# B&R Automation Studio project Panasonic_LinkaPowerCP2_A2021055 (part 2)

### IoMap.iom - 5PC900_TS17_00/IoMap.iom
```iecst
VAR_CONFIG
	Cyclic#1.P1_Pracovisko.IN.ModulWeidmuller_IO_KomOK AT %IX."P1_IOmodul_PowerlinkMaster".ModuleOk;
	Cyclic#1.P1_Pracovisko.IN.Robot_KomOK AT %IX."P1_Robot_IRB120_R1".ModuleOk;
	Cyclic#1.P1_Pracovisko.IN.Skrutkovacka_K30_KomOK AT %IX."P1_SkrutkovackaK30".ModuleOk;
	Cyclic#1.P1_Pracovisko.IN.Skrutkovacka_M5_KomOK AT %IX."P1_SkrutkovackaM5".ModuleOk;
	Cyclic#1.P1_Pracovisko.IN.Skrutkovacka_M4_KomOK AT %IX."P1_SkrutkovackaM4".ModuleOk;
	Cyclic#1.P1_Pracovisko.IN.ModulFesto_IO_KomOK AT %IX."P1_IOmaster".ModuleOk;
	Cyclic#1.::P1_Pracovisko.IN.SmartKamera3_KomOK AT %IX."P1_CAM_3".ModuleOk;
	Cyclic#1.P1_Pracovisko.IN.SmartKamera5_KomOK AT %IX."P1_CAM_5".ModuleOk;
	Cyclic#1.P1_Pracovisko.COM_Weidmuller.AB1_2_8DI AT %IB."P1_IOmodul_PowerlinkMaster".DigitalInput_I6000_S01;
	Cyclic#1.P1_Pracovisko.COM_Weidmuller.AB1_3_8DI AT %IB."P1_IOmodul_PowerlinkMaster".DigitalInput_I6000_S02;
	Cyclic#1.P1_Pracovisko.COM_Weidmuller.AB1_4_8DI AT %IB."P1_IOmodul_PowerlinkMaster".DigitalInput_I6000_S03;
	Cyclic#1.P1_Pracovisko.COM_Weidmuller.AB1_5_8DI AT %IB."P1_IOmodul_PowerlinkMaster".DigitalInput_I6000_S04;
	Cyclic#1.P1_Pracovisko.COM_Weidmuller.AB1_6_8DO AT %QB."P1_IOmodul_PowerlinkMaster".DigitalOutput_I6200_S01;
	Cyclic#1.P1_Pracovisko.COM_Weidmuller.AB1_7_8DO AT %QB."P1_IOmodul_PowerlinkMaster".DigitalOutput_I6200_S02;
	Cyclic#1.P1_Pracovisko.COM_Weidmuller.AB1_9_8DO AT %QB."P1_IOmodul_PowerlinkMaster".DigitalOutput_I6200_S03;
	Cyclic#1.P1_Pracovisko.COM_Weidmuller.AB1_10_8DO AT %QB."P1_IOmodul_PowerlinkMaster".DigitalOutput_I6200_S04;
	Cyclic#1.P1_Pracovisko.COM_Festo.DS1_1_Port0_IN[0] AT %IB."P1_IOmaster".Module007_Inputs001;
	Cyclic#1.P1_Pracovisko.COM_Festo.DS1_1_Port0_IN[1] AT %IB."P1_IOmaster".Module007_Inputs002;
	Cyclic#1.P1_Pracovisko.COM_Festo.DM1_1_4DI[0] AT %IX."P1_IOmaster".Module001_Bit_0_Bit_0;
	Cyclic#1.P1_Pracovisko.COM_Festo.DM1_1_4DI[1] AT %IX."P1_IOmaster".Module001_Bit_1_Bit_1;
	Cyclic#1.P1_Pracovisko.COM_Festo.DM1_1_4DI[2] AT %IX."P1_IOmaster".Module001_Bit_2_Bit_2;
	Cyclic#1.P1_Pracovisko.COM_Festo.DM1_1_4DI[3] AT %IX."P1_IOmaster".Module001_Bit_3_Bit_3;
	Cyclic#1.P1_Pracovisko.COM_Festo.DM1_1_4DO[0] AT %QX."P1_IOmaster".Module001_Bit_0_Bit_1;
	Cyclic#1.P1_Pracovisko.COM_Festo.DM1_1_4DO[1] AT %QX."P1_IOmaster".Module001_Bit_1_Bit_2;
	Cyclic#1.P1_Pracovisko.COM_Festo.DM1_1_4DO[2] AT %QX."P1_IOmaster".Module001_Bit_2_Bit_3;
	Cyclic#1.P1_Pracovisko.COM_Festo.DM1_1_4DO[3] AT %QX."P1_IOmaster".Module001_Bit_3_Bit_4;
	Cyclic#1.P1_Pracovisko.COM_Festo.DI1_1_8DI[0] AT %IX."P1_IOmaster".Module002_Bit_0_Bit_0;
	Cyclic#1.P1_Pracovisko.COM_Festo.DI1_1_8DI[1] AT %IX."P1_IOmaster".Module002_Bit_1_Bit_1;
	Cyclic#1.P1_Pracovisko.COM_Festo.DI1_1_8DI[2] AT %IX."P1_IOmaster".Module002_Bit_2_Bit_2;
	Cyclic#1.P1_Pracovisko.COM_Festo.DI1_1_8DI[3] AT %IX."P1_IOmaster".Module002_Bit_3_Bit_3;
	Cyclic#1.P1_Pracovisko.COM_Festo.DI1_1_8DI[4] AT %IX."P1_IOmaster".Module002_Bit_4_Bit_4;
	Cyclic#1.P1_Pracovisko.COM_Festo.DI1_1_8DI[5] AT %IX."P1_IOmaster".Module002_Bit_5_Bit_5;
	Cyclic#1.P1_Pracovisko.COM_Festo.DI1_1_8DI[6] AT %IX."P1_IOmaster".Module002_Bit_6_Bit_6;
	Cyclic#1.P1_Pracovisko.COM_Festo.DI1_1_8DI[7] AT %IX."P1_IOmaster".Module002_Bit_7_Bit_7;
	Cyclic#1.P1_Pracovisko.COM_Festo.DI1_5_8DI[0] AT %IX."P1_IOmaster".Module003_Bit_0_Bit_0;
	Cyclic#1.P1_Pracovisko.COM_Festo.DI1_5_8DI[1] AT %IX."P1_IOmaster".Module003_Bit_1_Bit_1;
	Cyclic#1.P1_Pracovisko.COM_Festo.DI1_5_8DI[2] AT %IX."P1_IOmaster".Module003_Bit_2_Bit_2;
	Cyclic#1.P1_Pracovisko.COM_Festo.DI1_5_8DI[3] AT %IX."P1_IOmaster".Module003_Bit_3_Bit_3;
	Cyclic#1.P1_Pracovisko.COM_Festo.DI1_5_8DI[4] AT %IX."P1_IOmaster".Module003_Bit_4_Bit_4;
	Cyclic#1.P1_Pracovisko.COM_Festo.DI1_5_8DI[5] AT %IX."P1_IOmaster".Module003_Bit_5_Bit_5;
	Cyclic#1.P1_Pracovisko.COM_Festo.DI1_5_8DI[6] AT %IX."P1_IOmaster".Module003_Bit_6_Bit_6;
	Cyclic#1.P1_Pracovisko.COM_Festo.DI1_5_8DI[7] AT %IX."P1_IOmaster".Module003_Bit_7_Bit_7;
	Cyclic#1.P1_Pracovisko.COM_Festo.DI1_3_8DI[0] AT %IX."P1_IOmaster".Module004_Bit_0_Bit_0;
	Cyclic#1.P1_Pracovisko.COM_Festo.DI1_3_8DI[1] AT %IX."P1_IOmaster".Module004_Bit_1_Bit_1;
	Cyclic#1.P1_Pracovisko.COM_Festo.DI1_3_8DI[2] AT %IX."P1_IOmaster".Module004_Bit_2_Bit_2;
	Cyclic#1.P1_Pracovisko.COM_Festo.DI1_3_8DI[3] AT %IX."P1_IOmaster".Module004_Bit_3_Bit_3;
	Cyclic#1.P1_Pracovisko.COM_Festo.DI1_3_8DI[4] AT %IX."P1_IOmaster".Module004_Bit_4_Bit_4;
	Cyclic#1.P1_Pracovisko.COM_Festo.DI1_3_8DI[5] AT %IX."P1_IOmaster".Module004_Bit_5_Bit_5;
	Cyclic#1.P1_Pracovisko.COM_Festo.DI1_3_8DI[6] AT %IX."P1_IOmaster".Module004_Bit_6_Bit_6;
	Cyclic#1.P1_Pracovisko.COM_Festo.DI1_3_8DI[7] AT %IX."P1_IOmaster".Module004_Bit_7_Bit_7;
	Cyclic#1.P1_Pracovisko.COM_Festo.DI1_4_8DI[0] AT %IX."P1_IOmaster".Module005_Bit_0_Bit_0;
	Cyclic#1.P1_Pracovisko.COM_Festo.DI1_4_8DI[1] AT %IX."P1_IOmaster".Module005_Bit_1_Bit_1;
	Cyclic#1.P1_Pracovisko.COM_Festo.DI1_4_8DI[2] AT %IX."P1_IOmaster".Module005_Bit_2_Bit_2;
	Cyclic#1.P1_Pracovisko.COM_Festo.DI1_4_8DI[3] AT %IX."P1_IOmaster".Module005_Bit_3_Bit_3;
	Cyclic#1.P1_Pracovisko.COM_Festo.DI1_4_8DI[4] AT %IX."P1_IOmaster".Module005_Bit_4_Bit_4;
	Cyclic#1.P1_Pracovisko.COM_Festo.DI1_4_8DI[5] AT %IX."P1_IOmaster".Module005_Bit_5_Bit_5;
	Cyclic#1.P1_Pracovisko.COM_Festo.DI1_4_8DI[6] AT %IX."P1_IOmaster".Module005_Bit_6_Bit_6;
	Cyclic#1.P1_Pracovisko.COM_Festo.DI1_4_8DI[7] AT %IX."P1_IOmaster".Module005_Bit_7_Bit_7;
	Cyclic#1.P1_Pracovisko.COM_Festo.DI1_2_8DI[0] AT %IX."P1_IOmaster".Module006_Bit_0_Bit_0;
	Cyclic#1.P1_Pracovisko.COM_Festo.DI1_2_8DI[1] AT %IX."P1_IOmaster".Module006_Bit_1_Bit_1;
	Cyclic#1.P1_Pracovisko.COM_Festo.DI1_2_8DI[2] AT %IX."P1_IOmaster".Module006_Bit_2_Bit_2;
	Cyclic#1.P1_Pracovisko.COM_Festo.DI1_2_8DI[3] AT %IX."P1_IOmaster".Module006_Bit_3_Bit_3;
	Cyclic#1.P1_Pracovisko.COM_Festo.DI1_2_8DI[4] AT %IX."P1_IOmaster".Module006_Bit_4_Bit_4;
	Cyclic#1.P1_Pracovisko.COM_Festo.DI1_2_8DI[5] AT %IX."P1_IOmaster".Module006_Bit_5_Bit_5;
	Cyclic#1.P1_Pracovisko.COM_Festo.DI1_2_8DI[6] AT %IX."P1_IOmaster".Module006_Bit_6_Bit_6;
	Cyclic#1.P1_Pracovisko.COM_Festo.DI1_2_8DI[7] AT %IX."P1_IOmaster".Module006_Bit_7_Bit_7;
	Cyclic#1.P1_Pracovisko.COM_Festo.DS1_1_Port0_OUT[0] AT %QB."P1_IOmaster".Module007_Outputs001;
	Cyclic#1.P1_Pracovisko.COM_Festo.DS1_1_Port0_OUT[1] AT %QB."P1_IOmaster".Module007_Outputs002;
	Cyclic#1.P1_Pracovisko.COM_Festo.DS1_1_Port1_IN[0] AT %IB."P1_IOmaster".Module007_Inputs003;
	Cyclic#1.P1_Pracovisko.COM_Festo.DS1_1_Port1_IN[1] AT %IB."P1_IOmaster".Module007_Inputs004;
	Cyclic#1.P1_Pracovisko.COM_Festo.DS1_1_Port1_IN[2] AT %IB."P1_IOmaster".Module007_Inputs005;
	Cyclic#1.P1_Pracovisko.COM_Festo.DS1_1_Port1_IN[3] AT %IB."P1_IOmaster".Module007_Inputs006;
	Cyclic#1.P1_Pracovisko.COM_Festo.DS1_1_Port1_IN[4] AT %IB."P1_IOmaster".Module007_Inputs007;
	Cyclic#1.P1_Pracovisko.COM_Festo.DS1_1_Port1_IN[5] AT %IB."P1_IOmaster".Module007_Inputs008;
	Cyclic#1.P1_Pracovisko.COM_Festo.DS1_1_Port1_IN[6] AT %IB."P1_IOmaster".Module007_Inputs009;
	Cyclic#1.P1_Pracovisko.COM_Festo.DS1_1_Port1_IN[7] AT %IB."P1_IOmaster".Module007_Inputs010;
	Cyclic#1.P1_Pracovisko.COM_Festo.DS1_1_Port1_IN[8] AT %IB."P1_IOmaster".Module007_Inputs011;
	Cyclic#1.P1_Pracovisko.COM_Festo.DS1_1_Port1_IN[9] AT %IB."P1_IOmaster".Module007_Inputs012;
	Cyclic#1.P1_Pracovisko.COM_Festo.DS1_1_Port1_IN[10] AT %IB."P1_IOmaster".Module007_Inputs013;
	Cyclic#1.P1_Pracovisko.COM_Festo.DS1_1_Port1_IN[11] AT %IB."P1_IOmaster".Module007_Inputs014;
	Cyclic#1.P1_Pracovisko.COM_Festo.DS1_1_Port1_IN[12] AT %IB."P1_IOmaster".Module007_Inputs015;
	Cyclic#1.P1_Pracovisko.COM_Festo.DS1_1_Port1_IN[13] AT %IB."P1_IOmaster".Module007_Inputs016;
	Cyclic#1.P1_Pracovisko.COM_Festo.DS1_1_Port1_IN[14] AT %IB."P1_IOmaster".Module007_Inputs017;
	Cyclic#1.P1_Pracovisko.COM_Festo.DS1_1_Port1_IN[15] AT %IB."P1_IOmaster".Module007_Inputs018;
	Cyclic#1.P1_Pracovisko.COM_Festo.DS1_1_Port1_OUT[0] AT %QB."P1_IOmaster".Module007_Outputs003;
	Cyclic#1.P1_Pracovisko.COM_Festo.DS1_1_Port1_OUT[1] AT %QB."P1_IOmaster".Module007_Outputs004;
	Cyclic#1.P1_Pracovisko.COM_Festo.DS1_1_Port1_OUT[2] AT %QB."P1_IOmaster".Module007_Outputs005;
	Cyclic#1.P1_Pracovisko.COM_Festo.DS1_1_Port1_OUT[3] AT %QB."P1_IOmaster".Module007_Outputs006;
	Cyclic#1.P1_Pracovisko.COM_Festo.DS1_1_Port1_OUT[4] AT %QB."P1_IOmaster".Module007_Outputs007;
	Cyclic#1.P1_Pracovisko.COM_Festo.DS1_1_Port1_OUT[5] AT %QB."P1_IOmaster".Module007_Outputs008;
	Cyclic#1.P1_Pracovisko.COM_Festo.DS1_1_Port1_OUT[6] AT %QB."P1_IOmaster".Module007_Outputs009;
	Cyclic#1.P1_Pracovisko.COM_Festo.DS1_1_Port1_OUT[7] AT %QB."P1_IOmaster".Module007_Outputs010;
	Cyclic#1.P1_Pracovisko.COM_Festo.DS1_1_Port1_OUT[8] AT %QB."P1_IOmaster".Module007_Outputs011;
	Cyclic#1.P1_Pracovisko.COM_Festo.DS1_1_Port1_OUT[9] AT %QB."P1_IOmaster".Module007_Outputs012;
	Cyclic#1.P1_Pracovisko.COM_Festo.DS1_1_Port1_OUT[10] AT %QB."P1_IOmaster".Module007_Outputs013;
	Cyclic#1.P1_Pracovisko.COM_Festo.DS1_1_Port1_OUT[11] AT %QB."P1_IOmaster".Module007_Outputs014;
	Cyclic#1.P1_Pracovisko.COM_Festo.DS1_1_Port1_OUT[12] AT %QB."P1_IOmaster".Module007_Outputs015;
	Cyclic#1.P1_Pracovisko.COM_Festo.DS1_1_Port1_OUT[13] AT %QB."P1_IOmaster".Module007_Outputs016;
	Cyclic#1.P1_Pracovisko.COM_Festo.DS1_1_Port1_OUT[14] AT %QB."P1_IOmaster".Module007_Outputs017;
	Cyclic#1.P1_Pracovisko.COM_Festo.DS1_1_Port1_OUT[15] AT %QB."P1_IOmaster".Module007_Outputs018;
	Cyclic#1.P1_Pracovisko.COM_Festo.DS1_1_Port2_IN[0] AT %IB."P1_IOmaster".Module007_Inputs019;
	Cyclic#1.P1_Pracovisko.COM_Festo.DS1_1_Port2_IN[1] AT %IB."P1_IOmaster".Module007_Inputs020;
	Cyclic#1.P1_Pracovisko.COM_Festo.DS1_1_Port2_IN[2] AT %IB."P1_IOmaster".Module007_Inputs021;
	Cyclic#1.P1_Pracovisko.COM_Festo.DS1_1_Port2_IN[3] AT %IB."P1_IOmaster".Module007_Inputs022;
	Cyclic#1.P1_Pracovisko.COM_Festo.DS1_1_Port2_IN[4] AT %IB."P1_IOmaster".Module007_Inputs023;
	Cyclic#1.P1_Pracovisko.COM_Festo.DS1_1_Port2_IN[5] AT %IB."P1_IOmaster".Module007_Inputs024;
	Cyclic#1.P1_Pracovisko.COM_Festo.DS1_1_Port2_IN[6] AT %IB."P1_IOmaster".Module007_Inputs025;
	Cyclic#1.P1_Pracovisko.COM_Festo.DS1_1_Port2_IN[7] AT %IB."P1_IOmaster".Module007_Inputs026;
	Cyclic#1.P1_Pracovisko.COM_Festo.DS1_1_Port2_IN[8] AT %IB."P1_IOmaster".Module007_Inputs027;
	Cyclic#1.P1_Pracovisko.COM_Festo.DS1_1_Port2_IN[9] AT %IB."P1_IOmaster".Module007_Inputs028;
	Cyclic#1.P1_Pracovisko.COM_Festo.DS1_1_Port2_IN[10] AT %IB."P1_IOmaster".Module007_Inputs029;
	Cyclic#1.P1_Pracovisko.COM_Festo.DS1_1_Port2_IN[11] AT %IB."P1_IOmaster".Module007_Inputs030;
	Cyclic#1.P1_Pracovisko.COM_Festo.DS1_1_Port2_IN[12] AT %IB."P1_IOmaster".Module007_Inputs031;
	Cyclic#1.P1_Pracovisko.COM_Festo.DS1_1_Port2_IN[13] AT %IB."P1_IOmaster".Module007_Inputs032;
	Cyclic#1.P1_Pracovisko.COM_Festo.DS1_1_Port2_IN[14] AT %IB."P1_IOmaster".Module007_Inputs033;
	Cyclic#1.P1_Pracovisko.COM_Festo.DS1_1_Port2_IN[15] AT %IB."P1_IOmaster".Module007_Inputs034;
	Cyclic#1.P1_Pracovisko.COM_Festo.DS1_1_Port2_IN[16] AT %IB."P1_IOmaster".Module007_Inputs035;
	Cyclic#1.P1_Pracovisko.COM_Festo.DS1_1_Port2_IN[17] AT %IB."P1_IOmaster".Module007_Inputs036;
	Cyclic#1.P1_Pracovisko.COM_Festo.DS1_1_Port2_IN[18] AT %IB."P1_IOmaster".Module007_Inputs037;
	Cyclic#1.P1_Pracovisko.COM_Festo.DS1_1_Port2_IN[19] AT %IB."P1_IOmaster".Module007_Inputs038;
	Cyclic#1.P1_Pracovisko.COM_Festo.DS1_1_Port2_IN[20] AT %IB."P1_IOmaster".Module007_Inputs039;
	Cyclic#1.P1_Pracovisko.COM_Festo.DS1_1_Port2_IN[21] AT %IB."P1_IOmaster".Module007_Inputs040;
	Cyclic#1.P1_Pracovisko.COM_Festo.DS1_1_Port2_IN[22] AT %IB."P1_IOmaster".Module007_Inputs041;
	Cyclic#1.P1_Pracovisko.COM_Festo.DS1_1_Port2_IN[23] AT %IB."P1_IOmaster".Module007_Inputs042;
	Cyclic#1.P1_Pracovisko.COM_Festo.DS1_1_Port2_IN[24] AT %IB."P1_IOmaster".Module007_Inputs043;
	Cyclic#1.P1_Pracovisko.COM_Festo.DS1_1_Port2_IN[25] AT %IB."P1_IOmaster".Module007_Inputs044;
	Cyclic#1.P1_Pracovisko.COM_Festo.DS1_1_Port2_IN[26] AT %IB."P1_IOmaster".Module007_Inputs045;
	Cyclic#1.P1_Pracovisko.COM_Festo.DS1_1_Port2_IN[27] AT %IB."P1_IOmaster".Module007_Inputs046;
	Cyclic#1.P1_Pracovisko.COM_Festo.DS1_1_Port2_IN[28] AT %IB."P1_IOmaster".Module007_Inputs047;
	Cyclic#1.P1_Pracovisko.COM_Festo.DS1_1_Port2_IN[29] AT %IB."P1_IOmaster".Module007_Inputs048;
	Cyclic#1.P1_Pracovisko.COM_Festo.DS1_1_Port2_IN[30] AT %IB."P1_IOmaster".Module007_Inputs049;
	Cyclic#1.P1_Pracovisko.COM_Festo.DS1_1_Port2_IN[31] AT %IB."P1_IOmaster".Module007_Inputs050;
	Cyclic#1.P1_Pracovisko.COM_Festo.DS1_1_Port2_OUT[0] AT %QB."P1_IOmaster".Module007_Outputs019;
	Cyclic#1.P1_Pracovisko.COM_Festo.DS1_1_Port2_OUT[1] AT %QB."P1_IOmaster".Module007_Outputs020;
	Cyclic#1.P1_Pracovisko.COM_Festo.DS1_1_Port2_OUT[2] AT %QB."P1_IOmaster".Module007_Outputs021;
	Cyclic#1.P1_Pracovisko.COM_Festo.DS1_1_Port2_OUT[3] AT %QB."P1_IOmaster".Module007_Outputs022;
	Cyclic#1.P1_Pracovisko.COM_Festo.DS1_1_Port2_OUT[4] AT %QB."P1_IOmaster".Module007_Outputs023;
	Cyclic#1.P1_Pracovisko.COM_Festo.DS1_1_Port2_OUT[5] AT %QB."P1_IOmaster".Module007_Outputs024;
	Cyclic#1.P1_Pracovisko.COM_Festo.DS1_1_Port2_OUT[6] AT %QB."P1_IOmaster".Module007_Outputs025;
	Cyclic#1.P1_Pracovisko.COM_Festo.DS1_1_Port2_OUT[7] AT %QB."P1_IOmaster".Module007_Outputs026;
	Cyclic#1.P1_Pracovisko.COM_Festo.DS1_1_Port2_OUT[8] AT %QB."P1_IOmaster".Module007_Outputs027;
	Cyclic#1.P1_Pracovisko.COM_Festo.DS1_1_Port2_OUT[9] AT %QB."P1_IOmaster".Module007_Outputs028;
	Cyclic#1.P1_Pracovisko.COM_Festo.DS1_1_Port2_OUT[10] AT %QB."P1_IOmaster".Module007_Outputs029;
	Cyclic#1.P1_Pracovisko.COM_Festo.DS1_1_Port2_OUT[11] AT %QB."P1_IOmaster".Module007_Outputs030;
	Cyclic#1.P1_Pracovisko.COM_Festo.DS1_1_Port2_OUT[12] AT %QB."P1_IOmaster".Module007_Outputs031;
	Cyclic#1.P1_Pracovisko.COM_Festo.DS1_1_Port2_OUT[13] AT %QB."P1_IOmaster".Module007_Outputs032;
	Cyclic#1.P1_Pracovisko.COM_Festo.DS1_1_Port2_OUT[14] AT %QB."P1_IOmaster".Module007_Outputs033;
	Cyclic#1.P1_Pracovisko.COM_Festo.DS1_1_Port2_OUT[15] AT %QB."P1_IOmaster".Module007_Outputs034;
	Cyclic#1.P1_Pracovisko.COM_Festo.DS1_1_Port2_OUT[16] AT %QB."P1_IOmaster".Module007_Outputs035;
	Cyclic#1.P1_Pracovisko.COM_Festo.DS1_1_Port2_OUT[17] AT %QB."P1_IOmaster".Module007_Outputs036;
	Cyclic#1.P1_Pracovisko.COM_Festo.DS1_1_Port2_OUT[18] AT %QB."P1_IOmaster".Module007_Outputs037;
	Cyclic#1.P1_Pracovisko.COM_Festo.DS1_1_Port2_OUT[19] AT %QB."P1_IOmaster".Module007_Outputs038;
	Cyclic#1.P1_Pracovisko.COM_Festo.DS1_1_Port2_OUT[20] AT %QB."P1_IOmaster".Module007_Outputs039;
	Cyclic#1.P1_Pracovisko.COM_Festo.DS1_1_Port2_OUT[21] AT %QB."P1_IOmaster".Module007_Outputs040;
	Cyclic#1.P1_Pracovisko.COM_Festo.DS1_1_Port2_OUT[22] AT %QB."P1_IOmaster".Module007_Outputs041;
	Cyclic#1.P1_Pracovisko.COM_Festo.DS1_1_Port2_OUT[23] AT %QB."P1_IOmaster".Module007_Outputs042;
	Cyclic#1.P1_Pracovisko.COM_Festo.DS1_1_Port2_OUT[24] AT %QB."P1_IOmaster".Module007_Outputs043;
	Cyclic#1.P1_Pracovisko.COM_Festo.DS1_1_Port2_OUT[25] AT %QB."P1_IOmaster".Module007_Outputs044;
	Cyclic#1.P1_Pracovisko.COM_Festo.DS1_1_Port2_OUT[26] AT %QB."P1_IOmaster".Module007_Outputs045;
	Cyclic#1.P1_Pracovisko.COM_Festo.DS1_1_Port2_OUT[27] AT %QB."P1_IOmaster".Module007_Outputs046;
	Cyclic#1.P1_Pracovisko.COM_Festo.DS1_1_Port2_OUT[28] AT %QB."P1_IOmaster".Module007_Outputs047;
	Cyclic#1.P1_Pracovisko.COM_Festo.DS1_1_Port2_OUT[29] AT %QB."P1_IOmaster".Module007_Outputs048;
	Cyclic#1.P1_Pracovisko.COM_Festo.DS1_1_Port2_OUT[30] AT %QB."P1_IOmaster".Module007_Outputs049;
	Cyclic#1.P1_Pracovisko.COM_Festo.DS1_1_Port2_OUT[31] AT %QB."P1_IOmaster".Module007_Outputs050;
	Cyclic#1.P1_Pracovisko.COM_Festo.DS1_1_Port3_IN[0] AT %IB."P1_IOmaster".Module007_Inputs051;
	Cyclic#1.P1_Pracovisko.COM_Festo.DS1_1_Port3_IN[1] AT %IB."P1_IOmaster".Module007_Inputs052;
	Cyclic#1.P1_Pracovisko.COM_Festo.DS1_1_Port3_IN[2] AT %IB."P1_IOmaster".Module007_Inputs053;
	Cyclic#1.P1_Pracovisko.COM_Festo.DS1_1_Port3_IN[3] AT %IB."P1_IOmaster".Module007_Inputs054;
	Cyclic#1.P1_Pracovisko.COM_Festo.DS1_1_Port3_IN[4] AT %IB."P1_IOmaster".Module007_Inputs055;
	Cyclic#1.P1_Pracovisko.COM_Festo.DS1_1_Port3_IN[5] AT %IB."P1_IOmaster".Module007_Inputs056;
	Cyclic#1.P1_Pracovisko.COM_Festo.DS1_1_Port3_IN[6] AT %IB."P1_IOmaster".Module007_Inputs057;
	Cyclic#1.P1_Pracovisko.COM_Festo.DS1_1_Port3_IN[7] AT %IB."P1_IOmaster".Module007_Inputs058;
	Cyclic#1.P1_Pracovisko.COM_Festo.DS1_1_Port3_IN[8] AT %IB."P1_IOmaster".Module007_Inputs059;
	Cyclic#1.P1_Pracovisko.COM_Festo.DS1_1_Port3_IN[9] AT %IB."P1_IOmaster".Module007_Inputs060;
	Cyclic#1.P1_Pracovisko.COM_Festo.DS1_1_Port3_IN[10] AT %IB."P1_IOmaster".Module007_Inputs061;
	Cyclic#1.P1_Pracovisko.COM_Festo.DS1_1_Port3_IN[11] AT %IB."P1_IOmaster".Module007_Inputs062;
	Cyclic#1.P1_Pracovisko.COM_Festo.DS1_1_Port3_IN[12] AT %IB."P1_IOmaster".Module007_Inputs063;
	Cyclic#1.P1_Pracovisko.COM_Festo.DS1_1_Port3_IN[13] AT %IB."P1_IOmaster".Module007_Inputs064;
	Cyclic#1.P1_Pracovisko.COM_Festo.DS1_1_Port3_IN[14] AT %IB."P1_IOmaster".Module007_Inputs065;
	Cyclic#1.P1_Pracovisko.COM_Festo.DS1_1_Port3_IN[15] AT %IB."P1_IOmaster".Module007_Inputs066;
	Cyclic#1.P1_Pracovisko.COM_Festo.DS1_1_Port3_IN[16] AT %IB."P1_IOmaster".Module007_Inputs067;
	Cyclic#1.P1_Pracovisko.COM_Festo.DS1_1_Port3_IN[17] AT %IB."P1_IOmaster".Module007_Inputs068;
	Cyclic#1.P1_Pracovisko.COM_Festo.DS1_1_Port3_IN[18] AT %IB."P1_IOmaster".Module007_Inputs069;
	Cyclic#1.P1_Pracovisko.COM_Festo.DS1_1_Port3_IN[19] AT %IB."P1_IOmaster".Module007_Inputs070;
	Cyclic#1.P1_Pracovisko.COM_Festo.DS1_1_Port3_IN[20] AT %IB."P1_IOmaster".Module007_Inputs071;
	Cyclic#1.P1_Pracovisko.COM_Festo.DS1_1_Port3_IN[21] AT %IB."P1_IOmaster".Module007_Inputs072;
	Cyclic#1.P1_Pracovisko.COM_Festo.DS1_1_Port3_IN[22] AT %IB."P1_IOmaster".Module007_Inputs073;
	Cyclic#1.P1_Pracovisko.COM_Festo.DS1_1_Port3_IN[23] AT %IB."P1_IOmaster".Module007_Inputs074;
	Cyclic#1.P1_Pracovisko.COM_Festo.DS1_1_Port3_IN[24] AT %IB."P1_IOmaster".Module007_Inputs075;
	Cyclic#1.P1_Pracovisko.COM_Festo.DS1_1_Port3_IN[25] AT %IB."P1_IOmaster".Module007_Inputs076;
	Cyclic#1.P1_Pracovisko.COM_Festo.DS1_1_Port3_IN[26] AT %IB."P1_IOmaster".Module007_Inputs077;
	Cyclic#1.P1_Pracovisko.COM_Festo.DS1_1_Port3_IN[27] AT %IB."P1_IOmaster".Module007_Inputs078;
	Cyclic#1.P1_Pracovisko.COM_Festo.DS1_1_Port3_IN[28] AT %IB."P1_IOmaster".Module007_Inputs079;
	Cyclic#1.P1_Pracovisko.COM_Festo.DS1_1_Port3_IN[29] AT %IB."P1_IOmaster".Module007_Inputs080;
	Cyclic#1.P1_Pracovisko.COM_Festo.DS1_1_Port3_IN[30] AT %IB."P1_IOmaster".Module007_Inputs081;
	Cyclic#1.P1_Pracovisko.COM_Festo.DS1_1_Port3_IN[31] AT %IB."P1_IOmaster".Module007_Inputs082;
	Cyclic#1.P1_Pracovisko.COM_Festo.DS1_1_Port3_OUT[0] AT %QB."P1_IOmaster".Module007_Outputs051;
	Cyclic#1.P1_Pracovisko.COM_Festo.DS1_1_Port3_OUT[1] AT %QB."P1_IOmaster".Module007_Outputs052;
	Cyclic#1.P1_Pracovisko.COM_Festo.DS1_1_Port3_OUT[2] AT %QB."P1_IOmaster".Module007_Outputs053;
	Cyclic#1.P1_Pracovisko.COM_Festo.DS1_1_Port3_OUT[3] AT %QB."P1_IOmaster".Module007_Outputs054;
	Cyclic#1.P1_Pracovisko.COM_Festo.DS1_1_Port3_OUT[4] AT %QB."P1_IOmaster".Module007_Outputs055;
	Cyclic#1.P1_Pracovisko.COM_Festo.DS1_1_Port3_OUT[5] AT %QB."P1_IOmaster".Module007_Outputs056;
	Cyclic#1.P1_Pracovisko.COM_Festo.DS1_1_Port3_OUT[6] AT %QB."P1_IOmaster".Module007_Outputs057;
	Cyclic#1.P1_Pracovisko.COM_Festo.DS1_1_Port3_OUT[7] AT %QB."P1_IOmaster".Module007_Outputs058;
	Cyclic#1.P1_Pracovisko.COM_Festo.DS1_1_Port3_OUT[8] AT %QB."P1_IOmaster".Module007_Outputs059;
	Cyclic#1.P1_Pracovisko.COM_Festo.DS1_1_Port3_OUT[9] AT %QB."P1_IOmaster".Module007_Outputs060;
	Cyclic#1.P1_Pracovisko.COM_Festo.DS1_1_Port3_OUT[10] AT %QB."P1_IOmaster".Module007_Outputs061;
	Cyclic#1.P1_Pracovisko.COM_Festo.DS1_1_Port3_OUT[11] AT %QB."P1_IOmaster".Module007_Outputs062;
	Cyclic#1.P1_Pracovisko.COM_Festo.DS1_1_Port3_OUT[12] AT %QB."P1_IOmaster".Module007_Outputs063;
	Cyclic#1.P1_Pracovisko.COM_Festo.DS1_1_Port3_OUT[13] AT %QB."P1_IOmaster".Module007_Outputs064;
	Cyclic#1.P1_Pracovisko.COM_Festo.DS1_1_Port3_OUT[14] AT %QB."P1_IOmaster".Module007_Outputs065;
	Cyclic#1.P1_Pracovisko.COM_Festo.DS1_1_Port3_OUT[15] AT %QB."P1_IOmaster".Module007_Outputs066;
	Cyclic#1.P1_Pracovisko.COM_Festo.DS1_1_Port3_OUT[16] AT %QB."P1_IOmaster".Module007_Outputs067;
	Cyclic#1.P1_Pracovisko.COM_Festo.DS1_1_Port3_OUT[17] AT %QB."P1_IOmaster".Module007_Outputs068;
	Cyclic#1.P1_Pracovisko.COM_Festo.DS1_1_Port3_OUT[18] AT %QB."P1_IOmaster".Module007_Outputs069;
	Cyclic#1.P1_Pracovisko.COM_Festo.DS1_1_Port3_OUT[19] AT %QB."P1_IOmaster".Module007_Outputs070;
	Cyclic#1.P1_Pracovisko.COM_Festo.DS1_1_Port3_OUT[20] AT %QB."P1_IOmaster".Module007_Outputs071;
	Cyclic#1.P1_Pracovisko.COM_Festo.DS1_1_Port3_OUT[21] AT %QB."P1_IOmaster".Module007_Outputs072;
	Cyclic#1.P1_Pracovisko.COM_Festo.DS1_1_Port3_OUT[22] AT %QB."P1_IOmaster".Module007_Outputs073;
	Cyclic#1.P1_Pracovisko.COM_Festo.DS1_1_Port3_OUT[23] AT %QB."P1_IOmaster".Module007_Outputs074;
	Cyclic#1.P1_Pracovisko.COM_Festo.DS1_1_Port3_OUT[24] AT %QB."P1_IOmaster".Module007_Outputs075;
	Cyclic#1.P1_Pracovisko.COM_Festo.DS1_1_Port3_OUT[25] AT %QB."P1_IOmaster".Module007_Outputs076;
	Cyclic#1.P1_Pracovisko.COM_Festo.DS1_1_Port3_OUT[26] AT %QB."P1_IOmaster".Module007_Outputs077;
	Cyclic#1.P1_Pracovisko.COM_Festo.DS1_1_Port3_OUT[27] AT %QB."P1_IOmaster".Module007_Outputs078;
	Cyclic#1.P1_Pracovisko.COM_Festo.DS1_1_Port3_OUT[28] AT %QB."P1_IOmaster".Module007_Outputs079;
	Cyclic#1.P1_Pracovisko.COM_Festo.DS1_1_Port3_OUT[29] AT %QB."P1_IOmaster".Module007_Outputs080;
	Cyclic#1.P1_Pracovisko.COM_Festo.DS1_1_Port3_OUT[30] AT %QB."P1_IOmaster".Module007_Outputs081;
	Cyclic#1.P1_Pracovisko.COM_Festo.DS1_1_Port3_OUT[31] AT %QB."P1_IOmaster".Module007_Outputs082;
	Cyclic#1.P1_Pracovisko.COM_Festo.DS1_2_Port0_IN[0] AT %IB."P1_IOmaster".Module008_Inputs001;
	Cyclic#1.P1_Pracovisko.COM_Festo.DS1_2_Port0_IN[1] AT %IB."P1_IOmaster".Module008_Inputs002;
	Cyclic#1.P1_Pracovisko.COM_Festo.DS1_2_Port0_OUT[0] AT %QB."P1_IOmaster".Module008_Outputs001;
	Cyclic#1.P1_Pracovisko.COM_Festo.DS1_2_Port0_OUT[1] AT %QB."P1_IOmaster".Module008_Outputs002;
	Cyclic#1.P3_Pracovisko.IN.ModulWeidmuller_IO_KomOK AT %IX."P3_IOmodul_PowerlinkMaster".ModuleOk;
	Cyclic#1.P3_Pracovisko.COM_Weidmuller.AB3_5_8DI AT %IB."P3_IOmodul_PowerlinkMaster".DigitalInput_I6000_S01;
	Cyclic#1.P3_Pracovisko.COM_Weidmuller.AB3_6_8DI AT %IB."P3_IOmodul_PowerlinkMaster".DigitalInput_I6000_S02;
	Cyclic#1.P3_Pracovisko.COM_Weidmuller.AB3_7_8DI AT %IB."P3_IOmodul_PowerlinkMaster".DigitalInput_I6000_S03;
	Cyclic#1.P3_Pracovisko.COM_Weidmuller.AB3_8_8DI AT %IB."P3_IOmodul_PowerlinkMaster".DigitalInput_I6000_S04;
	Cyclic#1.P3_Pracovisko.COM_Weidmuller.AB3_9_8DO AT %QB."P3_IOmodul_PowerlinkMaster".DigitalOutput_I6200_S01;
	Cyclic#1.P3_Pracovisko.COM_Weidmuller.AB3_10_8DO AT %QB."P3_IOmodul_PowerlinkMaster".DigitalOutput_I6200_S02;
	Cyclic#1.P3_Pracovisko.COM_Weidmuller.AB3_12_8DO AT %QB."P3_IOmodul_PowerlinkMaster".DigitalOutput_I6200_S03;
	Cyclic#1.P1_Robot.COM_IN.BYTE_IN[0] AT %IB."P1_Robot_IRB120_R1".Module001_Input_0;
	Cyclic#1.P1_Robot.COM_IN.BYTE_IN[1] AT %IB."P1_Robot_IRB120_R1".Module001_Input_1;
	Cyclic#1.P1_Robot.COM_IN.BYTE_IN[2] AT %IB."P1_Robot_IRB120_R1".Module001_Input_2;
	Cyclic#1.P1_Robot.COM_IN.BYTE_IN[3] AT %IB."P1_Robot_IRB120_R1".Module001_Input_3;
	Cyclic#1.P1_Robot.COM_IN.BYTE_IN[4] AT %IB."P1_Robot_IRB120_R1".Module001_Input_4;
	Cyclic#1.P1_Robot.COM_IN.BYTE_IN[5] AT %IB."P1_Robot_IRB120_R1".Module001_Input_5;
	Cyclic#1.P1_Robot.COM_IN.BYTE_IN[6] AT %IB."P1_Robot_IRB120_R1".Module001_Input_6;
	Cyclic#1.P1_Robot.COM_IN.BYTE_IN[7] AT %IB."P1_Robot_IRB120_R1".Module001_Input_7;
	Cyclic#1.P1_Robot.COM_IN.BYTE_IN[8] AT %IB."P1_Robot_IRB120_R1".Module001_Input_8;
	Cyclic#1.P1_Robot.COM_IN.BYTE_IN[9] AT %IB."P1_Robot_IRB120_R1".Module001_Input_9;
	Cyclic#1.P1_Robot.COM_IN.BYTE_IN[10] AT %IB."P1_Robot_IRB120_R1".Module001_Input_10;
	Cyclic#1.P1_Robot.COM_IN.BYTE_IN[11] AT %IB."P1_Robot_IRB120_R1".Module001_Input_11;
	Cyclic#1.P1_Robot.COM_IN.BYTE_IN[12] AT %IB."P1_Robot_IRB120_R1".Module001_Input_12;
	Cyclic#1.P1_Robot.COM_IN.BYTE_IN[13] AT %IB."P1_Robot_IRB120_R1".Module001_Input_13;
	Cyclic#1.P1_Robot.COM_IN.BYTE_IN[14] AT %IB."P1_Robot_IRB120_R1".Module001_Input_14;
	Cyclic#1.P1_Robot.COM_IN.BYTE_IN[15] AT %IB."P1_Robot_IRB120_R1".Module001_Input_15;
	Cyclic#1.P1_Robot.COM_IN.BYTE_IN[16] AT %IB."P1_Robot_IRB120_R1".Module001_Input_16;
	Cyclic#1.P1_Robot.COM_IN.BYTE_IN[17] AT %IB."P1_Robot_IRB120_R1".Module001_Input_17;
	Cyclic#1.P1_Robot.COM_IN.BYTE_IN[18] AT %IB."P1_Robot_IRB120_R1".Module001_Input_18;
	Cyclic#1.P1_Robot.COM_IN.BYTE_IN[19] AT %IB."P1_Robot_IRB120_R1".Module001_Input_19;
	Cyclic#1.P1_Robot.COM_IN.BYTE_IN[20] AT %IB."P1_Robot_IRB120_R1".Module001_Input_20;
	Cyclic#1.P1_Robot.COM_IN.BYTE_IN[21] AT %IB."P1_Robot_IRB120_R1".Module001_Input_21;
	Cyclic#1.P1_Robot.COM_IN.BYTE_IN[22] AT %IB."P1_Robot_IRB120_R1".Module001_Input_22;
	Cyclic#1.P1_Robot.COM_IN.BYTE_IN[23] AT %IB."P1_Robot_IRB120_R1".Module001_Input_23;
	Cyclic#1.P1_Robot.COM_IN.BYTE_IN[24] AT %IB."P1_Robot_IRB120_R1".Module001_Input_24;
	Cyclic#1.P1_Robot.COM_IN.BYTE_IN[25] AT %IB."P1_Robot_IRB120_R1".Module001_Input_25;
	Cyclic#1.P1_Robot.COM_IN.BYTE_IN[26] AT %IB."P1_Robot_IRB120_R1".Module001_Input_26;
	Cyclic#1.P1_Robot.COM_IN.BYTE_IN[27] AT %IB."P1_Robot_IRB120_R1".Module001_Input_27;
	Cyclic#1.P1_Robot.COM_IN.BYTE_IN[28] AT %IB."P1_Robot_IRB120_R1".Module001_Input_28;
	Cyclic#1.P1_Robot.COM_IN.BYTE_IN[29] AT %IB."P1_Robot_IRB120_R1".Module001_Input_29;
	Cyclic#1.P1_Robot.COM_IN.BYTE_IN[30] AT %IB."P1_Robot_IRB120_R1".Module001_Input_30;
	Cyclic#1.P1_Robot.COM_IN.BYTE_IN[31] AT %IB."P1_Robot_IRB120_R1".Module001_Input_31;
	Cyclic#1.P1_Robot.COM_IN.BYTE_IN[32] AT %IB."P1_Robot_IRB120_R1".Module001_Input_32;
	Cyclic#1.P1_Robot.COM_IN.BYTE_IN[33] AT %IB."P1_Robot_IRB120_R1".Module001_Input_33;
	Cyclic#1.P1_Robot.COM_IN.BYTE_IN[34] AT %IB."P1_Robot_IRB120_R1".Module001_Input_34;
	Cyclic#1.P1_Robot.COM_IN.BYTE_IN[35] AT %IB."P1_Robot_IRB120_R1".Module001_Input_35;
	Cyclic#1.P1_Robot.COM_IN.BYTE_IN[36] AT %IB."P1_Robot_IRB120_R1".Module001_Input_36;
	Cyclic#1.P1_Robot.COM_IN.BYTE_IN[37] AT %IB."P1_Robot_IRB120_R1".Module001_Input_37;
	Cyclic#1.P1_Robot.COM_IN.BYTE_IN[38] AT %IB."P1_Robot_IRB120_R1".Module001_Input_38;
	Cyclic#1.P1_Robot.COM_IN.BYTE_IN[39] AT %IB."P1_Robot_IRB120_R1".Module001_Input_39;
	Cyclic#1.P1_Robot.COM_IN.BYTE_IN[40] AT %IB."P1_Robot_IRB120_R1".Module001_Input_40;
	Cyclic#1.P1_Robot.COM_IN.BYTE_IN[41] AT %IB."P1_Robot_IRB120_R1".Module001_Input_41;
	Cyclic#1.P1_Robot.COM_IN.BYTE_IN[42] AT %IB."P1_Robot_IRB120_R1".Module001_Input_42;
	Cyclic#1.P1_Robot.COM_IN.BYTE_IN[43] AT %IB."P1_Robot_IRB120_R1".Module001_Input_43;
	Cyclic#1.P1_Robot.COM_IN.BYTE_IN[44] AT %IB."P1_Robot_IRB120_R1".Module001_Input_44;
	Cyclic#1.P1_Robot.COM_IN.BYTE_IN[45] AT %IB."P1_Robot_IRB120_R1".Module001_Input_45;
	Cyclic#1.P1_Robot.COM_IN.BYTE_IN[46] AT %IB."P1_Robot_IRB120_R1".Module001_Input_46;
	Cyclic#1.P1_Robot.COM_IN.BYTE_IN[47] AT %IB."P1_Robot_IRB120_R1".Module001_Input_47;
	Cyclic#1.P1_Robot.COM_IN.BYTE_IN[48] AT %IB."P1_Robot_IRB120_R1".Module001_Input_48;
	Cyclic#1.P1_Robot.COM_IN.BYTE_IN[49] AT %IB."P1_Robot_IRB120_R1".Module001_Input_49;
	Cyclic#1.P1_Robot.COM_IN.BYTE_IN[50] AT %IB."P1_Robot_IRB120_R1".Module001_Input_50;
	Cyclic#1.P1_Robot.COM_IN.BYTE_IN[51] AT %IB."P1_Robot_IRB120_R1".Module001_Input_51;
	Cyclic#1.P1_Robot.COM_IN.BYTE_IN[52] AT %IB."P1_Robot_IRB120_R1".Module001_Input_52;
	Cyclic#1.P1_Robot.COM_IN.BYTE_IN[53] AT %IB."P1_Robot_IRB120_R1".Module001_Input_53;
	Cyclic#1.P1_Robot.COM_IN.BYTE_IN[54] AT %IB."P1_Robot_IRB120_R1".Module001_Input_54;
	Cyclic#1.P1_Robot.COM_IN.BYTE_IN[55] AT %IB."P1_Robot_IRB120_R1".Module001_Input_55;
	Cyclic#1.P1_Robot.COM_IN.BYTE_IN[56] AT %IB."P1_Robot_IRB120_R1".Module001_Input_56;
	Cyclic#1.P1_Robot.COM_IN.BYTE_IN[57] AT %IB."P1_Robot_IRB120_R1".Module001_Input_57;
	Cyclic#1.P1_Robot.COM_IN.BYTE_IN[58] AT %IB."P1_Robot_IRB120_R1".Module001_Input_58;
	Cyclic#1.P1_Robot.COM_IN.BYTE_IN[59] AT %IB."P1_Robot_IRB120_R1".Module001_Input_59;
	Cyclic#1.P1_Robot.COM_IN.BYTE_IN[60] AT %IB."P1_Robot_IRB120_R1".Module001_Input_60;
	Cyclic#1.P1_Robot.COM_IN.BYTE_IN[61] AT %IB."P1_Robot_IRB120_R1".Module001_Input_61;
	Cyclic#1.P1_Robot.COM_IN.BYTE_IN[62] AT %IB."P1_Robot_IRB120_R1".Module001_Input_62;
	Cyclic#1.P1_Robot.COM_IN.BYTE_IN[63] AT %IB."P1_Robot_IRB120_R1".Module001_Input_63;
	Cyclic#1.P1_Robot.COM_OUT.BYTE_OUT[0] AT %QB."P1_Robot_IRB120_R1".Module002_Output_0;
	Cyclic#1.P1_Robot.COM_OUT.BYTE_OUT[1] AT %QB."P1_Robot_IRB120_R1".Module002_Output_1;
	Cyclic#1.P1_Robot.COM_OUT.BYTE_OUT[2] AT %QB."P1_Robot_IRB120_R1".Module002_Output_2;
	Cyclic#1.P1_Robot.COM_OUT.BYTE_OUT[3] AT %QB."P1_Robot_IRB120_R1".Module002_Output_3;
	Cyclic#1.P1_Robot.COM_OUT.BYTE_OUT[4] AT %QB."P1_Robot_IRB120_R1".Module002_Output_4;
	Cyclic#1.P1_Robot.COM_OUT.BYTE_OUT[5] AT %QB."P1_Robot_IRB120_R1".Module002_Output_5;
	Cyclic#1.P1_Robot.COM_OUT.BYTE_OUT[6] AT %QB."P1_Robot_IRB120_R1".Module002_Output_6;
	Cyclic#1.P1_Robot.COM_OUT.BYTE_OUT[7] AT %QB."P1_Robot_IRB120_R1".Module002_Output_7;
	Cyclic#1.P1_Robot.COM_OUT.BYTE_OUT[8] AT %QB."P1_Robot_IRB120_R1".Module002_Output_8;
	Cyclic#1.P1_Robot.COM_OUT.BYTE_OUT[9] AT %QB."P1_Robot_IRB120_R1".Module002_Output_9;
	Cyclic#1.P1_Robot.COM_OUT.BYTE_OUT[10] AT %QB."P1_Robot_IRB120_R1".Module002_Output_10;
	Cyclic#1.P1_Robot.COM_OUT.BYTE_OUT[11] AT %QB."P1_Robot_IRB120_R1".Module002_Output_11;
	Cyclic#1.P1_Robot.COM_OUT.BYTE_OUT[12] AT %QB."P1_Robot_IRB120_R1".Module002_Output_12;
	Cyclic#1.P1_Robot.COM_OUT.BYTE_OUT[13] AT %QB."P1_Robot_IRB120_R1".Module002_Output_13;
	Cyclic#1.P1_Robot.COM_OUT.BYTE_OUT[14] AT %QB."P1_Robot_IRB120_R1".Module002_Output_14;
	Cyclic#1.P1_Robot.COM_OUT.BYTE_OUT[15] AT %QB."P1_Robot_IRB120_R1".Module002_Output_15;
	Cyclic#1.P1_Robot.COM_OUT.BYTE_OUT[16] AT %QB."P1_Robot_IRB120_R1".Module002_Output_16;
	Cyclic#1.P1_Robot.COM_OUT.BYTE_OUT[17] AT %QB."P1_Robot_IRB120_R1".Module002_Output_17;
	Cyclic#1.P1_Robot.COM_OUT.BYTE_OUT[18] AT %QB."P1_Robot_IRB120_R1".Module002_Output_18;
	Cyclic#1.P1_Robot.COM_OUT.BYTE_OUT[19] AT %QB."P1_Robot_IRB120_R1".Module002_Output_19;
	Cyclic#1.P1_Robot.COM_OUT.BYTE_OUT[20] AT %QB."P1_Robot_IRB120_R1".Module002_Output_20;
	Cyclic#1.P1_Robot.COM_OUT.BYTE_OUT[21] AT %QB."P1_Robot_IRB120_R1".Module002_Output_21;
	Cyclic#1.P1_Robot.COM_OUT.BYTE_OUT[22] AT %QB."P1_Robot_IRB120_R1".Module002_Output_22;
	Cyclic#1.P1_Robot.COM_OUT.BYTE_OUT[23] AT %QB."P1_Robot_IRB120_R1".Module002_Output_23;
	Cyclic#1.P1_Robot.COM_OUT.BYTE_OUT[24] AT %QB."P1_Robot_IRB120_R1".Module002_Output_24;
	Cyclic#1.P1_Robot.COM_OUT.BYTE_OUT[25] AT %QB."P1_Robot_IRB120_R1".Module002_Output_25;
	Cyclic#1.P1_Robot.COM_OUT.BYTE_OUT[26] AT %QB."P1_Robot_IRB120_R1".Module002_Output_26;
	Cyclic#1.P1_Robot.COM_OUT.BYTE_OUT[27] AT %QB."P1_Robot_IRB120_R1".Module002_Output_27;
	Cyclic#1.P1_Robot.COM_OUT.BYTE_OUT[28] AT %QB."P1_Robot_IRB120_R1".Module002_Output_28;
	Cyclic#1.P1_Robot.COM_OUT.BYTE_OUT[29] AT %QB."P1_Robot_IRB120_R1".Module002_Output_29;
	Cyclic#1.P1_Robot.COM_OUT.BYTE_OUT[30] AT %QB."P1_Robot_IRB120_R1".Module002_Output_30;
	Cyclic#1.P1_Robot.COM_OUT.BYTE_OUT[31] AT %QB."P1_Robot_IRB120_R1".Module002_Output_31;
	Cyclic#1.P1_Robot.COM_OUT.BYTE_OUT[32] AT %QB."P1_Robot_IRB120_R1".Module002_Output_32;
	Cyclic#1.P1_Robot.COM_OUT.BYTE_OUT[33] AT %QB."P1_Robot_IRB120_R1".Module002_Output_33;
	Cyclic#1.P1_Robot.COM_OUT.BYTE_OUT[34] AT %QB."P1_Robot_IRB120_R1".Module002_Output_34;
	Cyclic#1.P1_Robot.COM_OUT.BYTE_OUT[35] AT %QB."P1_Robot_IRB120_R1".Module002_Output_35;
	Cyclic#1.P1_Robot.COM_OUT.BYTE_OUT[36] AT %QB."P1_Robot_IRB120_R1".Module002_Output_36;
	Cyclic#1.P1_Robot.COM_OUT.BYTE_OUT[37] AT %QB."P1_Robot_IRB120_R1".Module002_Output_37;
	Cyclic#1.P1_Robot.COM_OUT.BYTE_OUT[38] AT %QB."P1_Robot_IRB120_R1".Module002_Output_38;
	Cyclic#1.P1_Robot.COM_OUT.BYTE_OUT[39] AT %QB."P1_Robot_IRB120_R1".Module002_Output_39;
	Cyclic#1.P1_Robot.COM_OUT.BYTE_OUT[40] AT %QB."P1_Robot_IRB120_R1".Module002_Output_40;
	Cyclic#1.P1_Robot.COM_OUT.BYTE_OUT[41] AT %QB."P1_Robot_IRB120_R1".Module002_Output_41;
	Cyclic#1.P1_Robot.COM_OUT.BYTE_OUT[42] AT %QB."P1_Robot_IRB120_R1".Module002_Output_42;
	Cyclic#1.P1_Robot.COM_OUT.BYTE_OUT[43] AT %QB."P1_Robot_IRB120_R1".Module002_Output_43;
	Cyclic#1.P1_Robot.COM_OUT.BYTE_OUT[44] AT %QB."P1_Robot_IRB120_R1".Module002_Output_44;
	Cyclic#1.P1_Robot.COM_OUT.BYTE_OUT[45] AT %QB."P1_Robot_IRB120_R1".Module002_Output_45;
	Cyclic#1.P1_Robot.COM_OUT.BYTE_OUT[46] AT %QB."P1_Robot_IRB120_R1".Module002_Output_46;
	Cyclic#1.P1_Robot.COM_OUT.BYTE_OUT[47] AT %QB."P1_Robot_IRB120_R1".Module002_Output_47;
	Cyclic#1.P1_Robot.COM_OUT.BYTE_OUT[48] AT %QB."P1_Robot_IRB120_R1".Module002_Output_48;
	Cyclic#1.P1_Robot.COM_OUT.BYTE_OUT[49] AT %QB."P1_Robot_IRB120_R1".Module002_Output_49;
	Cyclic#1.P1_Robot.COM_OUT.BYTE_OUT[50] AT %QB."P1_Robot_IRB120_R1".Module002_Output_50;
	Cyclic#1.P1_Robot.COM_OUT.BYTE_OUT[51] AT %QB."P1_Robot_IRB120_R1".Module002_Output_51;
	Cyclic#1.P1_Robot.COM_OUT.BYTE_OUT[52] AT %QB."P1_Robot_IRB120_R1".Module002_Output_52;
	Cyclic#1.P1_Robot.COM_OUT.BYTE_OUT[53] AT %QB."P1_Robot_IRB120_R1".Module002_Output_53;
	Cyclic#1.P1_Robot.COM_OUT.BYTE_OUT[54] AT %QB."P1_Robot_IRB120_R1".Module002_Output_54;
	Cyclic#1.P1_Robot.COM_OUT.BYTE_OUT[55] AT %QB."P1_Robot_IRB120_R1".Module002_Output_55;
	Cyclic#1.P1_Robot.COM_OUT.BYTE_OUT[56] AT %QB."P1_Robot_IRB120_R1".Module002_Output_56;
	Cyclic#1.P1_Robot.COM_OUT.BYTE_OUT[57] AT %QB."P1_Robot_IRB120_R1".Module002_Output_57;
	Cyclic#1.P1_Robot.COM_OUT.BYTE_OUT[58] AT %QB."P1_Robot_IRB120_R1".Module002_Output_58;
	Cyclic#1.P1_Robot.COM_OUT.BYTE_OUT[59] AT %QB."P1_Robot_IRB120_R1".Module002_Output_59;
	Cyclic#1.P1_Robot.COM_OUT.BYTE_OUT[60] AT %QB."P1_Robot_IRB120_R1".Module002_Output_60;
	Cyclic#1.P1_Robot.COM_OUT.BYTE_OUT[61] AT %QB."P1_Robot_IRB120_R1".Module002_Output_61;
	Cyclic#1.P1_Robot.COM_OUT.BYTE_OUT[62] AT %QB."P1_Robot_IRB120_R1".Module002_Output_62;
	Cyclic#1.P1_Robot.COM_OUT.BYTE_OUT[63] AT %QB."P1_Robot_IRB120_R1".Module002_Output_63;
	Cyclic#1.P1_Srobovanie.PAR.K30_AtlasCopcoInputs[0] AT %ID."P1_SkrutkovackaK30".Module001_Input_I_00;
	Cyclic#1.P1_Srobovanie.PAR.K30_AtlasCopcoInputs[1] AT %ID."P1_SkrutkovackaK30".Module001_Input_I_01;
	Cyclic#1.P1_Srobovanie.PAR.K30_AtlasCopcoInputs[2] AT %ID."P1_SkrutkovackaK30".Module002_Input_I_00;
	Cyclic#1.P1_Srobovanie.PAR.K30_AtlasCopcoInputs[3] AT %ID."P1_SkrutkovackaK30".Module002_Input_I_01;
	Cyclic#1.P1_Srobovanie.PAR.K30_AtlasCopcoInputs[4] AT %ID."P1_SkrutkovackaK30".Module003_Input_I_00;
	Cyclic#1.P1_Srobovanie.PAR.K30_AtlasCopcoInputs[5] AT %ID."P1_SkrutkovackaK30".Module003_Input_I_01;
	Cyclic#1.P1_Srobovanie.PAR.K30_AtlasCopcoInputs[6] AT %ID."P1_SkrutkovackaK30".Module004_Input_I_00;
	Cyclic#1.P1_Srobovanie.PAR.K30_AtlasCopcoInputs[7] AT %ID."P1_SkrutkovackaK30".Module004_Input_I_01;
	Cyclic#1.P1_Srobovanie.PAR.K30_AtlasCopcoOutputs[0] AT %QD."P1_SkrutkovackaK30".Module005_Output_O_00;
	Cyclic#1.P1_Srobovanie.PAR.K30_AtlasCopcoOutputs[1] AT %QD."P1_SkrutkovackaK30".Module005_Output_O_01;
	Cyclic#1.P1_Srobovanie.PAR.K30_AtlasCopcoOutputs[2] AT %QD."P1_SkrutkovackaK30".Module006_Output_O_00;
	Cyclic#1.P1_Srobovanie.PAR.K30_AtlasCopcoOutputs[3] AT %QD."P1_SkrutkovackaK30".Module006_Output_O_01;
	Cyclic#1.P1_Srobovanie.PAR.K30_AtlasCopcoOutputs[4] AT %QD."P1_SkrutkovackaK30".Module007_Output_O_00;
	Cyclic#1.P1_Srobovanie.PAR.K30_AtlasCopcoOutputs[5] AT %QD."P1_SkrutkovackaK30".Module007_Output_O_01;
	Cyclic#1.P1_Srobovanie.PAR.K30_AtlasCopcoOutputs[6] AT %QD."P1_SkrutkovackaK30".Module008_Output_O_00;
	Cyclic#1.P1_Srobovanie.PAR.K30_AtlasCopcoOutputs[7] AT %QD."P1_SkrutkovackaK30".Module008_Output_O_01;
	Cyclic#1.P1_Srobovanie.PAR.M5_AtlasCopcoInputs[0] AT %ID."P1_SkrutkovackaM5".Module001_Input_I_00;
	Cyclic#1.P1_Srobovanie.PAR.M5_AtlasCopcoInputs[1] AT %ID."P1_SkrutkovackaM5".Module001_Input_I_01;
	Cyclic#1.P1_Srobovanie.PAR.M5_AtlasCopcoInputs[2] AT %ID."P1_SkrutkovackaM5".Module002_Input_I_00;
	Cyclic#1.P1_Srobovanie.PAR.M5_AtlasCopcoInputs[3] AT %ID."P1_SkrutkovackaM5".Module002_Input_I_01;
	Cyclic#1.P1_Srobovanie.PAR.M5_AtlasCopcoInputs[4] AT %ID."P1_SkrutkovackaM5".Module003_Input_I_00;
	Cyclic#1.P1_Srobovanie.PAR.M5_AtlasCopcoInputs[5] AT %ID."P1_SkrutkovackaM5".Module003_Input_I_01;
	Cyclic#1.P1_Srobovanie.PAR.M5_AtlasCopcoInputs[6] AT %ID."P1_SkrutkovackaM5".Module004_Input_I_00;
	Cyclic#1.P1_Srobovanie.PAR.M5_AtlasCopcoInputs[7] AT %ID."P1_SkrutkovackaM5".Module004_Input_I_01;
	Cyclic#1.P1_Srobovanie.PAR.M5_AtlasCopcoOutputs[0] AT %QD."P1_SkrutkovackaM5".Module005_Output_O_00;
	Cyclic#1.P1_Srobovanie.PAR.M5_AtlasCopcoOutputs[1] AT %QD."P1_SkrutkovackaM5".Module005_Output_O_01;
	Cyclic#1.P1_Srobovanie.PAR.M5_AtlasCopcoOutputs[2] AT %QD."P1_SkrutkovackaM5".Module006_Output_O_00;
	Cyclic#1.P1_Srobovanie.PAR.M5_AtlasCopcoOutputs[3] AT %QD."P1_SkrutkovackaM5".Module006_Output_O_01;
	Cyclic#1.P1_Srobovanie.PAR.M5_AtlasCopcoOutputs[4] AT %QD."P1_SkrutkovackaM5".Module007_Output_O_00;
	Cyclic#1.P1_Srobovanie.PAR.M5_AtlasCopcoOutputs[5] AT %QD."P1_SkrutkovackaM5".Module007_Output_O_01;
	Cyclic#1.P1_Srobovanie.PAR.M5_AtlasCopcoOutputs[6] AT %QD."P1_SkrutkovackaM5".Module008_Output_O_00;
	Cyclic#1.P1_Srobovanie.PAR.M5_AtlasCopcoOutputs[7] AT %QD."P1_SkrutkovackaM5".Module008_Output_O_01;
	Cyclic#1.P1_Srobovanie.PAR.M4_AtlasCopcoInputs[0] AT %ID."P1_SkrutkovackaM4".Module001_Input_I_00;
	Cyclic#1.P1_Srobovanie.PAR.M4_AtlasCopcoInputs[1] AT %ID."P1_SkrutkovackaM4".Module001_Input_I_01;
	Cyclic#1.P1_Srobovanie.PAR.M4_AtlasCopcoInputs[2] AT %ID."P1_SkrutkovackaM4".Module002_Input_I_00;
	Cyclic#1.P1_Srobovanie.PAR.M4_AtlasCopcoInputs[3] AT %ID."P1_SkrutkovackaM4".Module002_Input_I_01;
	Cyclic#1.P1_Srobovanie.PAR.M4_AtlasCopcoInputs[4] AT %ID."P1_SkrutkovackaM4".Module003_Input_I_00;
	Cyclic#1.P1_Srobovanie.PAR.M4_AtlasCopcoInputs[5] AT %ID."P1_SkrutkovackaM4".Module003_Input_I_01;
	Cyclic#1.P1_Srobovanie.PAR.M4_AtlasCopcoInputs[6] AT %ID."P1_SkrutkovackaM4".Module004_Input_I_00;
	Cyclic#1.P1_Srobovanie.PAR.M4_AtlasCopcoInputs[7] AT %ID."P1_SkrutkovackaM4".Module004_Input_I_01;
	Cyclic#1.P1_Srobovanie.PAR.M4_AtlasCopcoOutputs[0] AT %QD."P1_SkrutkovackaM4".Module005_Output_O_00;
	Cyclic#1.P1_Srobovanie.PAR.M4_AtlasCopcoOutputs[1] AT %QD."P1_SkrutkovackaM4".Module005_Output_O_01;
	Cyclic#1.P1_Srobovanie.PAR.M4_AtlasCopcoOutputs[2] AT %QD."P1_SkrutkovackaM4".Module006_Output_O_00;
	Cyclic#1.P1_Srobovanie.PAR.M4_AtlasCopcoOutputs[3] AT %QD."P1_SkrutkovackaM4".Module006_Output_O_01;
	Cyclic#1.P1_Srobovanie.PAR.M4_AtlasCopcoOutputs[4] AT %QD."P1_SkrutkovackaM4".Module007_Output_O_00;
	Cyclic#1.P1_Srobovanie.PAR.M4_AtlasCopcoOutputs[5] AT %QD."P1_SkrutkovackaM4".Module007_Output_O_01;
	Cyclic#1.P1_Srobovanie.PAR.M4_AtlasCopcoOutputs[6] AT %QD."P1_SkrutkovackaM4".Module008_Output_O_00;
	Cyclic#1.P1_Srobovanie.PAR.M4_AtlasCopcoOutputs[7] AT %QD."P1_SkrutkovackaM4".Module008_Output_O_01;
	Cyclic#1.P3_Pracovisko.IN.Skrutkovacka_K40_KomOK AT %IX."P3_SkrutkovackaK40".ModuleOk;
	Cyclic#1.P3_Pracovisko.IN.Skrutkovacka_M5_KomOK AT %IX."P3_SkrutkovackaM5".ModuleOk;
	Cyclic#1.P3_Srobovanie.PAR.K40_AtlasCopcoInputs[0] AT %ID."P3_SkrutkovackaK40".Module001_Input_I_00;
	Cyclic#1.P3_Srobovanie.PAR.K40_AtlasCopcoInputs[1] AT %ID."P3_SkrutkovackaK40".Module001_Input_I_01;
	Cyclic#1.P3_Srobovanie.PAR.K40_AtlasCopcoInputs[2] AT %ID."P3_SkrutkovackaK40".Module002_Input_I_00;
	Cyclic#1.P3_Srobovanie.PAR.K40_AtlasCopcoInputs[3] AT %ID."P3_SkrutkovackaK40".Module002_Input_I_01;
	Cyclic#1.P3_Srobovanie.PAR.K40_AtlasCopcoInputs[4] AT %ID."P3_SkrutkovackaK40".Module003_Input_I_00;
	Cyclic#1.P3_Srobovanie.PAR.K40_AtlasCopcoInputs[5] AT %ID."P3_SkrutkovackaK40".Module003_Input_I_01;
	Cyclic#1.P3_Srobovanie.PAR.K40_AtlasCopcoInputs[6] AT %ID."P3_SkrutkovackaK40".Module004_Input_I_00;
	Cyclic#1.P3_Srobovanie.PAR.K40_AtlasCopcoInputs[7] AT %ID."P3_SkrutkovackaK40".Module004_Input_I_01;
	Cyclic#1.P3_Srobovanie.PAR.K40_AtlasCopcoOutputs[0] AT %QD."P3_SkrutkovackaK40".Module005_Output_O_00;
	Cyclic#1.P3_Srobovanie.PAR.K40_AtlasCopcoOutputs[1] AT %QD."P3_SkrutkovackaK40".Module005_Output_O_01;
	Cyclic#1.P3_Srobovanie.PAR.K40_AtlasCopcoOutputs[2] AT %QD."P3_SkrutkovackaK40".Module006_Output_O_00;
	Cyclic#1.P3_Srobovanie.PAR.K40_AtlasCopcoOutputs[3] AT %QD."P3_SkrutkovackaK40".Module006_Output_O_01;
	Cyclic#1.P3_Srobovanie.PAR.K40_AtlasCopcoOutputs[4] AT %QD."P3_SkrutkovackaK40".Module007_Output_O_00;
	Cyclic#1.P3_Srobovanie.PAR.K40_AtlasCopcoOutputs[5] AT %QD."P3_SkrutkovackaK40".Module007_Output_O_01;
	Cyclic#1.P3_Srobovanie.PAR.K40_AtlasCopcoOutputs[6] AT %QD."P3_SkrutkovackaK40".Module008_Output_O_00;
	Cyclic#1.P3_Srobovanie.PAR.K40_AtlasCopcoOutputs[7] AT %QD."P3_SkrutkovackaK40".Module008_Output_O_01;
	Cyclic#1.P3_Srobovanie.PAR.M5_AtlasCopcoInputs[0] AT %ID."P3_SkrutkovackaM5".Module001_Input_I_00;
	Cyclic#1.P3_Srobovanie.PAR.M5_AtlasCopcoInputs[1] AT %ID."P3_SkrutkovackaM5".Module001_Input_I_01;
	Cyclic#1.P3_Srobovanie.PAR.M5_AtlasCopcoInputs[2] AT %ID."P3_SkrutkovackaM5".Module002_Input_I_00;
	Cyclic#1.P3_Srobovanie.PAR.M5_AtlasCopcoInputs[3] AT %ID."P3_SkrutkovackaM5".Module002_Input_I_01;
	Cyclic#1.P3_Srobovanie.PAR.M5_AtlasCopcoInputs[4] AT %ID."P3_SkrutkovackaM5".Module003_Input_I_00;
	Cyclic#1.P3_Srobovanie.PAR.M5_AtlasCopcoInputs[5] AT %ID."P3_SkrutkovackaM5".Module003_Input_I_01;
	Cyclic#1.P3_Srobovanie.PAR.M5_AtlasCopcoInputs[6] AT %ID."P3_SkrutkovackaM5".Module004_Input_I_00;
	Cyclic#1.P3_Srobovanie.PAR.M5_AtlasCopcoInputs[7] AT %ID."P3_SkrutkovackaM5".Module004_Input_I_01;
	Cyclic#1.P3_Srobovanie.PAR.M5_AtlasCopcoOutputs[0] AT %QD."P3_SkrutkovackaM5".Module005_Output_O_00;
	Cyclic#1.P3_Srobovanie.PAR.M5_AtlasCopcoOutputs[1] AT %QD."P3_SkrutkovackaM5".Module005_Output_O_01;
	Cyclic#1.P3_Srobovanie.PAR.M5_AtlasCopcoOutputs[2] AT %QD."P3_SkrutkovackaM5".Module006_Output_O_00;
	Cyclic#1.P3_Srobovanie.PAR.M5_AtlasCopcoOutputs[3] AT %QD."P3_SkrutkovackaM5".Module006_Output_O_01;
	Cyclic#1.P3_Srobovanie.PAR.M5_AtlasCopcoOutputs[4] AT %QD."P3_SkrutkovackaM5".Module007_Output_O_00;
	Cyclic#1.P3_Srobovanie.PAR.M5_AtlasCopcoOutputs[5] AT %QD."P3_SkrutkovackaM5".Module007_Output_O_01;
	Cyclic#1.P3_Srobovanie.PAR.M5_AtlasCopcoOutputs[6] AT %QD."P3_SkrutkovackaM5".Module008_Output_O_00;
	Cyclic#1.P3_Srobovanie.PAR.M5_AtlasCopcoOutputs[7] AT %QD."P3_SkrutkovackaM5".Module008_Output_O_01;
	Cyclic#1.P1_Pracovisko.IN.VentilovyTerminal_KomOK AT %IX."P1_VentilovyTerminal_VT1".ModuleOk;
	Cyclic#1.P1_Pracovisko.COM_VentilovyTerminal[0] AT %QB."P1_VentilovyTerminal_VT1".ValveCoils1_8_I2000_S01;
	Cyclic#1.P1_Pracovisko.COM_VentilovyTerminal[1] AT %QB."P1_VentilovyTerminal_VT1".ValveCoils9_16_I2000_S02;
	Cyclic#1.P1_Pracovisko.COM_VentilovyTerminal[2] AT %QB."P1_VentilovyTerminal_VT1".ValveCoils17_24_I2000_S03;
	Cyclic#1.P1_Pracovisko.COM_VentilovyTerminal[3] AT %QB."P1_VentilovyTerminal_VT1".ValveCoils25_32_I2000_S04;
	Cyclic#1.P1_Pracovisko.COM_VentilovyTerminal[4] AT %QB."P1_VentilovyTerminal_VT1".ValveCoils33_40_I2000_S05;
	Cyclic#1.P1_Pracovisko.COM_VentilovyTerminal[5] AT %QB."P1_VentilovyTerminal_VT1".ValveCoils41_48_I2000_S06;
	Cyclic#1.P3_Pracovisko.IN.VentilovyTerminal_KomOK AT %IX."P3_VentilovyTerminal_VT3".ModuleOk;
	Cyclic#1.P3_Pracovisko.COM_VentilovyTerminal[0] AT %QB."P3_VentilovyTerminal_VT3".ValveCoils1_8_I2000_S01;
	Cyclic#1.P3_Pracovisko.COM_VentilovyTerminal[1] AT %QB."P3_VentilovyTerminal_VT3".ValveCoils9_16_I2000_S02;
	Cyclic#1.P3_Pracovisko.COM_VentilovyTerminal[2] AT %QB."P3_VentilovyTerminal_VT3".ValveCoils17_24_I2000_S03;
	Cyclic#1.P3_Pracovisko.COM_VentilovyTerminal[3] AT %QB."P3_VentilovyTerminal_VT3".ValveCoils25_32_I2000_S04;
	Cyclic#1.P3_Pracovisko.COM_VentilovyTerminal[4] AT %QB."P3_VentilovyTerminal_VT3".ValveCoils33_40_I2000_S05;
	Cyclic#1.P3_Pracovisko.COM_VentilovyTerminal[5] AT %QB."P3_VentilovyTerminal_VT3".ValveCoils41_48_I2000_S06;
	Cyclic#1.P1_Pracovisko.IN.ServoZdvihuVytahu_KomOK AT %IX."P1_ServoZdvihuVstupVytahu".ModuleOk;
	Cyclic#1.P1_Vytah.ServoZdvihuVytahu.IN_forMapping.Status_word_1 AT %IW."P1_ServoZdvihuVstupVytahu".Module001_Status_word_1;
	Cyclic#1.P1_Vytah.ServoZdvihuVytahu.IN_forMapping.Position_Statusword_1 AT %IW."P1_ServoZdvihuVstupVytahu".Module001_Position_Statusword_1;
	Cyclic#1.P1_Vytah.ServoZdvihuVytahu.IN_forMapping.Position_Statusword_2 AT %IW."P1_ServoZdvihuVstupVytahu".Module001_Position_Statusword_2;
	Cyclic#1.P1_Vytah.ServoZdvihuVytahu.IN_forMapping.Status_word_2 AT %IW."P1_ServoZdvihuVstupVytahu".Module001_Status_word_2;
	Cyclic#1.P1_Vytah.ServoZdvihuVytahu.IN_forMapping.Report_word AT %IW."P1_ServoZdvihuVstupVytahu".Module001_Report_word;
	Cyclic#1.P1_Vytah.ServoZdvihuVytahu.IN_forMapping.Position_actual_value_A AT %ID."P1_ServoZdvihuVstupVytahu".Module001_Position_actual_value_A;
	Cyclic#1.P1_Vytah.ServoZdvihuVytahu.IN_forMapping.Speed_actual_value_B AT %ID."P1_ServoZdvihuVstupVytahu".Module001_Speed_actual_value_B;
	Cyclic#1.P1_Vytah.ServoZdvihuVytahu.IN_forMapping.Fault_Code AT %IW."P1_ServoZdvihuVstupVytahu".Module001_Fault_Code;
	Cyclic#1.P1_Vytah.ServoZdvihuVytahu.IN_forMapping.Warn_Code AT %IW."P1_ServoZdvihuVstupVytahu".Module001_Warn_Code;
	Cyclic#1.P1_Vytah.ServoZdvihuVytahu.IN_forMapping.User AT %IW."P1_ServoZdvihuVstupVytahu".Module001_User;
	Cyclic#1.P1_Vytah.ServoZdvihuVytahu.IN_forMapping.Status_word_or_actual_value_0 AT %IW."P1_ServoZdvihuVstupVytahu".Module001_Status_word_or_actual_value_I_00;
	Cyclic#1.P1_Vytah.ServoZdvihuVytahu.IN_forMapping.Status_word_or_actual_value_1 AT %IW."P1_ServoZdvihuVstupVytahu".Module001_Status_word_or_actual_value_I_01;
	Cyclic#1.P1_Vytah.ServoZdvihuVytahu.IN_forMapping.Status_word_or_actual_value_2 AT %IW."P1_ServoZdvihuVstupVytahu".Module001_Status_word_or_actual_value_I_02;
	Cyclic#1.P1_Vytah.ServoZdvihuVytahu.IN_forMapping.Status_word_or_actual_value_3 AT %IW."P1_ServoZdvihuVstupVytahu".Module001_Status_word_or_actual_value_I_03;
	Cyclic#1.P1_Vytah.ServoZdvihuVytahu.IN_forMapping.Status_word_or_actual_value_4 AT %IW."P1_ServoZdvihuVstupVytahu".Module001_Status_word_or_actual_value_I_04;
	Cyclic#1.P1_Vytah.ServoZdvihuVytahu.IN_forMapping.Status_word_or_actual_value_5 AT %IW."P1_ServoZdvihuVstupVytahu".Module001_Status_word_or_actual_value_I_05;
	Cyclic#1.P1_Vytah.ServoZdvihuVytahu.IN_forMapping.Status_word_or_actual_value_6 AT %IW."P1_ServoZdvihuVstupVytahu".Module001_Status_word_or_actual_value_I_06;
	Cyclic#1.P1_Vytah.ServoZdvihuVytahu.IN_forMapping.Status_word_or_actual_value_7 AT %IW."P1_ServoZdvihuVstupVytahu".Module001_Status_word_or_actual_value_I_07;
	Cyclic#1.P1_Vytah.ServoZdvihuVytahu.IN_forMapping.Status_word_or_actual_value_8 AT %IW."P1_ServoZdvihuVstupVytahu".Module001_Status_word_or_actual_value_I_08;
	Cyclic#1.P1_Vytah.ServoZdvihuVytahu.IN_forMapping.Status_word_or_actual_value_9 AT %IW."P1_ServoZdvihuVstupVytahu".Module001_Status_word_or_actual_value_I_09;
	Cyclic#1.P1_Vytah.ServoZdvihuVytahu.IN_forMapping.Status_word_or_actual_value_10 AT %IW."P1_ServoZdvihuVstupVytahu".Module001_Status_word_or_actual_value_I_10;
	Cyclic#1.P1_Vytah.ServoZdvihuVytahu.IN_forMapping.Status_word_or_actual_value_11 AT %IW."P1_ServoZdvihuVstupVytahu".Module001_Status_word_or_actual_value_I_11;
	Cyclic#1.P1_Vytah.ServoZdvihuVytahu.IN_forMapping.Status_word_or_actual_value_12 AT %IW."P1_ServoZdvihuVstupVytahu".Module001_Status_word_or_actual_value_I_12;
	Cyclic#1.P1_Vytah.ServoZdvihuVytahu.IN_forMapping.Status_word_or_actual_value_13 AT %IW."P1_ServoZdvihuVstupVytahu".Module001_Status_word_or_actual_value_I_13;
	Cyclic#1.P1_Vytah.ServoZdvihuVytahu.IN_forMapping.Status_word_or_actual_value_14 AT %IW."P1_ServoZdvihuVstupVytahu".Module001_Status_word_or_actual_value_I_14;
	Cyclic#1.P1_Vytah.ServoZdvihuVytahu.IN_forMapping.Status_word_or_actual_value_15 AT %IW."P1_ServoZdvihuVstupVytahu".Module001_Status_word_or_actual_value_I_15;
	Cyclic#1.P1_Vytah.ServoZdvihuVytahu.OUT_forMapping.Control_word_1 AT %QW."P1_ServoZdvihuVstupVytahu".Module001_Control_word_1;
	Cyclic#1.P1_Vytah.ServoZdvihuVytahu.OUT_forMapping.Position_Controlword_1 AT %QW."P1_ServoZdvihuVstupVytahu".Module001_Position_Controlword_1;
	Cyclic#1.P1_Vytah.ServoZdvihuVytahu.OUT_forMapping.Position_Controlword_2 AT %QW."P1_ServoZdvihuVstupVytahu".Module001_Position_Controlword_2;
	Cyclic#1.P1_Vytah.ServoZdvihuVytahu.OUT_forMapping.Control_word_2 AT %QW."P1_ServoZdvihuVstupVytahu".Module001_Control_word_2;
	Cyclic#1.P1_Vytah.ServoZdvihuVytahu.OUT_forMapping.Override AT %QW."P1_ServoZdvihuVstupVytahu".Module001_Override;
	Cyclic#1.P1_Vytah.ServoZdvihuVytahu.OUT_forMapping.MDI_target_position AT %QD."P1_ServoZdvihuVstupVytahu".Module001_MDI_target_position;
	Cyclic#1.P1_Vytah.ServoZdvihuVytahu.OUT_forMapping.MDI_velocity AT %QD."P1_ServoZdvihuVstupVytahu".Module001_MDI_velocity;
	Cyclic#1.P1_Vytah.ServoZdvihuVytahu.OUT_forMapping.MDI_acceleration AT %QW."P1_ServoZdvihuVstupVytahu".Module001_MDI_acceleartion;
	Cyclic#1.P1_Vytah.ServoZdvihuVytahu.OUT_forMapping.MDI_decceleration AT %QW."P1_ServoZdvihuVstupVytahu".Module001_MDI_deceleration;
	Cyclic#1.P1_Vytah.ServoZdvihuVytahu.OUT_forMapping.User1 AT %QW."P1_ServoZdvihuVstupVytahu".Module001_User1;
	Cyclic#1.P1_Vytah.ServoZdvihuVytahu.OUT_forMapping.Control_word_or_setpoint_0 AT %QW."P1_ServoZdvihuVstupVytahu".Module001_Control_word_or_setpoint_O_00;
	Cyclic#1.P1_Vytah.ServoZdvihuVytahu.OUT_forMapping.Control_word_or_setpoint_1 AT %QW."P1_ServoZdvihuVstupVytahu".Module001_Control_word_or_setpoint_O_01;
	Cyclic#1.P1_Vytah.ServoZdvihuVytahu.OUT_forMapping.Control_word_or_setpoint_2 AT %QW."P1_ServoZdvihuVstupVytahu".Module001_Control_word_or_setpoint_O_02;
	Cyclic#1.P1_Vytah.ServoZdvihuVytahu.OUT_forMapping.Control_word_or_setpoint_3 AT %QW."P1_ServoZdvihuVstupVytahu".Module001_Control_word_or_setpoint_O_03;
	Cyclic#1.P1_Vytah.ServoZdvihuVytahu.OUT_forMapping.Control_word_or_setpoint_4 AT %QW."P1_ServoZdvihuVstupVytahu".Module001_Control_word_or_setpoint_O_04;
	Cyclic#1.P1_Vytah.ServoZdvihuVytahu.OUT_forMapping.Control_word_or_setpoint_5 AT %QW."P1_ServoZdvihuVstupVytahu".Module001_Control_word_or_setpoint_O_05;
	Cyclic#1.P1_Vytah.ServoZdvihuVytahu.OUT_forMapping.Control_word_or_setpoint_6 AT %QW."P1_ServoZdvihuVstupVytahu".Module001_Control_word_or_setpoint_O_06;
	Cyclic#1.P1_Vytah.ServoZdvihuVytahu.OUT_forMapping.Control_word_or_setpoint_7 AT %QW."P1_ServoZdvihuVstupVytahu".Module001_Control_word_or_setpoint_O_07;
	Cyclic#1.P1_Vytah.ServoZdvihuVytahu.OUT_forMapping.Control_word_or_setpoint_8 AT %QW."P1_ServoZdvihuVstupVytahu".Module001_Control_word_or_setpoint_O_08;
	Cyclic#1.P1_Vytah.ServoZdvihuVytahu.OUT_forMapping.Control_word_or_setpoint_9 AT %QW."P1_ServoZdvihuVstupVytahu".Module001_Control_word_or_setpoint_O_09;
	Cyclic#1.P1_Vytah.ServoZdvihuVytahu.OUT_forMapping.Control_word_or_setpoint_10 AT %QW."P1_ServoZdvihuVstupVytahu".Module001_Control_word_or_setpoint_O_10;
	Cyclic#1.P1_Vytah.ServoZdvihuVytahu.OUT_forMapping.Control_word_or_setpoint_11 AT %QW."P1_ServoZdvihuVstupVytahu".Module001_Control_word_or_setpoint_O_11;
	Cyclic#1.P1_Vytah.ServoZdvihuVytahu.OUT_forMapping.Control_word_or_setpoint_12 AT %QW."P1_ServoZdvihuVstupVytahu".Module001_Control_word_or_setpoint_O_12;
	Cyclic#1.P1_Vytah.ServoZdvihuVytahu.OUT_forMapping.Control_word_or_setpoint_13 AT %QW."P1_ServoZdvihuVstupVytahu".Module001_Control_word_or_setpoint_O_13;
	Cyclic#1.P1_Vytah.ServoZdvihuVytahu.OUT_forMapping.Control_word_or_setpoint_14 AT %QW."P1_ServoZdvihuVstupVytahu".Module001_Control_word_or_setpoint_O_14;
	Cyclic#1.P1_Vytah.ServoZdvihuVytahu.OUT_forMapping.Control_word_or_setpoint_15 AT %QW."P1_ServoZdvihuVstupVytahu".Module001_Control_word_or_setpoint_O_15;
	Cyclic#1.P1_Pracovisko.IN.ServoManipulatorOsX_KomOK AT %IX."P1_ServoManipOsX".ModuleOk;
	Cyclic#1.P1_Srobovanie.ServoManipulOsX.IN_forMapping.Status_word_1 AT %IW."P1_ServoManipOsX".Module001_Status_word_1;
	Cyclic#1.P1_Srobovanie.ServoManipulOsX.IN_forMapping.Position_Statusword_1 AT %IW."P1_ServoManipOsX".Module001_Position_Statusword_1;
	Cyclic#1.P1_Srobovanie.ServoManipulOsX.IN_forMapping.Position_Statusword_2 AT %IW."P1_ServoManipOsX".Module001_Position_Statusword_2;
	Cyclic#1.P1_Srobovanie.ServoManipulOsX.IN_forMapping.Status_word_2 AT %IW."P1_ServoManipOsX".Module001_Status_word_2;
	Cyclic#1.P1_Srobovanie.ServoManipulOsX.IN_forMapping.Report_word AT %IW."P1_ServoManipOsX".Module001_Report_word;
	Cyclic#1.P1_Srobovanie.ServoManipulOsX.IN_forMapping.Position_actual_value_A AT %ID."P1_ServoManipOsX".Module001_Position_actual_value_A;
	Cyclic#1.P1_Srobovanie.ServoManipulOsX.IN_forMapping.Speed_actual_value_B AT %ID."P1_ServoManipOsX".Module001_Speed_actual_value_B;
	Cyclic#1.P1_Srobovanie.ServoManipulOsX.IN_forMapping.Fault_Code AT %IW."P1_ServoManipOsX".Module001_Fault_Code;
	Cyclic#1.P1_Srobovanie.ServoManipulOsX.IN_forMapping.Warn_Code AT %IW."P1_ServoManipOsX".Module001_Warn_Code;
	Cyclic#1.P1_Srobovanie.ServoManipulOsX.IN_forMapping.User AT %IW."P1_ServoManipOsX".Module001_User;
	Cyclic#1.P1_Srobovanie.ServoManipulOsX.IN_forMapping.Status_word_or_actual_value_0 AT %IW."P1_ServoManipOsX".Module001_Status_word_or_actual_value_I_00;
	Cyclic#1.P1_Srobovanie.ServoManipulOsX.IN_forMapping.Status_word_or_actual_value_1 AT %IW."P1_ServoManipOsX".Module001_Status_word_or_actual_value_I_01;
	Cyclic#1.P1_Srobovanie.ServoManipulOsX.IN_forMapping.Status_word_or_actual_value_2 AT %IW."P1_ServoManipOsX".Module001_Status_word_or_actual_value_I_02;
	Cyclic#1.P1_Srobovanie.ServoManipulOsX.IN_forMapping.Status_word_or_actual_value_3 AT %IW."P1_ServoManipOsX".Module001_Status_word_or_actual_value_I_03;
	Cyclic#1.P1_Srobovanie.ServoManipulOsX.IN_forMapping.Status_word_or_actual_value_4 AT %IW."P1_ServoManipOsX".Module001_Status_word_or_actual_value_I_04;
	Cyclic#1.P1_Srobovanie.ServoManipulOsX.IN_forMapping.Status_word_or_actual_value_5 AT %IW."P1_ServoManipOsX".Module001_Status_word_or_actual_value_I_05;
	Cyclic#1.P1_Srobovanie.ServoManipulOsX.IN_forMapping.Status_word_or_actual_value_6 AT %IW."P1_ServoManipOsX".Module001_Status_word_or_actual_value_I_06;
	Cyclic#1.P1_Srobovanie.ServoManipulOsX.IN_forMapping.Status_word_or_actual_value_7 AT %IW."P1_ServoManipOsX".Module001_Status_word_or_actual_value_I_07;
	Cyclic#1.P1_Srobovanie.ServoManipulOsX.IN_forMapping.Status_word_or_actual_value_8 AT %IW."P1_ServoManipOsX".Module001_Status_word_or_actual_value_I_08;
	Cyclic#1.P1_Srobovanie.ServoManipulOsX.IN_forMapping.Status_word_or_actual_value_9 AT %IW."P1_ServoManipOsX".Module001_Status_word_or_actual_value_I_09;
	Cyclic#1.P1_Srobovanie.ServoManipulOsX.IN_forMapping.Status_word_or_actual_value_10 AT %IW."P1_ServoManipOsX".Module001_Status_word_or_actual_value_I_10;
	Cyclic#1.P1_Srobovanie.ServoManipulOsX.IN_forMapping.Status_word_or_actual_value_11 AT %IW."P1_ServoManipOsX".Module001_Status_word_or_actual_value_I_11;
	Cyclic#1.P1_Srobovanie.ServoManipulOsX.IN_forMapping.Status_word_or_actual_value_12 AT %IW."P1_ServoManipOsX".Module001_Status_word_or_actual_value_I_12;
	Cyclic#1.P1_Srobovanie.ServoManipulOsX.IN_forMapping.Status_word_or_actual_value_13 AT %IW."P1_ServoManipOsX".Module001_Status_word_or_actual_value_I_13;
	Cyclic#1.P1_Srobovanie.ServoManipulOsX.IN_forMapping.Status_word_or_actual_value_14 AT %IW."P1_ServoManipOsX".Module001_Status_word_or_actual_value_I_14;
	Cyclic#1.P1_Srobovanie.ServoManipulOsX.IN_forMapping.Status_word_or_actual_value_15 AT %IW."P1_ServoManipOsX".Module001_Status_word_or_actual_value_I_15;
	Cyclic#1.P1_Srobovanie.ServoManipulOsX.OUT_forMapping.Control_word_1 AT %QW."P1_ServoManipOsX".Module001_Control_word_1;
	Cyclic#1.P1_Srobovanie.ServoManipulOsX.OUT_forMapping.Position_Controlword_1 AT %QW."P1_ServoManipOsX".Module001_Position_Controlword_1;
	Cyclic#1.P1_Srobovanie.ServoManipulOsX.OUT_forMapping.Position_Controlword_2 AT %QW."P1_ServoManipOsX".Module001_Position_Controlword_2;
	Cyclic#1.P1_Srobovanie.ServoManipulOsX.OUT_forMapping.Control_word_2 AT %QW."P1_ServoManipOsX".Module001_Control_word_2;
	Cyclic#1.P1_Srobovanie.ServoManipulOsX.OUT_forMapping.Override AT %QW."P1_ServoManipOsX".Module001_Override;
	Cyclic#1.P1_Srobovanie.ServoManipulOsX.OUT_forMapping.MDI_target_position AT %QD."P1_ServoManipOsX".Module001_MDI_target_position;
	Cyclic#1.P1_Srobovanie.ServoManipulOsX.OUT_forMapping.MDI_velocity AT %QD."P1_ServoManipOsX".Module001_MDI_velocity;
	Cyclic#1.P1_Srobovanie.ServoManipulOsX.OUT_forMapping.MDI_acceleration AT %QW."P1_ServoManipOsX".Module001_MDI_acceleartion;
	Cyclic#1.P1_Srobovanie.ServoManipulOsX.OUT_forMapping.MDI_decceleration AT %QW."P1_ServoManipOsX".Module001_MDI_deceleration;
	Cyclic#1.P1_Srobovanie.ServoManipulOsX.OUT_forMapping.User1 AT %QW."P1_ServoManipOsX".Module001_User1;
	Cyclic#1.P1_Srobovanie.ServoManipulOsX.OUT_forMapping.Control_word_or_setpoint_0 AT %QW."P1_ServoManipOsX".Module001_Control_word_or_setpoint_O_00;
	Cyclic#1.P1_Srobovanie.ServoManipulOsX.OUT_forMapping.Control_word_or_setpoint_1 AT %QW."P1_ServoManipOsX".Module001_Control_word_or_setpoint_O_01;
	Cyclic#1.P1_Srobovanie.ServoManipulOsX.OUT_forMapping.Control_word_or_setpoint_2 AT %QW."P1_ServoManipOsX".Module001_Control_word_or_setpoint_O_02;
	Cyclic#1.P1_Srobovanie.ServoManipulOsX.OUT_forMapping.Control_word_or_setpoint_3 AT %QW."P1_ServoManipOsX".Module001_Control_word_or_setpoint_O_03;
	Cyclic#1.P1_Srobovanie.ServoManipulOsX.OUT_forMapping.Control_word_or_setpoint_4 AT %QW."P1_ServoManipOsX".Module001_Control_word_or_setpoint_O_04;
	Cyclic#1.P1_Srobovanie.ServoManipulOsX.OUT_forMapping.Control_word_or_setpoint_5 AT %QW."P1_ServoManipOsX".Module001_Control_word_or_setpoint_O_05;
	Cyclic#1.P1_Srobovanie.ServoManipulOsX.OUT_forMapping.Control_word_or_setpoint_6 AT %QW."P1_ServoManipOsX".Module001_Control_word_or_setpoint_O_06;
	Cyclic#1.P1_Srobovanie.ServoManipulOsX.OUT_forMapping.Control_word_or_setpoint_7 AT %QW."P1_ServoManipOsX".Module001_Control_word_or_setpoint_O_07;
	Cyclic#1.P1_Srobovanie.ServoManipulOsX.OUT_forMapping.Control_word_or_setpoint_8 AT %QW."P1_ServoManipOsX".Module001_Control_word_or_setpoint_O_08;
	Cyclic#1.P1_Srobovanie.ServoManipulOsX.OUT_forMapping.Control_word_or_setpoint_9 AT %QW."P1_ServoManipOsX".Module001_Control_word_or_setpoint_O_09;
	Cyclic#1.P1_Srobovanie.ServoManipulOsX.OUT_forMapping.Control_word_or_setpoint_10 AT %QW."P1_ServoManipOsX".Module001_Control_word_or_setpoint_O_10;
	Cyclic#1.P1_Srobovanie.ServoManipulOsX.OUT_forMapping.Control_word_or_setpoint_11 AT %QW."P1_ServoManipOsX".Module001_Control_word_or_setpoint_O_11;
	Cyclic#1.P1_Srobovanie.ServoManipulOsX.OUT_forMapping.Control_word_or_setpoint_12 AT %QW."P1_ServoManipOsX".Module001_Control_word_or_setpoint_O_12;
	Cyclic#1.P1_Srobovanie.ServoManipulOsX.OUT_forMapping.Control_word_or_setpoint_13 AT %QW."P1_ServoManipOsX".Module001_Control_word_or_setpoint_O_13;
	Cyclic#1.P1_Srobovanie.ServoManipulOsX.OUT_forMapping.Control_word_or_setpoint_14 AT %QW."P1_ServoManipOsX".Module001_Control_word_or_setpoint_O_14;
	Cyclic#1.P1_Srobovanie.ServoManipulOsX.OUT_forMapping.Control_word_or_setpoint_15 AT %QW."P1_ServoManipOsX".Module001_Control_word_or_setpoint_O_15;
	Cyclic#1.P1_Pracovisko.IN.ServoManipulatorOsY_KomOK AT %IX."P1_ServoManipOsY".ModuleOk;
	Cyclic#1.P1_Srobovanie.ServoManipulOsY.IN_forMapping.Status_word_1 AT %IW."P1_ServoManipOsY".Module001_Status_word_1;
	Cyclic#1.P1_Srobovanie.ServoManipulOsY.IN_forMapping.Position_Statusword_1 AT %IW."P1_ServoManipOsY".Module001_Position_Statusword_1;
	Cyclic#1.P1_Srobovanie.ServoManipulOsY.IN_forMapping.Position_Statusword_2 AT %IW."P1_ServoManipOsY".Module001_Position_Statusword_2;
	Cyclic#1.P1_Srobovanie.ServoManipulOsY.IN_forMapping.Status_word_2 AT %IW."P1_ServoManipOsY".Module001_Status_word_2;
	Cyclic#1.P1_Srobovanie.ServoManipulOsY.IN_forMapping.Report_word AT %IW."P1_ServoManipOsY".Module001_Report_word;
	Cyclic#1.P1_Srobovanie.ServoManipulOsY.IN_forMapping.Position_actual_value_A AT %ID."P1_ServoManipOsY".Module001_Position_actual_value_A;
	Cyclic#1.P1_Srobovanie.ServoManipulOsY.IN_forMapping.Speed_actual_value_B AT %ID."P1_ServoManipOsY".Module001_Speed_actual_value_B;
	Cyclic#1.P1_Srobovanie.ServoManipulOsY.IN_forMapping.Fault_Code AT %IW."P1_ServoManipOsY".Module001_Fault_Code;
	Cyclic#1.P1_Srobovanie.ServoManipulOsY.IN_forMapping.Warn_Code AT %IW."P1_ServoManipOsY".Module001_Warn_Code;
	Cyclic#1.P1_Srobovanie.ServoManipulOsY.IN_forMapping.User AT %IW."P1_ServoManipOsY".Module001_User;
	Cyclic#1.P1_Srobovanie.ServoManipulOsY.IN_forMapping.Status_word_or_actual_value_0 AT %IW."P1_ServoManipOsY".Module001_Status_word_or_actual_value_I_00;
	Cyclic#1.P1_Srobovanie.ServoManipulOsY.IN_forMapping.Status_word_or_actual_value_1 AT %IW."P1_ServoManipOsY".Module001_Status_word_or_actual_value_I_01;
	Cyclic#1.P1_Srobovanie.ServoManipulOsY.IN_forMapping.Status_word_or_actual_value_2 AT %IW."P1_ServoManipOsY".Module001_Status_word_or_actual_value_I_02;
	Cyclic#1.P1_Srobovanie.ServoManipulOsY.IN_forMapping.Status_word_or_actual_value_3 AT %IW."P1_ServoManipOsY".Module001_Status_word_or_actual_value_I_03;
	Cyclic#1.P1_Srobovanie.ServoManipulOsY.IN_forMapping.Status_word_or_actual_value_4 AT %IW."P1_ServoManipOsY".Module001_Status_word_or_actual_value_I_04;
	Cyclic#1.P1_Srobovanie.ServoManipulOsY.IN_forMapping.Status_word_or_actual_value_5 AT %IW."P1_ServoManipOsY".Module001_Status_word_or_actual_value_I_05;
	Cyclic#1.P1_Srobovanie.ServoManipulOsY.IN_forMapping.Status_word_or_actual_value_6 AT %IW."P1_ServoManipOsY".Module001_Status_word_or_actual_value_I_06;
	Cyclic#1.P1_Srobovanie.ServoManipulOsY.IN_forMapping.Status_word_or_actual_value_7 AT %IW."P1_ServoManipOsY".Module001_Status_word_or_actual_value_I_07;
	Cyclic#1.P1_Srobovanie.ServoManipulOsY.IN_forMapping.Status_word_or_actual_value_8 AT %IW."P1_ServoManipOsY".Module001_Status_word_or_actual_value_I_08;
	Cyclic#1.P1_Srobovanie.ServoManipulOsY.IN_forMapping.Status_word_or_actual_value_9 AT %IW."P1_ServoManipOsY".Module001_Status_word_or_actual_value_I_09;
	Cyclic#1.P1_Srobovanie.ServoManipulOsY.IN_forMapping.Status_word_or_actual_value_10 AT %IW."P1_ServoManipOsY".Module001_Status_word_or_actual_value_I_10;
	Cyclic#1.P1_Srobovanie.ServoManipulOsY.IN_forMapping.Status_word_or_actual_value_11 AT %IW."P1_ServoManipOsY".Module001_Status_word_or_actual_value_I_11;
	Cyclic#1.P1_Srobovanie.ServoManipulOsY.IN_forMapping.Status_word_or_actual_value_12 AT %IW."P1_ServoManipOsY".Module001_Status_word_or_actual_value_I_12;
	Cyclic#1.P1_Srobovanie.ServoManipulOsY.IN_forMapping.Status_word_or_actual_value_13 AT %IW."P1_ServoManipOsY".Module001_Status_word_or_actual_value_I_13;
	Cyclic#1.P1_Srobovanie.ServoManipulOsY.IN_forMapping.Status_word_or_actual_value_14 AT %IW."P1_ServoManipOsY".Module001_Status_word_or_actual_value_I_14;
	Cyclic#1.P1_Srobovanie.ServoManipulOsY.IN_forMapping.Status_word_or_actual_value_15 AT %IW."P1_ServoManipOsY".Module001_Status_word_or_actual_value_I_15;
	Cyclic#1.P1_Srobovanie.ServoManipulOsY.OUT_forMapping.Control_word_1 AT %QW."P1_ServoManipOsY".Module001_Control_word_1;
	Cyclic#1.P1_Srobovanie.ServoManipulOsY.OUT_forMapping.Position_Controlword_1 AT %QW."P1_ServoManipOsY".Module001_Position_Controlword_1;
	Cyclic#1.P1_Srobovanie.ServoManipulOsY.OUT_forMapping.Position_Controlword_2 AT %QW."P1_ServoManipOsY".Module001_Position_Controlword_2;
	Cyclic#1.P1_Srobovanie.ServoManipulOsY.OUT_forMapping.Control_word_2 AT %QW."P1_ServoManipOsY".Module001_Control_word_2;
	Cyclic#1.P1_Srobovanie.ServoManipulOsY.OUT_forMapping.Override AT %QW."P1_ServoManipOsY".Module001_Override;
	Cyclic#1.P1_Srobovanie.ServoManipulOsY.OUT_forMapping.MDI_target_position AT %QD."P1_ServoManipOsY".Module001_MDI_target_position;
	Cyclic#1.P1_Srobovanie.ServoManipulOsY.OUT_forMapping.MDI_velocity AT %QD."P1_ServoManipOsY".Module001_MDI_velocity;
	Cyclic#1.P1_Srobovanie.ServoManipulOsY.OUT_forMapping.MDI_acceleration AT %QW."P1_ServoManipOsY".Module001_MDI_acceleartion;
	Cyclic#1.P1_Srobovanie.ServoManipulOsY.OUT_forMapping.MDI_decceleration AT %QW."P1_ServoManipOsY".Module001_MDI_deceleration;
	Cyclic#1.P1_Srobovanie.ServoManipulOsY.OUT_forMapping.User1 AT %QW."P1_ServoManipOsY".Module001_User1;
	Cyclic#1.P1_Srobovanie.ServoManipulOsY.OUT_forMapping.Control_word_or_setpoint_0 AT %QW."P1_ServoManipOsY".Module001_Control_word_or_setpoint_O_00;
	Cyclic#1.P1_Srobovanie.ServoManipulOsY.OUT_forMapping.Control_word_or_setpoint_1 AT %QW."P1_ServoManipOsY".Module001_Control_word_or_setpoint_O_01;
	Cyclic#1.P1_Srobovanie.ServoManipulOsY.OUT_forMapping.Control_word_or_setpoint_2 AT %QW."P1_ServoManipOsY".Module001_Control_word_or_setpoint_O_02;
	Cyclic#1.P1_Srobovanie.ServoManipulOsY.OUT_forMapping.Control_word_or_setpoint_3 AT %QW."P1_ServoManipOsY".Module001_Control_word_or_setpoint_O_03;
	Cyclic#1.P1_Srobovanie.ServoManipulOsY.OUT_forMapping.Control_word_or_setpoint_4 AT %QW."P1_ServoManipOsY".Module001_Control_word_or_setpoint_O_04;
	Cyclic#1.P1_Srobovanie.ServoManipulOsY.OUT_forMapping.Control_word_or_setpoint_5 AT %QW."P1_ServoManipOsY".Module001_Control_word_or_setpoint_O_05;
	Cyclic#1.P1_Srobovanie.ServoManipulOsY.OUT_forMapping.Control_word_or_setpoint_6 AT %QW."P1_ServoManipOsY".Module001_Control_word_or_setpoint_O_06;
	Cyclic#1.P1_Srobovanie.ServoManipulOsY.OUT_forMapping.Control_word_or_setpoint_7 AT %QW."P1_ServoManipOsY".Module001_Control_word_or_setpoint_O_07;
	Cyclic#1.P1_Srobovanie.ServoManipulOsY.OUT_forMapping.Control_word_or_setpoint_8 AT %QW."P1_ServoManipOsY".Module001_Control_word_or_setpoint_O_08;
	Cyclic#1.P1_Srobovanie.ServoManipulOsY.OUT_forMapping.Control_word_or_setpoint_9 AT %QW."P1_ServoManipOsY".Module001_Control_word_or_setpoint_O_09;
	Cyclic#1.P1_Srobovanie.ServoManipulOsY.OUT_forMapping.Control_word_or_setpoint_10 AT %QW."P1_ServoManipOsY".Module001_Control_word_or_setpoint_O_10;
	Cyclic#1.P1_Srobovanie.ServoManipulOsY.OUT_forMapping.Control_word_or_setpoint_11 AT %QW."P1_ServoManipOsY".Module001_Control_word_or_setpoint_O_11;
	Cyclic#1.P1_Srobovanie.ServoManipulOsY.OUT_forMapping.Control_word_or_setpoint_12 AT %QW."P1_ServoManipOsY".Module001_Control_word_or_setpoint_O_12;
	Cyclic#1.P1_Srobovanie.ServoManipulOsY.OUT_forMapping.Control_word_or_setpoint_13 AT %QW."P1_ServoManipOsY".Module001_Control_word_or_setpoint_O_13;
	Cyclic#1.P1_Srobovanie.ServoManipulOsY.OUT_forMapping.Control_word_or_setpoint_14 AT %QW."P1_ServoManipOsY".Module001_Control_word_or_setpoint_O_14;
	Cyclic#1.P1_Srobovanie.ServoManipulOsY.OUT_forMapping.Control_word_or_setpoint_15 AT %QW."P1_ServoManipOsY".Module001_Control_word_or_setpoint_O_15;
	Cyclic#1.P1_Pracovisko.IN.ServoManipulatorOsZ_M5_KomOK AT %IX."P1_ServoManipOsZ_M5".ModuleOk;
	Cyclic#1.P1_Srobovanie.ServoManipulOsZ_M5.IN_forMapping.Status_word_1 AT %IW."P1_ServoManipOsZ_M5".Module001_Status_word_1;
	Cyclic#1.P1_Srobovanie.ServoManipulOsZ_M5.IN_forMapping.Position_Statusword_1 AT %IW."P1_ServoManipOsZ_M5".Module001_Position_Statusword_1;
	Cyclic#1.P1_Srobovanie.ServoManipulOsZ_M5.IN_forMapping.Position_Statusword_2 AT %IW."P1_ServoManipOsZ_M5".Module001_Position_Statusword_2;
	Cyclic#1.P1_Srobovanie.ServoManipulOsZ_M5.IN_forMapping.Status_word_2 AT %IW."P1_ServoManipOsZ_M5".Module001_Status_word_2;
	Cyclic#1.P1_Srobovanie.ServoManipulOsZ_M5.IN_forMapping.Report_word AT %IW."P1_ServoManipOsZ_M5".Module001_Report_word;
	Cyclic#1.P1_Srobovanie.ServoManipulOsZ_M5.IN_forMapping.Position_actual_value_A AT %ID."P1_ServoManipOsZ_M5".Module001_Position_actual_value_A;
	Cyclic#1.P1_Srobovanie.ServoManipulOsZ_M5.IN_forMapping.Speed_actual_value_B AT %ID."P1_ServoManipOsZ_M5".Module001_Speed_actual_value_B;
	Cyclic#1.P1_Srobovanie.ServoManipulOsZ_M5.IN_forMapping.Fault_Code AT %IW."P1_ServoManipOsZ_M5".Module001_Fault_Code;
	Cyclic#1.P1_Srobovanie.ServoManipulOsZ_M5.IN_forMapping.Warn_Code AT %IW."P1_ServoManipOsZ_M5".Module001_Warn_Code;
	Cyclic#1.P1_Srobovanie.ServoManipulOsZ_M5.IN_forMapping.User AT %IW."P1_ServoManipOsZ_M5".Module001_User;
	Cyclic#1.P1_Srobovanie.ServoManipulOsZ_M5.IN_forMapping.Status_word_or_actual_value_0 AT %IW."P1_ServoManipOsZ_M5".Module001_Status_word_or_actual_value_I_00;
	Cyclic#1.P1_Srobovanie.ServoManipulOsZ_M5.IN_forMapping.Status_word_or_actual_value_1 AT %IW."P1_ServoManipOsZ_M5".Module001_Status_word_or_actual_value_I_01;
	Cyclic#1.P1_Srobovanie.ServoManipulOsZ_M5.IN_forMapping.Status_word_or_actual_value_2 AT %IW."P1_ServoManipOsZ_M5".Module001_Status_word_or_actual_value_I_02;
	Cyclic#1.P1_Srobovanie.ServoManipulOsZ_M5.IN_forMapping.Status_word_or_actual_value_3 AT %IW."P1_ServoManipOsZ_M5".Module001_Status_word_or_actual_value_I_03;
	Cyclic#1.P1_Srobovanie.ServoManipulOsZ_M5.IN_forMapping.Status_word_or_actual_value_4 AT %IW."P1_ServoManipOsZ_M5".Module001_Status_word_or_actual_value_I_04;
	Cyclic#1.P1_Srobovanie.ServoManipulOsZ_M5.IN_forMapping.Status_word_or_actual_value_5 AT %IW."P1_ServoManipOsZ_M5".Module001_Status_word_or_actual_value_I_05;
	Cyclic#1.P1_Srobovanie.ServoManipulOsZ_M5.IN_forMapping.Status_word_or_actual_value_6 AT %IW."P1_ServoManipOsZ_M5".Module001_Status_word_or_actual_value_I_06;
	Cyclic#1.P1_Srobovanie.ServoManipulOsZ_M5.IN_forMapping.Status_word_or_actual_value_7 AT %IW."P1_ServoManipOsZ_M5".Module001_Status_word_or_actual_value_I_07;
	Cyclic#1.P1_Srobovanie.ServoManipulOsZ_M5.IN_forMapping.Status_word_or_actual_value_8 AT %IW."P1_ServoManipOsZ_M5".Module001_Status_word_or_actual_value_I_08;
	Cyclic#1.P1_Srobovanie.ServoManipulOsZ_M5.IN_forMapping.Status_word_or_actual_value_9 AT %IW."P1_ServoManipOsZ_M5".Module001_Status_word_or_actual_value_I_09;
	Cyclic#1.P1_Srobovanie.ServoManipulOsZ_M5.IN_forMapping.Status_word_or_actual_value_10 AT %IW."P1_ServoManipOsZ_M5".Module001_Status_word_or_actual_value_I_10;
	Cyclic#1.P1_Srobovanie.ServoManipulOsZ_M5.IN_forMapping.Status_word_or_actual_value_11 AT %IW."P1_ServoManipOsZ_M5".Module001_Status_word_or_actual_value_I_11;
	Cyclic#1.P1_Srobovanie.ServoManipulOsZ_M5.IN_forMapping.Status_word_or_actual_value_12 AT %IW."P1_ServoManipOsZ_M5".Module001_Status_word_or_actual_value_I_12;
	Cyclic#1.P1_Srobovanie.ServoManipulOsZ_M5.IN_forMapping.Status_word_or_actual_value_13 AT %IW."P1_ServoManipOsZ_M5".Module001_Status_word_or_actual_value_I_13;
	Cyclic#1.P1_Srobovanie.ServoManipulOsZ_M5.IN_forMapping.Status_word_or_actual_value_14 AT %IW."P1_ServoManipOsZ_M5".Module001_Status_word_or_actual_value_I_14;
	Cyclic#1.P1_Srobovanie.ServoManipulOsZ_M5.IN_forMapping.Status_word_or_actual_value_15 AT %IW."P1_ServoManipOsZ_M5".Module001_Status_word_or_actual_value_I_15;
	Cyclic#1.P1_Srobovanie.ServoManipulOsZ_M5.OUT_forMapping.Control_word_1 AT %QW."P1_ServoManipOsZ_M5".Module001_Control_word_1;
	Cyclic#1.P1_Srobovanie.ServoManipulOsZ_M5.OUT_forMapping.Position_Controlword_1 AT %QW."P1_ServoManipOsZ_M5".Module001_Position_Controlword_1;
	Cyclic#1.P1_Srobovanie.ServoManipulOsZ_M5.OUT_forMapping.Position_Controlword_2 AT %QW."P1_ServoManipOsZ_M5".Module001_Position_Controlword_2;
	Cyclic#1.P1_Srobovanie.ServoManipulOsZ_M5.OUT_forMapping.Control_word_2 AT %QW."P1_ServoManipOsZ_M5".Module001_Control_word_2;
	Cyclic#1.P1_Srobovanie.ServoManipulOsZ_M5.OUT_forMapping.Override AT %QW."P1_ServoManipOsZ_M5".Module001_Override;
	Cyclic#1.P1_Srobovanie.ServoManipulOsZ_M5.OUT_forMapping.MDI_target_position AT %QD."P1_ServoManipOsZ_M5".Module001_MDI_target_position;
	Cyclic#1.P1_Srobovanie.ServoManipulOsZ_M5.OUT_forMapping.MDI_velocity AT %QD."P1_ServoManipOsZ_M5".Module001_MDI_velocity;
	Cyclic#1.P1_Srobovanie.ServoManipulOsZ_M5.OUT_forMapping.MDI_acceleration AT %QW."P1_ServoManipOsZ_M5".Module001_MDI_acceleartion;
	Cyclic#1.P1_Srobovanie.ServoManipulOsZ_M5.OUT_forMapping.MDI_decceleration AT %QW."P1_ServoManipOsZ_M5".Module001_MDI_deceleration;
	Cyclic#1.P1_Srobovanie.ServoManipulOsZ_M5.OUT_forMapping.User1 AT %QW."P1_ServoManipOsZ_M5".Module001_User1;
	Cyclic#1.P1_Srobovanie.ServoManipulOsZ_M5.OUT_forMapping.Control_word_or_setpoint_0 AT %QW."P1_ServoManipOsZ_M5".Module001_Control_word_or_setpoint_O_00;
	Cyclic#1.P1_Srobovanie.ServoManipulOsZ_M5.OUT_forMapping.Control_word_or_setpoint_1 AT %QW."P1_ServoManipOsZ_M5".Module001_Control_word_or_setpoint_O_01;
	Cyclic#1.P1_Srobovanie.ServoManipulOsZ_M5.OUT_forMapping.Control_word_or_setpoint_2 AT %QW."P1_ServoManipOsZ_M5".Module001_Control_word_or_setpoint_O_02;
	Cyclic#1.P1_Srobovanie.ServoManipulOsZ_M5.OUT_forMapping.Control_word_or_setpoint_3 AT %QW."P1_ServoManipOsZ_M5".Module001_Control_word_or_setpoint_O_03;
	Cyclic#1.P1_Srobovanie.ServoManipulOsZ_M5.OUT_forMapping.Control_word_or_setpoint_4 AT %QW."P1_ServoManipOsZ_M5".Module001_Control_word_or_setpoint_O_04;
	Cyclic#1.P1_Srobovanie.ServoManipulOsZ_M5.OUT_forMapping.Control_word_or_setpoint_5 AT %QW."P1_ServoManipOsZ_M5".Module001_Control_word_or_setpoint_O_05;
	Cyclic#1.P1_Srobovanie.ServoManipulOsZ_M5.OUT_forMapping.Control_word_or_setpoint_6 AT %QW."P1_ServoManipOsZ_M5".Module001_Control_word_or_setpoint_O_06;
	Cyclic#1.P1_Srobovanie.ServoManipulOsZ_M5.OUT_forMapping.Control_word_or_setpoint_7 AT %QW."P1_ServoManipOsZ_M5".Module001_Control_word_or_setpoint_O_07;
	Cyclic#1.P1_Srobovanie.ServoManipulOsZ_M5.OUT_forMapping.Control_word_or_setpoint_8 AT %QW."P1_ServoManipOsZ_M5".Module001_Control_word_or_setpoint_O_08;
	Cyclic#1.P1_Srobovanie.ServoManipulOsZ_M5.OUT_forMapping.Control_word_or_setpoint_9 AT %QW."P1_ServoManipOsZ_M5".Module001_Control_word_or_setpoint_O_09;
	Cyclic#1.P1_Srobovanie.ServoManipulOsZ_M5.OUT_forMapping.Control_word_or_setpoint_10 AT %QW."P1_ServoManipOsZ_M5".Module001_Control_word_or_setpoint_O_10;
	Cyclic#1.P1_Srobovanie.ServoManipulOsZ_M5.OUT_forMapping.Control_word_or_setpoint_11 AT %QW."P1_ServoManipOsZ_M5".Module001_Control_word_or_setpoint_O_11;
	Cyclic#1.P1_Srobovanie.ServoManipulOsZ_M5.OUT_forMapping.Control_word_or_setpoint_12 AT %QW."P1_ServoManipOsZ_M5".Module001_Control_word_or_setpoint_O_12;
	Cyclic#1.P1_Srobovanie.ServoManipulOsZ_M5.OUT_forMapping.Control_word_or_setpoint_13 AT %QW."P1_ServoManipOsZ_M5".Module001_Control_word_or_setpoint_O_13;
	Cyclic#1.P1_Srobovanie.ServoManipulOsZ_M5.OUT_forMapping.Control_word_or_setpoint_14 AT %QW."P1_ServoManipOsZ_M5".Module001_Control_word_or_setpoint_O_14;
	Cyclic#1.P1_Srobovanie.ServoManipulOsZ_M5.OUT_forMapping.Control_word_or_setpoint_15 AT %QW."P1_ServoManipOsZ_M5".Module001_Control_word_or_setpoint_O_15;
	Cyclic#1.P1_Pracovisko.IN.ServoManipulatorOsZ_M4_KomOK AT %IX."P1_ServoManipOsZ_M4".ModuleOk;
	Cyclic#1.P1_Srobovanie.ServoManipulOsZ_M4.IN_forMapping.Status_word_1 AT %IW."P1_ServoManipOsZ_M4".Module001_Status_word_1;
	Cyclic#1.P1_Srobovanie.ServoManipulOsZ_M4.IN_forMapping.Position_Statusword_1 AT %IW."P1_ServoManipOsZ_M4".Module001_Position_Statusword_1;
	Cyclic#1.P1_Srobovanie.ServoManipulOsZ_M4.IN_forMapping.Position_Statusword_2 AT %IW."P1_ServoManipOsZ_M4".Module001_Position_Statusword_2;
	Cyclic#1.P1_Srobovanie.ServoManipulOsZ_M4.IN_forMapping.Status_word_2 AT %IW."P1_ServoManipOsZ_M4".Module001_Status_word_2;
	Cyclic#1.P1_Srobovanie.ServoManipulOsZ_M4.IN_forMapping.Report_word AT %IW."P1_ServoManipOsZ_M4".Module001_Report_word;
	Cyclic#1.P1_Srobovanie.ServoManipulOsZ_M4.IN_forMapping.Position_actual_value_A AT %ID."P1_ServoManipOsZ_M4".Module001_Position_actual_value_A;
	Cyclic#1.P1_Srobovanie.ServoManipulOsZ_M4.IN_forMapping.Speed_actual_value_B AT %ID."P1_ServoManipOsZ_M4".Module001_Speed_actual_value_B;
	Cyclic#1.P1_Srobovanie.ServoManipulOsZ_M4.IN_forMapping.Fault_Code AT %IW."P1_ServoManipOsZ_M4".Module001_Fault_Code;
	Cyclic#1.P1_Srobovanie.ServoManipulOsZ_M4.IN_forMapping.Warn_Code AT %IW."P1_ServoManipOsZ_M4".Module001_Warn_Code;
	Cyclic#1.P1_Srobovanie.ServoManipulOsZ_M4.IN_forMapping.User AT %IW."P1_ServoManipOsZ_M4".Module001_User;
	Cyclic#1.P1_Srobovanie.ServoManipulOsZ_M4.IN_forMapping.Status_word_or_actual_value_0 AT %IW."P1_ServoManipOsZ_M4".Module001_Status_word_or_actual_value_I_00;
	Cyclic#1.P1_Srobovanie.ServoManipulOsZ_M4.IN_forMapping.Status_word_or_actual_value_1 AT %IW."P1_ServoManipOsZ_M4".Module001_Status_word_or_actual_value_I_01;
	Cyclic#1.P1_Srobovanie.ServoManipulOsZ_M4.IN_forMapping.Status_word_or_actual_value_2 AT %IW."P1_ServoManipOsZ_M4".Module001_Status_word_or_actual_value_I_02;
	Cyclic#1.P1_Srobovanie.ServoManipulOsZ_M4.IN_forMapping.Status_word_or_actual_value_3 AT %IW."P1_ServoManipOsZ_M4".Module001_Status_word_or_actual_value_I_03;
	Cyclic#1.P1_Srobovanie.ServoManipulOsZ_M4.IN_forMapping.Status_word_or_actual_value_4 AT %IW."P1_ServoManipOsZ_M4".Module001_Status_word_or_actual_value_I_04;
	Cyclic#1.P1_Srobovanie.ServoManipulOsZ_M4.IN_forMapping.Status_word_or_actual_value_5 AT %IW."P1_ServoManipOsZ_M4".Module001_Status_word_or_actual_value_I_05;
	Cyclic#1.P1_Srobovanie.ServoManipulOsZ_M4.IN_forMapping.Status_word_or_actual_value_6 AT %IW."P1_ServoManipOsZ_M4".Module001_Status_word_or_actual_value_I_06;
	Cyclic#1.P1_Srobovanie.ServoManipulOsZ_M4.IN_forMapping.Status_word_or_actual_value_7 AT %IW."P1_ServoManipOsZ_M4".Module001_Status_word_or_actual_value_I_07;
	Cyclic#1.P1_Srobovanie.ServoManipulOsZ_M4.IN_forMapping.Status_word_or_actual_value_8 AT %IW."P1_ServoManipOsZ_M4".Module001_Status_word_or_actual_value_I_08;
	Cyclic#1.P1_Srobovanie.ServoManipulOsZ_M4.IN_forMapping.Status_word_or_actual_value_9 AT %IW."P1_ServoManipOsZ_M4".Module001_Status_word_or_actual_value_I_09;
	Cyclic#1.P1_Srobovanie.ServoManipulOsZ_M4.IN_forMapping.Status_word_or_actual_value_10 AT %IW."P1_ServoManipOsZ_M4".Module001_Status_word_or_actual_value_I_10;
	Cyclic#1.P1_Srobovanie.ServoManipulOsZ_M4.IN_forMapping.Status_word_or_actual_value_11 AT %IW."P1_ServoManipOsZ_M4".Module001_Status_word_or_actual_value_I_11;
	Cyclic#1.P1_Srobovanie.ServoManipulOsZ_M4.IN_forMapping.Status_word_or_actual_value_12 AT %IW."P1_ServoManipOsZ_M4".Module001_Status_word_or_actual_value_I_12;
	Cyclic#1.P1_Srobovanie.ServoManipulOsZ_M4.IN_forMapping.Status_word_or_actual_value_13 AT %IW."P1_ServoManipOsZ_M4".Module001_Status_word_or_actual_value_I_13;
	Cyclic#1.P1_Srobovanie.ServoManipulOsZ_M4.IN_forMapping.Status_word_or_actual_value_14 AT %IW."P1_ServoManipOsZ_M4".Module001_Status_word_or_actual_value_I_14;
	Cyclic#1.P1_Srobovanie.ServoManipulOsZ_M4.IN_forMapping.Status_word_or_actual_value_15 AT %IW."P1_ServoManipOsZ_M4".Module001_Status_word_or_actual_value_I_15;
	Cyclic#1.P1_Srobovanie.ServoManipulOsZ_M4.OUT_forMapping.Control_word_1 AT %QW."P1_ServoManipOsZ_M4".Module001_Control_word_1;
	Cyclic#1.P1_Srobovanie.ServoManipulOsZ_M4.OUT_forMapping.Position_Controlword_1 AT %QW."P1_ServoManipOsZ_M4".Module001_Position_Controlword_1;
	Cyclic#1.P1_Srobovanie.ServoManipulOsZ_M4.OUT_forMapping.Position_Controlword_2 AT %QW."P1_ServoManipOsZ_M4".Module001_Position_Controlword_2;
	Cyclic#1.P1_Srobovanie.ServoManipulOsZ_M4.OUT_forMapping.Control_word_2 AT %QW."P1_ServoManipOsZ_M4".Module001_Control_word_2;
	Cyclic#1.P1_Srobovanie.ServoManipulOsZ_M4.OUT_forMapping.Override AT %QW."P1_ServoManipOsZ_M4".Module001_Override;
	Cyclic#1.P1_Srobovanie.ServoManipulOsZ_M4.OUT_forMapping.MDI_target_position AT %QD."P1_ServoManipOsZ_M4".Module001_MDI_target_position;
	Cyclic#1.P1_Srobovanie.ServoManipulOsZ_M4.OUT_forMapping.MDI_velocity AT %QD."P1_ServoManipOsZ_M4".Module001_MDI_velocity;
	Cyclic#1.P1_Srobovanie.ServoManipulOsZ_M4.OUT_forMapping.MDI_acceleration AT %QW."P1_ServoManipOsZ_M4".Module001_MDI_acceleartion;
	Cyclic#1.P1_Srobovanie.ServoManipulOsZ_M4.OUT_forMapping.MDI_decceleration AT %QW."P1_ServoManipOsZ_M4".Module001_MDI_deceleration;
	Cyclic#1.P1_Srobovanie.ServoManipulOsZ_M4.OUT_forMapping.User1 AT %QW."P1_ServoManipOsZ_M4".Module001_User1;
	Cyclic#1.P1_Srobovanie.ServoManipulOsZ_M4.OUT_forMapping.Control_word_or_setpoint_0 AT %QW."P1_ServoManipOsZ_M4".Module001_Control_word_or_setpoint_O_00;
	Cyclic#1.P1_Srobovanie.ServoManipulOsZ_M4.OUT_forMapping.Control_word_or_setpoint_1 AT %QW."P1_ServoManipOsZ_M4".Module001_Control_word_or_setpoint_O_01;
	Cyclic#1.P1_Srobovanie.ServoManipulOsZ_M4.OUT_forMapping.Control_word_or_setpoint_2 AT %QW."P1_ServoManipOsZ_M4".Module001_Control_word_or_setpoint_O_02;
	Cyclic#1.P1_Srobovanie.ServoManipulOsZ_M4.OUT_forMapping.Control_word_or_setpoint_3 AT %QW."P1_ServoManipOsZ_M4".Module001_Control_word_or_setpoint_O_03;
	Cyclic#1.P1_Srobovanie.ServoManipulOsZ_M4.OUT_forMapping.Control_word_or_setpoint_4 AT %QW."P1_ServoManipOsZ_M4".Module001_Control_word_or_setpoint_O_04;
	Cyclic#1.P1_Srobovanie.ServoManipulOsZ_M4.OUT_forMapping.Control_word_or_setpoint_5 AT %QW."P1_ServoManipOsZ_M4".Module001_Control_word_or_setpoint_O_05;
	Cyclic#1.P1_Srobovanie.ServoManipulOsZ_M4.OUT_forMapping.Control_word_or_setpoint_6 AT %QW."P1_ServoManipOsZ_M4".Module001_Control_word_or_setpoint_O_06;
	Cyclic#1.P1_Srobovanie.ServoManipulOsZ_M4.OUT_forMapping.Control_word_or_setpoint_7 AT %QW."P1_ServoManipOsZ_M4".Module001_Control_word_or_setpoint_O_07;
	Cyclic#1.P1_Srobovanie.ServoManipulOsZ_M4.OUT_forMapping.Control_word_or_setpoint_8 AT %QW."P1_ServoManipOsZ_M4".Module001_Control_word_or_setpoint_O_08;
	Cyclic#1.P1_Srobovanie.ServoManipulOsZ_M4.OUT_forMapping.Control_word_or_setpoint_9 AT %QW."P1_ServoManipOsZ_M4".Module001_Control_word_or_setpoint_O_09;
	Cyclic#1.P1_Srobovanie.ServoManipulOsZ_M4.OUT_forMapping.Control_word_or_setpoint_10 AT %QW."P1_ServoManipOsZ_M4".Module001_Control_word_or_setpoint_O_10;
	Cyclic#1.P1_Srobovanie.ServoManipulOsZ_M4.OUT_forMapping.Control_word_or_setpoint_11 AT %QW."P1_ServoManipOsZ_M4".Module001_Control_word_or_setpoint_O_11;
	Cyclic#1.P1_Srobovanie.ServoManipulOsZ_M4.OUT_forMapping.Control_word_or_setpoint_12 AT %QW."P1_ServoManipOsZ_M4".Module001_Control_word_or_setpoint_O_12;
	Cyclic#1.P1_Srobovanie.ServoManipulOsZ_M4.OUT_forMapping.Control_word_or_setpoint_13 AT %QW."P1_ServoManipOsZ_M4".Module001_Control_word_or_setpoint_O_13;
	Cyclic#1.P1_Srobovanie.ServoManipulOsZ_M4.OUT_forMapping.Control_word_or_setpoint_14 AT %QW."P1_ServoManipOsZ_M4".Module001_Control_word_or_setpoint_O_14;
	Cyclic#1.P1_Srobovanie.ServoManipulOsZ_M4.OUT_forMapping.Control_word_or_setpoint_15 AT %QW."P1_ServoManipOsZ_M4".Module001_Control_word_or_setpoint_O_15;
	Cyclic#1.P3_Pracovisko.IN.ServoManipulatorOsY_KomOK AT %IX."P3_ServoManipulatoraOsY".ModuleOk;
	Cyclic#1.P3_Srobovanie.ServoManipulOsY.IN_forMapping.Status_word_1 AT %IW."P3_ServoManipulatoraOsY".Module001_Status_word_1;
	Cyclic#1.P3_Srobovanie.ServoManipulOsY.IN_forMapping.Position_Statusword_1 AT %IW."P3_ServoManipulatoraOsY".Module001_Position_Statusword_1;
	Cyclic#1.P3_Srobovanie.ServoManipulOsY.IN_forMapping.Position_Statusword_2 AT %IW."P3_ServoManipulatoraOsY".Module001_Position_Statusword_2;
	Cyclic#1.P3_Srobovanie.ServoManipulOsY.IN_forMapping.Status_word_2 AT %IW."P3_ServoManipulatoraOsY".Module001_Status_word_2;
	Cyclic#1.P3_Srobovanie.ServoManipulOsY.IN_forMapping.Report_word AT %IW."P3_ServoManipulatoraOsY".Module001_Report_word;
	Cyclic#1.P3_Srobovanie.ServoManipulOsY.IN_forMapping.Position_actual_value_A AT %ID."P3_ServoManipulatoraOsY".Module001_Position_actual_value_A;
	Cyclic#1.P3_Srobovanie.ServoManipulOsY.IN_forMapping.Speed_actual_value_B AT %ID."P3_ServoManipulatoraOsY".Module001_Speed_actual_value_B;
	Cyclic#1.P3_Srobovanie.ServoManipulOsY.IN_forMapping.Fault_Code AT %IW."P3_ServoManipulatoraOsY".Module001_Fault_Code;
	Cyclic#1.P3_Srobovanie.ServoManipulOsY.IN_forMapping.Warn_Code AT %IW."P3_ServoManipulatoraOsY".Module001_Warn_Code;
	Cyclic#1.P3_Srobovanie.ServoManipulOsY.IN_forMapping.User AT %IW."P3_ServoManipulatoraOsY".Module001_User;
	Cyclic#1.P3_Srobovanie.ServoManipulOsY.IN_forMapping.Status_word_or_actual_value_0 AT %IW."P3_ServoManipulatoraOsY".Module001_Status_word_or_actual_value_I_00;
	Cyclic#1.P3_Srobovanie.ServoManipulOsY.IN_forMapping.Status_word_or_actual_value_1 AT %IW."P3_ServoManipulatoraOsY".Module001_Status_word_or_actual_value_I_01;
	Cyclic#1.P3_Srobovanie.ServoManipulOsY.IN_forMapping.Status_word_or_actual_value_2 AT %IW."P3_ServoManipulatoraOsY".Module001_Status_word_or_actual_value_I_02;
	Cyclic#1.P3_Srobovanie.ServoManipulOsY.IN_forMapping.Status_word_or_actual_value_3 AT %IW."P3_ServoManipulatoraOsY".Module001_Status_word_or_actual_value_I_03;
	Cyclic#1.P3_Srobovanie.ServoManipulOsY.IN_forMapping.Status_word_or_actual_value_4 AT %IW."P3_ServoManipulatoraOsY".Module001_Status_word_or_actual_value_I_04;
	Cyclic#1.P3_Srobovanie.ServoManipulOsY.IN_forMapping.Status_word_or_actual_value_5 AT %IW."P3_ServoManipulatoraOsY".Module001_Status_word_or_actual_value_I_05;
	Cyclic#1.P3_Srobovanie.ServoManipulOsY.IN_forMapping.Status_word_or_actual_value_6 AT %IW."P3_ServoManipulatoraOsY".Module001_Status_word_or_actual_value_I_06;
	Cyclic#1.P3_Srobovanie.ServoManipulOsY.IN_forMapping.Status_word_or_actual_value_7 AT %IW."P3_ServoManipulatoraOsY".Module001_Status_word_or_actual_value_I_07;
	Cyclic#1.P3_Srobovanie.ServoManipulOsY.IN_forMapping.Status_word_or_actual_value_8 AT %IW."P3_ServoManipulatoraOsY".Module001_Status_word_or_actual_value_I_08;
	Cyclic#1.P3_Srobovanie.ServoManipulOsY.IN_forMapping.Status_word_or_actual_value_9 AT %IW."P3_ServoManipulatoraOsY".Module001_Status_word_or_actual_value_I_09;
	Cyclic#1.P3_Srobovanie.ServoManipulOsY.IN_forMapping.Status_word_or_actual_value_10 AT %IW."P3_ServoManipulatoraOsY".Module001_Status_word_or_actual_value_I_10;
	Cyclic#1.P3_Srobovanie.ServoManipulOsY.IN_forMapping.Status_word_or_actual_value_11 AT %IW."P3_ServoManipulatoraOsY".Module001_Status_word_or_actual_value_I_11;
	Cyclic#1.P3_Srobovanie.ServoManipulOsY.IN_forMapping.Status_word_or_actual_value_12 AT %IW."P3_ServoManipulatoraOsY".Module001_Status_word_or_actual_value_I_12;
	Cyclic#1.P3_Srobovanie.ServoManipulOsY.IN_forMapping.Status_word_or_actual_value_13 AT %IW."P3_ServoManipulatoraOsY".Module001_Status_word_or_actual_value_I_13;
	Cyclic#1.P3_Srobovanie.ServoManipulOsY.IN_forMapping.Status_word_or_actual_value_14 AT %IW."P3_ServoManipulatoraOsY".Module001_Status_word_or_actual_value_I_14;
	Cyclic#1.P3_Srobovanie.ServoManipulOsY.IN_forMapping.Status_word_or_actual_value_15 AT %IW."P3_ServoManipulatoraOsY".Module001_Status_word_or_actual_value_I_15;
	Cyclic#1.P3_Srobovanie.ServoManipulOsY.OUT_forMapping.Control_word_1 AT %QW."P3_ServoManipulatoraOsY".Module001_Control_word_1;
	Cyclic#1.P3_Srobovanie.ServoManipulOsY.OUT_forMapping.Position_Controlword_1 AT %QW."P3_ServoManipulatoraOsY".Module001_Position_Controlword_1;
	Cyclic#1.P3_Srobovanie.ServoManipulOsY.OUT_forMapping.Position_Controlword_2 AT %QW."P3_ServoManipulatoraOsY".Module001_Position_Controlword_2;
	Cyclic#1.P3_Srobovanie.ServoManipulOsY.OUT_forMapping.Control_word_2 AT %QW."P3_ServoManipulatoraOsY".Module001_Control_word_2;
	Cyclic#1.P3_Srobovanie.ServoManipulOsY.OUT_forMapping.Override AT %QW."P3_ServoManipulatoraOsY".Module001_Override;
	Cyclic#1.P3_Srobovanie.ServoManipulOsY.OUT_forMapping.MDI_target_position AT %QD."P3_ServoManipulatoraOsY".Module001_MDI_target_position;
	Cyclic#1.P3_Srobovanie.ServoManipulOsY.OUT_forMapping.MDI_velocity AT %QD."P3_ServoManipulatoraOsY".Module001_MDI_velocity;
	Cyclic#1.P3_Srobovanie.ServoManipulOsY.OUT_forMapping.MDI_acceleration AT %QW."P3_ServoManipulatoraOsY".Module001_MDI_acceleartion;
	Cyclic#1.P3_Srobovanie.ServoManipulOsY.OUT_forMapping.MDI_decceleration AT %QW."P3_ServoManipulatoraOsY".Module001_MDI_deceleration;
	Cyclic#1.P3_Srobovanie.ServoManipulOsY.OUT_forMapping.User1 AT %QW."P3_ServoManipulatoraOsY".Module001_User1;
	Cyclic#1.P3_Srobovanie.ServoManipulOsY.OUT_forMapping.Control_word_or_setpoint_0 AT %QW."P3_ServoManipulatoraOsY".Module001_Control_word_or_setpoint_O_00;
	Cyclic#1.P3_Srobovanie.ServoManipulOsY.OUT_forMapping.Control_word_or_setpoint_1 AT %QW."P3_ServoManipulatoraOsY".Module001_Control_word_or_setpoint_O_01;
	Cyclic#1.P3_Srobovanie.ServoManipulOsY.OUT_forMapping.Control_word_or_setpoint_2 AT %QW."P3_ServoManipulatoraOsY".Module001_Control_word_or_setpoint_O_02;
	Cyclic#1.P3_Srobovanie.ServoManipulOsY.OUT_forMapping.Control_word_or_setpoint_3 AT %QW."P3_ServoManipulatoraOsY".Module001_Control_word_or_setpoint_O_03;
	Cyclic#1.P3_Srobovanie.ServoManipulOsY.OUT_forMapping.Control_word_or_setpoint_4 AT %QW."P3_ServoManipulatoraOsY".Module001_Control_word_or_setpoint_O_04;
	Cyclic#1.P3_Srobovanie.ServoManipulOsY.OUT_forMapping.Control_word_or_setpoint_5 AT %QW."P3_ServoManipulatoraOsY".Module001_Control_word_or_setpoint_O_05;
	Cyclic#1.P3_Srobovanie.ServoManipulOsY.OUT_forMapping.Control_word_or_setpoint_6 AT %QW."P3_ServoManipulatoraOsY".Module001_Control_word_or_setpoint_O_06;
	Cyclic#1.P3_Srobovanie.ServoManipulOsY.OUT_forMapping.Control_word_or_setpoint_7 AT %QW."P3_ServoManipulatoraOsY".Module001_Control_word_or_setpoint_O_07;
	Cyclic#1.P3_Srobovanie.ServoManipulOsY.OUT_forMapping.Control_word_or_setpoint_8 AT %QW."P3_ServoManipulatoraOsY".Module001_Control_word_or_setpoint_O_08;
	Cyclic#1.P3_Srobovanie.ServoManipulOsY.OUT_forMapping.Control_word_or_setpoint_9 AT %QW."P3_ServoManipulatoraOsY".Module001_Control_word_or_setpoint_O_09;
	Cyclic#1.P3_Srobovanie.ServoManipulOsY.OUT_forMapping.Control_word_or_setpoint_10 AT %QW."P3_ServoManipulatoraOsY".Module001_Control_word_or_setpoint_O_10;
	Cyclic#1.P3_Srobovanie.ServoManipulOsY.OUT_forMapping.Control_word_or_setpoint_11 AT %QW."P3_ServoManipulatoraOsY".Module001_Control_word_or_setpoint_O_11;
	Cyclic#1.P3_Srobovanie.ServoManipulOsY.OUT_forMapping.Control_word_or_setpoint_12 AT %QW."P3_ServoManipulatoraOsY".Module001_Control_word_or_setpoint_O_12;
	Cyclic#1.P3_Srobovanie.ServoManipulOsY.OUT_forMapping.Control_word_or_setpoint_13 AT %QW."P3_ServoManipulatoraOsY".Module001_Control_word_or_setpoint_O_13;
	Cyclic#1.P3_Srobovanie.ServoManipulOsY.OUT_forMapping.Control_word_or_setpoint_14 AT %QW."P3_ServoManipulatoraOsY".Module001_Control_word_or_setpoint_O_14;
	Cyclic#1.P3_Srobovanie.ServoManipulOsY.OUT_forMapping.Control_word_or_setpoint_15 AT %QW."P3_ServoManipulatoraOsY".Module001_Control_word_or_setpoint_O_15;
	Cyclic#1.P3_Pracovisko.IN.ServoManipulatorOsZ_M5_KomOK AT %IX."P3_ServoManipOsZ_M5".ModuleOk;
	Cyclic#1.P3_Srobovanie.ServoManipulOsZ_M5.IN_forMapping.Status_word_1 AT %IW."P3_ServoManipOsZ_M5".Module001_Status_word_1;
	Cyclic#1.P3_Srobovanie.ServoManipulOsZ_M5.IN_forMapping.Position_Statusword_1 AT %IW."P3_ServoManipOsZ_M5".Module001_Position_Statusword_1;
	Cyclic#1.P3_Srobovanie.ServoManipulOsZ_M5.IN_forMapping.Position_Statusword_2 AT %IW."P3_ServoManipOsZ_M5".Module001_Position_Statusword_2;
	Cyclic#1.P3_Srobovanie.ServoManipulOsZ_M5.IN_forMapping.Status_word_2 AT %IW."P3_ServoManipOsZ_M5".Module001_Status_word_2;
	Cyclic#1.P3_Srobovanie.ServoManipulOsZ_M5.IN_forMapping.Report_word AT %IW."P3_ServoManipOsZ_M5".Module001_Report_word;
	Cyclic#1.P3_Srobovanie.ServoManipulOsZ_M5.IN_forMapping.Position_actual_value_A AT %ID."P3_ServoManipOsZ_M5".Module001_Position_actual_value_A;
	Cyclic#1.P3_Srobovanie.ServoManipulOsZ_M5.IN_forMapping.Speed_actual_value_B AT %ID."P3_ServoManipOsZ_M5".Module001_Speed_actual_value_B;
	Cyclic#1.P3_Srobovanie.ServoManipulOsZ_M5.IN_forMapping.Fault_Code AT %IW."P3_ServoManipOsZ_M5".Module001_Fault_Code;
	Cyclic#1.P3_Srobovanie.ServoManipulOsZ_M5.IN_forMapping.Warn_Code AT %IW."P3_ServoManipOsZ_M5".Module001_Warn_Code;
	Cyclic#1.P3_Srobovanie.ServoManipulOsZ_M5.IN_forMapping.User AT %IW."P3_ServoManipOsZ_M5".Module001_User;
	Cyclic#1.P3_Srobovanie.ServoManipulOsZ_M5.IN_forMapping.Status_word_or_actual_value_0 AT %IW."P3_ServoManipOsZ_M5".Module001_Status_word_or_actual_value_I_00;
	Cyclic#1.P3_Srobovanie.ServoManipulOsZ_M5.IN_forMapping.Status_word_or_actual_value_1 AT %IW."P3_ServoManipOsZ_M5".Module001_Status_word_or_actual_value_I_01;
	Cyclic#1.P3_Srobovanie.ServoManipulOsZ_M5.IN_forMapping.Status_word_or_actual_value_2 AT %IW."P3_ServoManipOsZ_M5".Module001_Status_word_or_actual_value_I_02;
	Cyclic#1.P3_Srobovanie.ServoManipulOsZ_M5.IN_forMapping.Status_word_or_actual_value_3 AT %IW."P3_ServoManipOsZ_M5".Module001_Status_word_or_actual_value_I_03;
	Cyclic#1.P3_Srobovanie.ServoManipulOsZ_M5.IN_forMapping.Status_word_or_actual_value_4 AT %IW."P3_ServoManipOsZ_M5".Module001_Status_word_or_actual_value_I_04;
	Cyclic#1.P3_Srobovanie.ServoManipulOsZ_M5.IN_forMapping.Status_word_or_actual_value_5 AT %IW."P3_ServoManipOsZ_M5".Module001_Status_word_or_actual_value_I_05;
	Cyclic#1.P3_Srobovanie.ServoManipulOsZ_M5.IN_forMapping.Status_word_or_actual_value_6 AT %IW."P3_ServoManipOsZ_M5".Module001_Status_word_or_actual_value_I_06;
	Cyclic#1.P3_Srobovanie.ServoManipulOsZ_M5.IN_forMapping.Status_word_or_actual_value_7 AT %IW."P3_ServoManipOsZ_M5".Module001_Status_word_or_actual_value_I_07;
	Cyclic#1.P3_Srobovanie.ServoManipulOsZ_M5.IN_forMapping.Status_word_or_actual_value_8 AT %IW."P3_ServoManipOsZ_M5".Module001_Status_word_or_actual_value_I_08;
	Cyclic#1.P3_Srobovanie.ServoManipulOsZ_M5.IN_forMapping.Status_word_or_actual_value_9 AT %IW."P3_ServoManipOsZ_M5".Module001_Status_word_or_actual_value_I_09;
	Cyclic#1.P3_Srobovanie.ServoManipulOsZ_M5.IN_forMapping.Status_word_or_actual_value_10 AT %IW."P3_ServoManipOsZ_M5".Module001_Status_word_or_actual_value_I_10;
	Cyclic#1.P3_Srobovanie.ServoManipulOsZ_M5.IN_forMapping.Status_word_or_actual_value_11 AT %IW."P3_ServoManipOsZ_M5".Module001_Status_word_or_actual_value_I_11;
	Cyclic#1.P3_Srobovanie.ServoManipulOsZ_M5.IN_forMapping.Status_word_or_actual_value_12 AT %IW."P3_ServoManipOsZ_M5".Module001_Status_word_or_actual_value_I_12;
	Cyclic#1.P3_Srobovanie.ServoManipulOsZ_M5.IN_forMapping.Status_word_or_actual_value_13 AT %IW."P3_ServoManipOsZ_M5".Module001_Status_word_or_actual_value_I_13;
	Cyclic#1.P3_Srobovanie.ServoManipulOsZ_M5.IN_forMapping.Status_word_or_actual_value_14 AT %IW."P3_ServoManipOsZ_M5".Module001_Status_word_or_actual_value_I_14;
	Cyclic#1.P3_Srobovanie.ServoManipulOsZ_M5.IN_forMapping.Status_word_or_actual_value_15 AT %IW."P3_ServoManipOsZ_M5".Module001_Status_word_or_actual_value_I_15;
	Cyclic#1.P3_Srobovanie.ServoManipulOsZ_M5.OUT_forMapping.Control_word_1 AT %QW."P3_ServoManipOsZ_M5".Module001_Control_word_1;
	Cyclic#1.P3_Srobovanie.ServoManipulOsZ_M5.OUT_forMapping.Position_Controlword_1 AT %QW."P3_ServoManipOsZ_M5".Module001_Position_Controlword_1;
	Cyclic#1.P3_Srobovanie.ServoManipulOsZ_M5.OUT_forMapping.Position_Controlword_2 AT %QW."P3_ServoManipOsZ_M5".Module001_Position_Controlword_2;
	Cyclic#1.P3_Srobovanie.ServoManipulOsZ_M5.OUT_forMapping.Control_word_2 AT %QW."P3_ServoManipOsZ_M5".Module001_Control_word_2;
	Cyclic#1.P3_Srobovanie.ServoManipulOsZ_M5.OUT_forMapping.Override AT %QW."P3_ServoManipOsZ_M5".Module001_Override;
	Cyclic#1.P3_Srobovanie.ServoManipulOsZ_M5.OUT_forMapping.MDI_target_position AT %QD."P3_ServoManipOsZ_M5".Module001_MDI_target_position;
	Cyclic#1.P3_Srobovanie.ServoManipulOsZ_M5.OUT_forMapping.MDI_velocity AT %QD."P3_ServoManipOsZ_M5".Module001_MDI_velocity;
	Cyclic#1.P3_Srobovanie.ServoManipulOsZ_M5.OUT_forMapping.MDI_acceleration AT %QW."P3_ServoManipOsZ_M5".Module001_MDI_acceleartion;
	Cyclic#1.P3_Srobovanie.ServoManipulOsZ_M5.OUT_forMapping.MDI_decceleration AT %QW."P3_ServoManipOsZ_M5".Module001_MDI_deceleration;
	Cyclic#1.P3_Srobovanie.ServoManipulOsZ_M5.OUT_forMapping.User1 AT %QW."P3_ServoManipOsZ_M5".Module001_User1;
	Cyclic#1.P3_Srobovanie.ServoManipulOsZ_M5.OUT_forMapping.Control_word_or_setpoint_0 AT %QW."P3_ServoManipOsZ_M5".Module001_Control_word_or_setpoint_O_00;
	Cyclic#1.P3_Srobovanie.ServoManipulOsZ_M5.OUT_forMapping.Control_word_or_setpoint_1 AT %QW."P3_ServoManipOsZ_M5".Module001_Control_word_or_setpoint_O_01;
	Cyclic#1.P3_Srobovanie.ServoManipulOsZ_M5.OUT_forMapping.Control_word_or_setpoint_2 AT %QW."P3_ServoManipOsZ_M5".Module001_Control_word_or_setpoint_O_02;
	Cyclic#1.P3_Srobovanie.ServoManipulOsZ_M5.OUT_forMapping.Control_word_or_setpoint_3 AT %QW."P3_ServoManipOsZ_M5".Module001_Control_word_or_setpoint_O_03;
	Cyclic#1.P3_Srobovanie.ServoManipulOsZ_M5.OUT_forMapping.Control_word_or_setpoint_4 AT %QW."P3_ServoManipOsZ_M5".Module001_Control_word_or_setpoint_O_04;
	Cyclic#1.P3_Srobovanie.ServoManipulOsZ_M5.OUT_forMapping.Control_word_or_setpoint_5 AT %QW."P3_ServoManipOsZ_M5".Module001_Control_word_or_setpoint_O_05;
	Cyclic#1.P3_Srobovanie.ServoManipulOsZ_M5.OUT_forMapping.Control_word_or_setpoint_6 AT %QW."P3_ServoManipOsZ_M5".Module001_Control_word_or_setpoint_O_06;
	Cyclic#1.P3_Srobovanie.ServoManipulOsZ_M5.OUT_forMapping.Control_word_or_setpoint_7 AT %QW."P3_ServoManipOsZ_M5".Module001_Control_word_or_setpoint_O_07;
	Cyclic#1.P3_Srobovanie.ServoManipulOsZ_M5.OUT_forMapping.Control_word_or_setpoint_8 AT %QW."P3_ServoManipOsZ_M5".Module001_Control_word_or_setpoint_O_08;
	Cyclic#1.P3_Srobovanie.ServoManipulOsZ_M5.OUT_forMapping.Control_word_or_setpoint_9 AT %QW."P3_ServoManipOsZ_M5".Module001_Control_word_or_setpoint_O_09;
	Cyclic#1.P3_Srobovanie.ServoManipulOsZ_M5.OUT_forMapping.Control_word_or_setpoint_10 AT %QW."P3_ServoManipOsZ_M5".Module001_Control_word_or_setpoint_O_10;
	Cyclic#1.P3_Srobovanie.ServoManipulOsZ_M5.OUT_forMapping.Control_word_or_setpoint_11 AT %QW."P3_ServoManipOsZ_M5".Module001_Control_word_or_setpoint_O_11;
	Cyclic#1.P3_Srobovanie.ServoManipulOsZ_M5.OUT_forMapping.Control_word_or_setpoint_12 AT %QW."P3_ServoManipOsZ_M5".Module001_Control_word_or_setpoint_O_12;
	Cyclic#1.P3_Srobovanie.ServoManipulOsZ_M5.OUT_forMapping.Control_word_or_setpoint_13 AT %QW."P3_ServoManipOsZ_M5".Module001_Control_word_or_setpoint_O_13;
	Cyclic#1.P3_Srobovanie.ServoManipulOsZ_M5.OUT_forMapping.Control_word_or_setpoint_14 AT %QW."P3_ServoManipOsZ_M5".Module001_Control_word_or_setpoint_O_14;
	Cyclic#1.P3_Srobovanie.ServoManipulOsZ_M5.OUT_forMapping.Control_word_or_setpoint_15 AT %QW."P3_ServoManipOsZ_M5".Module001_Control_word_or_setpoint_O_15;
	Cyclic#1.P3_Pracovisko.IN.LeakageTesterA_KomOK AT %IX."P3_AteqLeakageTesterA".ModuleOk;
	Cyclic#1.AteqLeakageTester_A.Profinet_PLC_INPUTS[1] AT %IB."P3_AteqLeakageTesterA".Module001_Inputs001;
	Cyclic#1.AteqLeakageTester_A.Profinet_PLC_INPUTS[2] AT %IB."P3_AteqLeakageTesterA".Module001_Inputs002;
	Cyclic#1.AteqLeakageTester_A.Profinet_PLC_INPUTS[3] AT %IB."P3_AteqLeakageTesterA".Module001_Inputs003;
	Cyclic#1.AteqLeakageTester_A.Profinet_PLC_INPUTS[4] AT %IB."P3_AteqLeakageTesterA".Module001_Inputs004;
	Cyclic#1.AteqLeakageTester_A.Profinet_PLC_INPUTS[5] AT %IB."P3_AteqLeakageTesterA".Module001_Inputs005;
	Cyclic#1.AteqLeakageTester_A.Profinet_PLC_INPUTS[6] AT %IB."P3_AteqLeakageTesterA".Module001_Inputs006;
	Cyclic#1.AteqLeakageTester_A.Profinet_PLC_INPUTS[7] AT %IB."P3_AteqLeakageTesterA".Module001_Inputs007;
	Cyclic#1.AteqLeakageTester_A.Profinet_PLC_INPUTS[8] AT %IB."P3_AteqLeakageTesterA".Module001_Inputs008;
	Cyclic#1.AteqLeakageTester_A.Profinet_PLC_INPUTS[9] AT %IB."P3_AteqLeakageTesterA".Module001_Inputs009;
	Cyclic#1.AteqLeakageTester_A.Profinet_PLC_INPUTS[10] AT %IB."P3_AteqLeakageTesterA".Module001_Inputs010;
	Cyclic#1.AteqLeakageTester_A.Profinet_PLC_INPUTS[11] AT %IB."P3_AteqLeakageTesterA".Module001_Inputs011;
	Cyclic#1.AteqLeakageTester_A.Profinet_PLC_INPUTS[12] AT %IB."P3_AteqLeakageTesterA".Module001_Inputs012;
	Cyclic#1.AteqLeakageTester_A.Profinet_PLC_INPUTS[13] AT %IB."P3_AteqLeakageTesterA".Module001_Inputs013;
	Cyclic#1.AteqLeakageTester_A.Profinet_PLC_INPUTS[24] AT %IB."P3_AteqLeakageTesterA".Module001_Inputs024;
	Cyclic#1.AteqLeakageTester_A.Profinet_PLC_INPUTS[25] AT %IB."P3_AteqLeakageTesterA".Module001_Inputs025;
	Cyclic#1.AteqLeakageTester_A.Profinet_PLC_INPUTS[26] AT %IB."P3_AteqLeakageTesterA".Module001_Inputs026;
	Cyclic#1.AteqLeakageTester_A.Profinet_PLC_INPUTS[27] AT %IB."P3_AteqLeakageTesterA".Module001_Inputs027;
	Cyclic#1.AteqLeakageTester_A.Profinet_PLC_INPUTS[35] AT %IB."P3_AteqLeakageTesterA".Module001_Inputs035;
	Cyclic#1.AteqLeakageTester_A.Profinet_PLC_INPUTS[36] AT %IB."P3_AteqLeakageTesterA".Module001_Inputs036;
	Cyclic#1.AteqLeakageTester_A.Profinet_PLC_INPUTS[41] AT %IB."P3_AteqLeakageTesterA".Module001_Inputs041;
	Cyclic#1.AteqLeakageTester_A.Profinet_PLC_INPUTS[42] AT %IB."P3_AteqLeakageTesterA".Module001_Inputs042;
	Cyclic#1.AteqLeakageTester_A.Profinet_PLC_INPUTS[47] AT %IB."P3_AteqLeakageTesterA".Module001_Inputs047;
	Cyclic#1.AteqLeakageTester_A.Profinet_PLC_INPUTS[48] AT %IB."P3_AteqLeakageTesterA".Module001_Inputs048;
	Cyclic#1.AteqLeakageTester_A.Profinet_PLC_INPUTS[53] AT %IB."P3_AteqLeakageTesterA".Module001_Inputs053;
	Cyclic#1.AteqLeakageTester_A.Profinet_PLC_INPUTS[54] AT %IB."P3_AteqLeakageTesterA".Module001_Inputs054;
	Cyclic#1.AteqLeakageTester_A.Profinet_PLC_OUTPUTS[1] AT %QB."P3_AteqLeakageTesterA".Module005_Outputs001;
	Cyclic#1.AteqLeakageTester_A.Profinet_PLC_OUTPUTS[7] AT %QB."P3_AteqLeakageTesterA".Module005_Outputs007;
	Cyclic#1.AteqLeakageTester_A.Profinet_PLC_OUTPUTS[8] AT %QB."P3_AteqLeakageTesterA".Module005_Outputs008;
	Cyclic#1.AteqLeakageTester_A.PocetCitanychParametrov AT %QB."P3_AteqLeakageTesterA".Module005_Outputs033;
	Cyclic#1.AteqLeakageTester_A.IdentifikaciaParametra_1 AT %QB."P3_AteqLeakageTesterA".Module005_Outputs035;
	Cyclic#1.AteqLeakageTester_A.IdentifikaciaParametra_2 AT %QB."P3_AteqLeakageTesterA".Module005_Outputs037;
	Cyclic#1.AteqLeakageTester_A.IdentifikaciaParametra_3 AT %QB."P3_AteqLeakageTesterA".Module005_Outputs039;
	Cyclic#1.AteqLeakageTester_A.IdentifikaciaParametra_4 AT %QB."P3_AteqLeakageTesterA".Module005_Outputs041;
	Cyclic#1.P3_Pracovisko.IN.LeakageTesterB_KomOK AT %IX."P3_AteqLeakageTesterB".ModuleOk;
	Cyclic#1.AteqLeakageTester_B.Profinet_PLC_INPUTS[1] AT %IB."P3_AteqLeakageTesterB".Module001_Inputs001;
	Cyclic#1.AteqLeakageTester_B.Profinet_PLC_INPUTS[2] AT %IB."P3_AteqLeakageTesterB".Module001_Inputs002;
	Cyclic#1.AteqLeakageTester_B.Profinet_PLC_INPUTS[3] AT %IB."P3_AteqLeakageTesterB".Module001_Inputs003;
	Cyclic#1.AteqLeakageTester_B.Profinet_PLC_INPUTS[4] AT %IB."P3_AteqLeakageTesterB".Module001_Inputs004;
	Cyclic#1.AteqLeakageTester_B.Profinet_PLC_INPUTS[5] AT %IB."P3_AteqLeakageTesterB".Module001_Inputs005;
	Cyclic#1.AteqLeakageTester_B.Profinet_PLC_INPUTS[6] AT %IB."P3_AteqLeakageTesterB".Module001_Inputs006;
	Cyclic#1.AteqLeakageTester_B.Profinet_PLC_INPUTS[7] AT %IB."P3_AteqLeakageTesterB".Module001_Inputs007;
	Cyclic#1.AteqLeakageTester_B.Profinet_PLC_INPUTS[8] AT %IB."P3_AteqLeakageTesterB".Module001_Inputs008;
	Cyclic#1.AteqLeakageTester_B.Profinet_PLC_INPUTS[9] AT %IB."P3_AteqLeakageTesterB".Module001_Inputs009;
	Cyclic#1.AteqLeakageTester_B.Profinet_PLC_INPUTS[10] AT %IB."P3_AteqLeakageTesterB".Module001_Inputs010;
	Cyclic#1.AteqLeakageTester_B.Profinet_PLC_INPUTS[11] AT %IB."P3_AteqLeakageTesterB".Module001_Inputs011;
	Cyclic#1.AteqLeakageTester_B.Profinet_PLC_INPUTS[12] AT %IB."P3_AteqLeakageTesterB".Module001_Inputs012;
	Cyclic#1.AteqLeakageTester_B.Profinet_PLC_INPUTS[13] AT %IB."P3_AteqLeakageTesterB".Module001_Inputs013;
	Cyclic#1.AteqLeakageTester_B.Profinet_PLC_INPUTS[24] AT %IB."P3_AteqLeakageTesterB".Module001_Inputs024;
	Cyclic#1.AteqLeakageTester_B.Profinet_PLC_INPUTS[25] AT %IB."P3_AteqLeakageTesterB".Module001_Inputs025;
	Cyclic#1.AteqLeakageTester_B.Profinet_PLC_INPUTS[26] AT %IB."P3_AteqLeakageTesterB".Module001_Inputs026;
	Cyclic#1.AteqLeakageTester_B.Profinet_PLC_INPUTS[27] AT %IB."P3_AteqLeakageTesterB".Module001_Inputs027;
	Cyclic#1.AteqLeakageTester_B.Profinet_PLC_INPUTS[35] AT %IB."P3_AteqLeakageTesterB".Module001_Inputs035;
	Cyclic#1.AteqLeakageTester_B.Profinet_PLC_INPUTS[36] AT %IB."P3_AteqLeakageTesterB".Module001_Inputs036;
	Cyclic#1.AteqLeakageTester_B.Profinet_PLC_INPUTS[41] AT %IB."P3_AteqLeakageTesterB".Module001_Inputs041;
	Cyclic#1.AteqLeakageTester_B.Profinet_PLC_INPUTS[42] AT %IB."P3_AteqLeakageTesterB".Module001_Inputs042;
	Cyclic#1.AteqLeakageTester_B.Profinet_PLC_INPUTS[47] AT %IB."P3_AteqLeakageTesterB".Module001_Inputs047;
	Cyclic#1.AteqLeakageTester_B.Profinet_PLC_INPUTS[48] AT %IB."P3_AteqLeakageTesterB".Module001_Inputs048;
	Cyclic#1.AteqLeakageTester_B.Profinet_PLC_INPUTS[53] AT %IB."P3_AteqLeakageTesterB".Module001_Inputs053;
	Cyclic#1.AteqLeakageTester_B.Profinet_PLC_INPUTS[54] AT %IB."P3_AteqLeakageTesterB".Module001_Inputs054;
	Cyclic#1.AteqLeakageTester_B.Profinet_PLC_OUTPUTS[1] AT %QB."P3_AteqLeakageTesterB".Module005_Outputs001;
	Cyclic#1.AteqLeakageTester_B.Profinet_PLC_OUTPUTS[7] AT %QB."P3_AteqLeakageTesterB".Module005_Outputs007;
	Cyclic#1.AteqLeakageTester_B.Profinet_PLC_OUTPUTS[8] AT %QB."P3_AteqLeakageTesterB".Module005_Outputs008;
	Cyclic#1.AteqLeakageTester_B.PocetCitanychParametrov AT %QB."P3_AteqLeakageTesterB".Module005_Outputs033;
	Cyclic#1.AteqLeakageTester_B.IdentifikaciaParametra_1 AT %QB."P3_AteqLeakageTesterB".Module005_Outputs035;
	Cyclic#1.AteqLeakageTester_B.IdentifikaciaParametra_2 AT %QB."P3_AteqLeakageTesterB".Module005_Outputs037;
	Cyclic#1.AteqLeakageTester_B.IdentifikaciaParametra_3 AT %QB."P3_AteqLeakageTesterB".Module005_Outputs039;
	Cyclic#1.AteqLeakageTester_B.IdentifikaciaParametra_4 AT %QB."P3_AteqLeakageTesterB".Module005_Outputs041;
	Cyclic#1.P3_Pracovisko.COM_VentilovyTerminal[6] AT %QB."P3_VentilovyTerminal_VT3".ValveCoils49_56_I2000_S07;
	Cyclic#1.P3_Pracovisko.COM_VentilovyTerminal[7] AT %QB."P3_VentilovyTerminal_VT3".ValveCoils57_64_I2000_S08;
	Cyclic#1.P3_Pracovisko.COM_VentilovyTerminal[8] AT %QB."P3_VentilovyTerminal_VT3".ValveCoils65_72_I2000_S09;
	Cyclic#1.P2_Pracovisko.IN.ModulFesto_IO_KomOK AT %IX."P2_IOmaster".ModuleOk;
	Cyclic#1.P2_Pracovisko.COM_Festo.DI2_1_8DI[0] AT %IX."P2_IOmaster".Module001_Bit_0_Bit_0;
	Cyclic#1.P2_Pracovisko.COM_Festo.DI2_1_8DI[1] AT %IX."P2_IOmaster".Module001_Bit_1_Bit_1;
	Cyclic#1.P2_Pracovisko.COM_Festo.DI2_1_8DI[2] AT %IX."P2_IOmaster".Module001_Bit_2_Bit_2;
	Cyclic#1.P2_Pracovisko.COM_Festo.DI2_1_8DI[3] AT %IX."P2_IOmaster".Module001_Bit_3_Bit_3;
	Cyclic#1.P2_Pracovisko.COM_Festo.DI2_1_8DI[4] AT %IX."P2_IOmaster".Module001_Bit_4_Bit_4;
	Cyclic#1.P2_Pracovisko.COM_Festo.DI2_1_8DI[5] AT %IX."P2_IOmaster".Module001_Bit_5_Bit_5;
	Cyclic#1.P2_Pracovisko.COM_Festo.DI2_1_8DI[6] AT %IX."P2_IOmaster".Module001_Bit_6_Bit_6;
	Cyclic#1.P2_Pracovisko.COM_Festo.DI2_1_8DI[7] AT %IX."P2_IOmaster".Module001_Bit_7_Bit_7;
	Cyclic#1.P2_Pracovisko.COM_Festo.DI2_5_8DI[0] AT %IX."P2_IOmaster".Module002_Bit_0_Bit_0;
	Cyclic#1.P2_Pracovisko.COM_Festo.DI2_5_8DI[1] AT %IX."P2_IOmaster".Module002_Bit_1_Bit_1;
	Cyclic#1.P2_Pracovisko.COM_Festo.DI2_5_8DI[2] AT %IX."P2_IOmaster".Module002_Bit_2_Bit_2;
	Cyclic#1.P2_Pracovisko.COM_Festo.DI2_5_8DI[3] AT %IX."P2_IOmaster".Module002_Bit_3_Bit_3;
	Cyclic#1.P2_Pracovisko.COM_Festo.DI2_5_8DI[4] AT %IX."P2_IOmaster".Module002_Bit_4_Bit_4;
	Cyclic#1.P2_Pracovisko.COM_Festo.DI2_5_8DI[5] AT %IX."P2_IOmaster".Module002_Bit_5_Bit_5;
	Cyclic#1.P2_Pracovisko.COM_Festo.DI2_5_8DI[6] AT %IX."P2_IOmaster".Module002_Bit_6_Bit_6;
	Cyclic#1.P2_Pracovisko.COM_Festo.DI2_5_8DI[7] AT %IX."P2_IOmaster".Module002_Bit_7_Bit_7;
	Cyclic#1.P2_Pracovisko.COM_Festo.DI2_6_8DI[0] AT %IX."P2_IOmaster".Module003_Bit_0_Bit_0;
	Cyclic#1.P2_Pracovisko.COM_Festo.DI2_6_8DI[1] AT %IX."P2_IOmaster".Module003_Bit_1_Bit_1;
	Cyclic#1.P2_Pracovisko.COM_Festo.DI2_6_8DI[2] AT %IX."P2_IOmaster".Module003_Bit_2_Bit_2;
	Cyclic#1.P2_Pracovisko.COM_Festo.DI2_6_8DI[3] AT %IX."P2_IOmaster".Module003_Bit_3_Bit_3;
	Cyclic#1.P2_Pracovisko.COM_Festo.DI2_6_8DI[4] AT %IX."P2_IOmaster".Module003_Bit_4_Bit_4;
	Cyclic#1.P2_Pracovisko.COM_Festo.DI2_6_8DI[5] AT %IX."P2_IOmaster".Module003_Bit_5_Bit_5;
	Cyclic#1.P2_Pracovisko.COM_Festo.DI2_6_8DI[6] AT %IX."P2_IOmaster".Module003_Bit_6_Bit_6;
	Cyclic#1.P2_Pracovisko.COM_Festo.DI2_6_8DI[7] AT %IX."P2_IOmaster".Module003_Bit_7_Bit_7;
	Cyclic#1.P2_Pracovisko.COM_Festo.DI2_7_8DI[0] AT %IX."P2_IOmaster".Module004_Bit_0_Bit_0;
	Cyclic#1.P2_Pracovisko.COM_Festo.DI2_7_8DI[1] AT %IX."P2_IOmaster".Module004_Bit_1_Bit_1;
	Cyclic#1.P2_Pracovisko.COM_Festo.DI2_7_8DI[2] AT %IX."P2_IOmaster".Module004_Bit_2_Bit_2;
	Cyclic#1.P2_Pracovisko.COM_Festo.DI2_7_8DI[3] AT %IX."P2_IOmaster".Module004_Bit_3_Bit_3;
	Cyclic#1.P2_Pracovisko.COM_Festo.DI2_7_8DI[4] AT %IX."P2_IOmaster".Module004_Bit_4_Bit_4;
	Cyclic#1.P2_Pracovisko.COM_Festo.DI2_7_8DI[5] AT %IX."P2_IOmaster".Module004_Bit_5_Bit_5;
	Cyclic#1.P2_Pracovisko.COM_Festo.DI2_7_8DI[6] AT %IX."P2_IOmaster".Module004_Bit_6_Bit_6;
	Cyclic#1.P2_Pracovisko.COM_Festo.DI2_7_8DI[7] AT %IX."P2_IOmaster".Module004_Bit_7_Bit_7;
	Cyclic#1.P2_Pracovisko.COM_Festo.DI2_8_8DI[0] AT %IX."P2_IOmaster".Module005_Bit_0_Bit_0;
	Cyclic#1.P2_Pracovisko.COM_Festo.DI2_8_8DI[1] AT %IX."P2_IOmaster".Module005_Bit_1_Bit_1;
	Cyclic#1.P2_Pracovisko.COM_Festo.DI2_8_8DI[2] AT %IX."P2_IOmaster".Module005_Bit_2_Bit_2;
	Cyclic#1.P2_Pracovisko.COM_Festo.DI2_8_8DI[3] AT %IX."P2_IOmaster".Module005_Bit_3_Bit_3;
	Cyclic#1.P2_Pracovisko.COM_Festo.DI2_8_8DI[4] AT %IX."P2_IOmaster".Module005_Bit_4_Bit_4;
	Cyclic#1.P2_Pracovisko.COM_Festo.DI2_8_8DI[5] AT %IX."P2_IOmaster".Module005_Bit_5_Bit_5;
	Cyclic#1.P2_Pracovisko.COM_Festo.DI2_8_8DI[6] AT %IX."P2_IOmaster".Module005_Bit_6_Bit_6;
	Cyclic#1.P2_Pracovisko.COM_Festo.DI2_8_8DI[7] AT %IX."P2_IOmaster".Module005_Bit_7_Bit_7;
	Cyclic#1.P2_Pracovisko.COM_Festo.DM2_1_4DI[0] AT %IX."P2_IOmaster".Module006_Bit_0_Bit_0;
	Cyclic#1.P2_Pracovisko.COM_Festo.DM2_1_4DI[1] AT %IX."P2_IOmaster".Module006_Bit_1_Bit_1;
	Cyclic#1.P2_Pracovisko.COM_Festo.DM2_1_4DI[2] AT %IX."P2_IOmaster".Module006_Bit_2_Bit_2;
	Cyclic#1.P2_Pracovisko.COM_Festo.DM2_1_4DI[3] AT %IX."P2_IOmaster".Module006_Bit_3_Bit_3;
	Cyclic#1.P2_Pracovisko.COM_Festo.DM2_1_4DO[0] AT %QX."P2_IOmaster".Module006_Bit_0_Bit_1;
	Cyclic#1.P2_Pracovisko.COM_Festo.DM2_1_4DO[1] AT %QX."P2_IOmaster".Module006_Bit_1_Bit_2;
	Cyclic#1.P2_Pracovisko.COM_Festo.DM2_1_4DO[2] AT %QX."P2_IOmaster".Module006_Bit_2_Bit_3;
	Cyclic#1.P2_Pracovisko.COM_Festo.DM2_1_4DO[3] AT %QX."P2_IOmaster".Module006_Bit_3_Bit_4;
	Cyclic#1.P2_Pracovisko.COM_Festo.DI2_2_8DI[0] AT %IX."P2_IOmaster".Module007_Bit_0_Bit_0;
	Cyclic#1.P2_Pracovisko.COM_Festo.DI2_2_8DI[1] AT %IX."P2_IOmaster".Module007_Bit_1_Bit_1;
	Cyclic#1.P2_Pracovisko.COM_Festo.DI2_2_8DI[2] AT %IX."P2_IOmaster".Module007_Bit_2_Bit_2;
	Cyclic#1.P2_Pracovisko.COM_Festo.DI2_2_8DI[3] AT %IX."P2_IOmaster".Module007_Bit_3_Bit_3;
	Cyclic#1.P2_Pracovisko.COM_Festo.DI2_2_8DI[4] AT %IX."P2_IOmaster".Module007_Bit_4_Bit_4;
	Cyclic#1.P2_Pracovisko.COM_Festo.DI2_2_8DI[5] AT %IX."P2_IOmaster".Module007_Bit_5_Bit_5;
	Cyclic#1.P2_Pracovisko.COM_Festo.DI2_2_8DI[6] AT %IX."P2_IOmaster".Module007_Bit_6_Bit_6;
	Cyclic#1.P2_Pracovisko.COM_Festo.DI2_2_8DI[7] AT %IX."P2_IOmaster".Module007_Bit_7_Bit_7;
	Cyclic#1.P2_Pracovisko.COM_Festo.DI2_3_8DI[0] AT %IX."P2_IOmaster".Module008_Bit_0_Bit_0;
	Cyclic#1.P2_Pracovisko.COM_Festo.DI2_3_8DI[1] AT %IX."P2_IOmaster".Module008_Bit_1_Bit_1;
	Cyclic#1.P2_Pracovisko.COM_Festo.DI2_3_8DI[2] AT %IX."P2_IOmaster".Module008_Bit_2_Bit_2;
	Cyclic#1.P2_Pracovisko.COM_Festo.DI2_3_8DI[3] AT %IX."P2_IOmaster".Module008_Bit_3_Bit_3;
	Cyclic#1.P2_Pracovisko.COM_Festo.DI2_3_8DI[4] AT %IX."P2_IOmaster".Module008_Bit_4_Bit_4;
	Cyclic#1.P2_Pracovisko.COM_Festo.DI2_3_8DI[5] AT %IX."P2_IOmaster".Module008_Bit_5_Bit_5;
	Cyclic#1.P2_Pracovisko.COM_Festo.DI2_3_8DI[6] AT %IX."P2_IOmaster".Module008_Bit_6_Bit_6;
	Cyclic#1.P2_Pracovisko.COM_Festo.DI2_3_8DI[7] AT %IX."P2_IOmaster".Module008_Bit_7_Bit_7;
	Cyclic#1.P2_Pracovisko.COM_Festo.DI2_4_8DI[0] AT %IX."P2_IOmaster".Module009_Bit_0_Bit_0;
	Cyclic#1.P2_Pracovisko.COM_Festo.DI2_4_8DI[1] AT %IX."P2_IOmaster".Module009_Bit_1_Bit_1;
	Cyclic#1.P2_Pracovisko.COM_Festo.DI2_4_8DI[2] AT %IX."P2_IOmaster".Module009_Bit_2_Bit_2;
	Cyclic#1.P2_Pracovisko.COM_Festo.DI2_4_8DI[3] AT %IX."P2_IOmaster".Module009_Bit_3_Bit_3;
	Cyclic#1.P2_Pracovisko.COM_Festo.DI2_4_8DI[4] AT %IX."P2_IOmaster".Module009_Bit_4_Bit_4;
	Cyclic#1.P2_Pracovisko.COM_Festo.DI2_4_8DI[5] AT %IX."P2_IOmaster".Module009_Bit_5_Bit_5;
	Cyclic#1.P2_Pracovisko.COM_Festo.DI2_4_8DI[6] AT %IX."P2_IOmaster".Module009_Bit_6_Bit_6;
	Cyclic#1.P2_Pracovisko.COM_Festo.DI2_4_8DI[7] AT %IX."P2_IOmaster".Module009_Bit_7_Bit_7;
	Cyclic#1.P2_Pracovisko.COM_Festo.DS2_2_Port0_IN[0] AT %IB."P2_IOmaster".Module010_Inputs001;
	Cyclic#1.P2_Pracovisko.COM_Festo.DS2_2_Port0_IN[1] AT %IB."P2_IOmaster".Module010_Inputs002;
	Cyclic#1.P2_Pracovisko.COM_Festo.DS2_2_Port0_IN[2] AT %IB."P2_IOmaster".Module010_Inputs003;
	Cyclic#1.P2_Pracovisko.COM_Festo.DS2_2_Port0_IN[3] AT %IB."P2_IOmaster".Module010_Inputs004;
	Cyclic#1.P2_Pracovisko.COM_Festo.DS2_2_Port0_IN[4] AT %IB."P2_IOmaster".Module010_Inputs005;
	Cyclic#1.P2_Pracovisko.COM_Festo.DS2_2_Port0_IN[5] AT %IB."P2_IOmaster".Module010_Inputs006;
	Cyclic#1.P2_Pracovisko.COM_Festo.DS2_2_Port0_IN[6] AT %IB."P2_IOmaster".Module010_Inputs007;
	Cyclic#1.P2_Pracovisko.COM_Festo.DS2_2_Port0_IN[7] AT %IB."P2_IOmaster".Module010_Inputs008;
	Cyclic#1.P2_Pracovisko.COM_Festo.DS2_2_Port0_IN[8] AT %IB."P2_IOmaster".Module010_Inputs009;
	Cyclic#1.P2_Pracovisko.COM_Festo.DS2_2_Port0_IN[9] AT %IB."P2_IOmaster".Module010_Inputs010;
	Cyclic#1.P2_Pracovisko.COM_Festo.DS2_2_Port0_IN[10] AT %IB."P2_IOmaster".Module010_Inputs011;
	Cyclic#1.P2_Pracovisko.COM_Festo.DS2_2_Port0_IN[11] AT %IB."P2_IOmaster".Module010_Inputs012;
	Cyclic#1.P2_Pracovisko.COM_Festo.DS2_2_Port0_IN[12] AT %IB."P2_IOmaster".Module010_Inputs013;
	Cyclic#1.P2_Pracovisko.COM_Festo.DS2_2_Port0_IN[13] AT %IB."P2_IOmaster".Module010_Inputs014;
	Cyclic#1.P2_Pracovisko.COM_Festo.DS2_2_Port0_IN[14] AT %IB."P2_IOmaster".Module010_Inputs015;
	Cyclic#1.P2_Pracovisko.COM_Festo.DS2_2_Port0_IN[15] AT %IB."P2_IOmaster".Module010_Inputs016;
	Cyclic#1.P2_Pracovisko.COM_Festo.DS2_2_Port0_IN[16] AT %IB."P2_IOmaster".Module010_Inputs017;
	Cyclic#1.P2_Pracovisko.COM_Festo.DS2_2_Port0_IN[17] AT %IB."P2_IOmaster".Module010_Inputs018;
	Cyclic#1.P2_Pracovisko.COM_Festo.DS2_2_Port0_IN[18] AT %IB."P2_IOmaster".Module010_Inputs019;
	Cyclic#1.P2_Pracovisko.COM_Festo.DS2_2_Port0_IN[19] AT %IB."P2_IOmaster".Module010_Inputs020;
	Cyclic#1.P2_Pracovisko.COM_Festo.DS2_2_Port0_IN[20] AT %IB."P2_IOmaster".Module010_Inputs021;
	Cyclic#1.P2_Pracovisko.COM_Festo.DS2_2_Port0_IN[21] AT %IB."P2_IOmaster".Module010_Inputs022;
	Cyclic#1.P2_Pracovisko.COM_Festo.DS2_2_Port0_IN[22] AT %IB."P2_IOmaster".Module010_Inputs023;
	Cyclic#1.P2_Pracovisko.COM_Festo.DS2_2_Port0_IN[23] AT %IB."P2_IOmaster".Module010_Inputs024;
	Cyclic#1.P2_Pracovisko.COM_Festo.DS2_2_Port0_IN[24] AT %IB."P2_IOmaster".Module010_Inputs025;
	Cyclic#1.P2_Pracovisko.COM_Festo.DS2_2_Port0_IN[25] AT %IB."P2_IOmaster".Module010_Inputs026;
	Cyclic#1.P2_Pracovisko.COM_Festo.DS2_2_Port0_IN[26] AT %IB."P2_IOmaster".Module010_Inputs027;
	Cyclic#1.P2_Pracovisko.COM_Festo.DS2_2_Port0_IN[27] AT %IB."P2_IOmaster".Module010_Inputs028;
	Cyclic#1.P2_Pracovisko.COM_Festo.DS2_2_Port0_IN[28] AT %IB."P2_IOmaster".Module010_Inputs029;
	Cyclic#1.P2_Pracovisko.COM_Festo.DS2_2_Port0_IN[29] AT %IB."P2_IOmaster".Module010_Inputs030;
	Cyclic#1.P2_Pracovisko.COM_Festo.DS2_2_Port0_IN[30] AT %IB."P2_IOmaster".Module010_Inputs031;
	Cyclic#1.P2_Pracovisko.COM_Festo.DS2_2_Port0_IN[31] AT %IB."P2_IOmaster".Module010_Inputs032;
	Cyclic#1.P2_Pracovisko.COM_Festo.DS2_2_Port1_IN[0] AT %IB."P2_IOmaster".Module010_Inputs033;
	Cyclic#1.P2_Pracovisko.COM_Festo.DS2_2_Port1_IN[1] AT %IB."P2_IOmaster".Module010_Inputs034;
	Cyclic#1.P2_Pracovisko.COM_Festo.DS2_2_Port1_IN[2] AT %IB."P2_IOmaster".Module010_Inputs035;
	Cyclic#1.P2_Pracovisko.COM_Festo.DS2_2_Port1_IN[3] AT %IB."P2_IOmaster".Module010_Inputs036;
	Cyclic#1.P2_Pracovisko.COM_Festo.DS2_2_Port1_IN[4] AT %IB."P2_IOmaster".Module010_Inputs037;
	Cyclic#1.P2_Pracovisko.COM_Festo.DS2_2_Port1_IN[5] AT %IB."P2_IOmaster".Module010_Inputs038;
	Cyclic#1.P2_Pracovisko.COM_Festo.DS2_2_Port1_IN[6] AT %IB."P2_IOmaster".Module010_Inputs039;
	Cyclic#1.P2_Pracovisko.COM_Festo.DS2_2_Port1_IN[7] AT %IB."P2_IOmaster".Module010_Inputs040;
	Cyclic#1.P2_Pracovisko.COM_Festo.DS2_2_Port1_IN[8] AT %IB."P2_IOmaster".Module010_Inputs041;
	Cyclic#1.P2_Pracovisko.COM_Festo.DS2_2_Port1_IN[9] AT %IB."P2_IOmaster".Module010_Inputs042;
	Cyclic#1.P2_Pracovisko.COM_Festo.DS2_2_Port1_IN[10] AT %IB."P2_IOmaster".Module010_Inputs043;
	Cyclic#1.P2_Pracovisko.COM_Festo.DS2_2_Port1_IN[11] AT %IB."P2_IOmaster".Module010_Inputs044;
	Cyclic#1.P2_Pracovisko.COM_Festo.DS2_2_Port1_IN[12] AT %IB."P2_IOmaster".Module010_Inputs045;
	Cyclic#1.P2_Pracovisko.COM_Festo.DS2_2_Port1_IN[13] AT %IB."P2_IOmaster".Module010_Inputs046;
	Cyclic#1.P2_Pracovisko.COM_Festo.DS2_2_Port1_IN[14] AT %IB."P2_IOmaster".Module010_Inputs047;
	Cyclic#1.P2_Pracovisko.COM_Festo.DS2_2_Port1_IN[15] AT %IB."P2_IOmaster".Module010_Inputs048;
	Cyclic#1.P2_Pracovisko.COM_Festo.DS2_2_Port1_IN[16] AT %IB."P2_IOmaster".Module010_Inputs049;
	Cyclic#1.P2_Pracovisko.COM_Festo.DS2_2_Port1_IN[17] AT %IB."P2_IOmaster".Module010_Inputs050;
	Cyclic#1.P2_Pracovisko.COM_Festo.DS2_2_Port1_IN[18] AT %IB."P2_IOmaster".Module010_Inputs051;
	Cyclic#1.P2_Pracovisko.COM_Festo.DS2_2_Port1_IN[19] AT %IB."P2_IOmaster".Module010_Inputs052;
	Cyclic#1.P2_Pracovisko.COM_Festo.DS2_2_Port1_IN[20] AT %IB."P2_IOmaster".Module010_Inputs053;
	Cyclic#1.P2_Pracovisko.COM_Festo.DS2_2_Port1_IN[21] AT %IB."P2_IOmaster".Module010_Inputs054;
	Cyclic#1.P2_Pracovisko.COM_Festo.DS2_2_Port1_IN[22] AT %IB."P2_IOmaster".Module010_Inputs055;
	Cyclic#1.P2_Pracovisko.COM_Festo.DS2_2_Port1_IN[23] AT %IB."P2_IOmaster".Module010_Inputs056;
	Cyclic#1.P2_Pracovisko.COM_Festo.DS2_2_Port1_IN[24] AT %IB."P2_IOmaster".Module010_Inputs057;
	Cyclic#1.P2_Pracovisko.COM_Festo.DS2_2_Port1_IN[25] AT %IB."P2_IOmaster".Module010_Inputs058;
	Cyclic#1.P2_Pracovisko.COM_Festo.DS2_2_Port1_IN[26] AT %IB."P2_IOmaster".Module010_Inputs059;
	Cyclic#1.P2_Pracovisko.COM_Festo.DS2_2_Port1_IN[27] AT %IB."P2_IOmaster".Module010_Inputs060;
	Cyclic#1.P2_Pracovisko.COM_Festo.DS2_2_Port1_IN[28] AT %IB."P2_IOmaster".Module010_Inputs061;
	Cyclic#1.P2_Pracovisko.COM_Festo.DS2_2_Port1_IN[29] AT %IB."P2_IOmaster".Module010_Inputs062;
	Cyclic#1.P2_Pracovisko.COM_Festo.DS2_2_Port1_IN[30] AT %IB."P2_IOmaster".Module010_Inputs063;
	Cyclic#1.P2_Pracovisko.COM_Festo.DS2_2_Port1_IN[31] AT %IB."P2_IOmaster".Module010_Inputs064;
	Cyclic#1.P2_Pracovisko.COM_Festo.DS2_2_Port2_IN[0] AT %IB."P2_IOmaster".Module010_Inputs065;
	Cyclic#1.P2_Pracovisko.COM_Festo.DS2_2_Port2_IN[1] AT %IB."P2_IOmaster".Module010_Inputs066;
	Cyclic#1.P2_Pracovisko.COM_Festo.DS2_2_Port2_IN[2] AT %IB."P2_IOmaster".Module010_Inputs067;
	Cyclic#1.P2_Pracovisko.COM_Festo.DS2_2_Port2_IN[3] AT %IB."P2_IOmaster".Module010_Inputs068;
	Cyclic#1.P2_Pracovisko.COM_Festo.DS2_2_Port2_IN[4] AT %IB."P2_IOmaster".Module010_Inputs069;
	Cyclic#1.P2_Pracovisko.COM_Festo.DS2_2_Port2_IN[5] AT %IB."P2_IOmaster".Module010_Inputs070;
	Cyclic#1.P2_Pracovisko.COM_Festo.DS2_2_Port2_IN[6] AT %IB."P2_IOmaster".Module010_Inputs071;
	Cyclic#1.P2_Pracovisko.COM_Festo.DS2_2_Port2_IN[7] AT %IB."P2_IOmaster".Module010_Inputs072;
	Cyclic#1.P2_Pracovisko.COM_Festo.DS2_2_Port2_IN[8] AT %IB."P2_IOmaster".Module010_Inputs073;
	Cyclic#1.P2_Pracovisko.COM_Festo.DS2_2_Port2_IN[9] AT %IB."P2_IOmaster".Module010_Inputs074;
	Cyclic#1.P2_Pracovisko.COM_Festo.DS2_2_Port2_IN[10] AT %IB."P2_IOmaster".Module010_Inputs075;
	Cyclic#1.P2_Pracovisko.COM_Festo.DS2_2_Port2_IN[11] AT %IB."P2_IOmaster".Module010_Inputs076;
	Cyclic#1.P2_Pracovisko.COM_Festo.DS2_2_Port2_IN[12] AT %IB."P2_IOmaster".Module010_Inputs077;
	Cyclic#1.P2_Pracovisko.COM_Festo.DS2_2_Port2_IN[13] AT %IB."P2_IOmaster".Module010_Inputs078;
	Cyclic#1.P2_Pracovisko.COM_Festo.DS2_2_Port2_IN[14] AT %IB."P2_IOmaster".Module010_Inputs079;
	Cyclic#1.P2_Pracovisko.COM_Festo.DS2_2_Port2_IN[15] AT %IB."P2_IOmaster".Module010_Inputs080;
	Cyclic#1.P2_Pracovisko.COM_Festo.DS2_2_Port2_IN[16] AT %IB."P2_IOmaster".Module010_Inputs081;
	Cyclic#1.P2_Pracovisko.COM_Festo.DS2_2_Port2_IN[17] AT %IB."P2_IOmaster".Module010_Inputs082;
	Cyclic#1.P2_Pracovisko.COM_Festo.DS2_2_Port2_IN[18] AT %IB."P2_IOmaster".Module010_Inputs083;
	Cyclic#1.P2_Pracovisko.COM_Festo.DS2_2_Port2_IN[19] AT %IB."P2_IOmaster".Module010_Inputs084;
	Cyclic#1.P2_Pracovisko.COM_Festo.DS2_2_Port2_IN[20] AT %IB."P2_IOmaster".Module010_Inputs085;
	Cyclic#1.P2_Pracovisko.COM_Festo.DS2_2_Port2_IN[21] AT %IB."P2_IOmaster".Module010_Inputs086;
	Cyclic#1.P2_Pracovisko.COM_Festo.DS2_2_Port2_IN[22] AT %IB."P2_IOmaster".Module010_Inputs087;
	Cyclic#1.P2_Pracovisko.COM_Festo.DS2_2_Port2_IN[23] AT %IB."P2_IOmaster".Module010_Inputs088;
	Cyclic#1.P2_Pracovisko.COM_Festo.DS2_2_Port2_IN[24] AT %IB."P2_IOmaster".Module010_Inputs089;
	Cyclic#1.P2_Pracovisko.COM_Festo.DS2_2_Port2_IN[25] AT %IB."P2_IOmaster".Module010_Inputs090;
	Cyclic#1.P2_Pracovisko.COM_Festo.DS2_2_Port2_IN[26] AT %IB."P2_IOmaster".Module010_Inputs091;
	Cyclic#1.P2_Pracovisko.COM_Festo.DS2_2_Port2_IN[27] AT %IB."P2_IOmaster".Module010_Inputs092;
	Cyclic#1.P2_Pracovisko.COM_Festo.DS2_2_Port2_IN[28] AT %IB."P2_IOmaster".Module010_Inputs093;
	Cyclic#1.P2_Pracovisko.COM_Festo.DS2_2_Port2_IN[29] AT %IB."P2_IOmaster".Module010_Inputs094;
	Cyclic#1.P2_Pracovisko.COM_Festo.DS2_2_Port2_IN[30] AT %IB."P2_IOmaster".Module010_Inputs095;
	Cyclic#1.P2_Pracovisko.COM_Festo.DS2_2_Port2_IN[31] AT %IB."P2_IOmaster".Module010_Inputs096;
	Cyclic#1.P2_Pracovisko.COM_Festo.DS2_2_Port3_IN[0] AT %IB."P2_IOmaster".Module010_Inputs097;
	Cyclic#1.P2_Pracovisko.COM_Festo.DS2_2_Port3_IN[1] AT %IB."P2_IOmaster".Module010_Inputs098;
	Cyclic#1.P2_Pracovisko.COM_Festo.DS2_2_Port3_IN[2] AT %IB."P2_IOmaster".Module010_Inputs099;
	Cyclic#1.P2_Pracovisko.COM_Festo.DS2_2_Port3_IN[3] AT %IB."P2_IOmaster".Module010_Inputs100;
	Cyclic#1.P2_Pracovisko.COM_Festo.DS2_2_Port3_IN[4] AT %IB."P2_IOmaster".Module010_Inputs101;
	Cyclic#1.P2_Pracovisko.COM_Festo.DS2_2_Port3_IN[5] AT %IB."P2_IOmaster".Module010_Inputs102;
	Cyclic#1.P2_Pracovisko.COM_Festo.DS2_2_Port3_IN[6] AT %IB."P2_IOmaster".Module010_Inputs103;
	Cyclic#1.P2_Pracovisko.COM_Festo.DS2_2_Port3_IN[7] AT %IB."P2_IOmaster".Module010_Inputs104;
	Cyclic#1.P2_Pracovisko.COM_Festo.DS2_2_Port3_IN[8] AT %IB."P2_IOmaster".Module010_Inputs105;
	Cyclic#1.P2_Pracovisko.COM_Festo.DS2_2_Port3_IN[9] AT %IB."P2_IOmaster".Module010_Inputs106;
	Cyclic#1.P2_Pracovisko.COM_Festo.DS2_2_Port3_IN[10] AT %IB."P2_IOmaster".Module010_Inputs107;
	Cyclic#1.P2_Pracovisko.COM_Festo.DS2_2_Port3_IN[11] AT %IB."P2_IOmaster".Module010_Inputs108;
	Cyclic#1.P2_Pracovisko.COM_Festo.DS2_2_Port3_IN[12] AT %IB."P2_IOmaster".Module010_Inputs109;
	Cyclic#1.P2_Pracovisko.COM_Festo.DS2_2_Port3_IN[13] AT %IB."P2_IOmaster".Module010_Inputs110;
	Cyclic#1.P2_Pracovisko.COM_Festo.DS2_2_Port3_IN[14] AT %IB."P2_IOmaster".Module010_Inputs111;
	Cyclic#1.P2_Pracovisko.COM_Festo.DS2_2_Port3_IN[15] AT %IB."P2_IOmaster".Module010_Inputs112;
	Cyclic#1.P2_Pracovisko.COM_Festo.DS2_2_Port3_IN[16] AT %IB."P2_IOmaster".Module010_Inputs113;
	Cyclic#1.P2_Pracovisko.COM_Festo.DS2_2_Port3_IN[17] AT %IB."P2_IOmaster".Module010_Inputs114;
	Cyclic#1.P2_Pracovisko.COM_Festo.DS2_2_Port3_IN[18] AT %IB."P2_IOmaster".Module010_Inputs115;
	Cyclic#1.P2_Pracovisko.COM_Festo.DS2_2_Port3_IN[19] AT %IB."P2_IOmaster".Module010_Inputs116;
	Cyclic#1.P2_Pracovisko.COM_Festo.DS2_2_Port3_IN[20] AT %IB."P2_IOmaster".Module010_Inputs117;
	Cyclic#1.P2_Pracovisko.COM_Festo.DS2_2_Port3_IN[21] AT %IB."P2_IOmaster".Module010_Inputs118;
	Cyclic#1.P2_Pracovisko.COM_Festo.DS2_2_Port3_IN[22] AT %IB."P2_IOmaster".Module010_Inputs119;
	Cyclic#1.P2_Pracovisko.COM_Festo.DS2_2_Port3_IN[23] AT %IB."P2_IOmaster".Module010_Inputs120;
	Cyclic#1.P2_Pracovisko.COM_Festo.DS2_2_Port3_IN[24] AT %IB."P2_IOmaster".Module010_Inputs121;
	Cyclic#1.P2_Pracovisko.COM_Festo.DS2_2_Port3_IN[25] AT %IB."P2_IOmaster".Module010_Inputs122;
	Cyclic#1.P2_Pracovisko.COM_Festo.DS2_2_Port3_IN[26] AT %IB."P2_IOmaster".Module010_Inputs123;
	Cyclic#1.P2_Pracovisko.COM_Festo.DS2_2_Port3_IN[27] AT %IB."P2_IOmaster".Module010_Inputs124;
	Cyclic#1.P2_Pracovisko.COM_Festo.DS2_2_Port3_IN[28] AT %IB."P2_IOmaster".Module010_Inputs125;
	Cyclic#1.P2_Pracovisko.COM_Festo.DS2_2_Port3_IN[29] AT %IB."P2_IOmaster".Module010_Inputs126;
	Cyclic#1.P2_Pracovisko.COM_Festo.DS2_2_Port3_IN[30] AT %IB."P2_IOmaster".Module010_Inputs127;
	Cyclic#1.P2_Pracovisko.COM_Festo.DS2_2_Port3_IN[31] AT %IB."P2_IOmaster".Module010_Inputs128;
	Cyclic#1.P2_Pracovisko.COM_Festo.DS2_2_Port0_OUT[0] AT %QB."P2_IOmaster".Module010_Outputs001;
	Cyclic#1.P2_Pracovisko.COM_Festo.DS2_2_Port0_OUT[1] AT %QB."P2_IOmaster".Module010_Outputs002;
	Cyclic#1.P2_Pracovisko.COM_Festo.DS2_2_Port0_OUT[2] AT %QB."P2_IOmaster".Module010_Outputs003;
	Cyclic#1.P2_Pracovisko.COM_Festo.DS2_2_Port0_OUT[3] AT %QB."P2_IOmaster".Module010_Outputs004;
	Cyclic#1.P2_Pracovisko.COM_Festo.DS2_2_Port0_OUT[4] AT %QB."P2_IOmaster".Module010_Outputs005;
	Cyclic#1.P2_Pracovisko.COM_Festo.DS2_2_Port0_OUT[5] AT %QB."P2_IOmaster".Module010_Outputs006;
	Cyclic#1.P2_Pracovisko.COM_Festo.DS2_2_Port0_OUT[6] AT %QB."P2_IOmaster".Module010_Outputs007;
	Cyclic#1.P2_Pracovisko.COM_Festo.DS2_2_Port0_OUT[7] AT %QB."P2_IOmaster".Module010_Outputs008;
	Cyclic#1.P2_Pracovisko.COM_Festo.DS2_2_Port0_OUT[8] AT %QB."P2_IOmaster".Module010_Outputs009;
	Cyclic#1.P2_Pracovisko.COM_Festo.DS2_2_Port0_OUT[9] AT %QB."P2_IOmaster".Module010_Outputs010;
	Cyclic#1.P2_Pracovisko.COM_Festo.DS2_2_Port0_OUT[10] AT %QB."P2_IOmaster".Module010_Outputs011;
	Cyclic#1.P2_Pracovisko.COM_Festo.DS2_2_Port0_OUT[11] AT %QB."P2_IOmaster".Module010_Outputs012;
	Cyclic#1.P2_Pracovisko.COM_Festo.DS2_2_Port0_OUT[12] AT %QB."P2_IOmaster".Module010_Outputs013;
	Cyclic#1.P2_Pracovisko.COM_Festo.DS2_2_Port0_OUT[13] AT %QB."P2_IOmaster".Module010_Outputs014;
	Cyclic#1.P2_Pracovisko.COM_Festo.DS2_2_Port0_OUT[14] AT %QB."P2_IOmaster".Module010_Outputs015;
	Cyclic#1.P2_Pracovisko.COM_Festo.DS2_2_Port0_OUT[15] AT %QB."P2_IOmaster".Module010_Outputs016;
	Cyclic#1.P2_Pracovisko.COM_Festo.DS2_2_Port0_OUT[16] AT %QB."P2_IOmaster".Module010_Outputs017;
	Cyclic#1.P2_Pracovisko.COM_Festo.DS2_2_Port0_OUT[17] AT %QB."P2_IOmaster".Module010_Outputs018;
	Cyclic#1.P2_Pracovisko.COM_Festo.DS2_2_Port0_OUT[18] AT %QB."P2_IOmaster".Module010_Outputs019;
	Cyclic#1.P2_Pracovisko.COM_Festo.DS2_2_Port0_OUT[19] AT %QB."P2_IOmaster".Module010_Outputs020;
	Cyclic#1.P2_Pracovisko.COM_Festo.DS2_2_Port0_OUT[20] AT %QB."P2_IOmaster".Module010_Outputs021;
	Cyclic#1.P2_Pracovisko.COM_Festo.DS2_2_Port0_OUT[21] AT %QB."P2_IOmaster".Module010_Outputs022;
	Cyclic#1.P2_Pracovisko.COM_Festo.DS2_2_Port0_OUT[22] AT %QB."P2_IOmaster".Module010_Outputs023;
	Cyclic#1.P2_Pracovisko.COM_Festo.DS2_2_Port0_OUT[23] AT %QB."P2_IOmaster".Module010_Outputs024;
	Cyclic#1.P2_Pracovisko.COM_Festo.DS2_2_Port0_OUT[24] AT %QB."P2_IOmaster".Module010_Outputs025;
	Cyclic#1.P2_Pracovisko.COM_Festo.DS2_2_Port0_OUT[25] AT %QB."P2_IOmaster".Module010_Outputs026;
	Cyclic#1.P2_Pracovisko.COM_Festo.DS2_2_Port0_OUT[26] AT %QB."P2_IOmaster".Module010_Outputs027;
	Cyclic#1.P2_Pracovisko.COM_Festo.DS2_2_Port0_OUT[27] AT %QB."P2_IOmaster".Module010_Outputs028;
	Cyclic#1.P2_Pracovisko.COM_Festo.DS2_2_Port0_OUT[28] AT %QB."P2_IOmaster".Module010_Outputs029;
	Cyclic#1.P2_Pracovisko.COM_Festo.DS2_2_Port0_OUT[29] AT %QB."P2_IOmaster".Module010_Outputs030;
	Cyclic#1.P2_Pracovisko.COM_Festo.DS2_2_Port0_OUT[30] AT %QB."P2_IOmaster".Module010_Outputs031;
	Cyclic#1.P2_Pracovisko.COM_Festo.DS2_2_Port0_OUT[31] AT %QB."P2_IOmaster".Module010_Outputs032;
	Cyclic#1.P2_Pracovisko.COM_Festo.DS2_2_Port1_OUT[0] AT %QB."P2_IOmaster".Module010_Outputs033;
	Cyclic#1.P2_Pracovisko.COM_Festo.DS2_2_Port1_OUT[1] AT %QB."P2_IOmaster".Module010_Outputs034;
	Cyclic#1.P2_Pracovisko.COM_Festo.DS2_2_Port1_OUT[2] AT %QB."P2_IOmaster".Module010_Outputs035;
	Cyclic#1.P2_Pracovisko.COM_Festo.DS2_2_Port1_OUT[3] AT %QB."P2_IOmaster".Module010_Outputs036;
	Cyclic#1.P2_Pracovisko.COM_Festo.DS2_2_Port1_OUT[4] AT %QB."P2_IOmaster".Module010_Outputs037;
	Cyclic#1.P2_Pracovisko.COM_Festo.DS2_2_Port1_OUT[5] AT %QB."P2_IOmaster".Module010_Outputs038;
	Cyclic#1.P2_Pracovisko.COM_Festo.DS2_2_Port1_OUT[6] AT %QB."P2_IOmaster".Module010_Outputs039;
	Cyclic#1.P2_Pracovisko.COM_Festo.DS2_2_Port1_OUT[7] AT %QB."P2_IOmaster".Module010_Outputs040;
	Cyclic#1.P2_Pracovisko.COM_Festo.DS2_2_Port1_OUT[8] AT %QB."P2_IOmaster".Module010_Outputs041;
	Cyclic#1.P2_Pracovisko.COM_Festo.DS2_2_Port1_OUT[9] AT %QB."P2_IOmaster".Module010_Outputs042;
	Cyclic#1.P2_Pracovisko.COM_Festo.DS2_2_Port1_OUT[10] AT %QB."P2_IOmaster".Module010_Outputs043;
	Cyclic#1.P2_Pracovisko.COM_Festo.DS2_2_Port1_OUT[11] AT %QB."P2_IOmaster".Module010_Outputs044;
	Cyclic#1.P2_Pracovisko.COM_Festo.DS2_2_Port1_OUT[12] AT %QB."P2_IOmaster".Module010_Outputs045;
	Cyclic#1.P2_Pracovisko.COM_Festo.DS2_2_Port1_OUT[13] AT %QB."P2_IOmaster".Module010_Outputs046;
	Cyclic#1.P2_Pracovisko.COM_Festo.DS2_2_Port1_OUT[14] AT %QB."P2_IOmaster".Module010_Outputs047;
	Cyclic#1.P2_Pracovisko.COM_Festo.DS2_2_Port1_OUT[15] AT %QB."P2_IOmaster".Module010_Outputs048;
	Cyclic#1.P2_Pracovisko.COM_Festo.DS2_2_Port1_OUT[16] AT %QB."P2_IOmaster".Module010_Outputs049;
	Cyclic#1.P2_Pracovisko.COM_Festo.DS2_2_Port1_OUT[17] AT %QB."P2_IOmaster".Module010_Outputs050;
	Cyclic#1.P2_Pracovisko.COM_Festo.DS2_2_Port1_OUT[18] AT %QB."P2_IOmaster".Module010_Outputs051;
	Cyclic#1.P2_Pracovisko.COM_Festo.DS2_2_Port1_OUT[19] AT %QB."P2_IOmaster".Module010_Outputs052;
	Cyclic#1.P2_Pracovisko.COM_Festo.DS2_2_Port1_OUT[20] AT %QB."P2_IOmaster".Module010_Outputs053;
	Cyclic#1.P2_Pracovisko.COM_Festo.DS2_2_Port1_OUT[21] AT %QB."P2_IOmaster".Module010_Outputs054;
	Cyclic#1.P2_Pracovisko.COM_Festo.DS2_2_Port1_OUT[22] AT %QB."P2_IOmaster".Module010_Outputs055;
	Cyclic#1.P2_Pracovisko.COM_Festo.DS2_2_Port1_OUT[23] AT %QB."P2_IOmaster".Module010_Outputs056;
	Cyclic#1.P2_Pracovisko.COM_Festo.DS2_2_Port1_OUT[24] AT %QB."P2_IOmaster".Module010_Outputs057;
	Cyclic#1.P2_Pracovisko.COM_Festo.DS2_2_Port1_OUT[25] AT %QB."P2_IOmaster".Module010_Outputs058;
	Cyclic#1.P2_Pracovisko.COM_Festo.DS2_2_Port1_OUT[26] AT %QB."P2_IOmaster".Module010_Outputs059;
	Cyclic#1.P2_Pracovisko.COM_Festo.DS2_2_Port1_OUT[27] AT %QB."P2_IOmaster".Module010_Outputs060;
	Cyclic#1.P2_Pracovisko.COM_Festo.DS2_2_Port1_OUT[28] AT %QB."P2_IOmaster".Module010_Outputs061;
	Cyclic#1.P2_Pracovisko.COM_Festo.DS2_2_Port1_OUT[29] AT %QB."P2_IOmaster".Module010_Outputs062;
	Cyclic#1.P2_Pracovisko.COM_Festo.DS2_2_Port1_OUT[30] AT %QB."P2_IOmaster".Module010_Outputs063;
	Cyclic#1.P2_Pracovisko.COM_Festo.DS2_2_Port1_OUT[31] AT %QB."P2_IOmaster".Module010_Outputs064;
	Cyclic#1.P2_Pracovisko.COM_Festo.DS2_2_Port2_OUT[0] AT %QB."P2_IOmaster".Module010_Outputs065;
	Cyclic#1.P2_Pracovisko.COM_Festo.DS2_2_Port2_OUT[1] AT %QB."P2_IOmaster".Module010_Outputs066;
	Cyclic#1.P2_Pracovisko.COM_Festo.DS2_2_Port2_OUT[2] AT %QB."P2_IOmaster".Module010_Outputs067;
	Cyclic#1.P2_Pracovisko.COM_Festo.DS2_2_Port2_OUT[3] AT %QB."P2_IOmaster".Module010_Outputs068;
	Cyclic#1.P2_Pracovisko.COM_Festo.DS2_2_Port2_OUT[4] AT %QB."P2_IOmaster".Module010_Outputs069;
	Cyclic#1.P2_Pracovisko.COM_Festo.DS2_2_Port2_OUT[5] AT %QB."P2_IOmaster".Module010_Outputs070;
	Cyclic#1.P2_Pracovisko.COM_Festo.DS2_2_Port2_OUT[6] AT %QB."P2_IOmaster".Module010_Outputs071;
	Cyclic#1.P2_Pracovisko.COM_Festo.DS2_2_Port2_OUT[7] AT %QB."P2_IOmaster".Module010_Outputs072;
	Cyclic#1.P2_Pracovisko.COM_Festo.DS2_2_Port2_OUT[8] AT %QB."P2_IOmaster".Module010_Outputs073;
	Cyclic#1.P2_Pracovisko.COM_Festo.DS2_2_Port2_OUT[9] AT %QB."P2_IOmaster".Module010_Outputs074;
	Cyclic#1.P2_Pracovisko.COM_Festo.DS2_2_Port2_OUT[10] AT %QB."P2_IOmaster".Module010_Outputs075;
	Cyclic#1.P2_Pracovisko.COM_Festo.DS2_2_Port2_OUT[11] AT %QB."P2_IOmaster".Module010_Outputs076;
	Cyclic#1.P2_Pracovisko.COM_Festo.DS2_2_Port2_OUT[12] AT %QB."P2_IOmaster".Module010_Outputs077;
	Cyclic#1.P2_Pracovisko.COM_Festo.DS2_2_Port2_OUT[13] AT %QB."P2_IOmaster".Module010_Outputs078;
	Cyclic#1.P2_Pracovisko.COM_Festo.DS2_2_Port2_OUT[14] AT %QB."P2_IOmaster".Module010_Outputs079;
	Cyclic#1.P2_Pracovisko.COM_Festo.DS2_2_Port2_OUT[15] AT %QB."P2_IOmaster".Module010_Outputs080;
	Cyclic#1.P2_Pracovisko.COM_Festo.DS2_2_Port2_OUT[16] AT %QB."P2_IOmaster".Module010_Outputs081;
	Cyclic#1.P2_Pracovisko.COM_Festo.DS2_2_Port2_OUT[17] AT %QB."P2_IOmaster".Module010_Outputs082;
	Cyclic#1.P2_Pracovisko.COM_Festo.DS2_2_Port2_OUT[18] AT %QB."P2_IOmaster".Module010_Outputs083;
	Cyclic#1.P2_Pracovisko.COM_Festo.DS2_2_Port2_OUT[19] AT %QB."P2_IOmaster".Module010_Outputs084;
	Cyclic#1.P2_Pracovisko.COM_Festo.DS2_2_Port2_OUT[20] AT %QB."P2_IOmaster".Module010_Outputs085;
	Cyclic#1.P2_Pracovisko.COM_Festo.DS2_2_Port2_OUT[21] AT %QB."P2_IOmaster".Module010_Outputs086;
	Cyclic#1.P2_Pracovisko.COM_Festo.DS2_2_Port2_OUT[22] AT %QB."P2_IOmaster".Module010_Outputs087;
	Cyclic#1.P2_Pracovisko.COM_Festo.DS2_2_Port2_OUT[23] AT %QB."P2_IOmaster".Module010_Outputs088;
	Cyclic#1.P2_Pracovisko.COM_Festo.DS2_2_Port2_OUT[24] AT %QB."P2_IOmaster".Module010_Outputs089;
	Cyclic#1.P2_Pracovisko.COM_Festo.DS2_2_Port2_OUT[25] AT %QB."P2_IOmaster".Module010_Outputs090;
	Cyclic#1.P2_Pracovisko.COM_Festo.DS2_2_Port2_OUT[26] AT %QB."P2_IOmaster".Module010_Outputs091;
	Cyclic#1.P2_Pracovisko.COM_Festo.DS2_2_Port2_OUT[27] AT %QB."P2_IOmaster".Module010_Outputs092;
	Cyclic#1.P2_Pracovisko.COM_Festo.DS2_2_Port2_OUT[28] AT %QB."P2_IOmaster".Module010_Outputs093;
	Cyclic#1.P2_Pracovisko.COM_Festo.DS2_2_Port2_OUT[29] AT %QB."P2_IOmaster".Module010_Outputs094;
	Cyclic#1.P2_Pracovisko.COM_Festo.DS2_2_Port2_OUT[30] AT %QB."P2_IOmaster".Module010_Outputs095;
	Cyclic#1.P2_Pracovisko.COM_Festo.DS2_2_Port2_OUT[31] AT %QB."P2_IOmaster".Module010_Outputs096;
	Cyclic#1.P2_Pracovisko.COM_Festo.DS2_2_Port3_OUT[0] AT %QB."P2_IOmaster".Module010_Outputs097;
	Cyclic#1.P2_Pracovisko.COM_Festo.DS2_2_Port3_OUT[1] AT %QB."P2_IOmaster".Module010_Outputs098;
	Cyclic#1.P2_Pracovisko.COM_Festo.DS2_2_Port3_OUT[2] AT %QB."P2_IOmaster".Module010_Outputs099;
	Cyclic#1.P2_Pracovisko.COM_Festo.DS2_2_Port3_OUT[3] AT %QB."P2_IOmaster".Module010_Outputs100;
	Cyclic#1.P2_Pracovisko.COM_Festo.DS2_2_Port3_OUT[4] AT %QB."P2_IOmaster".Module010_Outputs101;
	Cyclic#1.P2_Pracovisko.COM_Festo.DS2_2_Port3_OUT[5] AT %QB."P2_IOmaster".Module010_Outputs102;
	Cyclic#1.P2_Pracovisko.COM_Festo.DS2_2_Port3_OUT[6] AT %QB."P2_IOmaster".Module010_Outputs103;
	Cyclic#1.P2_Pracovisko.COM_Festo.DS2_2_Port3_OUT[7] AT %QB."P2_IOmaster".Module010_Outputs104;
	Cyclic#1.P2_Pracovisko.COM_Festo.DS2_2_Port3_OUT[8] AT %QB."P2_IOmaster".Module010_Outputs105;
	Cyclic#1.P2_Pracovisko.COM_Festo.DS2_2_Port3_OUT[9] AT %QB."P2_IOmaster".Module010_Outputs106;
	Cyclic#1.P2_Pracovisko.COM_Festo.DS2_2_Port3_OUT[10] AT %QB."P2_IOmaster".Module010_Outputs107;
	Cyclic#1.P2_Pracovisko.COM_Festo.DS2_2_Port3_OUT[11] AT %QB."P2_IOmaster".Module010_Outputs108;
	Cyclic#1.P2_Pracovisko.COM_Festo.DS2_2_Port3_OUT[12] AT %QB."P2_IOmaster".Module010_Outputs109;
	Cyclic#1.P2_Pracovisko.COM_Festo.DS2_2_Port3_OUT[13] AT %QB."P2_IOmaster".Module010_Outputs110;
	Cyclic#1.P2_Pracovisko.COM_Festo.DS2_2_Port3_OUT[14] AT %QB."P2_IOmaster".Module010_Outputs111;
	Cyclic#1.P2_Pracovisko.COM_Festo.DS2_2_Port3_OUT[15] AT %QB."P2_IOmaster".Module010_Outputs112;
	Cyclic#1.P2_Pracovisko.COM_Festo.DS2_2_Port3_OUT[16] AT %QB."P2_IOmaster".Module010_Outputs113;
	Cyclic#1.P2_Pracovisko.COM_Festo.DS2_2_Port3_OUT[17] AT %QB."P2_IOmaster".Module010_Outputs114;
	Cyclic#1.P2_Pracovisko.COM_Festo.DS2_2_Port3_OUT[18] AT %QB."P2_IOmaster".Module010_Outputs115;
	Cyclic#1.P2_Pracovisko.COM_Festo.DS2_2_Port3_OUT[19] AT %QB."P2_IOmaster".Module010_Outputs116;
	Cyclic#1.P2_Pracovisko.COM_Festo.DS2_2_Port3_OUT[20] AT %QB."P2_IOmaster".Module010_Outputs117;
	Cyclic#1.P2_Pracovisko.COM_Festo.DS2_2_Port3_OUT[21] AT %QB."P2_IOmaster".Module010_Outputs118;
	Cyclic#1.P2_Pracovisko.COM_Festo.DS2_2_Port3_OUT[22] AT %QB."P2_IOmaster".Module010_Outputs119;
	Cyclic#1.P2_Pracovisko.COM_Festo.DS2_2_Port3_OUT[23] AT %QB."P2_IOmaster".Module010_Outputs120;
	Cyclic#1.P2_Pracovisko.COM_Festo.DS2_2_Port3_OUT[24] AT %QB."P2_IOmaster".Module010_Outputs121;
	Cyclic#1.P2_Pracovisko.COM_Festo.DS2_2_Port3_OUT[25] AT %QB."P2_IOmaster".Module010_Outputs122;
	Cyclic#1.P2_Pracovisko.COM_Festo.DS2_2_Port3_OUT[26] AT %QB."P2_IOmaster".Module010_Outputs123;
	Cyclic#1.P2_Pracovisko.COM_Festo.DS2_2_Port3_OUT[27] AT %QB."P2_IOmaster".Module010_Outputs124;
	Cyclic#1.P2_Pracovisko.COM_Festo.DS2_2_Port3_OUT[28] AT %QB."P2_IOmaster".Module010_Outputs125;
	Cyclic#1.P2_Pracovisko.COM_Festo.DS2_2_Port3_OUT[29] AT %QB."P2_IOmaster".Module010_Outputs126;
	Cyclic#1.P2_Pracovisko.COM_Festo.DS2_2_Port3_OUT[30] AT %QB."P2_IOmaster".Module010_Outputs127;
	Cyclic#1.P2_Pracovisko.COM_Festo.DS2_2_Port3_OUT[31] AT %QB."P2_IOmaster".Module010_Outputs128;
	Cyclic#1.P2_Pracovisko.COM_Festo.DS2_3_Port0_IN[0] AT %IB."P2_IOmaster".Module011_Inputs001;
	Cyclic#1.P2_Pracovisko.COM_Festo.DS2_3_Port0_IN[1] AT %IB."P2_IOmaster".Module011_Inputs002;
	Cyclic#1.P2_Pracovisko.COM_Festo.DS2_3_Port0_IN[2] AT %IB."P2_IOmaster".Module011_Inputs003;
	Cyclic#1.P2_Pracovisko.COM_Festo.DS2_3_Port0_IN[3] AT %IB."P2_IOmaster".Module011_Inputs004;
	Cyclic#1.P2_Pracovisko.COM_Festo.DS2_3_Port0_IN[4] AT %IB."P2_IOmaster".Module011_Inputs005;
	Cyclic#1.P2_Pracovisko.COM_Festo.DS2_3_Port0_IN[5] AT %IB."P2_IOmaster".Module011_Inputs006;
	Cyclic#1.P2_Pracovisko.COM_Festo.DS2_3_Port0_IN[6] AT %IB."P2_IOmaster".Module011_Inputs007;
	Cyclic#1.P2_Pracovisko.COM_Festo.DS2_3_Port0_IN[7] AT %IB."P2_IOmaster".Module011_Inputs008;
	Cyclic#1.P2_Pracovisko.COM_Festo.DS2_3_Port0_IN[8] AT %IB."P2_IOmaster".Module011_Inputs009;
	Cyclic#1.P2_Pracovisko.COM_Festo.DS2_3_Port0_IN[9] AT %IB."P2_IOmaster".Module011_Inputs010;
	Cyclic#1.P2_Pracovisko.COM_Festo.DS2_3_Port0_IN[10] AT %IB."P2_IOmaster".Module011_Inputs011;
	Cyclic#1.P2_Pracovisko.COM_Festo.DS2_3_Port0_IN[11] AT %IB."P2_IOmaster".Module011_Inputs012;
	Cyclic#1.P2_Pracovisko.COM_Festo.DS2_3_Port0_IN[12] AT %IB."P2_IOmaster".Module011_Inputs013;
	Cyclic#1.P2_Pracovisko.COM_Festo.DS2_3_Port0_IN[13] AT %IB."P2_IOmaster".Module011_Inputs014;
	Cyclic#1.P2_Pracovisko.COM_Festo.DS2_3_Port0_IN[14] AT %IB."P2_IOmaster".Module011_Inputs015;
	Cyclic#1.P2_Pracovisko.COM_Festo.DS2_3_Port0_IN[15] AT %IB."P2_IOmaster".Module011_Inputs016;
	Cyclic#1.P2_Pracovisko.COM_Festo.DS2_3_Port1_IN[0] AT %IB."P2_IOmaster".Module011_Inputs017;
	Cyclic#1.P2_Pracovisko.COM_Festo.DS2_3_Port1_IN[1] AT %IB."P2_IOmaster".Module011_Inputs018;
	Cyclic#1.P2_Pracovisko.COM_Festo.DS2_3_Port0_OUT[0] AT %QB."P2_IOmaster".Module011_Outputs001;
	Cyclic#1.P2_Pracovisko.COM_Festo.DS2_3_Port0_OUT[1] AT %QB."P2_IOmaster".Module011_Outputs002;
	Cyclic#1.P2_Pracovisko.COM_Festo.DS2_3_Port0_OUT[2] AT %QB."P2_IOmaster".Module011_Outputs003;
	Cyclic#1.P2_Pracovisko.COM_Festo.DS2_3_Port0_OUT[3] AT %QB."P2_IOmaster".Module011_Outputs004;
	Cyclic#1.P2_Pracovisko.COM_Festo.DS2_3_Port0_OUT[4] AT %QB."P2_IOmaster".Module011_Outputs005;
	Cyclic#1.P2_Pracovisko.COM_Festo.DS2_3_Port0_OUT[5] AT %QB."P2_IOmaster".Module011_Outputs006;
	Cyclic#1.P2_Pracovisko.COM_Festo.DS2_3_Port0_OUT[6] AT %QB."P2_IOmaster".Module011_Outputs007;
	Cyclic#1.P2_Pracovisko.COM_Festo.DS2_3_Port0_OUT[7] AT %QB."P2_IOmaster".Module011_Outputs008;
	Cyclic#1.P2_Pracovisko.COM_Festo.DS2_3_Port0_OUT[8] AT %QB."P2_IOmaster".Module011_Outputs009;
	Cyclic#1.P2_Pracovisko.COM_Festo.DS2_3_Port0_OUT[9] AT %QB."P2_IOmaster".Module011_Outputs010;
	Cyclic#1.P2_Pracovisko.COM_Festo.DS2_3_Port0_OUT[10] AT %QB."P2_IOmaster".Module011_Outputs011;
	Cyclic#1.P2_Pracovisko.COM_Festo.DS2_3_Port0_OUT[11] AT %QB."P2_IOmaster".Module011_Outputs012;
	Cyclic#1.P2_Pracovisko.COM_Festo.DS2_3_Port0_OUT[12] AT %QB."P2_IOmaster".Module011_Outputs013;
	Cyclic#1.P2_Pracovisko.COM_Festo.DS2_3_Port0_OUT[13] AT %QB."P2_IOmaster".Module011_Outputs014;
	Cyclic#1.P2_Pracovisko.COM_Festo.DS2_3_Port0_OUT[14] AT %QB."P2_IOmaster".Module011_Outputs015;
	Cyclic#1.P2_Pracovisko.COM_Festo.DS2_3_Port0_OUT[15] AT %QB."P2_IOmaster".Module011_Outputs016;
	Cyclic#1.P2_Pracovisko.COM_Festo.DS2_3_Port1_OUT[0] AT %QB."P2_IOmaster".Module011_Outputs017;
	Cyclic#1.P2_Pracovisko.COM_Festo.DS2_3_Port1_OUT[1] AT %QB."P2_IOmaster".Module011_Outputs018;
	Cyclic#1.P2_Pracovisko.COM_Festo.DS2_1_Port0_IN[0] AT %IB."P2_IOmaster".Module012_Inputs001;
	Cyclic#1.P2_Pracovisko.COM_Festo.DS2_1_Port0_IN[1] AT %IB."P2_IOmaster".Module012_Inputs002;
	Cyclic#1.P2_Pracovisko.COM_Festo.DS2_1_Port1_IN[0] AT %IB."P2_IOmaster".Module012_Inputs003;
	Cyclic#1.P2_Pracovisko.COM_Festo.DS2_1_Port1_IN[1] AT %IB."P2_IOmaster".Module012_Inputs004;
	Cyclic#1.P2_Pracovisko.COM_Festo.DS2_1_Port2_IN[0] AT %IB."P2_IOmaster".Module012_Inputs005;
	Cyclic#1.P2_Pracovisko.COM_Festo.DS2_1_Port2_IN[1] AT %IB."P2_IOmaster".Module012_Inputs006;
	Cyclic#1.P2_Pracovisko.COM_Festo.DS2_1_Port3_IN[0] AT %IB."P2_IOmaster".Module012_Inputs007;
	Cyclic#1.P2_Pracovisko.COM_Festo.DS2_1_Port3_IN[1] AT %IB."P2_IOmaster".Module012_Inputs008;
	Cyclic#1.P2_Pracovisko.COM_Festo.DS2_1_Port0_OUT[0] AT %QB."P2_IOmaster".Module012_Outputs001;
	Cyclic#1.P2_Pracovisko.COM_Festo.DS2_1_Port0_OUT[1] AT %QB."P2_IOmaster".Module012_Outputs002;
	Cyclic#1.P2_Pracovisko.COM_Festo.DS2_1_Port1_OUT[0] AT %QB."P2_IOmaster".Module012_Outputs003;
	Cyclic#1.P2_Pracovisko.COM_Festo.DS2_1_Port1_OUT[1] AT %QB."P2_IOmaster".Module012_Outputs004;
	Cyclic#1.P2_Pracovisko.COM_Festo.DS2_1_Port2_OUT[0] AT %QB."P2_IOmaster".Module012_Outputs005;
	Cyclic#1.P2_Pracovisko.COM_Festo.DS2_1_Port2_OUT[1] AT %QB."P2_IOmaster".Module012_Outputs006;
	Cyclic#1.P2_Pracovisko.COM_Festo.DS2_1_Port3_OUT[0] AT %QB."P2_IOmaster".Module012_Outputs007;
	Cyclic#1.P2_Pracovisko.COM_Festo.DS2_1_Port3_OUT[1] AT %QB."P2_IOmaster".Module012_Outputs008;
	Cyclic#1.P4_Pracovisko.IN.ModulWeidmuller_IO_KomOK AT %IX."P4_IOmodul_PowerlinkMaster".ModuleOk;
	Cyclic#1.P4_Pracovisko.COM_Weidmuller.AB4_2_8DI AT %IB."P4_IOmodul_PowerlinkMaster".DigitalInput_I6000_S01;
	Cyclic#1.P4_Pracovisko.COM_Weidmuller.AB4_3_8DI AT %IB."P4_IOmodul_PowerlinkMaster".DigitalInput_I6000_S02;
	Cyclic#1.P4_Pracovisko.COM_Weidmuller.AB4_4_8DI AT %IB."P4_IOmodul_PowerlinkMaster".DigitalInput_I6000_S03;
	Cyclic#1.P4_Pracovisko.COM_Weidmuller.AB4_5_8DO AT %QB."P4_IOmodul_PowerlinkMaster".DigitalOutput_I6200_S01;
	Cyclic#1.P4_Pracovisko.COM_Weidmuller.AB4_6_8DO AT %QB."P4_IOmodul_PowerlinkMaster".DigitalOutput_I6200_S02;
	Cyclic#1.P4_Pracovisko.COM_Weidmuller.AB4_8_8DO AT %QB."P4_IOmodul_PowerlinkMaster".DigitalOutput_I6200_S03;
	Cyclic#1.P3_Pracovisko.COM_VentilovyTerminal[9] AT %QB."P3_VentilovyTerminal_VT3".ValveCoils73_80_I2000_S0A;
	Cyclic#1.P2_Pracovisko.IN.VentilovyTerminal_KomOK AT %IX."P2_VentilovyTerminal_VT2".ModuleOk;
	Cyclic#1.P2_Pracovisko.COM_VentilovyTerminal[0] AT %QB."P2_VentilovyTerminal_VT2".ValveCoils1_8_I2000_S01;
	Cyclic#1.P2_Pracovisko.COM_VentilovyTerminal[1] AT %QB."P2_VentilovyTerminal_VT2".ValveCoils9_16_I2000_S02;
	Cyclic#1.P2_Pracovisko.COM_VentilovyTerminal[2] AT %QB."P2_VentilovyTerminal_VT2".ValveCoils17_24_I2000_S03;
	Cyclic#1.P2_Pracovisko.COM_VentilovyTerminal[3] AT %QB."P2_VentilovyTerminal_VT2".ValveCoils25_32_I2000_S04;
	Cyclic#1.P2_Pracovisko.COM_VentilovyTerminal[4] AT %QB."P2_VentilovyTerminal_VT2".ValveCoils33_40_I2000_S05;
	Cyclic#1.P2_Pracovisko.COM_VentilovyTerminal[5] AT %QB."P2_VentilovyTerminal_VT2".ValveCoils41_48_I2000_S06;
	Cyclic#1.P2_Pracovisko.COM_VentilovyTerminal[6] AT %QB."P2_VentilovyTerminal_VT2".ValveCoils49_56_I2000_S07;
	Cyclic#1.P2_Pracovisko.COM_VentilovyTerminal[7] AT %QB."P2_VentilovyTerminal_VT2".ValveCoils57_64_I2000_S08;
	Cyclic#1.P2_Pracovisko.COM_VentilovyTerminal[8] AT %QB."P2_VentilovyTerminal_VT2".ValveCoils65_72_I2000_S09;
	Cyclic#1.P2_Pracovisko.COM_VentilovyTerminal[9] AT %QB."P2_VentilovyTerminal_VT2".ValveCoils73_80_I2000_S0A;
	Cyclic#1.P2_Pracovisko.IN.ModulWeidmuller_IO_KomOK AT %IX."P2_IOmodul_PowerlinkMaster".ModuleOk;
	Cyclic#1.P2_Pracovisko.COM_Weidmuller.AB2_5_8DI AT %IB."P2_IOmodul_PowerlinkMaster".DigitalInput_I6000_S01;
	Cyclic#1.P2_Pracovisko.COM_Weidmuller.AB2_6_8DI AT %IB."P2_IOmodul_PowerlinkMaster".DigitalInput_I6000_S02;
	Cyclic#1.P2_Pracovisko.COM_Weidmuller.AB2_7_8DI AT %IB."P2_IOmodul_PowerlinkMaster".DigitalInput_I6000_S03;
	Cyclic#1.P2_Pracovisko.COM_Weidmuller.AB2_8_8DI AT %IB."P2_IOmodul_PowerlinkMaster".DigitalInput_I6000_S04;
	Cyclic#1.P2_Pracovisko.COM_Weidmuller.AB2_9_8DO AT %QB."P2_IOmodul_PowerlinkMaster".DigitalOutput_I6200_S01;
	Cyclic#1.P2_Pracovisko.COM_Weidmuller.AB2_10_8DO AT %QB."P2_IOmodul_PowerlinkMaster".DigitalOutput_I6200_S02;
	Cyclic#1.P2_Pracovisko.COM_Weidmuller.AB2_12_8DO AT %QB."P2_IOmodul_PowerlinkMaster".DigitalOutput_I6200_S03;
	Cyclic#1.P2_Pracovisko.COM_Weidmuller.AB2_13_8DO AT %QB."P2_IOmodul_PowerlinkMaster".DigitalOutput_I6200_S04;
	Cyclic#1.P2_Pracovisko.IN.Robot_KomOK AT %IX."P2_Robot_IRB1200".ModuleOk;
	Cyclic#1.P2_Robot.COM_IN.BYTE_IN[0] AT %IB."P2_Robot_IRB1200".Module001_Input_0;
	Cyclic#1.P2_Robot.COM_OUT.BYTE_OUT[0] AT %QB."P2_Robot_IRB1200".Module002_Output_0;
	Cyclic#1.P2_Robot.COM_IN.BYTE_IN[1] AT %IB."P2_Robot_IRB1200".Module001_Input_1;
	Cyclic#1.P2_Robot.COM_IN.BYTE_IN[2] AT %IB."P2_Robot_IRB1200".Module001_Input_2;
	Cyclic#1.P2_Robot.COM_IN.BYTE_IN[3] AT %IB."P2_Robot_IRB1200".Module001_Input_3;
	Cyclic#1.P2_Robot.COM_IN.BYTE_IN[4] AT %IB."P2_Robot_IRB1200".Module001_Input_4;
	Cyclic#1.P2_Robot.COM_IN.BYTE_IN[5] AT %IB."P2_Robot_IRB1200".Module001_Input_5;
	Cyclic#1.P2_Robot.COM_IN.BYTE_IN[6] AT %IB."P2_Robot_IRB1200".Module001_Input_6;
	Cyclic#1.P2_Robot.COM_IN.BYTE_IN[7] AT %IB."P2_Robot_IRB1200".Module001_Input_7;
	Cyclic#1.P2_Robot.COM_IN.BYTE_IN[8] AT %IB."P2_Robot_IRB1200".Module001_Input_8;
	Cyclic#1.P2_Robot.COM_IN.BYTE_IN[9] AT %IB."P2_Robot_IRB1200".Module001_Input_9;
	Cyclic#1.P2_Robot.COM_IN.BYTE_IN[10] AT %IB."P2_Robot_IRB1200".Module001_Input_10;
	Cyclic#1.P2_Robot.COM_IN.BYTE_IN[11] AT %IB."P2_Robot_IRB1200".Module001_Input_11;
	Cyclic#1.P2_Robot.COM_IN.BYTE_IN[12] AT %IB."P2_Robot_IRB1200".Module001_Input_12;
	Cyclic#1.P2_Robot.COM_IN.BYTE_IN[13] AT %IB."P2_Robot_IRB1200".Module001_Input_13;
	Cyclic#1.P2_Robot.COM_IN.BYTE_IN[14] AT %IB."P2_Robot_IRB1200".Module001_Input_14;
	Cyclic#1.P2_Robot.COM_IN.BYTE_IN[15] AT %IB."P2_Robot_IRB1200".Module001_Input_15;
	Cyclic#1.P2_Robot.COM_IN.BYTE_IN[16] AT %IB."P2_Robot_IRB1200".Module001_Input_16;
	Cyclic#1.P2_Robot.COM_IN.BYTE_IN[17] AT %IB."P2_Robot_IRB1200".Module001_Input_17;
	Cyclic#1.P2_Robot.COM_IN.BYTE_IN[18] AT %IB."P2_Robot_IRB1200".Module001_Input_18;
	Cyclic#1.P2_Robot.COM_IN.BYTE_IN[19] AT %IB."P2_Robot_IRB1200".Module001_Input_19;
	Cyclic#1.P2_Robot.COM_IN.BYTE_IN[20] AT %IB."P2_Robot_IRB1200".Module001_Input_20;
	Cyclic#1.P2_Robot.COM_IN.BYTE_IN[21] AT %IB."P2_Robot_IRB1200".Module001_Input_21;
	Cyclic#1.P2_Robot.COM_IN.BYTE_IN[22] AT %IB."P2_Robot_IRB1200".Module001_Input_22;
	Cyclic#1.P2_Robot.COM_IN.BYTE_IN[23] AT %IB."P2_Robot_IRB1200".Module001_Input_23;
	Cyclic#1.P2_Robot.COM_IN.BYTE_IN[24] AT %IB."P2_Robot_IRB1200".Module001_Input_24;
	Cyclic#1.P2_Robot.COM_IN.BYTE_IN[25] AT %IB."P2_Robot_IRB1200".Module001_Input_25;
	Cyclic#1.P2_Robot.COM_IN.BYTE_IN[26] AT %IB."P2_Robot_IRB1200".Module001_Input_26;
	Cyclic#1.P2_Robot.COM_IN.BYTE_IN[27] AT %IB."P2_Robot_IRB1200".Module001_Input_27;
	Cyclic#1.P2_Robot.COM_IN.BYTE_IN[28] AT %IB."P2_Robot_IRB1200".Module001_Input_28;
	Cyclic#1.P2_Robot.COM_IN.BYTE_IN[29] AT %IB."P2_Robot_IRB1200".Module001_Input_29;
	Cyclic#1.P2_Robot.COM_IN.BYTE_IN[30] AT %IB."P2_Robot_IRB1200".Module001_Input_30;
	Cyclic#1.P2_Robot.COM_IN.BYTE_IN[31] AT %IB."P2_Robot_IRB1200".Module001_Input_31;
	Cyclic#1.P2_Robot.COM_IN.BYTE_IN[32] AT %IB."P2_Robot_IRB1200".Module001_Input_32;
	Cyclic#1.P2_Robot.COM_IN.BYTE_IN[33] AT %IB."P2_Robot_IRB1200".Module001_Input_33;
	Cyclic#1.P2_Robot.COM_IN.BYTE_IN[34] AT %IB."P2_Robot_IRB1200".Module001_Input_34;
	Cyclic#1.P2_Robot.COM_IN.BYTE_IN[35] AT %IB."P2_Robot_IRB1200".Module001_Input_35;
	Cyclic#1.P2_Robot.COM_IN.BYTE_IN[36] AT %IB."P2_Robot_IRB1200".Module001_Input_36;
	Cyclic#1.P2_Robot.COM_IN.BYTE_IN[37] AT %IB."P2_Robot_IRB1200".Module001_Input_37;
	Cyclic#1.P2_Robot.COM_IN.BYTE_IN[38] AT %IB."P2_Robot_IRB1200".Module001_Input_38;
	Cyclic#1.P2_Robot.COM_IN.BYTE_IN[39] AT %IB."P2_Robot_IRB1200".Module001_Input_39;
	Cyclic#1.P2_Robot.COM_IN.BYTE_IN[40] AT %IB."P2_Robot_IRB1200".Module001_Input_40;
	Cyclic#1.P2_Robot.COM_IN.BYTE_IN[41] AT %IB."P2_Robot_IRB1200".Module001_Input_41;
	Cyclic#1.P2_Robot.COM_IN.BYTE_IN[42] AT %IB."P2_Robot_IRB1200".Module001_Input_42;
	Cyclic#1.P2_Robot.COM_IN.BYTE_IN[43] AT %IB."P2_Robot_IRB1200".Module001_Input_43;
	Cyclic#1.P2_Robot.COM_IN.BYTE_IN[44] AT %IB."P2_Robot_IRB1200".Module001_Input_44;
	Cyclic#1.P2_Robot.COM_IN.BYTE_IN[45] AT %IB."P2_Robot_IRB1200".Module001_Input_45;
	Cyclic#1.P2_Robot.COM_IN.BYTE_IN[46] AT %IB."P2_Robot_IRB1200".Module001_Input_46;
	Cyclic#1.P2_Robot.COM_IN.BYTE_IN[47] AT %IB."P2_Robot_IRB1200".Module001_Input_47;
	Cyclic#1.P2_Robot.COM_IN.BYTE_IN[48] AT %IB."P2_Robot_IRB1200".Module001_Input_48;
	Cyclic#1.P2_Robot.COM_IN.BYTE_IN[49] AT %IB."P2_Robot_IRB1200".Module001_Input_49;
	Cyclic#1.P2_Robot.COM_IN.BYTE_IN[50] AT %IB."P2_Robot_IRB1200".Module001_Input_50;
	Cyclic#1.P2_Robot.COM_IN.BYTE_IN[51] AT %IB."P2_Robot_IRB1200".Module001_Input_51;
	Cyclic#1.P2_Robot.COM_IN.BYTE_IN[52] AT %IB."P2_Robot_IRB1200".Module001_Input_52;
	Cyclic#1.P2_Robot.COM_IN.BYTE_IN[53] AT %IB."P2_Robot_IRB1200".Module001_Input_53;
	Cyclic#1.P2_Robot.COM_IN.BYTE_IN[54] AT %IB."P2_Robot_IRB1200".Module001_Input_54;
	Cyclic#1.P2_Robot.COM_IN.BYTE_IN[55] AT %IB."P2_Robot_IRB1200".Module001_Input_55;
	Cyclic#1.P2_Robot.COM_IN.BYTE_IN[56] AT %IB."P2_Robot_IRB1200".Module001_Input_56;
	Cyclic#1.P2_Robot.COM_IN.BYTE_IN[57] AT %IB."P2_Robot_IRB1200".Module001_Input_57;
	Cyclic#1.P2_Robot.COM_IN.BYTE_IN[58] AT %IB."P2_Robot_IRB1200".Module001_Input_58;
	Cyclic#1.P2_Robot.COM_IN.BYTE_IN[59] AT %IB."P2_Robot_IRB1200".Module001_Input_59;
	Cyclic#1.P2_Robot.COM_IN.BYTE_IN[60] AT %IB."P2_Robot_IRB1200".Module001_Input_60;
	Cyclic#1.P2_Robot.COM_IN.BYTE_IN[61] AT %IB."P2_Robot_IRB1200".Module001_Input_61;
	Cyclic#1.P2_Robot.COM_IN.BYTE_IN[62] AT %IB."P2_Robot_IRB1200".Module001_Input_62;
	Cyclic#1.P2_Robot.COM_IN.BYTE_IN[63] AT %IB."P2_Robot_IRB1200".Module001_Input_63;
	Cyclic#1.P2_Robot.COM_OUT.BYTE_OUT[1] AT %QB."P2_Robot_IRB1200".Module002_Output_1;
	Cyclic#1.P2_Robot.COM_OUT.BYTE_OUT[2] AT %QB."P2_Robot_IRB1200".Module002_Output_2;
	Cyclic#1.P2_Robot.COM_OUT.BYTE_OUT[3] AT %QB."P2_Robot_IRB1200".Module002_Output_3;
	Cyclic#1.P2_Robot.COM_OUT.BYTE_OUT[4] AT %QB."P2_Robot_IRB1200".Module002_Output_4;
	Cyclic#1.P2_Robot.COM_OUT.BYTE_OUT[5] AT %QB."P2_Robot_IRB1200".Module002_Output_5;
	Cyclic#1.P2_Robot.COM_OUT.BYTE_OUT[6] AT %QB."P2_Robot_IRB1200".Module002_Output_6;
	Cyclic#1.P2_Robot.COM_OUT.BYTE_OUT[7] AT %QB."P2_Robot_IRB1200".Module002_Output_7;
	Cyclic#1.P2_Robot.COM_OUT.BYTE_OUT[8] AT %QB."P2_Robot_IRB1200".Module002_Output_8;
	Cyclic#1.P2_Robot.COM_OUT.BYTE_OUT[9] AT %QB."P2_Robot_IRB1200".Module002_Output_9;
	Cyclic#1.P2_Robot.COM_OUT.BYTE_OUT[10] AT %QB."P2_Robot_IRB1200".Module002_Output_10;
	Cyclic#1.P2_Robot.COM_OUT.BYTE_OUT[11] AT %QB."P2_Robot_IRB1200".Module002_Output_11;
	Cyclic#1.P2_Robot.COM_OUT.BYTE_OUT[12] AT %QB."P2_Robot_IRB1200".Module002_Output_12;
	Cyclic#1.P2_Robot.COM_OUT.BYTE_OUT[13] AT %QB."P2_Robot_IRB1200".Module002_Output_13;
	Cyclic#1.P2_Robot.COM_OUT.BYTE_OUT[14] AT %QB."P2_Robot_IRB1200".Module002_Output_14;
	Cyclic#1.P2_Robot.COM_OUT.BYTE_OUT[15] AT %QB."P2_Robot_IRB1200".Module002_Output_15;
	Cyclic#1.P2_Robot.COM_OUT.BYTE_OUT[16] AT %QB."P2_Robot_IRB1200".Module002_Output_16;
	Cyclic#1.P2_Robot.COM_OUT.BYTE_OUT[17] AT %QB."P2_Robot_IRB1200".Module002_Output_17;
	Cyclic#1.P2_Robot.COM_OUT.BYTE_OUT[18] AT %QB."P2_Robot_IRB1200".Module002_Output_18;
	Cyclic#1.P2_Robot.COM_OUT.BYTE_OUT[19] AT %QB."P2_Robot_IRB1200".Module002_Output_19;
	Cyclic#1.P2_Robot.COM_OUT.BYTE_OUT[20] AT %QB."P2_Robot_IRB1200".Module002_Output_20;
	Cyclic#1.P2_Robot.COM_OUT.BYTE_OUT[21] AT %QB."P2_Robot_IRB1200".Module002_Output_21;
	Cyclic#1.P2_Robot.COM_OUT.BYTE_OUT[22] AT %QB."P2_Robot_IRB1200".Module002_Output_22;
	Cyclic#1.P2_Robot.COM_OUT.BYTE_OUT[23] AT %QB."P2_Robot_IRB1200".Module002_Output_23;
	Cyclic#1.P2_Robot.COM_OUT.BYTE_OUT[24] AT %QB."P2_Robot_IRB1200".Module002_Output_24;
	Cyclic#1.P2_Robot.COM_OUT.BYTE_OUT[25] AT %QB."P2_Robot_IRB1200".Module002_Output_25;
	Cyclic#1.P2_Robot.COM_OUT.BYTE_OUT[26] AT %QB."P2_Robot_IRB1200".Module002_Output_26;
	Cyclic#1.P2_Robot.COM_OUT.BYTE_OUT[27] AT %QB."P2_Robot_IRB1200".Module002_Output_27;
	Cyclic#1.P2_Robot.COM_OUT.BYTE_OUT[28] AT %QB."P2_Robot_IRB1200".Module002_Output_28;
	Cyclic#1.P2_Robot.COM_OUT.BYTE_OUT[29] AT %QB."P2_Robot_IRB1200".Module002_Output_29;
	Cyclic#1.P2_Robot.COM_OUT.BYTE_OUT[30] AT %QB."P2_Robot_IRB1200".Module002_Output_30;
	Cyclic#1.P2_Robot.COM_OUT.BYTE_OUT[31] AT %QB."P2_Robot_IRB1200".Module002_Output_31;
	Cyclic#1.P2_Robot.COM_OUT.BYTE_OUT[32] AT %QB."P2_Robot_IRB1200".Module002_Output_32;
	Cyclic#1.P2_Robot.COM_OUT.BYTE_OUT[33] AT %QB."P2_Robot_IRB1200".Module002_Output_33;
	Cyclic#1.P2_Robot.COM_OUT.BYTE_OUT[34] AT %QB."P2_Robot_IRB1200".Module002_Output_34;
	Cyclic#1.P2_Robot.COM_OUT.BYTE_OUT[35] AT %QB."P2_Robot_IRB1200".Module002_Output_35;
	Cyclic#1.P2_Robot.COM_OUT.BYTE_OUT[36] AT %QB."P2_Robot_IRB1200".Module002_Output_36;
	Cyclic#1.P2_Robot.COM_OUT.BYTE_OUT[37] AT %QB."P2_Robot_IRB1200".Module002_Output_37;
	Cyclic#1.P2_Robot.COM_OUT.BYTE_OUT[38] AT %QB."P2_Robot_IRB1200".Module002_Output_38;
	Cyclic#1.P2_Robot.COM_OUT.BYTE_OUT[39] AT %QB."P2_Robot_IRB1200".Module002_Output_39;
	Cyclic#1.P2_Robot.COM_OUT.BYTE_OUT[40] AT %QB."P2_Robot_IRB1200".Module002_Output_40;
	Cyclic#1.P2_Robot.COM_OUT.BYTE_OUT[41] AT %QB."P2_Robot_IRB1200".Module002_Output_41;
	Cyclic#1.P2_Robot.COM_OUT.BYTE_OUT[42] AT %QB."P2_Robot_IRB1200".Module002_Output_42;
	Cyclic#1.P2_Robot.COM_OUT.BYTE_OUT[43] AT %QB."P2_Robot_IRB1200".Module002_Output_43;
	Cyclic#1.P2_Robot.COM_OUT.BYTE_OUT[44] AT %QB."P2_Robot_IRB1200".Module002_Output_44;
	Cyclic#1.P2_Robot.COM_OUT.BYTE_OUT[45] AT %QB."P2_Robot_IRB1200".Module002_Output_45;
	Cyclic#1.P2_Robot.COM_OUT.BYTE_OUT[46] AT %QB."P2_Robot_IRB1200".Module002_Output_46;
	Cyclic#1.P2_Robot.COM_OUT.BYTE_OUT[47] AT %QB."P2_Robot_IRB1200".Module002_Output_47;
	Cyclic#1.P2_Robot.COM_OUT.BYTE_OUT[48] AT %QB."P2_Robot_IRB1200".Module002_Output_48;
	Cyclic#1.P2_Robot.COM_OUT.BYTE_OUT[49] AT %QB."P2_Robot_IRB1200".Module002_Output_49;
	Cyclic#1.P2_Robot.COM_OUT.BYTE_OUT[50] AT %QB."P2_Robot_IRB1200".Module002_Output_50;
	Cyclic#1.P2_Robot.COM_OUT.BYTE_OUT[51] AT %QB."P2_Robot_IRB1200".Module002_Output_51;
	Cyclic#1.P2_Robot.COM_OUT.BYTE_OUT[52] AT %QB."P2_Robot_IRB1200".Module002_Output_52;
	Cyclic#1.P2_Robot.COM_OUT.BYTE_OUT[53] AT %QB."P2_Robot_IRB1200".Module002_Output_53;
	Cyclic#1.P2_Robot.COM_OUT.BYTE_OUT[54] AT %QB."P2_Robot_IRB1200".Module002_Output_54;
	Cyclic#1.P2_Robot.COM_OUT.BYTE_OUT[55] AT %QB."P2_Robot_IRB1200".Module002_Output_55;
	Cyclic#1.P2_Robot.COM_OUT.BYTE_OUT[56] AT %QB."P2_Robot_IRB1200".Module002_Output_56;
	Cyclic#1.P2_Robot.COM_OUT.BYTE_OUT[57] AT %QB."P2_Robot_IRB1200".Module002_Output_57;
	Cyclic#1.P2_Robot.COM_OUT.BYTE_OUT[58] AT %QB."P2_Robot_IRB1200".Module002_Output_58;
	Cyclic#1.P2_Robot.COM_OUT.BYTE_OUT[59] AT %QB."P2_Robot_IRB1200".Module002_Output_59;
	Cyclic#1.P2_Robot.COM_OUT.BYTE_OUT[60] AT %QB."P2_Robot_IRB1200".Module002_Output_60;
	Cyclic#1.P2_Robot.COM_OUT.BYTE_OUT[61] AT %QB."P2_Robot_IRB1200".Module002_Output_61;
	Cyclic#1.P2_Robot.COM_OUT.BYTE_OUT[62] AT %QB."P2_Robot_IRB1200".Module002_Output_62;
	Cyclic#1.P2_Robot.COM_OUT.BYTE_OUT[63] AT %QB."P2_Robot_IRB1200".Module002_Output_63;
	Cyclic#1.P2_Pracovisko.IN.Maticovacka_M4_KomOK AT %IX."P2_MaticovackaM4".ModuleOk;
	Cyclic#1.P2_StoperMaticovacky.PAR.MaticeM4_AtlasCopcoInputs[0] AT %ID."P2_MaticovackaM4".Module001_Input_I_00;
	Cyclic#1.P2_StoperMaticovacky.PAR.MaticeM4_AtlasCopcoInputs[1] AT %ID."P2_MaticovackaM4".Module001_Input_I_01;
	Cyclic#1.P2_StoperMaticovacky.PAR.MaticeM4_AtlasCopcoInputs[2] AT %ID."P2_MaticovackaM4".Module002_Input_I_00;
	Cyclic#1.P2_StoperMaticovacky.PAR.MaticeM4_AtlasCopcoInputs[3] AT %ID."P2_MaticovackaM4".Module002_Input_I_01;
	Cyclic#1.P2_StoperMaticovacky.PAR.MaticeM4_AtlasCopcoInputs[4] AT %ID."P2_MaticovackaM4".Module003_Input_I_00;
	Cyclic#1.P2_StoperMaticovacky.PAR.MaticeM4_AtlasCopcoInputs[5] AT %ID."P2_MaticovackaM4".Module003_Input_I_01;
	Cyclic#1.P2_StoperMaticovacky.PAR.MaticeM4_AtlasCopcoInputs[6] AT %ID."P2_MaticovackaM4".Module004_Input_I_00;
	Cyclic#1.P2_StoperMaticovacky.PAR.MaticeM4_AtlasCopcoInputs[7] AT %ID."P2_MaticovackaM4".Module004_Input_I_01;
	Cyclic#1.P2_StoperMaticovacky.PAR.MaticeM4_AtlasCopcoOutputs[0] AT %QD."P2_MaticovackaM4".Module005_Output_O_00;
	Cyclic#1.P2_StoperMaticovacky.PAR.MaticeM4_AtlasCopcoOutputs[1] AT %QD."P2_MaticovackaM4".Module005_Output_O_01;
	Cyclic#1.P2_StoperMaticovacky.PAR.MaticeM4_AtlasCopcoOutputs[2] AT %QD."P2_MaticovackaM4".Module006_Output_O_00;
	Cyclic#1.P2_StoperMaticovacky.PAR.MaticeM4_AtlasCopcoOutputs[3] AT %QD."P2_MaticovackaM4".Module006_Output_O_01;
	Cyclic#1.P2_StoperMaticovacky.PAR.MaticeM4_AtlasCopcoOutputs[4] AT %QD."P2_MaticovackaM4".Module007_Output_O_00;
	Cyclic#1.P2_StoperMaticovacky.PAR.MaticeM4_AtlasCopcoOutputs[5] AT %QD."P2_MaticovackaM4".Module007_Output_O_01;
	Cyclic#1.P2_StoperMaticovacky.PAR.MaticeM4_AtlasCopcoOutputs[6] AT %QD."P2_MaticovackaM4".Module008_Output_O_00;
	Cyclic#1.P2_StoperMaticovacky.PAR.MaticeM4_AtlasCopcoOutputs[7] AT %QD."P2_MaticovackaM4".Module008_Output_O_01;
	Cyclic#1.P2_Pracovisko.IN.Skrutkovacka_M6_KomOK AT %IX."P2_SkrutkovackaM6".ModuleOk;
	Cyclic#1.P2_Srobovanie.PAR.M6_AtlasCopcoInputs[0] AT %ID."P2_SkrutkovackaM6".Module001_Input_I_00;
	Cyclic#1.P2_Srobovanie.PAR.M6_AtlasCopcoInputs[1] AT %ID."P2_SkrutkovackaM6".Module001_Input_I_01;
	Cyclic#1.P2_Srobovanie.PAR.M6_AtlasCopcoInputs[2] AT %ID."P2_SkrutkovackaM6".Module002_Input_I_00;
	Cyclic#1.P2_Srobovanie.PAR.M6_AtlasCopcoInputs[3] AT %ID."P2_SkrutkovackaM6".Module002_Input_I_01;
	Cyclic#1.P2_Srobovanie.PAR.M6_AtlasCopcoInputs[4] AT %ID."P2_SkrutkovackaM6".Module003_Input_I_00;
	Cyclic#1.P2_Srobovanie.PAR.M6_AtlasCopcoInputs[5] AT %ID."P2_SkrutkovackaM6".Module003_Input_I_01;
	Cyclic#1.P2_Srobovanie.PAR.M6_AtlasCopcoInputs[6] AT %ID."P2_SkrutkovackaM6".Module004_Input_I_00;
	Cyclic#1.P2_Srobovanie.PAR.M6_AtlasCopcoInputs[7] AT %ID."P2_SkrutkovackaM6".Module004_Input_I_01;
	Cyclic#1.P2_Srobovanie.PAR.M6_AtlasCopcoOutputs[0] AT %QD."P2_SkrutkovackaM6".Module005_Output_O_00;
	Cyclic#1.P2_Srobovanie.PAR.M6_AtlasCopcoOutputs[1] AT %QD."P2_SkrutkovackaM6".Module005_Output_O_01;
	Cyclic#1.P2_Srobovanie.PAR.M6_AtlasCopcoOutputs[2] AT %QD."P2_SkrutkovackaM6".Module006_Output_O_00;
	Cyclic#1.P2_Srobovanie.PAR.M6_AtlasCopcoOutputs[3] AT %QD."P2_SkrutkovackaM6".Module006_Output_O_01;
	Cyclic#1.P2_Srobovanie.PAR.M6_AtlasCopcoOutputs[4] AT %QD."P2_SkrutkovackaM6".Module007_Output_O_00;
	Cyclic#1.P2_Srobovanie.PAR.M6_AtlasCopcoOutputs[5] AT %QD."P2_SkrutkovackaM6".Module007_Output_O_01;
	Cyclic#1.P2_Srobovanie.PAR.M6_AtlasCopcoOutputs[6] AT %QD."P2_SkrutkovackaM6".Module008_Output_O_00;
	Cyclic#1.P2_Srobovanie.PAR.M6_AtlasCopcoOutputs[7] AT %QD."P2_SkrutkovackaM6".Module008_Output_O_01;
	Cyclic#1.P2_Pracovisko.IN.Skrutkovacka_M4_KomOK AT %IX."P2_SkrutkovackaM4".ModuleOk;
	Cyclic#1.P2_Srobovanie.PAR.M4_AtlasCopcoInputs[0] AT %ID."P2_SkrutkovackaM4".Module001_Input_I_00;
	Cyclic#1.P2_Srobovanie.PAR.M4_AtlasCopcoInputs[1] AT %ID."P2_SkrutkovackaM4".Module001_Input_I_01;
	Cyclic#1.P2_Srobovanie.PAR.M4_AtlasCopcoInputs[2] AT %ID."P2_SkrutkovackaM4".Module002_Input_I_00;
	Cyclic#1.P2_Srobovanie.PAR.M4_AtlasCopcoInputs[3] AT %ID."P2_SkrutkovackaM4".Module002_Input_I_01;
	Cyclic#1.P2_Srobovanie.PAR.M4_AtlasCopcoInputs[4] AT %ID."P2_SkrutkovackaM4".Module003_Input_I_00;
	Cyclic#1.P2_Srobovanie.PAR.M4_AtlasCopcoInputs[5] AT %ID."P2_SkrutkovackaM4".Module003_Input_I_01;
	Cyclic#1.P2_Srobovanie.PAR.M4_AtlasCopcoInputs[6] AT %ID."P2_SkrutkovackaM4".Module004_Input_I_00;
	Cyclic#1.P2_Srobovanie.PAR.M4_AtlasCopcoInputs[7] AT %ID."P2_SkrutkovackaM4".Module004_Input_I_01;
	Cyclic#1.P2_Srobovanie.PAR.M4_AtlasCopcoOutputs[0] AT %QD."P2_SkrutkovackaM4".Module005_Output_O_00;
	Cyclic#1.P2_Srobovanie.PAR.M4_AtlasCopcoOutputs[1] AT %QD."P2_SkrutkovackaM4".Module005_Output_O_01;
	Cyclic#1.P2_Srobovanie.PAR.M4_AtlasCopcoOutputs[2] AT %QD."P2_SkrutkovackaM4".Module006_Output_O_00;
	Cyclic#1.P2_Srobovanie.PAR.M4_AtlasCopcoOutputs[3] AT %QD."P2_SkrutkovackaM4".Module006_Output_O_01;
	Cyclic#1.P2_Srobovanie.PAR.M4_AtlasCopcoOutputs[4] AT %QD."P2_SkrutkovackaM4".Module007_Output_O_00;
	Cyclic#1.P2_Srobovanie.PAR.M4_AtlasCopcoOutputs[5] AT %QD."P2_SkrutkovackaM4".Module007_Output_O_01;
	Cyclic#1.P2_Srobovanie.PAR.M4_AtlasCopcoOutputs[6] AT %QD."P2_SkrutkovackaM4".Module008_Output_O_00;
	Cyclic#1.P2_Srobovanie.PAR.M4_AtlasCopcoOutputs[7] AT %QD."P2_SkrutkovackaM4".Module008_Output_O_01;
	Cyclic#1.P2_Pracovisko.IN.Skrutkovacka_M5_KomOK AT %IX."P2_SkrutkovackaM5".ModuleOk;
	Cyclic#1.P2_Srobovanie.PAR.M5_AtlasCopcoInputs[0] AT %ID."P2_SkrutkovackaM5".Module001_Input_I_00;
	Cyclic#1.P2_Srobovanie.PAR.M5_AtlasCopcoInputs[1] AT %ID."P2_SkrutkovackaM5".Module001_Input_I_01;
	Cyclic#1.P2_Srobovanie.PAR.M5_AtlasCopcoInputs[2] AT %ID."P2_SkrutkovackaM5".Module002_Input_I_00;
	Cyclic#1.P2_Srobovanie.PAR.M5_AtlasCopcoInputs[3] AT %ID."P2_SkrutkovackaM5".Module002_Input_I_01;
	Cyclic#1.P2_Srobovanie.PAR.M5_AtlasCopcoInputs[4] AT %ID."P2_SkrutkovackaM5".Module003_Input_I_00;
	Cyclic#1.P2_Srobovanie.PAR.M5_AtlasCopcoInputs[5] AT %ID."P2_SkrutkovackaM5".Module003_Input_I_01;
	Cyclic#1.P2_Srobovanie.PAR.M5_AtlasCopcoInputs[6] AT %ID."P2_SkrutkovackaM5".Module004_Input_I_00;
	Cyclic#1.P2_Srobovanie.PAR.M5_AtlasCopcoInputs[7] AT %ID."P2_SkrutkovackaM5".Module004_Input_I_01;
	Cyclic#1.P2_Srobovanie.PAR.M5_AtlasCopcoOutputs[0] AT %QD."P2_SkrutkovackaM5".Module005_Output_O_00;
	Cyclic#1.P2_Srobovanie.PAR.M5_AtlasCopcoOutputs[1] AT %QD."P2_SkrutkovackaM5".Module005_Output_O_01;
	Cyclic#1.P2_Srobovanie.PAR.M5_AtlasCopcoOutputs[2] AT %QD."P2_SkrutkovackaM5".Module006_Output_O_00;
	Cyclic#1.P2_Srobovanie.PAR.M5_AtlasCopcoOutputs[3] AT %QD."P2_SkrutkovackaM5".Module006_Output_O_01;
	Cyclic#1.P2_Srobovanie.PAR.M5_AtlasCopcoOutputs[4] AT %QD."P2_SkrutkovackaM5".Module007_Output_O_00;
	Cyclic#1.P2_Srobovanie.PAR.M5_AtlasCopcoOutputs[5] AT %QD."P2_SkrutkovackaM5".Module007_Output_O_01;
	Cyclic#1.P2_Srobovanie.PAR.M5_AtlasCopcoOutputs[6] AT %QD."P2_SkrutkovackaM5".Module008_Output_O_00;
	Cyclic#1.P2_Srobovanie.PAR.M5_AtlasCopcoOutputs[7] AT %QD."P2_SkrutkovackaM5".Module008_Output_O_01;
	Cyclic#1.P2_Pracovisko.IN.SmartKamera8_KomOK AT %IX."P2_CAM_8".ModuleOk;
	Cyclic#1.P2_Pracovisko.IN.SmartKamera9_KomOK AT %IX."P2_CAM_9".ModuleOk;
	Cyclic#1.P4_Pracovisko.IN.VentilovyTerminal_KomOK AT %IX."P4_VentilovyTerminal_VT4".ModuleOk;
	Cyclic#1.P4_Pracovisko.COM_VentilovyTerminal[0] AT %QB."P4_VentilovyTerminal_VT4".ValveCoils1_8_I2000_S01;
	Cyclic#1.P4_Pracovisko.COM_VentilovyTerminal[1] AT %QB."P4_VentilovyTerminal_VT4".ValveCoils9_16_I2000_S02;
	Cyclic#1.P4_Pracovisko.COM_VentilovyTerminal[2] AT %QB."P4_VentilovyTerminal_VT4".ValveCoils17_24_I2000_S03;
	Cyclic#1.P4_Pracovisko.COM_VentilovyTerminal[3] AT %QB."P4_VentilovyTerminal_VT4".ValveCoils25_32_I2000_S04;
	Cyclic#1.P4_Pracovisko.COM_VentilovyTerminal[4] AT %QB."P4_VentilovyTerminal_VT4".ValveCoils33_40_I2000_S05;
	Cyclic#1.P4_Pracovisko.COM_VentilovyTerminal[5] AT %QB."P4_VentilovyTerminal_VT4".ValveCoils41_48_I2000_S06;
	Cyclic#1.P4_Pracovisko.COM_VentilovyTerminal[6] AT %QB."P4_VentilovyTerminal_VT4".ValveCoils49_56_I2000_S07;
	Cyclic#1.P4_Pracovisko.IN.ModulFesto_IO_KomOK AT %IX."P4_IOmaster".ModuleOk;
	Cyclic#1.P2_Pracovisko.IN.ServoManipulatorOsX_KomOK AT %IX."P2_ServoManipOsX".ModuleOk;
	Cyclic#1.P2_Srobovanie.ServoManipulOsX.IN_forMapping.Status_word_1 AT %IW."P2_ServoManipOsX".Module001_Status_word_1;
	Cyclic#1.P2_Srobovanie.ServoManipulOsX.IN_forMapping.Position_Statusword_1 AT %IW."P2_ServoManipOsX".Module001_Position_Statusword_1;
	Cyclic#1.P2_Srobovanie.ServoManipulOsX.IN_forMapping.Position_Statusword_2 AT %IW."P2_ServoManipOsX".Module001_Position_Statusword_2;
	Cyclic#1.P2_Srobovanie.ServoManipulOsX.IN_forMapping.Status_word_2 AT %IW."P2_ServoManipOsX".Module001_Status_word_2;
	Cyclic#1.P2_Srobovanie.ServoManipulOsX.IN_forMapping.Report_word AT %IW."P2_ServoManipOsX".Module001_Report_word;
	Cyclic#1.P2_Srobovanie.ServoManipulOsX.IN_forMapping.Position_actual_value_A AT %ID."P2_ServoManipOsX".Module001_Position_actual_value_A;
	Cyclic#1.P2_Srobovanie.ServoManipulOsX.IN_forMapping.Speed_actual_value_B AT %ID."P2_ServoManipOsX".Module001_Speed_actual_value_B;
	Cyclic#1.P2_Srobovanie.ServoManipulOsX.IN_forMapping.Fault_Code AT %IW."P2_ServoManipOsX".Module001_Fault_Code;
	Cyclic#1.P2_Srobovanie.ServoManipulOsX.IN_forMapping.Warn_Code AT %IW."P2_ServoManipOsX".Module001_Warn_Code;
	Cyclic#1.P2_Srobovanie.ServoManipulOsX.IN_forMapping.User AT %IW."P2_ServoManipOsX".Module001_User;
	Cyclic#1.P2_Srobovanie.ServoManipulOsX.IN_forMapping.Status_word_or_actual_value_0 AT %IW."P2_ServoManipOsX".Module001_Status_word_or_actual_value_I_00;
	Cyclic#1.P2_Srobovanie.ServoManipulOsX.IN_forMapping.Status_word_or_actual_value_1 AT %IW."P2_ServoManipOsX".Module001_Status_word_or_actual_value_I_01;
	Cyclic#1.P2_Srobovanie.ServoManipulOsX.IN_forMapping.Status_word_or_actual_value_2 AT %IW."P2_ServoManipOsX".Module001_Status_word_or_actual_value_I_02;
	Cyclic#1.P2_Srobovanie.ServoManipulOsX.IN_forMapping.Status_word_or_actual_value_3 AT %IW."P2_ServoManipOsX".Module001_Status_word_or_actual_value_I_03;
	Cyclic#1.P2_Srobovanie.ServoManipulOsX.IN_forMapping.Status_word_or_actual_value_4 AT %IW."P2_ServoManipOsX".Module001_Status_word_or_actual_value_I_04;
	Cyclic#1.P2_Srobovanie.ServoManipulOsX.IN_forMapping.Status_word_or_actual_value_5 AT %IW."P2_ServoManipOsX".Module001_Status_word_or_actual_value_I_05;
	Cyclic#1.P2_Srobovanie.ServoManipulOsX.IN_forMapping.Status_word_or_actual_value_6 AT %IW."P2_ServoManipOsX".Module001_Status_word_or_actual_value_I_06;
	Cyclic#1.P2_Srobovanie.ServoManipulOsX.IN_forMapping.Status_word_or_actual_value_7 AT %IW."P2_ServoManipOsX".Module001_Status_word_or_actual_value_I_07;
	Cyclic#1.P2_Srobovanie.ServoManipulOsX.IN_forMapping.Status_word_or_actual_value_8 AT %IW."P2_ServoManipOsX".Module001_Status_word_or_actual_value_I_08;
	Cyclic#1.P2_Srobovanie.ServoManipulOsX.IN_forMapping.Status_word_or_actual_value_9 AT %IW."P2_ServoManipOsX".Module001_Status_word_or_actual_value_I_09;
	Cyclic#1.P2_Srobovanie.ServoManipulOsX.IN_forMapping.Status_word_or_actual_value_10 AT %IW."P2_ServoManipOsX".Module001_Status_word_or_actual_value_I_10;
	Cyclic#1.P2_Srobovanie.ServoManipulOsX.IN_forMapping.Status_word_or_actual_value_11 AT %IW."P2_ServoManipOsX".Module001_Status_word_or_actual_value_I_11;
	Cyclic#1.P2_Srobovanie.ServoManipulOsX.IN_forMapping.Status_word_or_actual_value_12 AT %IW."P2_ServoManipOsX".Module001_Status_word_or_actual_value_I_12;
	Cyclic#1.P2_Srobovanie.ServoManipulOsX.IN_forMapping.Status_word_or_actual_value_13 AT %IW."P2_ServoManipOsX".Module001_Status_word_or_actual_value_I_13;
	Cyclic#1.P2_Srobovanie.ServoManipulOsX.IN_forMapping.Status_word_or_actual_value_14 AT %IW."P2_ServoManipOsX".Module001_Status_word_or_actual_value_I_14;
	Cyclic#1.P2_Srobovanie.ServoManipulOsX.IN_forMapping.Status_word_or_actual_value_15 AT %IW."P2_ServoManipOsX".Module001_Status_word_or_actual_value_I_15;
	Cyclic#1.P2_Srobovanie.ServoManipulOsX.OUT_forMapping.Control_word_1 AT %QW."P2_ServoManipOsX".Module001_Control_word_1;
	Cyclic#1.P2_Srobovanie.ServoManipulOsX.OUT_forMapping.Position_Controlword_1 AT %QW."P2_ServoManipOsX".Module001_Position_Controlword_1;
	Cyclic#1.P2_Srobovanie.ServoManipulOsX.OUT_forMapping.Position_Controlword_2 AT %QW."P2_ServoManipOsX".Module001_Position_Controlword_2;
	Cyclic#1.P2_Srobovanie.ServoManipulOsX.OUT_forMapping.Control_word_2 AT %QW."P2_ServoManipOsX".Module001_Control_word_2;
	Cyclic#1.P2_Srobovanie.ServoManipulOsX.OUT_forMapping.Override AT %QW."P2_ServoManipOsX".Module001_Override;
	Cyclic#1.P2_Srobovanie.ServoManipulOsX.OUT_forMapping.MDI_target_position AT %QD."P2_ServoManipOsX".Module001_MDI_target_position;
	Cyclic#1.P2_Srobovanie.ServoManipulOsX.OUT_forMapping.MDI_velocity AT %QD."P2_ServoManipOsX".Module001_MDI_velocity;
	Cyclic#1.P2_Srobovanie.ServoManipulOsX.OUT_forMapping.MDI_acceleration AT %QW."P2_ServoManipOsX".Module001_MDI_acceleartion;
	Cyclic#1.P2_Srobovanie.ServoManipulOsX.OUT_forMapping.MDI_decceleration AT %QW."P2_ServoManipOsX".Module001_MDI_deceleration;
	Cyclic#1.P2_Srobovanie.ServoManipulOsX.OUT_forMapping.User1 AT %QW."P2_ServoManipOsX".Module001_User1;
	Cyclic#1.P2_Srobovanie.ServoManipulOsX.OUT_forMapping.Control_word_or_setpoint_0 AT %QW."P2_ServoManipOsX".Module001_Control_word_or_setpoint_O_00;
	Cyclic#1.P2_Srobovanie.ServoManipulOsX.OUT_forMapping.Control_word_or_setpoint_1 AT %QW."P2_ServoManipOsX".Module001_Control_word_or_setpoint_O_01;
	Cyclic#1.P2_Srobovanie.ServoManipulOsX.OUT_forMapping.Control_word_or_setpoint_2 AT %QW."P2_ServoManipOsX".Module001_Control_word_or_setpoint_O_02;
	Cyclic#1.P2_Srobovanie.ServoManipulOsX.OUT_forMapping.Control_word_or_setpoint_3 AT %QW."P2_ServoManipOsX".Module001_Control_word_or_setpoint_O_03;
	Cyclic#1.P2_Srobovanie.ServoManipulOsX.OUT_forMapping.Control_word_or_setpoint_4 AT %QW."P2_ServoManipOsX".Module001_Control_word_or_setpoint_O_04;
	Cyclic#1.P2_Srobovanie.ServoManipulOsX.OUT_forMapping.Control_word_or_setpoint_5 AT %QW."P2_ServoManipOsX".Module001_Control_word_or_setpoint_O_05;
	Cyclic#1.P2_Srobovanie.ServoManipulOsX.OUT_forMapping.Control_word_or_setpoint_6 AT %QW."P2_ServoManipOsX".Module001_Control_word_or_setpoint_O_06;
	Cyclic#1.P2_Srobovanie.ServoManipulOsX.OUT_forMapping.Control_word_or_setpoint_7 AT %QW."P2_ServoManipOsX".Module001_Control_word_or_setpoint_O_07;
	Cyclic#1.P2_Srobovanie.ServoManipulOsX.OUT_forMapping.Control_word_or_setpoint_8 AT %QW."P2_ServoManipOsX".Module001_Control_word_or_setpoint_O_08;
	Cyclic#1.P2_Srobovanie.ServoManipulOsX.OUT_forMapping.Control_word_or_setpoint_9 AT %QW."P2_ServoManipOsX".Module001_Control_word_or_setpoint_O_09;
	Cyclic#1.P2_Srobovanie.ServoManipulOsX.OUT_forMapping.Control_word_or_setpoint_10 AT %QW."P2_ServoManipOsX".Module001_Control_word_or_setpoint_O_10;
	Cyclic#1.P2_Srobovanie.ServoManipulOsX.OUT_forMapping.Control_word_or_setpoint_11 AT %QW."P2_ServoManipOsX".Module001_Control_word_or_setpoint_O_11;
	Cyclic#1.P2_Srobovanie.ServoManipulOsX.OUT_forMapping.Control_word_or_setpoint_12 AT %QW."P2_ServoManipOsX".Module001_Control_word_or_setpoint_O_12;
	Cyclic#1.P2_Srobovanie.ServoManipulOsX.OUT_forMapping.Control_word_or_setpoint_13 AT %QW."P2_ServoManipOsX".Module001_Control_word_or_setpoint_O_13;
	Cyclic#1.P2_Srobovanie.ServoManipulOsX.OUT_forMapping.Control_word_or_setpoint_14 AT %QW."P2_ServoManipOsX".Module001_Control_word_or_setpoint_O_14;
	Cyclic#1.P2_Srobovanie.ServoManipulOsX.OUT_forMapping.Control_word_or_setpoint_15 AT %QW."P2_ServoManipOsX".Module001_Control_word_or_setpoint_O_15;
	Cyclic#1.P2_Pracovisko.IN.ServoManipulatorOsY_KomOK AT %IX."P2_ServoManipOsY".ModuleOk;
	Cyclic#1.P2_Srobovanie.ServoManipulOsY.IN_forMapping.Status_word_1 AT %IW."P2_ServoManipOsY".Module001_Status_word_1;
	Cyclic#1.P2_Srobovanie.ServoManipulOsY.IN_forMapping.Position_Statusword_1 AT %IW."P2_ServoManipOsY".Module001_Position_Statusword_1;
	Cyclic#1.P2_Srobovanie.ServoManipulOsY.IN_forMapping.Position_Statusword_2 AT %IW."P2_ServoManipOsY".Module001_Position_Statusword_2;
	Cyclic#1.P2_Srobovanie.ServoManipulOsY.IN_forMapping.Status_word_2 AT %IW."P2_ServoManipOsY".Module001_Status_word_2;
	Cyclic#1.P2_Srobovanie.ServoManipulOsY.IN_forMapping.Report_word AT %IW."P2_ServoManipOsY".Module001_Report_word;
	Cyclic#1.P2_Srobovanie.ServoManipulOsY.IN_forMapping.Position_actual_value_A AT %ID."P2_ServoManipOsY".Module001_Position_actual_value_A;
	Cyclic#1.P2_Srobovanie.ServoManipulOsY.IN_forMapping.Speed_actual_value_B AT %ID."P2_ServoManipOsY".Module001_Speed_actual_value_B;
	Cyclic#1.P2_Srobovanie.ServoManipulOsY.IN_forMapping.Fault_Code AT %IW."P2_ServoManipOsY".Module001_Fault_Code;
	Cyclic#1.P2_Srobovanie.ServoManipulOsY.IN_forMapping.Warn_Code AT %IW."P2_ServoManipOsY".Module001_Warn_Code;
	Cyclic#1.P2_Srobovanie.ServoManipulOsY.IN_forMapping.User AT %IW."P2_ServoManipOsY".Module001_User;
	Cyclic#1.P2_Srobovanie.ServoManipulOsY.IN_forMapping.Status_word_or_actual_value_0 AT %IW."P2_ServoManipOsY".Module001_Status_word_or_actual_value_I_00;
	Cyclic#1.P2_Srobovanie.ServoManipulOsY.IN_forMapping.Status_word_or_actual_value_1 AT %IW."P2_ServoManipOsY".Module001_Status_word_or_actual_value_I_01;
	Cyclic#1.P2_Srobovanie.ServoManipulOsY.IN_forMapping.Status_word_or_actual_value_2 AT %IW."P2_ServoManipOsY".Module001_Status_word_or_actual_value_I_02;
	Cyclic#1.P2_Srobovanie.ServoManipulOsY.IN_forMapping.Status_word_or_actual_value_3 AT %IW."P2_ServoManipOsY".Module001_Status_word_or_actual_value_I_03;
	Cyclic#1.P2_Srobovanie.ServoManipulOsY.IN_forMapping.Status_word_or_actual_value_4 AT %IW."P2_ServoManipOsY".Module001_Status_word_or_actual_value_I_04;
	Cyclic#1.P2_Srobovanie.ServoManipulOsY.IN_forMapping.Status_word_or_actual_value_5 AT %IW."P2_ServoManipOsY".Module001_Status_word_or_actual_value_I_05;
	Cyclic#1.P2_Srobovanie.ServoManipulOsY.IN_forMapping.Status_word_or_actual_value_6 AT %IW."P2_ServoManipOsY".Module001_Status_word_or_actual_value_I_06;
	Cyclic#1.P2_Srobovanie.ServoManipulOsY.IN_forMapping.Status_word_or_actual_value_7 AT %IW."P2_ServoManipOsY".Module001_Status_word_or_actual_value_I_07;
	Cyclic#1.P2_Srobovanie.ServoManipulOsY.IN_forMapping.Status_word_or_actual_value_8 AT %IW."P2_ServoManipOsY".Module001_Status_word_or_actual_value_I_08;
	Cyclic#1.P2_Srobovanie.ServoManipulOsY.IN_forMapping.Status_word_or_actual_value_9 AT %IW."P2_ServoManipOsY".Module001_Status_word_or_actual_value_I_09;
	Cyclic#1.P2_Srobovanie.ServoManipulOsY.IN_forMapping.Status_word_or_actual_value_10 AT %IW."P2_ServoManipOsY".Module001_Status_word_or_actual_value_I_10;
	Cyclic#1.P2_Srobovanie.ServoManipulOsY.IN_forMapping.Status_word_or_actual_value_11 AT %IW."P2_ServoManipOsY".Module001_Status_word_or_actual_value_I_11;
	Cyclic#1.P2_Srobovanie.ServoManipulOsY.IN_forMapping.Status_word_or_actual_value_12 AT %IW."P2_ServoManipOsY".Module001_Status_word_or_actual_value_I_12;
	Cyclic#1.P2_Srobovanie.ServoManipulOsY.IN_forMapping.Status_word_or_actual_value_13 AT %IW."P2_ServoManipOsY".Module001_Status_word_or_actual_value_I_13;
	Cyclic#1.P2_Srobovanie.ServoManipulOsY.IN_forMapping.Status_word_or_actual_value_14 AT %IW."P2_ServoManipOsY".Module001_Status_word_or_actual_value_I_14;
	Cyclic#1.P2_Srobovanie.ServoManipulOsY.IN_forMapping.Status_word_or_actual_value_15 AT %IW."P2_ServoManipOsY".Module001_Status_word_or_actual_value_I_15;
	Cyclic#1.P2_Srobovanie.ServoManipulOsY.OUT_forMapping.Control_word_1 AT %QW."P2_ServoManipOsY".Module001_Control_word_1;
	Cyclic#1.P2_Srobovanie.ServoManipulOsY.OUT_forMapping.Position_Controlword_1 AT %QW."P2_ServoManipOsY".Module001_Position_Controlword_1;
	Cyclic#1.P2_Srobovanie.ServoManipulOsY.OUT_forMapping.Position_Controlword_2 AT %QW."P2_ServoManipOsY".Module001_Position_Controlword_2;
	Cyclic#1.P2_Srobovanie.ServoManipulOsY.OUT_forMapping.Control_word_2 AT %QW."P2_ServoManipOsY".Module001_Control_word_2;
	Cyclic#1.P2_Srobovanie.ServoManipulOsY.OUT_forMapping.Override AT %QW."P2_ServoManipOsY".Module001_Override;
	Cyclic#1.P2_Srobovanie.ServoManipulOsY.OUT_forMapping.MDI_target_position AT %QD."P2_ServoManipOsY".Module001_MDI_target_position;
	Cyclic#1.P2_Srobovanie.ServoManipulOsY.OUT_forMapping.MDI_velocity AT %QD."P2_ServoManipOsY".Module001_MDI_velocity;
	Cyclic#1.P2_Srobovanie.ServoManipulOsY.OUT_forMapping.MDI_acceleration AT %QW."P2_ServoManipOsY".Module001_MDI_acceleartion;
	Cyclic#1.P2_Srobovanie.ServoManipulOsY.OUT_forMapping.MDI_decceleration AT %QW."P2_ServoManipOsY".Module001_MDI_deceleration;
	Cyclic#1.P2_Srobovanie.ServoManipulOsY.OUT_forMapping.User1 AT %QW."P2_ServoManipOsY".Module001_User1;
	Cyclic#1.P2_Srobovanie.ServoManipulOsY.OUT_forMapping.Control_word_or_setpoint_0 AT %QW."P2_ServoManipOsY".Module001_Control_word_or_setpoint_O_00;
	Cyclic#1.P2_Srobovanie.ServoManipulOsY.OUT_forMapping.Control_word_or_setpoint_1 AT %QW."P2_ServoManipOsY".Module001_Control_word_or_setpoint_O_01;
	Cyclic#1.P2_Srobovanie.ServoManipulOsY.OUT_forMapping.Control_word_or_setpoint_2 AT %QW."P2_ServoManipOsY".Module001_Control_word_or_setpoint_O_02;
	Cyclic#1.P2_Srobovanie.ServoManipulOsY.OUT_forMapping.Control_word_or_setpoint_3 AT %QW."P2_ServoManipOsY".Module001_Control_word_or_setpoint_O_03;
	Cyclic#1.P2_Srobovanie.ServoManipulOsY.OUT_forMapping.Control_word_or_setpoint_4 AT %QW."P2_ServoManipOsY".Module001_Control_word_or_setpoint_O_04;
	Cyclic#1.P2_Srobovanie.ServoManipulOsY.OUT_forMapping.Control_word_or_setpoint_5 AT %QW."P2_ServoManipOsY".Module001_Control_word_or_setpoint_O_05;
	Cyclic#1.P2_Srobovanie.ServoManipulOsY.OUT_forMapping.Control_word_or_setpoint_6 AT %QW."P2_ServoManipOsY".Module001_Control_word_or_setpoint_O_06;
	Cyclic#1.P2_Srobovanie.ServoManipulOsY.OUT_forMapping.Control_word_or_setpoint_7 AT %QW."P2_ServoManipOsY".Module001_Control_word_or_setpoint_O_07;
	Cyclic#1.P2_Srobovanie.ServoManipulOsY.OUT_forMapping.Control_word_or_setpoint_8 AT %QW."P2_ServoManipOsY".Module001_Control_word_or_setpoint_O_08;
	Cyclic#1.P2_Srobovanie.ServoManipulOsY.OUT_forMapping.Control_word_or_setpoint_9 AT %QW."P2_ServoManipOsY".Module001_Control_word_or_setpoint_O_09;
	Cyclic#1.P2_Srobovanie.ServoManipulOsY.OUT_forMapping.Control_word_or_setpoint_10 AT %QW."P2_ServoManipOsY".Module001_Control_word_or_setpoint_O_10;
	Cyclic#1.P2_Srobovanie.ServoManipulOsY.OUT_forMapping.Control_word_or_setpoint_11 AT %QW."P2_ServoManipOsY".Module001_Control_word_or_setpoint_O_11;
	Cyclic#1.P2_Srobovanie.ServoManipulOsY.OUT_forMapping.Control_word_or_setpoint_12 AT %QW."P2_ServoManipOsY".Module001_Control_word_or_setpoint_O_12;
	Cyclic#1.P2_Srobovanie.ServoManipulOsY.OUT_forMapping.Control_word_or_setpoint_13 AT %QW."P2_ServoManipOsY".Module001_Control_word_or_setpoint_O_13;
	Cyclic#1.P2_Srobovanie.ServoManipulOsY.OUT_forMapping.Control_word_or_setpoint_14 AT %QW."P2_ServoManipOsY".Module001_Control_word_or_setpoint_O_14;
	Cyclic#1.P2_Srobovanie.ServoManipulOsY.OUT_forMapping.Control_word_or_setpoint_15 AT %QW."P2_ServoManipOsY".Module001_Control_word_or_setpoint_O_15;
	Cyclic#1.P2_Pracovisko.IN.ServoManipulatorOsZ_M4_KomOK AT %IX."P2_ServoManipOsZ_M4".ModuleOk;
	Cyclic#1.P2_Srobovanie.ServoManipulOsZ_M4.IN_forMapping.Status_word_1 AT %IW."P2_ServoManipOsZ_M4".Module001_Status_word_1;
	Cyclic#1.P2_Srobovanie.ServoManipulOsZ_M4.IN_forMapping.Position_Statusword_1 AT %IW."P2_ServoManipOsZ_M4".Module001_Position_Statusword_1;
	Cyclic#1.P2_Srobovanie.ServoManipulOsZ_M4.IN_forMapping.Position_Statusword_2 AT %IW."P2_ServoManipOsZ_M4".Module001_Position_Statusword_2;
	Cyclic#1.P2_Srobovanie.ServoManipulOsZ_M4.IN_forMapping.Status_word_2 AT %IW."P2_ServoManipOsZ_M4".Module001_Status_word_2;
	Cyclic#1.P2_Srobovanie.ServoManipulOsZ_M4.IN_forMapping.Report_word AT %IW."P2_ServoManipOsZ_M4".Module001_Report_word;
	Cyclic#1.P2_Srobovanie.ServoManipulOsZ_M4.IN_forMapping.Position_actual_value_A AT %ID."P2_ServoManipOsZ_M4".Module001_Position_actual_value_A;
	Cyclic#1.P2_Srobovanie.ServoManipulOsZ_M4.IN_forMapping.Speed_actual_value_B AT %ID."P2_ServoManipOsZ_M4".Module001_Speed_actual_value_B;
	Cyclic#1.P2_Srobovanie.ServoManipulOsZ_M4.IN_forMapping.Fault_Code AT %IW."P2_ServoManipOsZ_M4".Module001_Fault_Code;
	Cyclic#1.P2_Srobovanie.ServoManipulOsZ_M4.IN_forMapping.Warn_Code AT %IW."P2_ServoManipOsZ_M4".Module001_Warn_Code;
	Cyclic#1.P2_Srobovanie.ServoManipulOsZ_M4.IN_forMapping.User AT %IW."P2_ServoManipOsZ_M4".Module001_User;
	Cyclic#1.P2_Srobovanie.ServoManipulOsZ_M4.IN_forMapping.Status_word_or_actual_value_0 AT %IW."P2_ServoManipOsZ_M4".Module001_Status_word_or_actual_value_I_00;
	Cyclic#1.P2_Srobovanie.ServoManipulOsZ_M4.IN_forMapping.Status_word_or_actual_value_1 AT %IW."P2_ServoManipOsZ_M4".Module001_Status_word_or_actual_value_I_01;
	Cyclic#1.P2_Srobovanie.ServoManipulOsZ_M4.IN_forMapping.Status_word_or_actual_value_2 AT %IW."P2_ServoManipOsZ_M4".Module001_Status_word_or_actual_value_I_02;
	Cyclic#1.P2_Srobovanie.ServoManipulOsZ_M4.IN_forMapping.Status_word_or_actual_value_3 AT %IW."P2_ServoManipOsZ_M4".Module001_Status_word_or_actual_value_I_03;
	Cyclic#1.P2_Srobovanie.ServoManipulOsZ_M4.IN_forMapping.Status_word_or_actual_value_4 AT %IW."P2_ServoManipOsZ_M4".Module001_Status_word_or_actual_value_I_04;
	Cyclic#1.P2_Srobovanie.ServoManipulOsZ_M4.IN_forMapping.Status_word_or_actual_value_5 AT %IW."P2_ServoManipOsZ_M4".Module001_Status_word_or_actual_value_I_05;
	Cyclic#1.P2_Srobovanie.ServoManipulOsZ_M4.IN_forMapping.Status_word_or_actual_value_6 AT %IW."P2_ServoManipOsZ_M4".Module001_Status_word_or_actual_value_I_06;
	Cyclic#1.P2_Srobovanie.ServoManipulOsZ_M4.IN_forMapping.Status_word_or_actual_value_7 AT %IW."P2_ServoManipOsZ_M4".Module001_Status_word_or_actual_value_I_07;
	Cyclic#1.P2_Srobovanie.ServoManipulOsZ_M4.IN_forMapping.Status_word_or_actual_value_8 AT %IW."P2_ServoManipOsZ_M4".Module001_Status_word_or_actual_value_I_08;
	Cyclic#1.P2_Srobovanie.ServoManipulOsZ_M4.IN_forMapping.Status_word_or_actual_value_9 AT %IW."P2_ServoManipOsZ_M4".Module001_Status_word_or_actual_value_I_09;
	Cyclic#1.P2_Srobovanie.ServoManipulOsZ_M4.IN_forMapping.Status_word_or_actual_value_10 AT %IW."P2_ServoManipOsZ_M4".Module001_Status_word_or_actual_value_I_10;
	Cyclic#1.P2_Srobovanie.ServoManipulOsZ_M4.IN_forMapping.Status_word_or_actual_value_11 AT %IW."P2_ServoManipOsZ_M4".Module001_Status_word_or_actual_value_I_11;
	Cyclic#1.P2_Srobovanie.ServoManipulOsZ_M4.IN_forMapping.Status_word_or_actual_value_12 AT %IW."P2_ServoManipOsZ_M4".Module001_Status_word_or_actual_value_I_12;
	Cyclic#1.P2_Srobovanie.ServoManipulOsZ_M4.IN_forMapping.Status_word_or_actual_value_13 AT %IW."P2_ServoManipOsZ_M4".Module001_Status_word_or_actual_value_I_13;
	Cyclic#1.P2_Srobovanie.ServoManipulOsZ_M4.IN_forMapping.Status_word_or_actual_value_14 AT %IW."P2_ServoManipOsZ_M4".Module001_Status_word_or_actual_value_I_14;
	Cyclic#1.P2_Srobovanie.ServoManipulOsZ_M4.IN_forMapping.Status_word_or_actual_value_15 AT %IW."P2_ServoManipOsZ_M4".Module001_Status_word_or_actual_value_I_15;
	Cyclic#1.P2_Srobovanie.ServoManipulOsZ_M4.OUT_forMapping.Control_word_1 AT %QW."P2_ServoManipOsZ_M4".Module001_Control_word_1;
	Cyclic#1.P2_Srobovanie.ServoManipulOsZ_M4.OUT_forMapping.Position_Controlword_1 AT %QW."P2_ServoManipOsZ_M4".Module001_Position_Controlword_1;
	Cyclic#1.P2_Srobovanie.ServoManipulOsZ_M4.OUT_forMapping.Position_Controlword_2 AT %QW."P2_ServoManipOsZ_M4".Module001_Position_Controlword_2;
	Cyclic#1.P2_Srobovanie.ServoManipulOsZ_M4.OUT_forMapping.Control_word_2 AT %QW."P2_ServoManipOsZ_M4".Module001_Control_word_2;
	Cyclic#1.P2_Srobovanie.ServoManipulOsZ_M4.OUT_forMapping.Override AT %QW."P2_ServoManipOsZ_M4".Module001_Override;
	Cyclic#1.P2_Srobovanie.ServoManipulOsZ_M4.OUT_forMapping.MDI_target_position AT %QD."P2_ServoManipOsZ_M4".Module001_MDI_target_position;
	Cyclic#1.P2_Srobovanie.ServoManipulOsZ_M4.OUT_forMapping.MDI_velocity AT %QD."P2_ServoManipOsZ_M4".Module001_MDI_velocity;
	Cyclic#1.P2_Srobovanie.ServoManipulOsZ_M4.OUT_forMapping.MDI_acceleration AT %QW."P2_ServoManipOsZ_M4".Module001_MDI_acceleartion;
	Cyclic#1.P2_Srobovanie.ServoManipulOsZ_M4.OUT_forMapping.MDI_decceleration AT %QW."P2_ServoManipOsZ_M4".Module001_MDI_deceleration;
	Cyclic#1.P2_Srobovanie.ServoManipulOsZ_M4.OUT_forMapping.User1 AT %QW."P2_ServoManipOsZ_M4".Module001_User1;
	Cyclic#1.P2_Srobovanie.ServoManipulOsZ_M4.OUT_forMapping.Control_word_or_setpoint_0 AT %QW."P2_ServoManipOsZ_M4".Module001_Control_word_or_setpoint_O_00;
	Cyclic#1.P2_Srobovanie.ServoManipulOsZ_M4.OUT_forMapping.Control_word_or_setpoint_1 AT %QW."P2_ServoManipOsZ_M4".Module001_Control_word_or_setpoint_O_01;
	Cyclic#1.P2_Srobovanie.ServoManipulOsZ_M4.OUT_forMapping.Control_word_or_setpoint_2 AT %QW."P2_ServoManipOsZ_M4".Module001_Control_word_or_setpoint_O_02;
	Cyclic#1.P2_Srobovanie.ServoManipulOsZ_M4.OUT_forMapping.Control_word_or_setpoint_3 AT %QW."P2_ServoManipOsZ_M4".Module001_Control_word_or_setpoint_O_03;
	Cyclic#1.P2_Srobovanie.ServoManipulOsZ_M4.OUT_forMapping.Control_word_or_setpoint_4 AT %QW."P2_ServoManipOsZ_M4".Module001_Control_word_or_setpoint_O_04;
	Cyclic#1.P2_Srobovanie.ServoManipulOsZ_M4.OUT_forMapping.Control_word_or_setpoint_5 AT %QW."P2_ServoManipOsZ_M4".Module001_Control_word_or_setpoint_O_05;
	Cyclic#1.P2_Srobovanie.ServoManipulOsZ_M4.OUT_forMapping.Control_word_or_setpoint_6 AT %QW."P2_ServoManipOsZ_M4".Module001_Control_word_or_setpoint_O_06;
	Cyclic#1.P2_Srobovanie.ServoManipulOsZ_M4.OUT_forMapping.Control_word_or_setpoint_7 AT %QW."P2_ServoManipOsZ_M4".Module001_Control_word_or_setpoint_O_07;
	Cyclic#1.P2_Srobovanie.ServoManipulOsZ_M4.OUT_forMapping.Control_word_or_setpoint_8 AT %QW."P2_ServoManipOsZ_M4".Module001_Control_word_or_setpoint_O_08;
	Cyclic#1.P2_Srobovanie.ServoManipulOsZ_M4.OUT_forMapping.Control_word_or_setpoint_9 AT %QW."P2_ServoManipOsZ_M4".Module001_Control_word_or_setpoint_O_09;
	Cyclic#1.P2_Srobovanie.ServoManipulOsZ_M4.OUT_forMapping.Control_word_or_setpoint_10 AT %QW."P2_ServoManipOsZ_M4".Module001_Control_word_or_setpoint_O_10;
	Cyclic#1.P2_Srobovanie.ServoManipulOsZ_M4.OUT_forMapping.Control_word_or_setpoint_11 AT %QW."P2_ServoManipOsZ_M4".Module001_Control_word_or_setpoint_O_11;
	Cyclic#1.P2_Srobovanie.ServoManipulOsZ_M4.OUT_forMapping.Control_word_or_setpoint_12 AT %QW."P2_ServoManipOsZ_M4".Module001_Control_word_or_setpoint_O_12;
	Cyclic#1.P2_Srobovanie.ServoManipulOsZ_M4.OUT_forMapping.Control_word_or_setpoint_13 AT %QW."P2_ServoManipOsZ_M4".Module001_Control_word_or_setpoint_O_13;
	Cyclic#1.P2_Srobovanie.ServoManipulOsZ_M4.OUT_forMapping.Control_word_or_setpoint_14 AT %QW."P2_ServoManipOsZ_M4".Module001_Control_word_or_setpoint_O_14;
	Cyclic#1.P2_Srobovanie.ServoManipulOsZ_M4.OUT_forMapping.Control_word_or_setpoint_15 AT %QW."P2_ServoManipOsZ_M4".Module001_Control_word_or_setpoint_O_15;
	Cyclic#1.P2_Pracovisko.IN.ServoZaklTesneniaZdvih_KomOK AT %IX."P2_ServoZatlTesneniaZdvih".ModuleOk;
	Cyclic#1.P2_ZakladacTesnenia.ServoZdvihuZakladaca.IN_forMapping.Status_word_1 AT %IW."P2_ServoZatlTesneniaZdvih".Module001_Status_word_1;
	Cyclic#1.P2_ZakladacTesnenia.ServoZdvihuZakladaca.IN_forMapping.Position_Statusword_1 AT %IW."P2_ServoZatlTesneniaZdvih".Module001_Position_Statusword_1;
	Cyclic#1.P2_ZakladacTesnenia.ServoZdvihuZakladaca.IN_forMapping.Position_Statusword_2 AT %IW."P2_ServoZatlTesneniaZdvih".Module001_Position_Statusword_2;
	Cyclic#1.P2_ZakladacTesnenia.ServoZdvihuZakladaca.IN_forMapping.Status_word_2 AT %IW."P2_ServoZatlTesneniaZdvih".Module001_Status_word_2;
	Cyclic#1.P2_ZakladacTesnenia.ServoZdvihuZakladaca.IN_forMapping.Report_word AT %IW."P2_ServoZatlTesneniaZdvih".Module001_Report_word;
	Cyclic#1.P2_ZakladacTesnenia.ServoZdvihuZakladaca.IN_forMapping.Position_actual_value_A AT %ID."P2_ServoZatlTesneniaZdvih".Module001_Position_actual_value_A;
	Cyclic#1.P2_ZakladacTesnenia.ServoZdvihuZakladaca.IN_forMapping.Speed_actual_value_B AT %ID."P2_ServoZatlTesneniaZdvih".Module001_Speed_actual_value_B;
	Cyclic#1.P2_ZakladacTesnenia.ServoZdvihuZakladaca.IN_forMapping.Fault_Code AT %IW."P2_ServoZatlTesneniaZdvih".Module001_Fault_Code;
	Cyclic#1.P2_ZakladacTesnenia.ServoZdvihuZakladaca.IN_forMapping.Warn_Code AT %IW."P2_ServoZatlTesneniaZdvih".Module001_Warn_Code;
	Cyclic#1.P2_ZakladacTesnenia.ServoZdvihuZakladaca.IN_forMapping.User AT %IW."P2_ServoZatlTesneniaZdvih".Module001_User;
	Cyclic#1.P2_ZakladacTesnenia.ServoZdvihuZakladaca.IN_forMapping.Status_word_or_actual_value_0 AT %IW."P2_ServoZatlTesneniaZdvih".Module001_Status_word_or_actual_value_I_00;
	Cyclic#1.P2_ZakladacTesnenia.ServoZdvihuZakladaca.IN_forMapping.Status_word_or_actual_value_1 AT %IW."P2_ServoZatlTesneniaZdvih".Module001_Status_word_or_actual_value_I_01;
	Cyclic#1.P2_ZakladacTesnenia.ServoZdvihuZakladaca.IN_forMapping.Status_word_or_actual_value_2 AT %IW."P2_ServoZatlTesneniaZdvih".Module001_Status_word_or_actual_value_I_02;
	Cyclic#1.P2_ZakladacTesnenia.ServoZdvihuZakladaca.IN_forMapping.Status_word_or_actual_value_3 AT %IW."P2_ServoZatlTesneniaZdvih".Module001_Status_word_or_actual_value_I_03;
	Cyclic#1.P2_ZakladacTesnenia.ServoZdvihuZakladaca.IN_forMapping.Status_word_or_actual_value_4 AT %IW."P2_ServoZatlTesneniaZdvih".Module001_Status_word_or_actual_value_I_04;
	Cyclic#1.P2_ZakladacTesnenia.ServoZdvihuZakladaca.IN_forMapping.Status_word_or_actual_value_5 AT %IW."P2_ServoZatlTesneniaZdvih".Module001_Status_word_or_actual_value_I_05;
	Cyclic#1.P2_ZakladacTesnenia.ServoZdvihuZakladaca.IN_forMapping.Status_word_or_actual_value_6 AT %IW."P2_ServoZatlTesneniaZdvih".Module001_Status_word_or_actual_value_I_06;
	Cyclic#1.P2_ZakladacTesnenia.ServoZdvihuZakladaca.IN_forMapping.Status_word_or_actual_value_7 AT %IW."P2_ServoZatlTesneniaZdvih".Module001_Status_word_or_actual_value_I_07;
	Cyclic#1.P2_ZakladacTesnenia.ServoZdvihuZakladaca.IN_forMapping.Status_word_or_actual_value_8 AT %IW."P2_ServoZatlTesneniaZdvih".Module001_Status_word_or_actual_value_I_08;
	Cyclic#1.P2_ZakladacTesnenia.ServoZdvihuZakladaca.IN_forMapping.Status_word_or_actual_value_9 AT %IW."P2_ServoZatlTesneniaZdvih".Module001_Status_word_or_actual_value_I_09;
	Cyclic#1.P2_ZakladacTesnenia.ServoZdvihuZakladaca.IN_forMapping.Status_word_or_actual_value_10 AT %IW."P2_ServoZatlTesneniaZdvih".Module001_Status_word_or_actual_value_I_10;
	Cyclic#1.P2_ZakladacTesnenia.ServoZdvihuZakladaca.IN_forMapping.Status_word_or_actual_value_11 AT %IW."P2_ServoZatlTesneniaZdvih".Module001_Status_word_or_actual_value_I_11;
	Cyclic#1.P2_ZakladacTesnenia.ServoZdvihuZakladaca.IN_forMapping.Status_word_or_actual_value_12 AT %IW."P2_ServoZatlTesneniaZdvih".Module001_Status_word_or_actual_value_I_12;
	Cyclic#1.P2_ZakladacTesnenia.ServoZdvihuZakladaca.IN_forMapping.Status_word_or_actual_value_13 AT %IW."P2_ServoZatlTesneniaZdvih".Module001_Status_word_or_actual_value_I_13;
	Cyclic#1.P2_ZakladacTesnenia.ServoZdvihuZakladaca.IN_forMapping.Status_word_or_actual_value_14 AT %IW."P2_ServoZatlTesneniaZdvih".Module001_Status_word_or_actual_value_I_14;
	Cyclic#1.P2_ZakladacTesnenia.ServoZdvihuZakladaca.IN_forMapping.Status_word_or_actual_value_15 AT %IW."P2_ServoZatlTesneniaZdvih".Module001_Status_word_or_actual_value_I_15;
	Cyclic#1.P2_ZakladacTesnenia.ServoZdvihuZakladaca.OUT_forMapping.Control_word_1 AT %QW."P2_ServoZatlTesneniaZdvih".Module001_Control_word_1;
	Cyclic#1.P2_ZakladacTesnenia.ServoZdvihuZakladaca.OUT_forMapping.Position_Controlword_1 AT %QW."P2_ServoZatlTesneniaZdvih".Module001_Position_Controlword_1;
	Cyclic#1.P2_ZakladacTesnenia.ServoZdvihuZakladaca.OUT_forMapping.Position_Controlword_2 AT %QW."P2_ServoZatlTesneniaZdvih".Module001_Position_Controlword_2;
	Cyclic#1.P2_ZakladacTesnenia.ServoZdvihuZakladaca.OUT_forMapping.Control_word_2 AT %QW."P2_ServoZatlTesneniaZdvih".Module001_Control_word_2;
	Cyclic#1.P2_ZakladacTesnenia.ServoZdvihuZakladaca.OUT_forMapping.Override AT %QW."P2_ServoZatlTesneniaZdvih".Module001_Override;
	Cyclic#1.P2_ZakladacTesnenia.ServoZdvihuZakladaca.OUT_forMapping.MDI_target_position AT %QD."P2_ServoZatlTesneniaZdvih".Module001_MDI_target_position;
	Cyclic#1.P2_ZakladacTesnenia.ServoZdvihuZakladaca.OUT_forMapping.MDI_velocity AT %QD."P2_ServoZatlTesneniaZdvih".Module001_MDI_velocity;
	Cyclic#1.P2_ZakladacTesnenia.ServoZdvihuZakladaca.OUT_forMapping.MDI_acceleration AT %QW."P2_ServoZatlTesneniaZdvih".Module001_MDI_acceleartion;
	Cyclic#1.P2_ZakladacTesnenia.ServoZdvihuZakladaca.OUT_forMapping.MDI_decceleration AT %QW."P2_ServoZatlTesneniaZdvih".Module001_MDI_deceleration;
	Cyclic#1.P2_ZakladacTesnenia.ServoZdvihuZakladaca.OUT_forMapping.User1 AT %QW."P2_ServoZatlTesneniaZdvih".Module001_User1;
	Cyclic#1.P2_ZakladacTesnenia.ServoZdvihuZakladaca.OUT_forMapping.Control_word_or_setpoint_0 AT %QW."P2_ServoZatlTesneniaZdvih".Module001_Control_word_or_setpoint_O_00;
	Cyclic#1.P2_ZakladacTesnenia.ServoZdvihuZakladaca.OUT_forMapping.Control_word_or_setpoint_1 AT %QW."P2_ServoZatlTesneniaZdvih".Module001_Control_word_or_setpoint_O_01;
	Cyclic#1.P2_ZakladacTesnenia.ServoZdvihuZakladaca.OUT_forMapping.Control_word_or_setpoint_2 AT %QW."P2_ServoZatlTesneniaZdvih".Module001_Control_word_or_setpoint_O_02;
	Cyclic#1.P2_ZakladacTesnenia.ServoZdvihuZakladaca.OUT_forMapping.Control_word_or_setpoint_3 AT %QW."P2_ServoZatlTesneniaZdvih".Module001_Control_word_or_setpoint_O_03;
	Cyclic#1.P2_ZakladacTesnenia.ServoZdvihuZakladaca.OUT_forMapping.Control_word_or_setpoint_4 AT %QW."P2_ServoZatlTesneniaZdvih".Module001_Control_word_or_setpoint_O_04;
	Cyclic#1.P2_ZakladacTesnenia.ServoZdvihuZakladaca.OUT_forMapping.Control_word_or_setpoint_5 AT %QW."P2_ServoZatlTesneniaZdvih".Module001_Control_word_or_setpoint_O_05;
	Cyclic#1.P2_ZakladacTesnenia.ServoZdvihuZakladaca.OUT_forMapping.Control_word_or_setpoint_6 AT %QW."P2_ServoZatlTesneniaZdvih".Module001_Control_word_or_setpoint_O_06;
	Cyclic#1.P2_ZakladacTesnenia.ServoZdvihuZakladaca.OUT_forMapping.Control_word_or_setpoint_7 AT %QW."P2_ServoZatlTesneniaZdvih".Module001_Control_word_or_setpoint_O_07;
	Cyclic#1.P2_ZakladacTesnenia.ServoZdvihuZakladaca.OUT_forMapping.Control_word_or_setpoint_8 AT %QW."P2_ServoZatlTesneniaZdvih".Module001_Control_word_or_setpoint_O_08;
	Cyclic#1.P2_ZakladacTesnenia.ServoZdvihuZakladaca.OUT_forMapping.Control_word_or_setpoint_9 AT %QW."P2_ServoZatlTesneniaZdvih".Module001_Control_word_or_setpoint_O_09;
	Cyclic#1.P2_ZakladacTesnenia.ServoZdvihuZakladaca.OUT_forMapping.Control_word_or_setpoint_10 AT %QW."P2_ServoZatlTesneniaZdvih".Module001_Control_word_or_setpoint_O_10;
	Cyclic#1.P2_ZakladacTesnenia.ServoZdvihuZakladaca.OUT_forMapping.Control_word_or_setpoint_11 AT %QW."P2_ServoZatlTesneniaZdvih".Module001_Control_word_or_setpoint_O_11;
	Cyclic#1.P2_ZakladacTesnenia.ServoZdvihuZakladaca.OUT_forMapping.Control_word_or_setpoint_12 AT %QW."P2_ServoZatlTesneniaZdvih".Module001_Control_word_or_setpoint_O_12;
	Cyclic#1.P2_ZakladacTesnenia.ServoZdvihuZakladaca.OUT_forMapping.Control_word_or_setpoint_13 AT %QW."P2_ServoZatlTesneniaZdvih".Module001_Control_word_or_setpoint_O_13;
	Cyclic#1.P2_ZakladacTesnenia.ServoZdvihuZakladaca.OUT_forMapping.Control_word_or_setpoint_14 AT %QW."P2_ServoZatlTesneniaZdvih".Module001_Control_word_or_setpoint_O_14;
	Cyclic#1.P2_ZakladacTesnenia.ServoZdvihuZakladaca.OUT_forMapping.Control_word_or_setpoint_15 AT %QW."P2_ServoZatlTesneniaZdvih".Module001_Control_word_or_setpoint_O_15;
	Cyclic#1.P2_Pracovisko.IN.ServoZaklTesneniaPojazd_KomOK AT %IX."P2_ServoZatlTesneniaPojazd".ModuleOk;
	Cyclic#1.P2_ZakladacTesnenia.ServoPojazduZakladaca.IN_forMapping.Status_word_1 AT %IW."P2_ServoZatlTesneniaPojazd".Module001_Status_word_1;
	Cyclic#1.P2_ZakladacTesnenia.ServoPojazduZakladaca.IN_forMapping.Position_Statusword_1 AT %IW."P2_ServoZatlTesneniaPojazd".Module001_Position_Statusword_1;
	Cyclic#1.P2_ZakladacTesnenia.ServoPojazduZakladaca.IN_forMapping.Position_Statusword_2 AT %IW."P2_ServoZatlTesneniaPojazd".Module001_Position_Statusword_2;
	Cyclic#1.P2_ZakladacTesnenia.ServoPojazduZakladaca.IN_forMapping.Status_word_2 AT %IW."P2_ServoZatlTesneniaPojazd".Module001_Status_word_2;
	Cyclic#1.P2_ZakladacTesnenia.ServoPojazduZakladaca.IN_forMapping.Report_word AT %IW."P2_ServoZatlTesneniaPojazd".Module001_Report_word;
	Cyclic#1.P2_ZakladacTesnenia.ServoPojazduZakladaca.IN_forMapping.Position_actual_value_A AT %ID."P2_ServoZatlTesneniaPojazd".Module001_Position_actual_value_A;
	Cyclic#1.P2_ZakladacTesnenia.ServoPojazduZakladaca.IN_forMapping.Speed_actual_value_B AT %ID."P2_ServoZatlTesneniaPojazd".Module001_Speed_actual_value_B;
	Cyclic#1.P2_ZakladacTesnenia.ServoPojazduZakladaca.IN_forMapping.Fault_Code AT %IW."P2_ServoZatlTesneniaPojazd".Module001_Fault_Code;
	Cyclic#1.P2_ZakladacTesnenia.ServoPojazduZakladaca.IN_forMapping.Warn_Code AT %IW."P2_ServoZatlTesneniaPojazd".Module001_Warn_Code;
	Cyclic#1.P2_ZakladacTesnenia.ServoPojazduZakladaca.IN_forMapping.User AT %IW."P2_ServoZatlTesneniaPojazd".Module001_User;
	Cyclic#1.P2_ZakladacTesnenia.ServoPojazduZakladaca.IN_forMapping.Status_word_or_actual_value_0 AT %IW."P2_ServoZatlTesneniaPojazd".Module001_Status_word_or_actual_value_I_00;
	Cyclic#1.P2_ZakladacTesnenia.ServoPojazduZakladaca.IN_forMapping.Status_word_or_actual_value_1 AT %IW."P2_ServoZatlTesneniaPojazd".Module001_Status_word_or_actual_value_I_01;
	Cyclic#1.P2_ZakladacTesnenia.ServoPojazduZakladaca.IN_forMapping.Status_word_or_actual_value_2 AT %IW."P2_ServoZatlTesneniaPojazd".Module001_Status_word_or_actual_value_I_02;
	Cyclic#1.P2_ZakladacTesnenia.ServoPojazduZakladaca.IN_forMapping.Status_word_or_actual_value_3 AT %IW."P2_ServoZatlTesneniaPojazd".Module001_Status_word_or_actual_value_I_03;
	Cyclic#1.P2_ZakladacTesnenia.ServoPojazduZakladaca.IN_forMapping.Status_word_or_actual_value_4 AT %IW."P2_ServoZatlTesneniaPojazd".Module001_Status_word_or_actual_value_I_04;
	Cyclic#1.P2_ZakladacTesnenia.ServoPojazduZakladaca.IN_forMapping.Status_word_or_actual_value_5 AT %IW."P2_ServoZatlTesneniaPojazd".Module001_Status_word_or_actual_value_I_05;
	Cyclic#1.P2_ZakladacTesnenia.ServoPojazduZakladaca.IN_forMapping.Status_word_or_actual_value_6 AT %IW."P2_ServoZatlTesneniaPojazd".Module001_Status_word_or_actual_value_I_06;
	Cyclic#1.P2_ZakladacTesnenia.ServoPojazduZakladaca.IN_forMapping.Status_word_or_actual_value_7 AT %IW."P2_ServoZatlTesneniaPojazd".Module001_Status_word_or_actual_value_I_07;
	Cyclic#1.P2_ZakladacTesnenia.ServoPojazduZakladaca.IN_forMapping.Status_word_or_actual_value_8 AT %IW."P2_ServoZatlTesneniaPojazd".Module001_Status_word_or_actual_value_I_08;
	Cyclic#1.P2_ZakladacTesnenia.ServoPojazduZakladaca.IN_forMapping.Status_word_or_actual_value_9 AT %IW."P2_ServoZatlTesneniaPojazd".Module001_Status_word_or_actual_value_I_09;
	Cyclic#1.P2_ZakladacTesnenia.ServoPojazduZakladaca.IN_forMapping.Status_word_or_actual_value_10 AT %IW."P2_ServoZatlTesneniaPojazd".Module001_Status_word_or_actual_value_I_10;
	Cyclic#1.P2_ZakladacTesnenia.ServoPojazduZakladaca.IN_forMapping.Status_word_or_actual_value_11 AT %IW."P2_ServoZatlTesneniaPojazd".Module001_Status_word_or_actual_value_I_11;
	Cyclic#1.P2_ZakladacTesnenia.ServoPojazduZakladaca.IN_forMapping.Status_word_or_actual_value_12 AT %IW."P2_ServoZatlTesneniaPojazd".Module001_Status_word_or_actual_value_I_12;
	Cyclic#1.P2_ZakladacTesnenia.ServoPojazduZakladaca.IN_forMapping.Status_word_or_actual_value_13 AT %IW."P2_ServoZatlTesneniaPojazd".Module001_Status_word_or_actual_value_I_13;
	Cyclic#1.P2_ZakladacTesnenia.ServoPojazduZakladaca.IN_forMapping.Status_word_or_actual_value_14 AT %IW."P2_ServoZatlTesneniaPojazd".Module001_Status_word_or_actual_value_I_14;
	Cyclic#1.P2_ZakladacTesnenia.ServoPojazduZakladaca.IN_forMapping.Status_word_or_actual_value_15 AT %IW."P2_ServoZatlTesneniaPojazd".Module001_Status_word_or_actual_value_I_15;
	Cyclic#1.P2_ZakladacTesnenia.ServoPojazduZakladaca.OUT_forMapping.Control_word_1 AT %QW."P2_ServoZatlTesneniaPojazd".Module001_Control_word_1;
	Cyclic#1.P2_ZakladacTesnenia.ServoPojazduZakladaca.OUT_forMapping.Position_Controlword_1 AT %QW."P2_ServoZatlTesneniaPojazd".Module001_Position_Controlword_1;
	Cyclic#1.P2_ZakladacTesnenia.ServoPojazduZakladaca.OUT_forMapping.Position_Controlword_2 AT %QW."P2_ServoZatlTesneniaPojazd".Module001_Position_Controlword_2;
	Cyclic#1.P2_ZakladacTesnenia.ServoPojazduZakladaca.OUT_forMapping.Control_word_2 AT %QW."P2_ServoZatlTesneniaPojazd".Module001_Control_word_2;
	Cyclic#1.P2_ZakladacTesnenia.ServoPojazduZakladaca.OUT_forMapping.Override AT %QW."P2_ServoZatlTesneniaPojazd".Module001_Override;
	Cyclic#1.P2_ZakladacTesnenia.ServoPojazduZakladaca.OUT_forMapping.MDI_target_position AT %QD."P2_ServoZatlTesneniaPojazd".Module001_MDI_target_position;
	Cyclic#1.P2_ZakladacTesnenia.ServoPojazduZakladaca.OUT_forMapping.MDI_velocity AT %QD."P2_ServoZatlTesneniaPojazd".Module001_MDI_velocity;
	Cyclic#1.P2_ZakladacTesnenia.ServoPojazduZakladaca.OUT_forMapping.MDI_acceleration AT %QW."P2_ServoZatlTesneniaPojazd".Module001_MDI_acceleartion;
	Cyclic#1.P2_ZakladacTesnenia.ServoPojazduZakladaca.OUT_forMapping.MDI_decceleration AT %QW."P2_ServoZatlTesneniaPojazd".Module001_MDI_deceleration;
	Cyclic#1.P2_ZakladacTesnenia.ServoPojazduZakladaca.OUT_forMapping.User1 AT %QW."P2_ServoZatlTesneniaPojazd".Module001_User1;
	Cyclic#1.P2_ZakladacTesnenia.ServoPojazduZakladaca.OUT_forMapping.Control_word_or_setpoint_0 AT %QW."P2_ServoZatlTesneniaPojazd".Module001_Control_word_or_setpoint_O_00;
	Cyclic#1.P2_ZakladacTesnenia.ServoPojazduZakladaca.OUT_forMapping.Control_word_or_setpoint_1 AT %QW."P2_ServoZatlTesneniaPojazd".Module001_Control_word_or_setpoint_O_01;
	Cyclic#1.P2_ZakladacTesnenia.ServoPojazduZakladaca.OUT_forMapping.Control_word_or_setpoint_2 AT %QW."P2_ServoZatlTesneniaPojazd".Module001_Control_word_or_setpoint_O_02;
	Cyclic#1.P2_ZakladacTesnenia.ServoPojazduZakladaca.OUT_forMapping.Control_word_or_setpoint_3 AT %QW."P2_ServoZatlTesneniaPojazd".Module001_Control_word_or_setpoint_O_03;
	Cyclic#1.P2_ZakladacTesnenia.ServoPojazduZakladaca.OUT_forMapping.Control_word_or_setpoint_4 AT %QW."P2_ServoZatlTesneniaPojazd".Module001_Control_word_or_setpoint_O_04;
	Cyclic#1.P2_ZakladacTesnenia.ServoPojazduZakladaca.OUT_forMapping.Control_word_or_setpoint_5 AT %QW."P2_ServoZatlTesneniaPojazd".Module001_Control_word_or_setpoint_O_05;
	Cyclic#1.P2_ZakladacTesnenia.ServoPojazduZakladaca.OUT_forMapping.Control_word_or_setpoint_6 AT %QW."P2_ServoZatlTesneniaPojazd".Module001_Control_word_or_setpoint_O_06;
	Cyclic#1.P2_ZakladacTesnenia.ServoPojazduZakladaca.OUT_forMapping.Control_word_or_setpoint_7 AT %QW."P2_ServoZatlTesneniaPojazd".Module001_Control_word_or_setpoint_O_07;
	Cyclic#1.P2_ZakladacTesnenia.ServoPojazduZakladaca.OUT_forMapping.Control_word_or_setpoint_8 AT %QW."P2_ServoZatlTesneniaPojazd".Module001_Control_word_or_setpoint_O_08;
	Cyclic#1.P2_ZakladacTesnenia.ServoPojazduZakladaca.OUT_forMapping.Control_word_or_setpoint_9 AT %QW."P2_ServoZatlTesneniaPojazd".Module001_Control_word_or_setpoint_O_09;
	Cyclic#1.P2_ZakladacTesnenia.ServoPojazduZakladaca.OUT_forMapping.Control_word_or_setpoint_10 AT %QW."P2_ServoZatlTesneniaPojazd".Module001_Control_word_or_setpoint_O_10;
	Cyclic#1.P2_ZakladacTesnenia.ServoPojazduZakladaca.OUT_forMapping.Control_word_or_setpoint_11 AT %QW."P2_ServoZatlTesneniaPojazd".Module001_Control_word_or_setpoint_O_11;
	Cyclic#1.P2_ZakladacTesnenia.ServoPojazduZakladaca.OUT_forMapping.Control_word_or_setpoint_12 AT %QW."P2_ServoZatlTesneniaPojazd".Module001_Control_word_or_setpoint_O_12;
	Cyclic#1.P2_ZakladacTesnenia.ServoPojazduZakladaca.OUT_forMapping.Control_word_or_setpoint_13 AT %QW."P2_ServoZatlTesneniaPojazd".Module001_Control_word_or_setpoint_O_13;
	Cyclic#1.P2_ZakladacTesnenia.ServoPojazduZakladaca.OUT_forMapping.Control_word_or_setpoint_14 AT %QW."P2_ServoZatlTesneniaPojazd".Module001_Control_word_or_setpoint_O_14;
	Cyclic#1.P2_ZakladacTesnenia.ServoPojazduZakladaca.OUT_forMapping.Control_word_or_setpoint_15 AT %QW."P2_ServoZatlTesneniaPojazd".Module001_Control_word_or_setpoint_O_15;
	Cyclic#1.P2_Pracovisko.IN.ServoZvaraniaOsZ_KomOK AT %IX."P2_ServoZvaraniaOsZ".ModuleOk;
	Cyclic#1.P2_Zvaranie.ServoZdvihuZvarania.IN_forMapping.Status_word_1 AT %IW."P2_ServoZvaraniaOsZ".Module001_Status_word_1;
	Cyclic#1.P2_Zvaranie.ServoZdvihuZvarania.IN_forMapping.Position_Statusword_1 AT %IW."P2_ServoZvaraniaOsZ".Module001_Position_Statusword_1;
	Cyclic#1.P2_Zvaranie.ServoZdvihuZvarania.IN_forMapping.Position_Statusword_2 AT %IW."P2_ServoZvaraniaOsZ".Module001_Position_Statusword_2;
	Cyclic#1.P2_Zvaranie.ServoZdvihuZvarania.IN_forMapping.Status_word_2 AT %IW."P2_ServoZvaraniaOsZ".Module001_Status_word_2;
	Cyclic#1.P2_Zvaranie.ServoZdvihuZvarania.IN_forMapping.Report_word AT %IW."P2_ServoZvaraniaOsZ".Module001_Report_word;
	Cyclic#1.P2_Zvaranie.ServoZdvihuZvarania.IN_forMapping.Position_actual_value_A AT %ID."P2_ServoZvaraniaOsZ".Module001_Position_actual_value_A;
	Cyclic#1.P2_Zvaranie.ServoZdvihuZvarania.IN_forMapping.Speed_actual_value_B AT %ID."P2_ServoZvaraniaOsZ".Module001_Speed_actual_value_B;
	Cyclic#1.P2_Zvaranie.ServoZdvihuZvarania.IN_forMapping.Fault_Code AT %IW."P2_ServoZvaraniaOsZ".Module001_Fault_Code;
	Cyclic#1.P2_Zvaranie.ServoZdvihuZvarania.IN_forMapping.Warn_Code AT %IW."P2_ServoZvaraniaOsZ".Module001_Warn_Code;
	Cyclic#1.P2_Zvaranie.ServoZdvihuZvarania.IN_forMapping.User AT %IW."P2_ServoZvaraniaOsZ".Module001_User;
	Cyclic#1.P2_Zvaranie.ServoZdvihuZvarania.IN_forMapping.Status_word_or_actual_value_0 AT %IW."P2_ServoZvaraniaOsZ".Module001_Status_word_or_actual_value_I_00;
	Cyclic#1.P2_Zvaranie.ServoZdvihuZvarania.IN_forMapping.Status_word_or_actual_value_1 AT %IW."P2_ServoZvaraniaOsZ".Module001_Status_word_or_actual_value_I_01;
	Cyclic#1.P2_Zvaranie.ServoZdvihuZvarania.IN_forMapping.Status_word_or_actual_value_2 AT %IW."P2_ServoZvaraniaOsZ".Module001_Status_word_or_actual_value_I_02;
	Cyclic#1.P2_Zvaranie.ServoZdvihuZvarania.IN_forMapping.Status_word_or_actual_value_3 AT %IW."P2_ServoZvaraniaOsZ".Module001_Status_word_or_actual_value_I_03;
	Cyclic#1.P2_Zvaranie.ServoZdvihuZvarania.IN_forMapping.Status_word_or_actual_value_4 AT %IW."P2_ServoZvaraniaOsZ".Module001_Status_word_or_actual_value_I_04;
	Cyclic#1.P2_Zvaranie.ServoZdvihuZvarania.IN_forMapping.Status_word_or_actual_value_5 AT %IW."P2_ServoZvaraniaOsZ".Module001_Status_word_or_actual_value_I_05;
	Cyclic#1.P2_Zvaranie.ServoZdvihuZvarania.IN_forMapping.Status_word_or_actual_value_6 AT %IW."P2_ServoZvaraniaOsZ".Module001_Status_word_or_actual_value_I_06;
	Cyclic#1.P2_Zvaranie.ServoZdvihuZvarania.IN_forMapping.Status_word_or_actual_value_7 AT %IW."P2_ServoZvaraniaOsZ".Module001_Status_word_or_actual_value_I_07;
	Cyclic#1.P2_Zvaranie.ServoZdvihuZvarania.IN_forMapping.Status_word_or_actual_value_8 AT %IW."P2_ServoZvaraniaOsZ".Module001_Status_word_or_actual_value_I_08;
	Cyclic#1.P2_Zvaranie.ServoZdvihuZvarania.IN_forMapping.Status_word_or_actual_value_9 AT %IW."P2_ServoZvaraniaOsZ".Module001_Status_word_or_actual_value_I_09;
	Cyclic#1.P2_Zvaranie.ServoZdvihuZvarania.IN_forMapping.Status_word_or_actual_value_10 AT %IW."P2_ServoZvaraniaOsZ".Module001_Status_word_or_actual_value_I_10;
	Cyclic#1.P2_Zvaranie.ServoZdvihuZvarania.IN_forMapping.Status_word_or_actual_value_11 AT %IW."P2_ServoZvaraniaOsZ".Module001_Status_word_or_actual_value_I_11;
	Cyclic#1.P2_Zvaranie.ServoZdvihuZvarania.IN_forMapping.Status_word_or_actual_value_12 AT %IW."P2_ServoZvaraniaOsZ".Module001_Status_word_or_actual_value_I_12;
	Cyclic#1.P2_Zvaranie.ServoZdvihuZvarania.IN_forMapping.Status_word_or_actual_value_13 AT %IW."P2_ServoZvaraniaOsZ".Module001_Status_word_or_actual_value_I_13;
	Cyclic#1.P2_Zvaranie.ServoZdvihuZvarania.IN_forMapping.Status_word_or_actual_value_14 AT %IW."P2_ServoZvaraniaOsZ".Module001_Status_word_or_actual_value_I_14;
	Cyclic#1.P2_Zvaranie.ServoZdvihuZvarania.IN_forMapping.Status_word_or_actual_value_15 AT %IW."P2_ServoZvaraniaOsZ".Module001_Status_word_or_actual_value_I_15;
	Cyclic#1.P2_Zvaranie.ServoZdvihuZvarania.OUT_forMapping.Control_word_1 AT %QW."P2_ServoZvaraniaOsZ".Module001_Control_word_1;
	Cyclic#1.P2_Zvaranie.ServoZdvihuZvarania.OUT_forMapping.Position_Controlword_1 AT %QW."P2_ServoZvaraniaOsZ".Module001_Position_Controlword_1;
	Cyclic#1.P2_Zvaranie.ServoZdvihuZvarania.OUT_forMapping.Position_Controlword_2 AT %QW."P2_ServoZvaraniaOsZ".Module001_Position_Controlword_2;
	Cyclic#1.P2_Zvaranie.ServoZdvihuZvarania.OUT_forMapping.Control_word_2 AT %QW."P2_ServoZvaraniaOsZ".Module001_Control_word_2;
	Cyclic#1.P2_Zvaranie.ServoZdvihuZvarania.OUT_forMapping.Override AT %QW."P2_ServoZvaraniaOsZ".Module001_Override;
	Cyclic#1.P2_Zvaranie.ServoZdvihuZvarania.OUT_forMapping.MDI_target_position AT %QD."P2_ServoZvaraniaOsZ".Module001_MDI_target_position;
	Cyclic#1.P2_Zvaranie.ServoZdvihuZvarania.OUT_forMapping.MDI_velocity AT %QD."P2_ServoZvaraniaOsZ".Module001_MDI_velocity;
	Cyclic#1.P2_Zvaranie.ServoZdvihuZvarania.OUT_forMapping.MDI_acceleration AT %QW."P2_ServoZvaraniaOsZ".Module001_MDI_acceleartion;
	Cyclic#1.P2_Zvaranie.ServoZdvihuZvarania.OUT_forMapping.MDI_decceleration AT %QW."P2_ServoZvaraniaOsZ".Module001_MDI_deceleration;
	Cyclic#1.P2_Zvaranie.ServoZdvihuZvarania.OUT_forMapping.User1 AT %QW."P2_ServoZvaraniaOsZ".Module001_User1;
	Cyclic#1.P2_Zvaranie.ServoZdvihuZvarania.OUT_forMapping.Control_word_or_setpoint_0 AT %QW."P2_ServoZvaraniaOsZ".Module001_Control_word_or_setpoint_O_00;
	Cyclic#1.P2_Zvaranie.ServoZdvihuZvarania.OUT_forMapping.Control_word_or_setpoint_1 AT %QW."P2_ServoZvaraniaOsZ".Module001_Control_word_or_setpoint_O_01;
	Cyclic#1.P2_Zvaranie.ServoZdvihuZvarania.OUT_forMapping.Control_word_or_setpoint_2 AT %QW."P2_ServoZvaraniaOsZ".Module001_Control_word_or_setpoint_O_02;
	Cyclic#1.P2_Zvaranie.ServoZdvihuZvarania.OUT_forMapping.Control_word_or_setpoint_3 AT %QW."P2_ServoZvaraniaOsZ".Module001_Control_word_or_setpoint_O_03;
	Cyclic#1.P2_Zvaranie.ServoZdvihuZvarania.OUT_forMapping.Control_word_or_setpoint_4 AT %QW."P2_ServoZvaraniaOsZ".Module001_Control_word_or_setpoint_O_04;
	Cyclic#1.P2_Zvaranie.ServoZdvihuZvarania.OUT_forMapping.Control_word_or_setpoint_5 AT %QW."P2_ServoZvaraniaOsZ".Module001_Control_word_or_setpoint_O_05;
	Cyclic#1.P2_Zvaranie.ServoZdvihuZvarania.OUT_forMapping.Control_word_or_setpoint_6 AT %QW."P2_ServoZvaraniaOsZ".Module001_Control_word_or_setpoint_O_06;
	Cyclic#1.P2_Zvaranie.ServoZdvihuZvarania.OUT_forMapping.Control_word_or_setpoint_7 AT %QW."P2_ServoZvaraniaOsZ".Module001_Control_word_or_setpoint_O_07;
	Cyclic#1.P2_Zvaranie.ServoZdvihuZvarania.OUT_forMapping.Control_word_or_setpoint_8 AT %QW."P2_ServoZvaraniaOsZ".Module001_Control_word_or_setpoint_O_08;
	Cyclic#1.P2_Zvaranie.ServoZdvihuZvarania.OUT_forMapping.Control_word_or_setpoint_9 AT %QW."P2_ServoZvaraniaOsZ".Module001_Control_word_or_setpoint_O_09;
	Cyclic#1.P2_Zvaranie.ServoZdvihuZvarania.OUT_forMapping.Control_word_or_setpoint_10 AT %QW."P2_ServoZvaraniaOsZ".Module001_Control_word_or_setpoint_O_10;
	Cyclic#1.P2_Zvaranie.ServoZdvihuZvarania.OUT_forMapping.Control_word_or_setpoint_11 AT %QW."P2_ServoZvaraniaOsZ".Module001_Control_word_or_setpoint_O_11;
	Cyclic#1.P2_Zvaranie.ServoZdvihuZvarania.OUT_forMapping.Control_word_or_setpoint_12 AT %QW."P2_ServoZvaraniaOsZ".Module001_Control_word_or_setpoint_O_12;
	Cyclic#1.P2_Zvaranie.ServoZdvihuZvarania.OUT_forMapping.Control_word_or_setpoint_13 AT %QW."P2_ServoZvaraniaOsZ".Module001_Control_word_or_setpoint_O_13;
	Cyclic#1.P2_Zvaranie.ServoZdvihuZvarania.OUT_forMapping.Control_word_or_setpoint_14 AT %QW."P2_ServoZvaraniaOsZ".Module001_Control_word_or_setpoint_O_14;
	Cyclic#1.P2_Zvaranie.ServoZdvihuZvarania.OUT_forMapping.Control_word_or_setpoint_15 AT %QW."P2_ServoZvaraniaOsZ".Module001_Control_word_or_setpoint_O_15;
	Cyclic#1.P4_Pracovisko.IN.ServoZdvihuAplikEtikiet_KomOK AT %IX."P4_ServoAplikatoraEtikietOsZ".ModuleOk;
	Cyclic#1.P4_Etiketovacka.ServoZdvihuAplikatora.IN_forMapping.Status_word_1 AT %IW."P4_ServoAplikatoraEtikietOsZ".Module001_Status_word_1;
	Cyclic#1.P4_Etiketovacka.ServoZdvihuAplikatora.IN_forMapping.Position_Statusword_1 AT %IW."P4_ServoAplikatoraEtikietOsZ".Module001_Position_Statusword_1;
	Cyclic#1.P4_Etiketovacka.ServoZdvihuAplikatora.IN_forMapping.Position_Statusword_2 AT %IW."P4_ServoAplikatoraEtikietOsZ".Module001_Position_Statusword_2;
	Cyclic#1.P4_Etiketovacka.ServoZdvihuAplikatora.IN_forMapping.Status_word_2 AT %IW."P4_ServoAplikatoraEtikietOsZ".Module001_Status_word_2;
	Cyclic#1.P4_Etiketovacka.ServoZdvihuAplikatora.IN_forMapping.Report_word AT %IW."P4_ServoAplikatoraEtikietOsZ".Module001_Report_word;
	Cyclic#1.P4_Etiketovacka.ServoZdvihuAplikatora.IN_forMapping.Position_actual_value_A AT %ID."P4_ServoAplikatoraEtikietOsZ".Module001_Position_actual_value_A;
	Cyclic#1.P4_Etiketovacka.ServoZdvihuAplikatora.IN_forMapping.Speed_actual_value_B AT %ID."P4_ServoAplikatoraEtikietOsZ".Module001_Speed_actual_value_B;
	Cyclic#1.P4_Etiketovacka.ServoZdvihuAplikatora.IN_forMapping.Fault_Code AT %IW."P4_ServoAplikatoraEtikietOsZ".Module001_Fault_Code;
	Cyclic#1.P4_Etiketovacka.ServoZdvihuAplikatora.IN_forMapping.Warn_Code AT %IW."P4_ServoAplikatoraEtikietOsZ".Module001_Warn_Code;
	Cyclic#1.P4_Etiketovacka.ServoZdvihuAplikatora.IN_forMapping.User AT %IW."P4_ServoAplikatoraEtikietOsZ".Module001_User;
	Cyclic#1.P4_Etiketovacka.ServoZdvihuAplikatora.IN_forMapping.Status_word_or_actual_value_0 AT %IW."P4_ServoAplikatoraEtikietOsZ".Module001_Status_word_or_actual_value_I_00;
	Cyclic#1.P4_Etiketovacka.ServoZdvihuAplikatora.IN_forMapping.Status_word_or_actual_value_1 AT %IW."P4_ServoAplikatoraEtikietOsZ".Module001_Status_word_or_actual_value_I_01;
	Cyclic#1.P4_Etiketovacka.ServoZdvihuAplikatora.IN_forMapping.Status_word_or_actual_value_2 AT %IW."P4_ServoAplikatoraEtikietOsZ".Module001_Status_word_or_actual_value_I_02;
	Cyclic#1.P4_Etiketovacka.ServoZdvihuAplikatora.IN_forMapping.Status_word_or_actual_value_3 AT %IW."P4_ServoAplikatoraEtikietOsZ".Module001_Status_word_or_actual_value_I_03;
	Cyclic#1.P4_Etiketovacka.ServoZdvihuAplikatora.IN_forMapping.Status_word_or_actual_value_4 AT %IW."P4_ServoAplikatoraEtikietOsZ".Module001_Status_word_or_actual_value_I_04;
	Cyclic#1.P4_Etiketovacka.ServoZdvihuAplikatora.IN_forMapping.Status_word_or_actual_value_5 AT %IW."P4_ServoAplikatoraEtikietOsZ".Module001_Status_word_or_actual_value_I_05;
	Cyclic#1.P4_Etiketovacka.ServoZdvihuAplikatora.IN_forMapping.Status_word_or_actual_value_6 AT %IW."P4_ServoAplikatoraEtikietOsZ".Module001_Status_word_or_actual_value_I_06;
	Cyclic#1.P4_Etiketovacka.ServoZdvihuAplikatora.IN_forMapping.Status_word_or_actual_value_7 AT %IW."P4_ServoAplikatoraEtikietOsZ".Module001_Status_word_or_actual_value_I_07;
	Cyclic#1.P4_Etiketovacka.ServoZdvihuAplikatora.IN_forMapping.Status_word_or_actual_value_8 AT %IW."P4_ServoAplikatoraEtikietOsZ".Module001_Status_word_or_actual_value_I_08;
	Cyclic#1.P4_Etiketovacka.ServoZdvihuAplikatora.IN_forMapping.Status_word_or_actual_value_9 AT %IW."P4_ServoAplikatoraEtikietOsZ".Module001_Status_word_or_actual_value_I_09;
	Cyclic#1.P4_Etiketovacka.ServoZdvihuAplikatora.IN_forMapping.Status_word_or_actual_value_10 AT %IW."P4_ServoAplikatoraEtikietOsZ".Module001_Status_word_or_actual_value_I_10;
	Cyclic#1.P4_Etiketovacka.ServoZdvihuAplikatora.IN_forMapping.Status_word_or_actual_value_11 AT %IW."P4_ServoAplikatoraEtikietOsZ".Module001_Status_word_or_actual_value_I_11;
	Cyclic#1.P4_Etiketovacka.ServoZdvihuAplikatora.IN_forMapping.Status_word_or_actual_value_12 AT %IW."P4_ServoAplikatoraEtikietOsZ".Module001_Status_word_or_actual_value_I_12;
	Cyclic#1.P4_Etiketovacka.ServoZdvihuAplikatora.IN_forMapping.Status_word_or_actual_value_13 AT %IW."P4_ServoAplikatoraEtikietOsZ".Module001_Status_word_or_actual_value_I_13;
	Cyclic#1.P4_Etiketovacka.ServoZdvihuAplikatora.IN_forMapping.Status_word_or_actual_value_14 AT %IW."P4_ServoAplikatoraEtikietOsZ".Module001_Status_word_or_actual_value_I_14;
	Cyclic#1.P4_Etiketovacka.ServoZdvihuAplikatora.IN_forMapping.Status_word_or_actual_value_15 AT %IW."P4_ServoAplikatoraEtikietOsZ".Module001_Status_word_or_actual_value_I_15;
	Cyclic#1.P4_Etiketovacka.ServoZdvihuAplikatora.OUT_forMapping.Control_word_1 AT %QW."P4_ServoAplikatoraEtikietOsZ".Module001_Control_word_1;
	Cyclic#1.P4_Etiketovacka.ServoZdvihuAplikatora.OUT_forMapping.Position_Controlword_1 AT %QW."P4_ServoAplikatoraEtikietOsZ".Module001_Position_Controlword_1;
	Cyclic#1.P4_Etiketovacka.ServoZdvihuAplikatora.OUT_forMapping.Position_Controlword_2 AT %QW."P4_ServoAplikatoraEtikietOsZ".Module001_Position_Controlword_2;
	Cyclic#1.P4_Etiketovacka.ServoZdvihuAplikatora.OUT_forMapping.Control_word_2 AT %QW."P4_ServoAplikatoraEtikietOsZ".Module001_Control_word_2;
	Cyclic#1.P4_Etiketovacka.ServoZdvihuAplikatora.OUT_forMapping.Override AT %QW."P4_ServoAplikatoraEtikietOsZ".Module001_Override;
	Cyclic#1.P4_Etiketovacka.ServoZdvihuAplikatora.OUT_forMapping.MDI_target_position AT %QD."P4_ServoAplikatoraEtikietOsZ".Module001_MDI_target_position;
	Cyclic#1.P4_Etiketovacka.ServoZdvihuAplikatora.OUT_forMapping.MDI_velocity AT %QD."P4_ServoAplikatoraEtikietOsZ".Module001_MDI_velocity;
	Cyclic#1.P4_Etiketovacka.ServoZdvihuAplikatora.OUT_forMapping.MDI_acceleration AT %QW."P4_ServoAplikatoraEtikietOsZ".Module001_MDI_acceleartion;
	Cyclic#1.P4_Etiketovacka.ServoZdvihuAplikatora.OUT_forMapping.MDI_decceleration AT %QW."P4_ServoAplikatoraEtikietOsZ".Module001_MDI_deceleration;
	Cyclic#1.P4_Etiketovacka.ServoZdvihuAplikatora.OUT_forMapping.User1 AT %QW."P4_ServoAplikatoraEtikietOsZ".Module001_User1;
	Cyclic#1.P4_Etiketovacka.ServoZdvihuAplikatora.OUT_forMapping.Control_word_or_setpoint_0 AT %QW."P4_ServoAplikatoraEtikietOsZ".Module001_Control_word_or_setpoint_O_00;
	Cyclic#1.P4_Etiketovacka.ServoZdvihuAplikatora.OUT_forMapping.Control_word_or_setpoint_1 AT %QW."P4_ServoAplikatoraEtikietOsZ".Module001_Control_word_or_setpoint_O_01;
	Cyclic#1.P4_Etiketovacka.ServoZdvihuAplikatora.OUT_forMapping.Control_word_or_setpoint_2 AT %QW."P4_ServoAplikatoraEtikietOsZ".Module001_Control_word_or_setpoint_O_02;
	Cyclic#1.P4_Etiketovacka.ServoZdvihuAplikatora.OUT_forMapping.Control_word_or_setpoint_3 AT %QW."P4_ServoAplikatoraEtikietOsZ".Module001_Control_word_or_setpoint_O_03;
	Cyclic#1.P4_Etiketovacka.ServoZdvihuAplikatora.OUT_forMapping.Control_word_or_setpoint_4 AT %QW."P4_ServoAplikatoraEtikietOsZ".Module001_Control_word_or_setpoint_O_04;
	Cyclic#1.P4_Etiketovacka.ServoZdvihuAplikatora.OUT_forMapping.Control_word_or_setpoint_5 AT %QW."P4_ServoAplikatoraEtikietOsZ".Module001_Control_word_or_setpoint_O_05;
	Cyclic#1.P4_Etiketovacka.ServoZdvihuAplikatora.OUT_forMapping.Control_word_or_setpoint_6 AT %QW."P4_ServoAplikatoraEtikietOsZ".Module001_Control_word_or_setpoint_O_06;
	Cyclic#1.P4_Etiketovacka.ServoZdvihuAplikatora.OUT_forMapping.Control_word_or_setpoint_7 AT %QW."P4_ServoAplikatoraEtikietOsZ".Module001_Control_word_or_setpoint_O_07;
	Cyclic#1.P4_Etiketovacka.ServoZdvihuAplikatora.OUT_forMapping.Control_word_or_setpoint_8 AT %QW."P4_ServoAplikatoraEtikietOsZ".Module001_Control_word_or_setpoint_O_08;
	Cyclic#1.P4_Etiketovacka.ServoZdvihuAplikatora.OUT_forMapping.Control_word_or_setpoint_9 AT %QW."P4_ServoAplikatoraEtikietOsZ".Module001_Control_word_or_setpoint_O_09;
	Cyclic#1.P4_Etiketovacka.ServoZdvihuAplikatora.OUT_forMapping.Control_word_or_setpoint_10 AT %QW."P4_ServoAplikatoraEtikietOsZ".Module001_Control_word_or_setpoint_O_10;
	Cyclic#1.P4_Etiketovacka.ServoZdvihuAplikatora.OUT_forMapping.Control_word_or_setpoint_11 AT %QW."P4_ServoAplikatoraEtikietOsZ".Module001_Control_word_or_setpoint_O_11;
	Cyclic#1.P4_Etiketovacka.ServoZdvihuAplikatora.OUT_forMapping.Control_word_or_setpoint_12 AT %QW."P4_ServoAplikatoraEtikietOsZ".Module001_Control_word_or_setpoint_O_12;
	Cyclic#1.P4_Etiketovacka.ServoZdvihuAplikatora.OUT_forMapping.Control_word_or_setpoint_13 AT %QW."P4_ServoAplikatoraEtikietOsZ".Module001_Control_word_or_setpoint_O_13;
	Cyclic#1.P4_Etiketovacka.ServoZdvihuAplikatora.OUT_forMapping.Control_word_or_setpoint_14 AT %QW."P4_ServoAplikatoraEtikietOsZ".Module001_Control_word_or_setpoint_O_14;
	Cyclic#1.P4_Etiketovacka.ServoZdvihuAplikatora.OUT_forMapping.Control_word_or_setpoint_15 AT %QW."P4_ServoAplikatoraEtikietOsZ".Module001_Control_word_or_setpoint_O_15;
	Cyclic#1.P4_Pracovisko.IN.ServoZdvihuVytahu_KomOK AT %IX."P4_ServoZdvihuVystupVytahu".ModuleOk;
	Cyclic#1.P4_Vytah.ServoZdvihuVytahu.IN_forMapping.Status_word_1 AT %IW."P4_ServoZdvihuVystupVytahu".Module001_Status_word_1;
	Cyclic#1.P4_Vytah.ServoZdvihuVytahu.IN_forMapping.Position_Statusword_1 AT %IW."P4_ServoZdvihuVystupVytahu".Module001_Position_Statusword_1;
	Cyclic#1.P4_Vytah.ServoZdvihuVytahu.IN_forMapping.Position_Statusword_2 AT %IW."P4_ServoZdvihuVystupVytahu".Module001_Position_Statusword_2;
	Cyclic#1.P4_Vytah.ServoZdvihuVytahu.IN_forMapping.Status_word_2 AT %IW."P4_ServoZdvihuVystupVytahu".Module001_Status_word_2;
	Cyclic#1.P4_Vytah.ServoZdvihuVytahu.IN_forMapping.Report_word AT %IW."P4_ServoZdvihuVystupVytahu".Module001_Report_word;
	Cyclic#1.P4_Vytah.ServoZdvihuVytahu.IN_forMapping.Position_actual_value_A AT %ID."P4_ServoZdvihuVystupVytahu".Module001_Position_actual_value_A;
	Cyclic#1.P4_Vytah.ServoZdvihuVytahu.IN_forMapping.Speed_actual_value_B AT %ID."P4_ServoZdvihuVystupVytahu".Module001_Speed_actual_value_B;
	Cyclic#1.P4_Vytah.ServoZdvihuVytahu.IN_forMapping.Fault_Code AT %IW."P4_ServoZdvihuVystupVytahu".Module001_Fault_Code;
	Cyclic#1.P4_Vytah.ServoZdvihuVytahu.IN_forMapping.Warn_Code AT %IW."P4_ServoZdvihuVystupVytahu".Module001_Warn_Code;
	Cyclic#1.P4_Vytah.ServoZdvihuVytahu.IN_forMapping.User AT %IW."P4_ServoZdvihuVystupVytahu".Module001_User;
	Cyclic#1.P4_Vytah.ServoZdvihuVytahu.IN_forMapping.Status_word_or_actual_value_0 AT %IW."P4_ServoZdvihuVystupVytahu".Module001_Status_word_or_actual_value_I_00;
	Cyclic#1.P4_Vytah.ServoZdvihuVytahu.IN_forMapping.Status_word_or_actual_value_1 AT %IW."P4_ServoZdvihuVystupVytahu".Module001_Status_word_or_actual_value_I_01;
	Cyclic#1.P4_Vytah.ServoZdvihuVytahu.IN_forMapping.Status_word_or_actual_value_2 AT %IW."P4_ServoZdvihuVystupVytahu".Module001_Status_word_or_actual_value_I_02;
	Cyclic#1.P4_Vytah.ServoZdvihuVytahu.IN_forMapping.Status_word_or_actual_value_3 AT %IW."P4_ServoZdvihuVystupVytahu".Module001_Status_word_or_actual_value_I_03;
	Cyclic#1.P4_Vytah.ServoZdvihuVytahu.IN_forMapping.Status_word_or_actual_value_4 AT %IW."P4_ServoZdvihuVystupVytahu".Module001_Status_word_or_actual_value_I_04;
	Cyclic#1.P4_Vytah.ServoZdvihuVytahu.IN_forMapping.Status_word_or_actual_value_5 AT %IW."P4_ServoZdvihuVystupVytahu".Module001_Status_word_or_actual_value_I_05;
	Cyclic#1.P4_Vytah.ServoZdvihuVytahu.IN_forMapping.Status_word_or_actual_value_6 AT %IW."P4_ServoZdvihuVystupVytahu".Module001_Status_word_or_actual_value_I_06;
	Cyclic#1.P4_Vytah.ServoZdvihuVytahu.IN_forMapping.Status_word_or_actual_value_7 AT %IW."P4_ServoZdvihuVystupVytahu".Module001_Status_word_or_actual_value_I_07;
	Cyclic#1.P4_Vytah.ServoZdvihuVytahu.IN_forMapping.Status_word_or_actual_value_8 AT %IW."P4_ServoZdvihuVystupVytahu".Module001_Status_word_or_actual_value_I_08;
	Cyclic#1.P4_Vytah.ServoZdvihuVytahu.IN_forMapping.Status_word_or_actual_value_9 AT %IW."P4_ServoZdvihuVystupVytahu".Module001_Status_word_or_actual_value_I_09;
	Cyclic#1.P4_Vytah.ServoZdvihuVytahu.IN_forMapping.Status_word_or_actual_value_10 AT %IW."P4_ServoZdvihuVystupVytahu".Module001_Status_word_or_actual_value_I_10;
	Cyclic#1.P4_Vytah.ServoZdvihuVytahu.IN_forMapping.Status_word_or_actual_value_11 AT %IW."P4_ServoZdvihuVystupVytahu".Module001_Status_word_or_actual_value_I_11;
	Cyclic#1.P4_Vytah.ServoZdvihuVytahu.IN_forMapping.Status_word_or_actual_value_12 AT %IW."P4_ServoZdvihuVystupVytahu".Module001_Status_word_or_actual_value_I_12;
	Cyclic#1.P4_Vytah.ServoZdvihuVytahu.IN_forMapping.Status_word_or_actual_value_13 AT %IW."P4_ServoZdvihuVystupVytahu".Module001_Status_word_or_actual_value_I_13;
	Cyclic#1.P4_Vytah.ServoZdvihuVytahu.IN_forMapping.Status_word_or_actual_value_14 AT %IW."P4_ServoZdvihuVystupVytahu".Module001_Status_word_or_actual_value_I_14;
	Cyclic#1.P4_Vytah.ServoZdvihuVytahu.IN_forMapping.Status_word_or_actual_value_15 AT %IW."P4_ServoZdvihuVystupVytahu".Module001_Status_word_or_actual_value_I_15;
	Cyclic#1.P4_Vytah.ServoZdvihuVytahu.OUT_forMapping.Control_word_1 AT %QW."P4_ServoZdvihuVystupVytahu".Module001_Control_word_1;
	Cyclic#1.P4_Vytah.ServoZdvihuVytahu.OUT_forMapping.Position_Controlword_1 AT %QW."P4_ServoZdvihuVystupVytahu".Module001_Position_Controlword_1;
	Cyclic#1.P4_Vytah.ServoZdvihuVytahu.OUT_forMapping.Position_Controlword_2 AT %QW."P4_ServoZdvihuVystupVytahu".Module001_Position_Controlword_2;
	Cyclic#1.P4_Vytah.ServoZdvihuVytahu.OUT_forMapping.Control_word_2 AT %QW."P4_ServoZdvihuVystupVytahu".Module001_Control_word_2;
	Cyclic#1.P4_Vytah.ServoZdvihuVytahu.OUT_forMapping.Override AT %QW."P4_ServoZdvihuVystupVytahu".Module001_Override;
	Cyclic#1.P4_Vytah.ServoZdvihuVytahu.OUT_forMapping.MDI_target_position AT %QD."P4_ServoZdvihuVystupVytahu".Module001_MDI_target_position;
	Cyclic#1.P4_Vytah.ServoZdvihuVytahu.OUT_forMapping.MDI_velocity AT %QD."P4_ServoZdvihuVystupVytahu".Module001_MDI_velocity;
	Cyclic#1.P4_Vytah.ServoZdvihuVytahu.OUT_forMapping.MDI_acceleration AT %QW."P4_ServoZdvihuVystupVytahu".Module001_MDI_acceleartion;
	Cyclic#1.P4_Vytah.ServoZdvihuVytahu.OUT_forMapping.MDI_decceleration AT %QW."P4_ServoZdvihuVystupVytahu".Module001_MDI_deceleration;
	Cyclic#1.P4_Vytah.ServoZdvihuVytahu.OUT_forMapping.User1 AT %QW."P4_ServoZdvihuVystupVytahu".Module001_User1;
	Cyclic#1.P4_Vytah.ServoZdvihuVytahu.OUT_forMapping.Control_word_or_setpoint_0 AT %QW."P4_ServoZdvihuVystupVytahu".Module001_Control_word_or_setpoint_O_00;
	Cyclic#1.P4_Vytah.ServoZdvihuVytahu.OUT_forMapping.Control_word_or_setpoint_1 AT %QW."P4_ServoZdvihuVystupVytahu".Module001_Control_word_or_setpoint_O_01;
	Cyclic#1.P4_Vytah.ServoZdvihuVytahu.OUT_forMapping.Control_word_or_setpoint_2 AT %QW."P4_ServoZdvihuVystupVytahu".Module001_Control_word_or_setpoint_O_02;
	Cyclic#1.P4_Vytah.ServoZdvihuVytahu.OUT_forMapping.Control_word_or_setpoint_3 AT %QW."P4_ServoZdvihuVystupVytahu".Module001_Control_word_or_setpoint_O_03;
	Cyclic#1.P4_Vytah.ServoZdvihuVytahu.OUT_forMapping.Control_word_or_setpoint_4 AT %QW."P4_ServoZdvihuVystupVytahu".Module001_Control_word_or_setpoint_O_04;
	Cyclic#1.P4_Vytah.ServoZdvihuVytahu.OUT_forMapping.Control_word_or_setpoint_5 AT %QW."P4_ServoZdvihuVystupVytahu".Module001_Control_word_or_setpoint_O_05;
	Cyclic#1.P4_Vytah.ServoZdvihuVytahu.OUT_forMapping.Control_word_or_setpoint_6 AT %QW."P4_ServoZdvihuVystupVytahu".Module001_Control_word_or_setpoint_O_06;
	Cyclic#1.P4_Vytah.ServoZdvihuVytahu.OUT_forMapping.Control_word_or_setpoint_7 AT %QW."P4_ServoZdvihuVystupVytahu".Module001_Control_word_or_setpoint_O_07;
	Cyclic#1.P4_Vytah.ServoZdvihuVytahu.OUT_forMapping.Control_word_or_setpoint_8 AT %QW."P4_ServoZdvihuVystupVytahu".Module001_Control_word_or_setpoint_O_08;
	Cyclic#1.P4_Vytah.ServoZdvihuVytahu.OUT_forMapping.Control_word_or_setpoint_9 AT %QW."P4_ServoZdvihuVystupVytahu".Module001_Control_word_or_setpoint_O_09;
	Cyclic#1.P4_Vytah.ServoZdvihuVytahu.OUT_forMapping.Control_word_or_setpoint_10 AT %QW."P4_ServoZdvihuVystupVytahu".Module001_Control_word_or_setpoint_O_10;
	Cyclic#1.P4_Vytah.ServoZdvihuVytahu.OUT_forMapping.Control_word_or_setpoint_11 AT %QW."P4_ServoZdvihuVystupVytahu".Module001_Control_word_or_setpoint_O_11;
	Cyclic#1.P4_Vytah.ServoZdvihuVytahu.OUT_forMapping.Control_word_or_setpoint_12 AT %QW."P4_ServoZdvihuVystupVytahu".Module001_Control_word_or_setpoint_O_12;
	Cyclic#1.P4_Vytah.ServoZdvihuVytahu.OUT_forMapping.Control_word_or_setpoint_13 AT %QW."P4_ServoZdvihuVystupVytahu".Module001_Control_word_or_setpoint_O_13;
	Cyclic#1.P4_Vytah.ServoZdvihuVytahu.OUT_forMapping.Control_word_or_setpoint_14 AT %QW."P4_ServoZdvihuVystupVytahu".Module001_Control_word_or_setpoint_O_14;
	Cyclic#1.P4_Vytah.ServoZdvihuVytahu.OUT_forMapping.Control_word_or_setpoint_15 AT %QW."P4_ServoZdvihuVystupVytahu".Module001_Control_word_or_setpoint_O_15;
	Cyclic#1.P4_Pracovisko.COM_Festo.DM4_1_4DI[0] AT %IX."P4_IOmaster".Module001_Bit_0_Bit_0;
	Cyclic#1.P4_Pracovisko.COM_Festo.DM4_1_4DI[1] AT %IX."P4_IOmaster".Module001_Bit_1_Bit_1;
	Cyclic#1.P4_Pracovisko.COM_Festo.DM4_1_4DI[2] AT %IX."P4_IOmaster".Module001_Bit_2_Bit_2;
	Cyclic#1.P4_Pracovisko.COM_Festo.DM4_1_4DI[3] AT %IX."P4_IOmaster".Module001_Bit_3_Bit_3;
	Cyclic#1.P4_Pracovisko.COM_Festo.DM4_1_4DO[0] AT %QX."P4_IOmaster".Module001_Bit_0_Bit_1;
	Cyclic#1.P4_Pracovisko.COM_Festo.DM4_1_4DO[1] AT %QX."P4_IOmaster".Module001_Bit_1_Bit_2;
	Cyclic#1.P4_Pracovisko.COM_Festo.DM4_1_4DO[2] AT %QX."P4_IOmaster".Module001_Bit_2_Bit_3;
	Cyclic#1.P4_Pracovisko.COM_Festo.DM4_1_4DO[3] AT %QX."P4_IOmaster".Module001_Bit_3_Bit_4;
	Cyclic#1.P4_Pracovisko.COM_Festo.DI4_2_8DI[0] AT %IX."P4_IOmaster".Module002_Bit_0_Bit_0;
	Cyclic#1.P4_Pracovisko.COM_Festo.DI4_2_8DI[1] AT %IX."P4_IOmaster".Module002_Bit_1_Bit_1;
	Cyclic#1.P4_Pracovisko.COM_Festo.DI4_2_8DI[2] AT %IX."P4_IOmaster".Module002_Bit_2_Bit_2;
	Cyclic#1.P4_Pracovisko.COM_Festo.DI4_2_8DI[3] AT %IX."P4_IOmaster".Module002_Bit_3_Bit_3;
	Cyclic#1.P4_Pracovisko.COM_Festo.DI4_2_8DI[4] AT %IX."P4_IOmaster".Module002_Bit_4_Bit_4;
	Cyclic#1.P4_Pracovisko.COM_Festo.DI4_2_8DI[5] AT %IX."P4_IOmaster".Module002_Bit_5_Bit_5;
	Cyclic#1.P4_Pracovisko.COM_Festo.DI4_2_8DI[6] AT %IX."P4_IOmaster".Module002_Bit_6_Bit_6;
	Cyclic#1.P4_Pracovisko.COM_Festo.DI4_2_8DI[7] AT %IX."P4_IOmaster".Module002_Bit_7_Bit_7;
	Cyclic#1.P4_Pracovisko.COM_Festo.DI4_5_8DI[0] AT %IX."P4_IOmaster".Module003_Bit_0_Bit_0;
	Cyclic#1.P4_Pracovisko.COM_Festo.DI4_5_8DI[1] AT %IX."P4_IOmaster".Module003_Bit_1_Bit_1;
	Cyclic#1.P4_Pracovisko.COM_Festo.DI4_5_8DI[2] AT %IX."P4_IOmaster".Module003_Bit_2_Bit_2;
	Cyclic#1.P4_Pracovisko.COM_Festo.DI4_5_8DI[3] AT %IX."P4_IOmaster".Module003_Bit_3_Bit_3;
	Cyclic#1.P4_Pracovisko.COM_Festo.DI4_5_8DI[4] AT %IX."P4_IOmaster".Module003_Bit_4_Bit_4;
	Cyclic#1.P4_Pracovisko.COM_Festo.DI4_5_8DI[5] AT %IX."P4_IOmaster".Module003_Bit_5_Bit_5;
	Cyclic#1.P4_Pracovisko.COM_Festo.DI4_5_8DI[6] AT %IX."P4_IOmaster".Module003_Bit_6_Bit_6;
	Cyclic#1.P4_Pracovisko.COM_Festo.DI4_5_8DI[7] AT %IX."P4_IOmaster".Module003_Bit_7_Bit_7;
	Cyclic#1.P4_Pracovisko.COM_Festo.DI4_1_8DI[0] AT %IX."P4_IOmaster".Module004_Bit_0_Bit_0;
	Cyclic#1.P4_Pracovisko.COM_Festo.DI4_1_8DI[1] AT %IX."P4_IOmaster".Module004_Bit_1_Bit_1;
	Cyclic#1.P4_Pracovisko.COM_Festo.DI4_1_8DI[2] AT %IX."P4_IOmaster".Module004_Bit_2_Bit_2;
	Cyclic#1.P4_Pracovisko.COM_Festo.DI4_1_8DI[3] AT %IX."P4_IOmaster".Module004_Bit_3_Bit_3;
	Cyclic#1.P4_Pracovisko.COM_Festo.DI4_1_8DI[4] AT %IX."P4_IOmaster".Module004_Bit_4_Bit_4;
	Cyclic#1.P4_Pracovisko.COM_Festo.DI4_1_8DI[5] AT %IX."P4_IOmaster".Module004_Bit_5_Bit_5;
	Cyclic#1.P4_Pracovisko.COM_Festo.DI4_1_8DI[6] AT %IX."P4_IOmaster".Module004_Bit_6_Bit_6;
	Cyclic#1.P4_Pracovisko.COM_Festo.DI4_1_8DI[7] AT %IX."P4_IOmaster".Module004_Bit_7_Bit_7;
	Cyclic#1.P4_Pracovisko.COM_Festo.DI4_4_8DI[0] AT %IX."P4_IOmaster".Module005_Bit_0_Bit_0;
	Cyclic#1.P4_Pracovisko.COM_Festo.DI4_4_8DI[1] AT %IX."P4_IOmaster".Module005_Bit_1_Bit_1;
	Cyclic#1.P4_Pracovisko.COM_Festo.DI4_4_8DI[2] AT %IX."P4_IOmaster".Module005_Bit_2_Bit_2;
	Cyclic#1.P4_Pracovisko.COM_Festo.DI4_4_8DI[3] AT %IX."P4_IOmaster".Module005_Bit_3_Bit_3;
	Cyclic#1.P4_Pracovisko.COM_Festo.DI4_4_8DI[4] AT %IX."P4_IOmaster".Module005_Bit_4_Bit_4;
	Cyclic#1.P4_Pracovisko.COM_Festo.DI4_4_8DI[5] AT %IX."P4_IOmaster".Module005_Bit_5_Bit_5;
	Cyclic#1.P4_Pracovisko.COM_Festo.DI4_4_8DI[6] AT %IX."P4_IOmaster".Module005_Bit_6_Bit_6;
	Cyclic#1.P4_Pracovisko.COM_Festo.DI4_4_8DI[7] AT %IX."P4_IOmaster".Module005_Bit_7_Bit_7;
	Cyclic#1.P4_Pracovisko.COM_Festo.DI4_3_8DI[0] AT %IX."P4_IOmaster".Module006_Bit_0_Bit_0;
	Cyclic#1.P4_Pracovisko.COM_Festo.DI4_3_8DI[1] AT %IX."P4_IOmaster".Module006_Bit_1_Bit_1;
	Cyclic#1.P4_Pracovisko.COM_Festo.DI4_3_8DI[2] AT %IX."P4_IOmaster".Module006_Bit_2_Bit_2;
	Cyclic#1.P4_Pracovisko.COM_Festo.DI4_3_8DI[3] AT %IX."P4_IOmaster".Module006_Bit_3_Bit_3;
	Cyclic#1.P4_Pracovisko.COM_Festo.DI4_3_8DI[4] AT %IX."P4_IOmaster".Module006_Bit_4_Bit_4;
	Cyclic#1.P4_Pracovisko.COM_Festo.DI4_3_8DI[5] AT %IX."P4_IOmaster".Module006_Bit_5_Bit_5;
	Cyclic#1.P4_Pracovisko.COM_Festo.DI4_3_8DI[6] AT %IX."P4_IOmaster".Module006_Bit_6_Bit_6;
	Cyclic#1.P4_Pracovisko.COM_Festo.DI4_3_8DI[7] AT %IX."P4_IOmaster".Module006_Bit_7_Bit_7;
	Cyclic#1.P4_Pracovisko.COM_Festo.DS4_1_Port0_IN[0] AT %IB."P4_IOmaster".Module007_Inputs001;
	Cyclic#1.P4_Pracovisko.COM_Festo.DS4_1_Port0_IN[1] AT %IB."P4_IOmaster".Module007_Inputs002;
	Cyclic#1.P4_Pracovisko.COM_Festo.DS4_1_Port0_IN[2] AT %IB."P4_IOmaster".Module007_Inputs003;
	Cyclic#1.P4_Pracovisko.COM_Festo.DS4_1_Port0_IN[3] AT %IB."P4_IOmaster".Module007_Inputs004;
	Cyclic#1.P4_Pracovisko.COM_Festo.DS4_1_Port0_IN[4] AT %IB."P4_IOmaster".Module007_Inputs005;
	Cyclic#1.P4_Pracovisko.COM_Festo.DS4_1_Port0_IN[5] AT %IB."P4_IOmaster".Module007_Inputs006;
	Cyclic#1.P4_Pracovisko.COM_Festo.DS4_1_Port0_IN[6] AT %IB."P4_IOmaster".Module007_Inputs007;
	Cyclic#1.P4_Pracovisko.COM_Festo.DS4_1_Port0_IN[7] AT %IB."P4_IOmaster".Module007_Inputs008;
	Cyclic#1.P4_Pracovisko.COM_Festo.DS4_1_Port0_IN[8] AT %IB."P4_IOmaster".Module007_Inputs009;
	Cyclic#1.P4_Pracovisko.COM_Festo.DS4_1_Port0_IN[9] AT %IB."P4_IOmaster".Module007_Inputs010;
	Cyclic#1.P4_Pracovisko.COM_Festo.DS4_1_Port0_IN[10] AT %IB."P4_IOmaster".Module007_Inputs011;
	Cyclic#1.P4_Pracovisko.COM_Festo.DS4_1_Port0_IN[11] AT %IB."P4_IOmaster".Module007_Inputs012;
	Cyclic#1.P4_Pracovisko.COM_Festo.DS4_1_Port0_IN[12] AT %IB."P4_IOmaster".Module007_Inputs013;
	Cyclic#1.P4_Pracovisko.COM_Festo.DS4_1_Port0_IN[13] AT %IB."P4_IOmaster".Module007_Inputs014;
	Cyclic#1.P4_Pracovisko.COM_Festo.DS4_1_Port0_IN[14] AT %IB."P4_IOmaster".Module007_Inputs015;
	Cyclic#1.P4_Pracovisko.COM_Festo.DS4_1_Port0_IN[15] AT %IB."P4_IOmaster".Module007_Inputs016;
	Cyclic#1.P4_Pracovisko.COM_Festo.DS4_1_Port0_IN[16] AT %IB."P4_IOmaster".Module007_Inputs017;
	Cyclic#1.P4_Pracovisko.COM_Festo.DS4_1_Port0_IN[17] AT %IB."P4_IOmaster".Module007_Inputs018;
	Cyclic#1.P4_Pracovisko.COM_Festo.DS4_1_Port0_IN[18] AT %IB."P4_IOmaster".Module007_Inputs019;
	Cyclic#1.P4_Pracovisko.COM_Festo.DS4_1_Port0_IN[19] AT %IB."P4_IOmaster".Module007_Inputs020;
	Cyclic#1.P4_Pracovisko.COM_Festo.DS4_1_Port0_IN[20] AT %IB."P4_IOmaster".Module007_Inputs021;
	Cyclic#1.P4_Pracovisko.COM_Festo.DS4_1_Port0_IN[21] AT %IB."P4_IOmaster".Module007_Inputs022;
	Cyclic#1.P4_Pracovisko.COM_Festo.DS4_1_Port0_IN[22] AT %IB."P4_IOmaster".Module007_Inputs023;
	Cyclic#1.P4_Pracovisko.COM_Festo.DS4_1_Port0_IN[23] AT %IB."P4_IOmaster".Module007_Inputs024;
	Cyclic#1.P4_Pracovisko.COM_Festo.DS4_1_Port0_IN[24] AT %IB."P4_IOmaster".Module007_Inputs025;
	Cyclic#1.P4_Pracovisko.COM_Festo.DS4_1_Port0_IN[25] AT %IB."P4_IOmaster".Module007_Inputs026;
	Cyclic#1.P4_Pracovisko.COM_Festo.DS4_1_Port0_IN[26] AT %IB."P4_IOmaster".Module007_Inputs027;
	Cyclic#1.P4_Pracovisko.COM_Festo.DS4_1_Port0_IN[27] AT %IB."P4_IOmaster".Module007_Inputs028;
	Cyclic#1.P4_Pracovisko.COM_Festo.DS4_1_Port0_IN[28] AT %IB."P4_IOmaster".Module007_Inputs029;
	Cyclic#1.P4_Pracovisko.COM_Festo.DS4_1_Port0_IN[29] AT %IB."P4_IOmaster".Module007_Inputs030;
	Cyclic#1.P4_Pracovisko.COM_Festo.DS4_1_Port0_IN[30] AT %IB."P4_IOmaster".Module007_Inputs031;
	Cyclic#1.P4_Pracovisko.COM_Festo.DS4_1_Port0_IN[31] AT %IB."P4_IOmaster".Module007_Inputs032;
	Cyclic#1.P4_Pracovisko.COM_Festo.DS4_1_Port1_IN[0] AT %IB."P4_IOmaster".Module007_Inputs033;
	Cyclic#1.P4_Pracovisko.COM_Festo.DS4_1_Port1_IN[1] AT %IB."P4_IOmaster".Module007_Inputs034;
	Cyclic#1.P4_Pracovisko.COM_Festo.DS4_1_Port1_IN[2] AT %IB."P4_IOmaster".Module007_Inputs035;
	Cyclic#1.P4_Pracovisko.COM_Festo.DS4_1_Port1_IN[3] AT %IB."P4_IOmaster".Module007_Inputs036;
	Cyclic#1.P4_Pracovisko.COM_Festo.DS4_1_Port1_IN[4] AT %IB."P4_IOmaster".Module007_Inputs037;
	Cyclic#1.P4_Pracovisko.COM_Festo.DS4_1_Port1_IN[5] AT %IB."P4_IOmaster".Module007_Inputs038;
	Cyclic#1.P4_Pracovisko.COM_Festo.DS4_1_Port1_IN[6] AT %IB."P4_IOmaster".Module007_Inputs039;
	Cyclic#1.P4_Pracovisko.COM_Festo.DS4_1_Port1_IN[7] AT %IB."P4_IOmaster".Module007_Inputs040;
	Cyclic#1.P4_Pracovisko.COM_Festo.DS4_1_Port1_IN[8] AT %IB."P4_IOmaster".Module007_Inputs041;
	Cyclic#1.P4_Pracovisko.COM_Festo.DS4_1_Port1_IN[9] AT %IB."P4_IOmaster".Module007_Inputs042;
	Cyclic#1.P4_Pracovisko.COM_Festo.DS4_1_Port1_IN[10] AT %IB."P4_IOmaster".Module007_Inputs043;
	Cyclic#1.P4_Pracovisko.COM_Festo.DS4_1_Port1_IN[11] AT %IB."P4_IOmaster".Module007_Inputs044;
	Cyclic#1.P4_Pracovisko.COM_Festo.DS4_1_Port1_IN[12] AT %IB."P4_IOmaster".Module007_Inputs045;
	Cyclic#1.P4_Pracovisko.COM_Festo.DS4_1_Port1_IN[13] AT %IB."P4_IOmaster".Module007_Inputs046;
	Cyclic#1.P4_Pracovisko.COM_Festo.DS4_1_Port1_IN[14] AT %IB."P4_IOmaster".Module007_Inputs047;
	Cyclic#1.P4_Pracovisko.COM_Festo.DS4_1_Port1_IN[15] AT %IB."P4_IOmaster".Module007_Inputs048;
	Cyclic#1.P4_Pracovisko.COM_Festo.DS4_1_Port1_IN[16] AT %IB."P4_IOmaster".Module007_Inputs049;
	Cyclic#1.P4_Pracovisko.COM_Festo.DS4_1_Port1_IN[17] AT %IB."P4_IOmaster".Module007_Inputs050;
	Cyclic#1.P4_Pracovisko.COM_Festo.DS4_1_Port1_IN[18] AT %IB."P4_IOmaster".Module007_Inputs051;
	Cyclic#1.P4_Pracovisko.COM_Festo.DS4_1_Port1_IN[19] AT %IB."P4_IOmaster".Module007_Inputs052;
	Cyclic#1.P4_Pracovisko.COM_Festo.DS4_1_Port1_IN[20] AT %IB."P4_IOmaster".Module007_Inputs053;
	Cyclic#1.P4_Pracovisko.COM_Festo.DS4_1_Port1_IN[21] AT %IB."P4_IOmaster".Module007_Inputs054;
	Cyclic#1.P4_Pracovisko.COM_Festo.DS4_1_Port1_IN[22] AT %IB."P4_IOmaster".Module007_Inputs055;
	Cyclic#1.P4_Pracovisko.COM_Festo.DS4_1_Port1_IN[23] AT %IB."P4_IOmaster".Module007_Inputs056;
	Cyclic#1.P4_Pracovisko.COM_Festo.DS4_1_Port1_IN[24] AT %IB."P4_IOmaster".Module007_Inputs057;
	Cyclic#1.P4_Pracovisko.COM_Festo.DS4_1_Port1_IN[25] AT %IB."P4_IOmaster".Module007_Inputs058;
	Cyclic#1.P4_Pracovisko.COM_Festo.DS4_1_Port1_IN[26] AT %IB."P4_IOmaster".Module007_Inputs059;
	Cyclic#1.P4_Pracovisko.COM_Festo.DS4_1_Port1_IN[27] AT %IB."P4_IOmaster".Module007_Inputs060;
	Cyclic#1.P4_Pracovisko.COM_Festo.DS4_1_Port1_IN[28] AT %IB."P4_IOmaster".Module007_Inputs061;
	Cyclic#1.P4_Pracovisko.COM_Festo.DS4_1_Port1_IN[29] AT %IB."P4_IOmaster".Module007_Inputs062;
	Cyclic#1.P4_Pracovisko.COM_Festo.DS4_1_Port1_IN[30] AT %IB."P4_IOmaster".Module007_Inputs063;
	Cyclic#1.P4_Pracovisko.COM_Festo.DS4_1_Port1_IN[31] AT %IB."P4_IOmaster".Module007_Inputs064;
	Cyclic#1.P4_Pracovisko.COM_Festo.DS4_1_Port2_IN[0] AT %IB."P4_IOmaster".Module007_Inputs065;
	Cyclic#1.P4_Pracovisko.COM_Festo.DS4_1_Port2_IN[1] AT %IB."P4_IOmaster".Module007_Inputs066;
	Cyclic#1.P4_Pracovisko.COM_Festo.DS4_1_Port2_IN[2] AT %IB."P4_IOmaster".Module007_Inputs067;
	Cyclic#1.P4_Pracovisko.COM_Festo.DS4_1_Port2_IN[3] AT %IB."P4_IOmaster".Module007_Inputs068;
	Cyclic#1.P4_Pracovisko.COM_Festo.DS4_1_Port2_IN[4] AT %IB."P4_IOmaster".Module007_Inputs069;
	Cyclic#1.P4_Pracovisko.COM_Festo.DS4_1_Port2_IN[5] AT %IB."P4_IOmaster".Module007_Inputs070;
	Cyclic#1.P4_Pracovisko.COM_Festo.DS4_1_Port2_IN[6] AT %IB."P4_IOmaster".Module007_Inputs071;
	Cyclic#1.P4_Pracovisko.COM_Festo.DS4_1_Port2_IN[7] AT %IB."P4_IOmaster".Module007_Inputs072;
	Cyclic#1.P4_Pracovisko.COM_Festo.DS4_1_Port2_IN[8] AT %IB."P4_IOmaster".Module007_Inputs073;
	Cyclic#1.P4_Pracovisko.COM_Festo.DS4_1_Port2_IN[9] AT %IB."P4_IOmaster".Module007_Inputs074;
	Cyclic#1.P4_Pracovisko.COM_Festo.DS4_1_Port2_IN[10] AT %IB."P4_IOmaster".Module007_Inputs075;
	Cyclic#1.P4_Pracovisko.COM_Festo.DS4_1_Port2_IN[11] AT %IB."P4_IOmaster".Module007_Inputs076;
	Cyclic#1.P4_Pracovisko.COM_Festo.DS4_1_Port2_IN[12] AT %IB."P4_IOmaster".Module007_Inputs077;
	Cyclic#1.P4_Pracovisko.COM_Festo.DS4_1_Port2_IN[13] AT %IB."P4_IOmaster".Module007_Inputs078;
	Cyclic#1.P4_Pracovisko.COM_Festo.DS4_1_Port2_IN[14] AT %IB."P4_IOmaster".Module007_Inputs079;
	Cyclic#1.P4_Pracovisko.COM_Festo.DS4_1_Port2_IN[15] AT %IB."P4_IOmaster".Module007_Inputs080;
	Cyclic#1.P4_Pracovisko.COM_Festo.DS4_1_Port2_IN[16] AT %IB."P4_IOmaster".Module007_Inputs081;
	Cyclic#1.P4_Pracovisko.COM_Festo.DS4_1_Port2_IN[17] AT %IB."P4_IOmaster".Module007_Inputs082;
	Cyclic#1.P4_Pracovisko.COM_Festo.DS4_1_Port2_IN[18] AT %IB."P4_IOmaster".Module007_Inputs083;
	Cyclic#1.P4_Pracovisko.COM_Festo.DS4_1_Port2_IN[19] AT %IB."P4_IOmaster".Module007_Inputs084;
	Cyclic#1.P4_Pracovisko.COM_Festo.DS4_1_Port2_IN[20] AT %IB."P4_IOmaster".Module007_Inputs085;
	Cyclic#1.P4_Pracovisko.COM_Festo.DS4_1_Port2_IN[21] AT %IB."P4_IOmaster".Module007_Inputs086;
	Cyclic#1.P4_Pracovisko.COM_Festo.DS4_1_Port2_IN[22] AT %IB."P4_IOmaster".Module007_Inputs087;
	Cyclic#1.P4_Pracovisko.COM_Festo.DS4_1_Port2_IN[23] AT %IB."P4_IOmaster".Module007_Inputs088;
	Cyclic#1.P4_Pracovisko.COM_Festo.DS4_1_Port2_IN[24] AT %IB."P4_IOmaster".Module007_Inputs089;
	Cyclic#1.P4_Pracovisko.COM_Festo.DS4_1_Port2_IN[25] AT %IB."P4_IOmaster".Module007_Inputs090;
	Cyclic#1.P4_Pracovisko.COM_Festo.DS4_1_Port2_IN[26] AT %IB."P4_IOmaster".Module007_Inputs091;
	Cyclic#1.P4_Pracovisko.COM_Festo.DS4_1_Port2_IN[27] AT %IB."P4_IOmaster".Module007_Inputs092;
	Cyclic#1.P4_Pracovisko.COM_Festo.DS4_1_Port2_IN[28] AT %IB."P4_IOmaster".Module007_Inputs093;
	Cyclic#1.P4_Pracovisko.COM_Festo.DS4_1_Port2_IN[29] AT %IB."P4_IOmaster".Module007_Inputs094;
	Cyclic#1.P4_Pracovisko.COM_Festo.DS4_1_Port2_IN[30] AT %IB."P4_IOmaster".Module007_Inputs095;
	Cyclic#1.P4_Pracovisko.COM_Festo.DS4_1_Port2_IN[31] AT %IB."P4_IOmaster".Module007_Inputs096;
	Cyclic#1.P4_Pracovisko.COM_Festo.DS4_1_Port0_OUT[0] AT %QB."P4_IOmaster".Module007_Outputs001;
	Cyclic#1.P4_Pracovisko.COM_Festo.DS4_1_Port0_OUT[1] AT %QB."P4_IOmaster".Module007_Outputs002;
	Cyclic#1.P4_Pracovisko.COM_Festo.DS4_1_Port0_OUT[2] AT %QB."P4_IOmaster".Module007_Outputs003;
	Cyclic#1.P4_Pracovisko.COM_Festo.DS4_1_Port0_OUT[3] AT %QB."P4_IOmaster".Module007_Outputs004;
	Cyclic#1.P4_Pracovisko.COM_Festo.DS4_1_Port0_OUT[4] AT %QB."P4_IOmaster".Module007_Outputs005;
	Cyclic#1.P4_Pracovisko.COM_Festo.DS4_1_Port0_OUT[5] AT %QB."P4_IOmaster".Module007_Outputs006;
	Cyclic#1.P4_Pracovisko.COM_Festo.DS4_1_Port0_OUT[6] AT %QB."P4_IOmaster".Module007_Outputs007;
	Cyclic#1.P4_Pracovisko.COM_Festo.DS4_1_Port0_OUT[7] AT %QB."P4_IOmaster".Module007_Outputs008;
	Cyclic#1.P4_Pracovisko.COM_Festo.DS4_1_Port0_OUT[8] AT %QB."P4_IOmaster".Module007_Outputs009;
	Cyclic#1.P4_Pracovisko.COM_Festo.DS4_1_Port0_OUT[9] AT %QB."P4_IOmaster".Module007_Outputs010;
	Cyclic#1.P4_Pracovisko.COM_Festo.DS4_1_Port0_OUT[10] AT %QB."P4_IOmaster".Module007_Outputs011;
	Cyclic#1.P4_Pracovisko.COM_Festo.DS4_1_Port0_OUT[11] AT %QB."P4_IOmaster".Module007_Outputs012;
	Cyclic#1.P4_Pracovisko.COM_Festo.DS4_1_Port0_OUT[12] AT %QB."P4_IOmaster".Module007_Outputs013;
	Cyclic#1.P4_Pracovisko.COM_Festo.DS4_1_Port0_OUT[13] AT %QB."P4_IOmaster".Module007_Outputs014;
	Cyclic#1.P4_Pracovisko.COM_Festo.DS4_1_Port0_OUT[14] AT %QB."P4_IOmaster".Module007_Outputs015;
	Cyclic#1.P4_Pracovisko.COM_Festo.DS4_1_Port0_OUT[15] AT %QB."P4_IOmaster".Module007_Outputs016;
	Cyclic#1.P4_Pracovisko.COM_Festo.DS4_1_Port0_OUT[16] AT %QB."P4_IOmaster".Module007_Outputs017;
	Cyclic#1.P4_Pracovisko.COM_Festo.DS4_1_Port0_OUT[17] AT %QB."P4_IOmaster".Module007_Outputs018;
	Cyclic#1.P4_Pracovisko.COM_Festo.DS4_1_Port0_OUT[18] AT %QB."P4_IOmaster".Module007_Outputs019;
	Cyclic#1.P4_Pracovisko.COM_Festo.DS4_1_Port0_OUT[19] AT %QB."P4_IOmaster".Module007_Outputs020;
	Cyclic#1.P4_Pracovisko.COM_Festo.DS4_1_Port0_OUT[20] AT %QB."P4_IOmaster".Module007_Outputs021;
	Cyclic#1.P4_Pracovisko.COM_Festo.DS4_1_Port0_OUT[21] AT %QB."P4_IOmaster".Module007_Outputs022;
	Cyclic#1.P4_Pracovisko.COM_Festo.DS4_1_Port0_OUT[22] AT %QB."P4_IOmaster".Module007_Outputs023;
	Cyclic#1.P4_Pracovisko.COM_Festo.DS4_1_Port0_OUT[23] AT %QB."P4_IOmaster".Module007_Outputs024;
	Cyclic#1.P4_Pracovisko.COM_Festo.DS4_1_Port0_OUT[24] AT %QB."P4_IOmaster".Module007_Outputs025;
	Cyclic#1.P4_Pracovisko.COM_Festo.DS4_1_Port0_OUT[25] AT %QB."P4_IOmaster".Module007_Outputs026;
	Cyclic#1.P4_Pracovisko.COM_Festo.DS4_1_Port0_OUT[26] AT %QB."P4_IOmaster".Module007_Outputs027;
	Cyclic#1.P4_Pracovisko.COM_Festo.DS4_1_Port0_OUT[27] AT %QB."P4_IOmaster".Module007_Outputs028;
	Cyclic#1.P4_Pracovisko.COM_Festo.DS4_1_Port0_OUT[28] AT %QB."P4_IOmaster".Module007_Outputs029;
	Cyclic#1.P4_Pracovisko.COM_Festo.DS4_1_Port0_OUT[29] AT %QB."P4_IOmaster".Module007_Outputs030;
	Cyclic#1.P4_Pracovisko.COM_Festo.DS4_1_Port0_OUT[30] AT %QB."P4_IOmaster".Module007_Outputs031;
	Cyclic#1.P4_Pracovisko.COM_Festo.DS4_1_Port0_OUT[31] AT %QB."P4_IOmaster".Module007_Outputs032;
	Cyclic#1.P4_Pracovisko.COM_Festo.DS4_1_Port1_OUT[0] AT %QB."P4_IOmaster".Module007_Outputs033;
	Cyclic#1.P4_Pracovisko.COM_Festo.DS4_1_Port1_OUT[1] AT %QB."P4_IOmaster".Module007_Outputs034;
	Cyclic#1.P4_Pracovisko.COM_Festo.DS4_1_Port1_OUT[2] AT %QB."P4_IOmaster".Module007_Outputs035;
	Cyclic#1.P4_Pracovisko.COM_Festo.DS4_1_Port1_OUT[3] AT %QB."P4_IOmaster".Module007_Outputs036;
	Cyclic#1.P4_Pracovisko.COM_Festo.DS4_1_Port1_OUT[4] AT %QB."P4_IOmaster".Module007_Outputs037;
	Cyclic#1.P4_Pracovisko.COM_Festo.DS4_1_Port1_OUT[5] AT %QB."P4_IOmaster".Module007_Outputs038;
	Cyclic#1.P4_Pracovisko.COM_Festo.DS4_1_Port1_OUT[6] AT %QB."P4_IOmaster".Module007_Outputs039;
	Cyclic#1.P4_Pracovisko.COM_Festo.DS4_1_Port1_OUT[7] AT %QB."P4_IOmaster".Module007_Outputs040;
	Cyclic#1.P4_Pracovisko.COM_Festo.DS4_1_Port1_OUT[8] AT %QB."P4_IOmaster".Module007_Outputs041;
	Cyclic#1.P4_Pracovisko.COM_Festo.DS4_1_Port1_OUT[9] AT %QB."P4_IOmaster".Module007_Outputs042;
	Cyclic#1.P4_Pracovisko.COM_Festo.DS4_1_Port1_OUT[10] AT %QB."P4_IOmaster".Module007_Outputs043;
	Cyclic#1.P4_Pracovisko.COM_Festo.DS4_1_Port1_OUT[11] AT %QB."P4_IOmaster".Module007_Outputs044;
	Cyclic#1.P4_Pracovisko.COM_Festo.DS4_1_Port1_OUT[12] AT %QB."P4_IOmaster".Module007_Outputs045;
	Cyclic#1.P4_Pracovisko.COM_Festo.DS4_1_Port1_OUT[13] AT %QB."P4_IOmaster".Module007_Outputs046;
	Cyclic#1.P4_Pracovisko.COM_Festo.DS4_1_Port1_OUT[14] AT %QB."P4_IOmaster".Module007_Outputs047;
	Cyclic#1.P4_Pracovisko.COM_Festo.DS4_1_Port1_OUT[15] AT %QB."P4_IOmaster".Module007_Outputs048;
	Cyclic#1.P4_Pracovisko.COM_Festo.DS4_1_Port1_OUT[16] AT %QB."P4_IOmaster".Module007_Outputs049;
	Cyclic#1.P4_Pracovisko.COM_Festo.DS4_1_Port1_OUT[17] AT %QB."P4_IOmaster".Module007_Outputs050;
	Cyclic#1.P4_Pracovisko.COM_Festo.DS4_1_Port1_OUT[18] AT %QB."P4_IOmaster".Module007_Outputs051;
	Cyclic#1.P4_Pracovisko.COM_Festo.DS4_1_Port1_OUT[19] AT %QB."P4_IOmaster".Module007_Outputs052;
	Cyclic#1.P4_Pracovisko.COM_Festo.DS4_1_Port1_OUT[20] AT %QB."P4_IOmaster".Module007_Outputs053;
	Cyclic#1.P4_Pracovisko.COM_Festo.DS4_1_Port1_OUT[21] AT %QB."P4_IOmaster".Module007_Outputs054;
	Cyclic#1.P4_Pracovisko.COM_Festo.DS4_1_Port1_OUT[22] AT %QB."P4_IOmaster".Module007_Outputs055;
	Cyclic#1.P4_Pracovisko.COM_Festo.DS4_1_Port1_OUT[23] AT %QB."P4_IOmaster".Module007_Outputs056;
	Cyclic#1.P4_Pracovisko.COM_Festo.DS4_1_Port1_OUT[24] AT %QB."P4_IOmaster".Module007_Outputs057;
	Cyclic#1.P4_Pracovisko.COM_Festo.DS4_1_Port1_OUT[25] AT %QB."P4_IOmaster".Module007_Outputs058;
	Cyclic#1.P4_Pracovisko.COM_Festo.DS4_1_Port1_OUT[26] AT %QB."P4_IOmaster".Module007_Outputs059;
	Cyclic#1.P4_Pracovisko.COM_Festo.DS4_1_Port1_OUT[27] AT %QB."P4_IOmaster".Module007_Outputs060;
	Cyclic#1.P4_Pracovisko.COM_Festo.DS4_1_Port1_OUT[28] AT %QB."P4_IOmaster".Module007_Outputs061;
	Cyclic#1.P4_Pracovisko.COM_Festo.DS4_1_Port1_OUT[29] AT %QB."P4_IOmaster".Module007_Outputs062;
	Cyclic#1.P4_Pracovisko.COM_Festo.DS4_1_Port1_OUT[30] AT %QB."P4_IOmaster".Module007_Outputs063;
	Cyclic#1.P4_Pracovisko.COM_Festo.DS4_1_Port1_OUT[31] AT %QB."P4_IOmaster".Module007_Outputs064;
	Cyclic#1.P4_Pracovisko.COM_Festo.DS4_1_Port2_OUT[0] AT %QB."P4_IOmaster".Module007_Outputs065;
	Cyclic#1.P4_Pracovisko.COM_Festo.DS4_1_Port2_OUT[1] AT %QB."P4_IOmaster".Module007_Outputs066;
	Cyclic#1.P4_Pracovisko.COM_Festo.DS4_1_Port2_OUT[2] AT %QB."P4_IOmaster".Module007_Outputs067;
	Cyclic#1.P4_Pracovisko.COM_Festo.DS4_1_Port2_OUT[3] AT %QB."P4_IOmaster".Module007_Outputs068;
	Cyclic#1.P4_Pracovisko.COM_Festo.DS4_1_Port2_OUT[4] AT %QB."P4_IOmaster".Module007_Outputs069;
	Cyclic#1.P4_Pracovisko.COM_Festo.DS4_1_Port2_OUT[5] AT %QB."P4_IOmaster".Module007_Outputs070;
	Cyclic#1.P4_Pracovisko.COM_Festo.DS4_1_Port2_OUT[6] AT %QB."P4_IOmaster".Module007_Outputs071;
	Cyclic#1.P4_Pracovisko.COM_Festo.DS4_1_Port2_OUT[7] AT %QB."P4_IOmaster".Module007_Outputs072;
	Cyclic#1.P4_Pracovisko.COM_Festo.DS4_1_Port2_OUT[8] AT %QB."P4_IOmaster".Module007_Outputs073;
	Cyclic#1.P4_Pracovisko.COM_Festo.DS4_1_Port2_OUT[9] AT %QB."P4_IOmaster".Module007_Outputs074;
	Cyclic#1.P4_Pracovisko.COM_Festo.DS4_1_Port2_OUT[10] AT %QB."P4_IOmaster".Module007_Outputs075;
	Cyclic#1.P4_Pracovisko.COM_Festo.DS4_1_Port2_OUT[11] AT %QB."P4_IOmaster".Module007_Outputs076;
	Cyclic#1.P4_Pracovisko.COM_Festo.DS4_1_Port2_OUT[12] AT %QB."P4_IOmaster".Module007_Outputs077;
	Cyclic#1.P4_Pracovisko.COM_Festo.DS4_1_Port2_OUT[13] AT %QB."P4_IOmaster".Module007_Outputs078;
	Cyclic#1.P4_Pracovisko.COM_Festo.DS4_1_Port2_OUT[14] AT %QB."P4_IOmaster".Module007_Outputs079;
	Cyclic#1.P4_Pracovisko.COM_Festo.DS4_1_Port2_OUT[15] AT %QB."P4_IOmaster".Module007_Outputs080;
	Cyclic#1.P4_Pracovisko.COM_Festo.DS4_1_Port2_OUT[16] AT %QB."P4_IOmaster".Module007_Outputs081;
	Cyclic#1.P4_Pracovisko.COM_Festo.DS4_1_Port2_OUT[17] AT %QB."P4_IOmaster".Module007_Outputs082;
	Cyclic#1.P4_Pracovisko.COM_Festo.DS4_1_Port2_OUT[18] AT %QB."P4_IOmaster".Module007_Outputs083;
	Cyclic#1.P4_Pracovisko.COM_Festo.DS4_1_Port2_OUT[19] AT %QB."P4_IOmaster".Module007_Outputs084;
	Cyclic#1.P4_Pracovisko.COM_Festo.DS4_1_Port2_OUT[20] AT %QB."P4_IOmaster".Module007_Outputs085;
	Cyclic#1.P4_Pracovisko.COM_Festo.DS4_1_Port2_OUT[21] AT %QB."P4_IOmaster".Module007_Outputs086;
	Cyclic#1.P4_Pracovisko.COM_Festo.DS4_1_Port2_OUT[22] AT %QB."P4_IOmaster".Module007_Outputs087;
	Cyclic#1.P4_Pracovisko.COM_Festo.DS4_1_Port2_OUT[23] AT %QB."P4_IOmaster".Module007_Outputs088;
	Cyclic#1.P4_Pracovisko.COM_Festo.DS4_1_Port2_OUT[24] AT %QB."P4_IOmaster".Module007_Outputs089;
	Cyclic#1.P4_Pracovisko.COM_Festo.DS4_1_Port2_OUT[25] AT %QB."P4_IOmaster".Module007_Outputs090;
	Cyclic#1.P4_Pracovisko.COM_Festo.DS4_1_Port2_OUT[26] AT %QB."P4_IOmaster".Module007_Outputs091;
	Cyclic#1.P4_Pracovisko.COM_Festo.DS4_1_Port2_OUT[27] AT %QB."P4_IOmaster".Module007_Outputs092;
	Cyclic#1.P4_Pracovisko.COM_Festo.DS4_1_Port2_OUT[28] AT %QB."P4_IOmaster".Module007_Outputs093;
	Cyclic#1.P4_Pracovisko.COM_Festo.DS4_1_Port2_OUT[29] AT %QB."P4_IOmaster".Module007_Outputs094;
	Cyclic#1.P4_Pracovisko.COM_Festo.DS4_1_Port2_OUT[30] AT %QB."P4_IOmaster".Module007_Outputs095;
	Cyclic#1.P4_Pracovisko.COM_Festo.DS4_1_Port2_OUT[31] AT %QB."P4_IOmaster".Module007_Outputs096;
	Cyclic#1.P4_Pracovisko.COM_Festo.DS4_2_Port0_IN[0] AT %IB."P4_IOmaster".Module008_Inputs001;
	Cyclic#1.P4_Pracovisko.COM_Festo.DS4_2_Port0_IN[1] AT %IB."P4_IOmaster".Module008_Inputs002;
	Cyclic#1.P4_Pracovisko.COM_Festo.DS4_2_Port0_IN[2] AT %IB."P4_IOmaster".Module008_Inputs003;
	Cyclic#1.P4_Pracovisko.COM_Festo.DS4_2_Port0_IN[3] AT %IB."P4_IOmaster".Module008_Inputs004;
	Cyclic#1.P4_Pracovisko.COM_Festo.DS4_2_Port0_IN[4] AT %IB."P4_IOmaster".Module008_Inputs005;
	Cyclic#1.P4_Pracovisko.COM_Festo.DS4_2_Port0_IN[5] AT %IB."P4_IOmaster".Module008_Inputs006;
	Cyclic#1.P4_Pracovisko.COM_Festo.DS4_2_Port0_IN[6] AT %IB."P4_IOmaster".Module008_Inputs007;
	Cyclic#1.P4_Pracovisko.COM_Festo.DS4_2_Port0_IN[7] AT %IB."P4_IOmaster".Module008_Inputs008;
	Cyclic#1.P4_Pracovisko.COM_Festo.DS4_2_Port0_IN[8] AT %IB."P4_IOmaster".Module008_Inputs009;
	Cyclic#1.P4_Pracovisko.COM_Festo.DS4_2_Port0_IN[9] AT %IB."P4_IOmaster".Module008_Inputs010;
	Cyclic#1.P4_Pracovisko.COM_Festo.DS4_2_Port0_IN[10] AT %IB."P4_IOmaster".Module008_Inputs011;
	Cyclic#1.P4_Pracovisko.COM_Festo.DS4_2_Port0_IN[11] AT %IB."P4_IOmaster".Module008_Inputs012;
	Cyclic#1.P4_Pracovisko.COM_Festo.DS4_2_Port0_IN[12] AT %IB."P4_IOmaster".Module008_Inputs013;
	Cyclic#1.P4_Pracovisko.COM_Festo.DS4_2_Port0_IN[13] AT %IB."P4_IOmaster".Module008_Inputs014;
	Cyclic#1.P4_Pracovisko.COM_Festo.DS4_2_Port0_IN[14] AT %IB."P4_IOmaster".Module008_Inputs015;
	Cyclic#1.P4_Pracovisko.COM_Festo.DS4_2_Port0_IN[15] AT %IB."P4_IOmaster".Module008_Inputs016;
	Cyclic#1.P4_Pracovisko.COM_Festo.DS4_2_Port1_IN[0] AT %IB."P4_IOmaster".Module008_Inputs017;
	Cyclic#1.P4_Pracovisko.COM_Festo.DS4_2_Port1_IN[1] AT %IB."P4_IOmaster".Module008_Inputs018;
	Cyclic#1.P4_Pracovisko.COM_Festo.DS4_2_Port1_IN[2] AT %IB."P4_IOmaster".Module008_Inputs019;
	Cyclic#1.P4_Pracovisko.COM_Festo.DS4_2_Port1_IN[3] AT %IB."P4_IOmaster".Module008_Inputs020;
	Cyclic#1.P4_Pracovisko.COM_Festo.DS4_2_Port1_IN[4] AT %IB."P4_IOmaster".Module008_Inputs021;
	Cyclic#1.P4_Pracovisko.COM_Festo.DS4_2_Port1_IN[5] AT %IB."P4_IOmaster".Module008_Inputs022;
	Cyclic#1.P4_Pracovisko.COM_Festo.DS4_2_Port1_IN[6] AT %IB."P4_IOmaster".Module008_Inputs023;
	Cyclic#1.P4_Pracovisko.COM_Festo.DS4_2_Port1_IN[7] AT %IB."P4_IOmaster".Module008_Inputs024;
	Cyclic#1.P4_Pracovisko.COM_Festo.DS4_2_Port1_IN[8] AT %IB."P4_IOmaster".Module008_Inputs025;
	Cyclic#1.P4_Pracovisko.COM_Festo.DS4_2_Port1_IN[9] AT %IB."P4_IOmaster".Module008_Inputs026;
	Cyclic#1.P4_Pracovisko.COM_Festo.DS4_2_Port1_IN[10] AT %IB."P4_IOmaster".Module008_Inputs027;
	Cyclic#1.P4_Pracovisko.COM_Festo.DS4_2_Port1_IN[11] AT %IB."P4_IOmaster".Module008_Inputs028;
	Cyclic#1.P4_Pracovisko.COM_Festo.DS4_2_Port1_IN[12] AT %IB."P4_IOmaster".Module008_Inputs029;
	Cyclic#1.P4_Pracovisko.COM_Festo.DS4_2_Port1_IN[13] AT %IB."P4_IOmaster".Module008_Inputs030;
	Cyclic#1.P4_Pracovisko.COM_Festo.DS4_2_Port1_IN[14] AT %IB."P4_IOmaster".Module008_Inputs031;
	Cyclic#1.P4_Pracovisko.COM_Festo.DS4_2_Port1_IN[15] AT %IB."P4_IOmaster".Module008_Inputs032;
	Cyclic#1.P4_Pracovisko.COM_Festo.DS4_2_Port1_IN[16] AT %IB."P4_IOmaster".Module008_Inputs033;
	Cyclic#1.P4_Pracovisko.COM_Festo.DS4_2_Port1_IN[17] AT %IB."P4_IOmaster".Module008_Inputs034;
	Cyclic#1.P4_Pracovisko.COM_Festo.DS4_2_Port1_IN[18] AT %IB."P4_IOmaster".Module008_Inputs035;
	Cyclic#1.P4_Pracovisko.COM_Festo.DS4_2_Port1_IN[19] AT %IB."P4_IOmaster".Module008_Inputs036;
	Cyclic#1.P4_Pracovisko.COM_Festo.DS4_2_Port1_IN[20] AT %IB."P4_IOmaster".Module008_Inputs037;
	Cyclic#1.P4_Pracovisko.COM_Festo.DS4_2_Port1_IN[21] AT %IB."P4_IOmaster".Module008_Inputs038;
	Cyclic#1.P4_Pracovisko.COM_Festo.DS4_2_Port1_IN[22] AT %IB."P4_IOmaster".Module008_Inputs039;
	Cyclic#1.P4_Pracovisko.COM_Festo.DS4_2_Port1_IN[23] AT %IB."P4_IOmaster".Module008_Inputs040;
	Cyclic#1.P4_Pracovisko.COM_Festo.DS4_2_Port1_IN[24] AT %IB."P4_IOmaster".Module008_Inputs041;
	Cyclic#1.P4_Pracovisko.COM_Festo.DS4_2_Port1_IN[25] AT %IB."P4_IOmaster".Module008_Inputs042;
	Cyclic#1.P4_Pracovisko.COM_Festo.DS4_2_Port1_IN[26] AT %IB."P4_IOmaster".Module008_Inputs043;
	Cyclic#1.P4_Pracovisko.COM_Festo.DS4_2_Port1_IN[27] AT %IB."P4_IOmaster".Module008_Inputs044;
	Cyclic#1.P4_Pracovisko.COM_Festo.DS4_2_Port1_IN[28] AT %IB."P4_IOmaster".Module008_Inputs045;
	Cyclic#1.P4_Pracovisko.COM_Festo.DS4_2_Port1_IN[29] AT %IB."P4_IOmaster".Module008_Inputs046;
	Cyclic#1.P4_Pracovisko.COM_Festo.DS4_2_Port1_IN[30] AT %IB."P4_IOmaster".Module008_Inputs047;
	Cyclic#1.P4_Pracovisko.COM_Festo.DS4_2_Port1_IN[31] AT %IB."P4_IOmaster".Module008_Inputs048;
	Cyclic#1.P4_Pracovisko.COM_Festo.DS4_2_Port0_OUT[0] AT %QB."P4_IOmaster".Module008_Outputs001;
	Cyclic#1.P4_Pracovisko.COM_Festo.DS4_2_Port0_OUT[1] AT %QB."P4_IOmaster".Module008_Outputs002;
	Cyclic#1.P4_Pracovisko.COM_Festo.DS4_2_Port0_OUT[2] AT %QB."P4_IOmaster".Module008_Outputs003;
	Cyclic#1.P4_Pracovisko.COM_Festo.DS4_2_Port0_OUT[3] AT %QB."P4_IOmaster".Module008_Outputs004;
	Cyclic#1.P4_Pracovisko.COM_Festo.DS4_2_Port0_OUT[4] AT %QB."P4_IOmaster".Module008_Outputs005;
	Cyclic#1.P4_Pracovisko.COM_Festo.DS4_2_Port0_OUT[5] AT %QB."P4_IOmaster".Module008_Outputs006;
	Cyclic#1.P4_Pracovisko.COM_Festo.DS4_2_Port0_OUT[6] AT %QB."P4_IOmaster".Module008_Outputs007;
	Cyclic#1.P4_Pracovisko.COM_Festo.DS4_2_Port0_OUT[7] AT %QB."P4_IOmaster".Module008_Outputs008;
	Cyclic#1.P4_Pracovisko.COM_Festo.DS4_2_Port0_OUT[8] AT %QB."P4_IOmaster".Module008_Outputs009;
	Cyclic#1.P4_Pracovisko.COM_Festo.DS4_2_Port0_OUT[9] AT %QB."P4_IOmaster".Module008_Outputs010;
	Cyclic#1.P4_Pracovisko.COM_Festo.DS4_2_Port0_OUT[10] AT %QB."P4_IOmaster".Module008_Outputs011;
	Cyclic#1.P4_Pracovisko.COM_Festo.DS4_2_Port0_OUT[11] AT %QB."P4_IOmaster".Module008_Outputs012;
	Cyclic#1.P4_Pracovisko.COM_Festo.DS4_2_Port0_OUT[12] AT %QB."P4_IOmaster".Module008_Outputs013;
	Cyclic#1.P4_Pracovisko.COM_Festo.DS4_2_Port0_OUT[13] AT %QB."P4_IOmaster".Module008_Outputs014;
	Cyclic#1.P4_Pracovisko.COM_Festo.DS4_2_Port0_OUT[14] AT %QB."P4_IOmaster".Module008_Outputs015;
	Cyclic#1.P4_Pracovisko.COM_Festo.DS4_2_Port0_OUT[15] AT %QB."P4_IOmaster".Module008_Outputs016;
	Cyclic#1.P4_Pracovisko.COM_Festo.DS4_2_Port1_OUT[0] AT %QB."P4_IOmaster".Module008_Outputs017;
	Cyclic#1.P4_Pracovisko.COM_Festo.DS4_2_Port1_OUT[1] AT %QB."P4_IOmaster".Module008_Outputs018;
	Cyclic#1.P4_Pracovisko.COM_Festo.DS4_2_Port1_OUT[2] AT %QB."P4_IOmaster".Module008_Outputs019;
	Cyclic#1.P4_Pracovisko.COM_Festo.DS4_2_Port1_OUT[3] AT %QB."P4_IOmaster".Module008_Outputs020;
	Cyclic#1.P4_Pracovisko.COM_Festo.DS4_2_Port1_OUT[4] AT %QB."P4_IOmaster".Module008_Outputs021;
	Cyclic#1.P4_Pracovisko.COM_Festo.DS4_2_Port1_OUT[5] AT %QB."P4_IOmaster".Module008_Outputs022;
	Cyclic#1.P4_Pracovisko.COM_Festo.DS4_2_Port1_OUT[6] AT %QB."P4_IOmaster".Module008_Outputs023;
	Cyclic#1.P4_Pracovisko.COM_Festo.DS4_2_Port1_OUT[7] AT %QB."P4_IOmaster".Module008_Outputs024;
	Cyclic#1.P4_Pracovisko.COM_Festo.DS4_2_Port1_OUT[8] AT %QB."P4_IOmaster".Module008_Outputs025;
	Cyclic#1.P4_Pracovisko.COM_Festo.DS4_2_Port1_OUT[9] AT %QB."P4_IOmaster".Module008_Outputs026;
	Cyclic#1.P4_Pracovisko.COM_Festo.DS4_2_Port1_OUT[10] AT %QB."P4_IOmaster".Module008_Outputs027;
	Cyclic#1.P4_Pracovisko.COM_Festo.DS4_2_Port1_OUT[11] AT %QB."P4_IOmaster".Module008_Outputs028;
	Cyclic#1.P4_Pracovisko.COM_Festo.DS4_2_Port1_OUT[12] AT %QB."P4_IOmaster".Module008_Outputs029;
	Cyclic#1.P4_Pracovisko.COM_Festo.DS4_2_Port1_OUT[13] AT %QB."P4_IOmaster".Module008_Outputs030;
	Cyclic#1.P4_Pracovisko.COM_Festo.DS4_2_Port1_OUT[14] AT %QB."P4_IOmaster".Module008_Outputs031;
	Cyclic#1.P4_Pracovisko.COM_Festo.DS4_2_Port1_OUT[15] AT %QB."P4_IOmaster".Module008_Outputs032;
	Cyclic#1.P4_Pracovisko.COM_Festo.DS4_2_Port1_OUT[16] AT %QB."P4_IOmaster".Module008_Outputs033;
	Cyclic#1.P4_Pracovisko.COM_Festo.DS4_2_Port1_OUT[17] AT %QB."P4_IOmaster".Module008_Outputs034;
	Cyclic#1.P4_Pracovisko.COM_Festo.DS4_2_Port1_OUT[18] AT %QB."P4_IOmaster".Module008_Outputs035;
	Cyclic#1.P4_Pracovisko.COM_Festo.DS4_2_Port1_OUT[19] AT %QB."P4_IOmaster".Module008_Outputs036;
	Cyclic#1.P4_Pracovisko.COM_Festo.DS4_2_Port1_OUT[20] AT %QB."P4_IOmaster".Module008_Outputs037;
	Cyclic#1.P4_Pracovisko.COM_Festo.DS4_2_Port1_OUT[21] AT %QB."P4_IOmaster".Module008_Outputs038;
	Cyclic#1.P4_Pracovisko.COM_Festo.DS4_2_Port1_OUT[22] AT %QB."P4_IOmaster".Module008_Outputs039;
	Cyclic#1.P4_Pracovisko.COM_Festo.DS4_2_Port1_OUT[23] AT %QB."P4_IOmaster".Module008_Outputs040;
	Cyclic#1.P4_Pracovisko.COM_Festo.DS4_2_Port1_OUT[24] AT %QB."P4_IOmaster".Module008_Outputs041;
	Cyclic#1.P4_Pracovisko.COM_Festo.DS4_2_Port1_OUT[25] AT %QB."P4_IOmaster".Module008_Outputs042;
	Cyclic#1.P4_Pracovisko.COM_Festo.DS4_2_Port1_OUT[26] AT %QB."P4_IOmaster".Module008_Outputs043;
	Cyclic#1.P4_Pracovisko.COM_Festo.DS4_2_Port1_OUT[27] AT %QB."P4_IOmaster".Module008_Outputs044;
	Cyclic#1.P4_Pracovisko.COM_Festo.DS4_2_Port1_OUT[28] AT %QB."P4_IOmaster".Module008_Outputs045;
	Cyclic#1.P4_Pracovisko.COM_Festo.DS4_2_Port1_OUT[29] AT %QB."P4_IOmaster".Module008_Outputs046;
	Cyclic#1.P4_Pracovisko.COM_Festo.DS4_2_Port1_OUT[30] AT %QB."P4_IOmaster".Module008_Outputs047;
	Cyclic#1.P4_Pracovisko.COM_Festo.DS4_2_Port1_OUT[31] AT %QB."P4_IOmaster".Module008_Outputs048;
	Cyclic#1.Linka.IN.SafetyMaster_OK AT %IX."P2_SafetyMaster".ModuleOk;
	Cyclic#1.Safety.Mapping_BYTE_OUT[0] AT %QB."P2_SafetyMaster".Module001_External_Input_signal_EI_byte_0;
	Cyclic#1.Safety.Mapping_BYTE_OUT[1] AT %QB."P2_SafetyMaster".Module001_External_Input_signal_EI_byte_1;
	Cyclic#1.Safety.Mapping_BYTE_OUT[2] AT %QB."P2_SafetyMaster".Module001_External_Input_signal_EI_byte_2;
	Cyclic#1.Safety.Mapping_BYTE_OUT[3] AT %QB."P2_SafetyMaster".Module001_External_Input_signal_EI_byte_3;
	Cyclic#1.Safety.Mapping_BYTE_IN[0] AT %IB."P2_SafetyMaster".Module002_Input_status_byte_0;
	Cyclic#1.Safety.Mapping_BYTE_IN[1] AT %IB."P2_SafetyMaster".Module002_Input_status_byte_1;
	Cyclic#1.Safety.Mapping_BYTE_IN[2] AT %IB."P2_SafetyMaster".Module002_Input_status_byte_2;
	Cyclic#1.Safety.Mapping_BYTE_IN[3] AT %IB."P2_SafetyMaster".Module002_Input_status_byte_3;
	Cyclic#1.Safety.Mapping_BYTE_IN[4] AT %IB."P2_SafetyMaster".Module002_Input_status_byte_4;
	Cyclic#1.Safety.Mapping_BYTE_IN[5] AT %IB."P2_SafetyMaster".Module002_Input_status_byte_5;
	Cyclic#1.Safety.Mapping_BYTE_IN[6] AT %IB."P2_SafetyMaster".Module002_Input_status_byte_6;
	Cyclic#1.Safety.Mapping_BYTE_IN[7] AT %IB."P2_SafetyMaster".Module002_Input_status_byte_7;
	Cyclic#1.Safety.Mapping_BYTE_IN[8] AT %IB."P2_SafetyMaster".Module002_Input_status_byte_8;
	Cyclic#1.Safety.Mapping_BYTE_IN[9] AT %IB."P2_SafetyMaster".Module002_Input_status_byte_9;
	Cyclic#1.Safety.Mapping_BYTE_IN[10] AT %IB."P2_SafetyMaster".Module002_Input_status_byte_10;
	Cyclic#1.Safety.Mapping_BYTE_IN[11] AT %IB."P2_SafetyMaster".Module002_Input_status_byte_11;
	Cyclic#1.Safety.Mapping_BYTE_IN[12] AT %IB."P2_SafetyMaster".Module002_Input_status_byte_12;
	Cyclic#1.Safety.Mapping_BYTE_IN[13] AT %IB."P2_SafetyMaster".Module002_Input_status_byte_13;
	Cyclic#1.Safety.Mapping_BYTE_IN[14] AT %IB."P2_SafetyMaster".Module002_Input_status_byte_14;
	Cyclic#1.Safety.Mapping_BYTE_IN[15] AT %IB."P2_SafetyMaster".Module002_Input_status_byte_15;
	Cyclic#1.P2_Pracovisko.COM_VentilovyTerminal[10] AT %QB."P2_VentilovyTerminal_VT2".ValveCoils81_88_I2000_S0B;
	Cyclic#1.P2_Pracovisko.COM_Festo.DS2_1_Port3_IN[2] AT %IB."P2_IOmaster".Module012_Inputs009;
	Cyclic#1.P2_Pracovisko.COM_Festo.DS2_1_Port3_IN[3] AT %IB."P2_IOmaster".Module012_Inputs010;
	Cyclic#1.P2_Pracovisko.COM_Festo.DS2_1_Port3_IN[4] AT %IB."P2_IOmaster".Module012_Inputs011;
	Cyclic#1.P2_Pracovisko.COM_Festo.DS2_1_Port3_IN[5] AT %IB."P2_IOmaster".Module012_Inputs012;
	Cyclic#1.P2_Pracovisko.COM_Festo.DS2_1_Port3_IN[6] AT %IB."P2_IOmaster".Module012_Inputs013;
	Cyclic#1.P2_Pracovisko.COM_Festo.DS2_1_Port3_IN[7] AT %IB."P2_IOmaster".Module012_Inputs014;
	Cyclic#1.P2_Pracovisko.COM_Festo.DS2_1_Port3_IN[8] AT %IB."P2_IOmaster".Module012_Inputs015;
	Cyclic#1.P2_Pracovisko.COM_Festo.DS2_1_Port3_IN[9] AT %IB."P2_IOmaster".Module012_Inputs016;
	Cyclic#1.P2_Pracovisko.COM_Festo.DS2_1_Port3_IN[10] AT %IB."P2_IOmaster".Module012_Inputs017;
	Cyclic#1.P2_Pracovisko.COM_Festo.DS2_1_Port3_IN[11] AT %IB."P2_IOmaster".Module012_Inputs018;
	Cyclic#1.P2_Pracovisko.COM_Festo.DS2_1_Port3_IN[12] AT %IB."P2_IOmaster".Module012_Inputs019;
	Cyclic#1.P2_Pracovisko.COM_Festo.DS2_1_Port3_IN[13] AT %IB."P2_IOmaster".Module012_Inputs020;
	Cyclic#1.P2_Pracovisko.COM_Festo.DS2_1_Port3_IN[14] AT %IB."P2_IOmaster".Module012_Inputs021;
	Cyclic#1.P2_Pracovisko.COM_Festo.DS2_1_Port3_IN[15] AT %IB."P2_IOmaster".Module012_Inputs022;
	Cyclic#1.P2_Pracovisko.COM_Festo.DS2_1_Port3_IN[16] AT %IB."P2_IOmaster".Module012_Inputs023;
	Cyclic#1.P2_Pracovisko.COM_Festo.DS2_1_Port3_IN[17] AT %IB."P2_IOmaster".Module012_Inputs024;
	Cyclic#1.P2_Pracovisko.COM_Festo.DS2_1_Port3_IN[18] AT %IB."P2_IOmaster".Module012_Inputs025;
	Cyclic#1.P2_Pracovisko.COM_Festo.DS2_1_Port3_IN[19] AT %IB."P2_IOmaster".Module012_Inputs026;
	Cyclic#1.P2_Pracovisko.COM_Festo.DS2_1_Port3_IN[20] AT %IB."P2_IOmaster".Module012_Inputs027;
	Cyclic#1.P2_Pracovisko.COM_Festo.DS2_1_Port3_IN[21] AT %IB."P2_IOmaster".Module012_Inputs028;
	Cyclic#1.P2_Pracovisko.COM_Festo.DS2_1_Port3_IN[22] AT %IB."P2_IOmaster".Module012_Inputs029;
	Cyclic#1.P2_Pracovisko.COM_Festo.DS2_1_Port3_IN[23] AT %IB."P2_IOmaster".Module012_Inputs030;
	Cyclic#1.P2_Pracovisko.COM_Festo.DS2_1_Port3_IN[24] AT %IB."P2_IOmaster".Module012_Inputs031;
	Cyclic#1.P2_Pracovisko.COM_Festo.DS2_1_Port3_IN[25] AT %IB."P2_IOmaster".Module012_Inputs032;
	Cyclic#1.P2_Pracovisko.COM_Festo.DS2_1_Port3_IN[26] AT %IB."P2_IOmaster".Module012_Inputs033;
	Cyclic#1.P2_Pracovisko.COM_Festo.DS2_1_Port3_IN[27] AT %IB."P2_IOmaster".Module012_Inputs034;
	Cyclic#1.P2_Pracovisko.COM_Festo.DS2_1_Port3_IN[28] AT %IB."P2_IOmaster".Module012_Inputs035;
	Cyclic#1.P2_Pracovisko.COM_Festo.DS2_1_Port3_IN[29] AT %IB."P2_IOmaster".Module012_Inputs036;
	Cyclic#1.P2_Pracovisko.COM_Festo.DS2_1_Port3_IN[30] AT %IB."P2_IOmaster".Module012_Inputs037;
	Cyclic#1.P2_Pracovisko.COM_Festo.DS2_1_Port3_IN[31] AT %IB."P2_IOmaster".Module012_Inputs038;
	Cyclic#1.P2_Pracovisko.COM_Festo.DS2_1_Port3_OUT[2] AT %QB."P2_IOmaster".Module012_Outputs009;
	Cyclic#1.P2_Pracovisko.COM_Festo.DS2_1_Port3_OUT[3] AT %QB."P2_IOmaster".Module012_Outputs010;
	Cyclic#1.P2_Pracovisko.COM_Festo.DS2_1_Port3_OUT[4] AT %QB."P2_IOmaster".Module012_Outputs011;
	Cyclic#1.P2_Pracovisko.COM_Festo.DS2_1_Port3_OUT[5] AT %QB."P2_IOmaster".Module012_Outputs012;
	Cyclic#1.P2_Pracovisko.COM_Festo.DS2_1_Port3_OUT[6] AT %QB."P2_IOmaster".Module012_Outputs013;
	Cyclic#1.P2_Pracovisko.COM_Festo.DS2_1_Port3_OUT[7] AT %QB."P2_IOmaster".Module012_Outputs014;
	Cyclic#1.P2_Pracovisko.COM_Festo.DS2_1_Port3_OUT[8] AT %QB."P2_IOmaster".Module012_Outputs015;
	Cyclic#1.P2_Pracovisko.COM_Festo.DS2_1_Port3_OUT[9] AT %QB."P2_IOmaster".Module012_Outputs016;
	Cyclic#1.P2_Pracovisko.COM_Festo.DS2_1_Port3_OUT[10] AT %QB."P2_IOmaster".Module012_Outputs017;
	Cyclic#1.P2_Pracovisko.COM_Festo.DS2_1_Port3_OUT[11] AT %QB."P2_IOmaster".Module012_Outputs018;
	Cyclic#1.P2_Pracovisko.COM_Festo.DS2_1_Port3_OUT[12] AT %QB."P2_IOmaster".Module012_Outputs019;
	Cyclic#1.P2_Pracovisko.COM_Festo.DS2_1_Port3_OUT[13] AT %QB."P2_IOmaster".Module012_Outputs020;
	Cyclic#1.P2_Pracovisko.COM_Festo.DS2_1_Port3_OUT[14] AT %QB."P2_IOmaster".Module012_Outputs021;
	Cyclic#1.P2_Pracovisko.COM_Festo.DS2_1_Port3_OUT[15] AT %QB."P2_IOmaster".Module012_Outputs022;
	Cyclic#1.P2_Pracovisko.COM_Festo.DS2_1_Port3_OUT[16] AT %QB."P2_IOmaster".Module012_Outputs023;
	Cyclic#1.P2_Pracovisko.COM_Festo.DS2_1_Port3_OUT[17] AT %QB."P2_IOmaster".Module012_Outputs024;
	Cyclic#1.P2_Pracovisko.COM_Festo.DS2_1_Port3_OUT[18] AT %QB."P2_IOmaster".Module012_Outputs025;
	Cyclic#1.P2_Pracovisko.COM_Festo.DS2_1_Port3_OUT[19] AT %QB."P2_IOmaster".Module012_Outputs026;
	Cyclic#1.P2_Pracovisko.COM_Festo.DS2_1_Port3_OUT[20] AT %QB."P2_IOmaster".Module012_Outputs027;
	Cyclic#1.P2_Pracovisko.COM_Festo.DS2_1_Port3_OUT[21] AT %QB."P2_IOmaster".Module012_Outputs028;
	Cyclic#1.P2_Pracovisko.COM_Festo.DS2_1_Port3_OUT[22] AT %QB."P2_IOmaster".Module012_Outputs029;
	Cyclic#1.P2_Pracovisko.COM_Festo.DS2_1_Port3_OUT[23] AT %QB."P2_IOmaster".Module012_Outputs030;
	Cyclic#1.P2_Pracovisko.COM_Festo.DS2_1_Port3_OUT[24] AT %QB."P2_IOmaster".Module012_Outputs031;
	Cyclic#1.P2_Pracovisko.COM_Festo.DS2_1_Port3_OUT[25] AT %QB."P2_IOmaster".Module012_Outputs032;
	Cyclic#1.P2_Pracovisko.COM_Festo.DS2_1_Port3_OUT[26] AT %QB."P2_IOmaster".Module012_Outputs033;
	Cyclic#1.P2_Pracovisko.COM_Festo.DS2_1_Port3_OUT[27] AT %QB."P2_IOmaster".Module012_Outputs034;
	Cyclic#1.P2_Pracovisko.COM_Festo.DS2_1_Port3_OUT[28] AT %QB."P2_IOmaster".Module012_Outputs035;
	Cyclic#1.P2_Pracovisko.COM_Festo.DS2_1_Port3_OUT[29] AT %QB."P2_IOmaster".Module012_Outputs036;
	Cyclic#1.P2_Pracovisko.COM_Festo.DS2_1_Port3_OUT[30] AT %QB."P2_IOmaster".Module012_Outputs037;
	Cyclic#1.P2_Pracovisko.COM_Festo.DS2_1_Port3_OUT[31] AT %QB."P2_IOmaster".Module012_Outputs038;
	Cyclic#1.P4_Pracovisko.IN.SmartKamera14_KomOK AT %IX."P4_CAM_14".ModuleOk;
	Cyclic#1.P3_Pracovisko.IN.ModulFesto_IO_KomOK AT %IX."P3_IO_Master".ModuleOk;
	Cyclic#1.P3_Pracovisko.COM_Festo.DI3_1_8DI[0] AT %IX."P3_IO_Master".Module001_Bit_0_Bit_0;
	Cyclic#1.P3_Pracovisko.COM_Festo.DI3_1_8DI[1] AT %IX."P3_IO_Master".Module001_Bit_1_Bit_1;
	Cyclic#1.P3_Pracovisko.COM_Festo.DI3_1_8DI[2] AT %IX."P3_IO_Master".Module001_Bit_2_Bit_2;
	Cyclic#1.P3_Pracovisko.COM_Festo.DI3_1_8DI[3] AT %IX."P3_IO_Master".Module001_Bit_3_Bit_3;
	Cyclic#1.P3_Pracovisko.COM_Festo.DI3_1_8DI[4] AT %IX."P3_IO_Master".Module001_Bit_4_Bit_4;
	Cyclic#1.P3_Pracovisko.COM_Festo.DI3_1_8DI[5] AT %IX."P3_IO_Master".Module001_Bit_5_Bit_5;
	Cyclic#1.P3_Pracovisko.COM_Festo.DI3_1_8DI[6] AT %IX."P3_IO_Master".Module001_Bit_6_Bit_6;
	Cyclic#1.P3_Pracovisko.COM_Festo.DI3_1_8DI[7] AT %IX."P3_IO_Master".Module001_Bit_7_Bit_7;
	Cyclic#1.P3_Pracovisko.COM_Festo.DM3_1_4DI[0] AT %IX."P3_IO_Master".Module002_Bit_0_Bit_0;
	Cyclic#1.P3_Pracovisko.COM_Festo.DM3_1_4DI[1] AT %IX."P3_IO_Master".Module002_Bit_1_Bit_1;
	Cyclic#1.P3_Pracovisko.COM_Festo.DM3_1_4DI[2] AT %IX."P3_IO_Master".Module002_Bit_2_Bit_2;
	Cyclic#1.P3_Pracovisko.COM_Festo.DM3_1_4DI[3] AT %IX."P3_IO_Master".Module002_Bit_3_Bit_3;
	Cyclic#1.P3_Pracovisko.COM_Festo.DM3_1_4DO[0] AT %QX."P3_IO_Master".Module002_Bit_0_Bit_1;
	Cyclic#1.P3_Pracovisko.COM_Festo.DM3_1_4DO[1] AT %QX."P3_IO_Master".Module002_Bit_1_Bit_2;
	Cyclic#1.P3_Pracovisko.COM_Festo.DM3_1_4DO[2] AT %QX."P3_IO_Master".Module002_Bit_2_Bit_3;
	Cyclic#1.P3_Pracovisko.COM_Festo.DM3_1_4DO[3] AT %QX."P3_IO_Master".Module002_Bit_3_Bit_4;
	Cyclic#1.P3_Pracovisko.COM_Festo.DI3_4_8DI[0] AT %IX."P3_IO_Master".Module003_Bit_0_Bit_0;
	Cyclic#1.P3_Pracovisko.COM_Festo.DI3_4_8DI[1] AT %IX."P3_IO_Master".Module003_Bit_1_Bit_1;
	Cyclic#1.P3_Pracovisko.COM_Festo.DI3_4_8DI[2] AT %IX."P3_IO_Master".Module003_Bit_2_Bit_2;
	Cyclic#1.P3_Pracovisko.COM_Festo.DI3_4_8DI[3] AT %IX."P3_IO_Master".Module003_Bit_3_Bit_3;
	Cyclic#1.P3_Pracovisko.COM_Festo.DI3_4_8DI[4] AT %IX."P3_IO_Master".Module003_Bit_4_Bit_4;
	Cyclic#1.P3_Pracovisko.COM_Festo.DI3_4_8DI[5] AT %IX."P3_IO_Master".Module003_Bit_5_Bit_5;
	Cyclic#1.P3_Pracovisko.COM_Festo.DI3_4_8DI[6] AT %IX."P3_IO_Master".Module003_Bit_6_Bit_6;
	Cyclic#1.P3_Pracovisko.COM_Festo.DI3_4_8DI[7] AT %IX."P3_IO_Master".Module003_Bit_7_Bit_7;
	Cyclic#1.P3_Pracovisko.COM_Festo.DI3_8_8DI[0] AT %IX."P3_IO_Master".Module004_Bit_0_Bit_0;
	Cyclic#1.P3_Pracovisko.COM_Festo.DI3_8_8DI[1] AT %IX."P3_IO_Master".Module004_Bit_1_Bit_1;
	Cyclic#1.P3_Pracovisko.COM_Festo.DI3_8_8DI[2] AT %IX."P3_IO_Master".Module004_Bit_2_Bit_2;
	Cyclic#1.P3_Pracovisko.COM_Festo.DI3_8_8DI[3] AT %IX."P3_IO_Master".Module004_Bit_3_Bit_3;
	Cyclic#1.P3_Pracovisko.COM_Festo.DI3_8_8DI[4] AT %IX."P3_IO_Master".Module004_Bit_4_Bit_4;
	Cyclic#1.P3_Pracovisko.COM_Festo.DI3_8_8DI[5] AT %IX."P3_IO_Master".Module004_Bit_5_Bit_5;
	Cyclic#1.P3_Pracovisko.COM_Festo.DI3_8_8DI[6] AT %IX."P3_IO_Master".Module004_Bit_6_Bit_6;
	Cyclic#1.P3_Pracovisko.COM_Festo.DI3_8_8DI[7] AT %IX."P3_IO_Master".Module004_Bit_7_Bit_7;
	Cyclic#1.P3_Pracovisko.COM_Festo.DI3_9_8DI[0] AT %IX."P3_IO_Master".Module005_Bit_0_Bit_0;
	Cyclic#1.P3_Pracovisko.COM_Festo.DI3_9_8DI[1] AT %IX."P3_IO_Master".Module005_Bit_1_Bit_1;
	Cyclic#1.P3_Pracovisko.COM_Festo.DI3_9_8DI[2] AT %IX."P3_IO_Master".Module005_Bit_2_Bit_2;
	Cyclic#1.P3_Pracovisko.COM_Festo.DI3_9_8DI[3] AT %IX."P3_IO_Master".Module005_Bit_3_Bit_3;
	Cyclic#1.P3_Pracovisko.COM_Festo.DI3_9_8DI[4] AT %IX."P3_IO_Master".Module005_Bit_4_Bit_4;
	Cyclic#1.P3_Pracovisko.COM_Festo.DI3_9_8DI[5] AT %IX."P3_IO_Master".Module005_Bit_5_Bit_5;
	Cyclic#1.P3_Pracovisko.COM_Festo.DI3_9_8DI[6] AT %IX."P3_IO_Master".Module005_Bit_6_Bit_6;
	Cyclic#1.P3_Pracovisko.COM_Festo.DI3_9_8DI[7] AT %IX."P3_IO_Master".Module005_Bit_7_Bit_7;
	Cyclic#1.P3_Pracovisko.COM_Festo.DI3_10_8DI[0] AT %IX."P3_IO_Master".Module006_Bit_0_Bit_0;
	Cyclic#1.P3_Pracovisko.COM_Festo.DI3_10_8DI[1] AT %IX."P3_IO_Master".Module006_Bit_1_Bit_1;
	Cyclic#1.P3_Pracovisko.COM_Festo.DI3_10_8DI[2] AT %IX."P3_IO_Master".Module006_Bit_2_Bit_2;
	Cyclic#1.P3_Pracovisko.COM_Festo.DI3_10_8DI[3] AT %IX."P3_IO_Master".Module006_Bit_3_Bit_3;
	Cyclic#1.P3_Pracovisko.COM_Festo.DI3_10_8DI[4] AT %IX."P3_IO_Master".Module006_Bit_4_Bit_4;
	Cyclic#1.P3_Pracovisko.COM_Festo.DI3_10_8DI[5] AT %IX."P3_IO_Master".Module006_Bit_5_Bit_5;
	Cyclic#1.P3_Pracovisko.COM_Festo.DI3_10_8DI[6] AT %IX."P3_IO_Master".Module006_Bit_6_Bit_6;
	Cyclic#1.P3_Pracovisko.COM_Festo.DI3_10_8DI[7] AT %IX."P3_IO_Master".Module006_Bit_7_Bit_7;
	Cyclic#1.P3_Pracovisko.COM_Festo.DI3_3_8DI[0] AT %IX."P3_IO_Master".Module007_Bit_0_Bit_0;
	Cyclic#1.P3_Pracovisko.COM_Festo.DI3_3_8DI[1] AT %IX."P3_IO_Master".Module007_Bit_1_Bit_1;
	Cyclic#1.P3_Pracovisko.COM_Festo.DI3_3_8DI[2] AT %IX."P3_IO_Master".Module007_Bit_2_Bit_2;
	Cyclic#1.P3_Pracovisko.COM_Festo.DI3_3_8DI[3] AT %IX."P3_IO_Master".Module007_Bit_3_Bit_3;
	Cyclic#1.P3_Pracovisko.COM_Festo.DI3_3_8DI[4] AT %IX."P3_IO_Master".Module007_Bit_4_Bit_4;
	Cyclic#1.P3_Pracovisko.COM_Festo.DI3_3_8DI[5] AT %IX."P3_IO_Master".Module007_Bit_5_Bit_5;
	Cyclic#1.P3_Pracovisko.COM_Festo.DI3_3_8DI[6] AT %IX."P3_IO_Master".Module007_Bit_6_Bit_6;
	Cyclic#1.P3_Pracovisko.COM_Festo.DI3_3_8DI[7] AT %IX."P3_IO_Master".Module007_Bit_7_Bit_7;
	Cyclic#1.P3_Pracovisko.COM_Festo.DI3_2_8DI[0] AT %IX."P3_IO_Master".Module008_Bit_0_Bit_0;
	Cyclic#1.P3_Pracovisko.COM_Festo.DI3_2_8DI[1] AT %IX."P3_IO_Master".Module008_Bit_1_Bit_1;
	Cyclic#1.P3_Pracovisko.COM_Festo.DI3_2_8DI[2] AT %IX."P3_IO_Master".Module008_Bit_2_Bit_2;
	Cyclic#1.P3_Pracovisko.COM_Festo.DI3_2_8DI[3] AT %IX."P3_IO_Master".Module008_Bit_3_Bit_3;
	Cyclic#1.P3_Pracovisko.COM_Festo.DI3_2_8DI[4] AT %IX."P3_IO_Master".Module008_Bit_4_Bit_4;
	Cyclic#1.P3_Pracovisko.COM_Festo.DI3_2_8DI[5] AT %IX."P3_IO_Master".Module008_Bit_5_Bit_5;
	Cyclic#1.P3_Pracovisko.COM_Festo.DI3_2_8DI[6] AT %IX."P3_IO_Master".Module008_Bit_6_Bit_6;
	Cyclic#1.P3_Pracovisko.COM_Festo.DI3_2_8DI[7] AT %IX."P3_IO_Master".Module008_Bit_7_Bit_7;
	Cyclic#1.P3_Pracovisko.COM_Festo.DI3_7_8DI[0] AT %IX."P3_IO_Master".Module009_Bit_0_Bit_0;
	Cyclic#1.P3_Pracovisko.COM_Festo.DI3_7_8DI[1] AT %IX."P3_IO_Master".Module009_Bit_1_Bit_1;
	Cyclic#1.P3_Pracovisko.COM_Festo.DI3_7_8DI[2] AT %IX."P3_IO_Master".Module009_Bit_2_Bit_2;
	Cyclic#1.P3_Pracovisko.COM_Festo.DI3_7_8DI[3] AT %IX."P3_IO_Master".Module009_Bit_3_Bit_3;
	Cyclic#1.P3_Pracovisko.COM_Festo.DI3_7_8DI[4] AT %IX."P3_IO_Master".Module009_Bit_4_Bit_4;
	Cyclic#1.P3_Pracovisko.COM_Festo.DI3_7_8DI[5] AT %IX."P3_IO_Master".Module009_Bit_5_Bit_5;
	Cyclic#1.P3_Pracovisko.COM_Festo.DI3_7_8DI[6] AT %IX."P3_IO_Master".Module009_Bit_6_Bit_6;
	Cyclic#1.P3_Pracovisko.COM_Festo.DI3_7_8DI[7] AT %IX."P3_IO_Master".Module009_Bit_7_Bit_7;
	Cyclic#1.P3_Pracovisko.COM_Festo.DI3_5_8DI[0] AT %IX."P3_IO_Master".Module010_Bit_0_Bit_0;
	Cyclic#1.P3_Pracovisko.COM_Festo.DI3_5_8DI[1] AT %IX."P3_IO_Master".Module010_Bit_1_Bit_1;
	Cyclic#1.P3_Pracovisko.COM_Festo.DI3_5_8DI[2] AT %IX."P3_IO_Master".Module010_Bit_2_Bit_2;
	Cyclic#1.P3_Pracovisko.COM_Festo.DI3_5_8DI[3] AT %IX."P3_IO_Master".Module010_Bit_3_Bit_3;
	Cyclic#1.P3_Pracovisko.COM_Festo.DI3_5_8DI[4] AT %IX."P3_IO_Master".Module010_Bit_4_Bit_4;
	Cyclic#1.P3_Pracovisko.COM_Festo.DI3_5_8DI[5] AT %IX."P3_IO_Master".Module010_Bit_5_Bit_5;
	Cyclic#1.P3_Pracovisko.COM_Festo.DI3_5_8DI[6] AT %IX."P3_IO_Master".Module010_Bit_6_Bit_6;
	Cyclic#1.P3_Pracovisko.COM_Festo.DI3_5_8DI[7] AT %IX."P3_IO_Master".Module010_Bit_7_Bit_7;
	Cyclic#1.P3_Pracovisko.COM_Festo.DI3_6_8DI[0] AT %IX."P3_IO_Master".Module011_Bit_0_Bit_0;
	Cyclic#1.P3_Pracovisko.COM_Festo.DI3_6_8DI[1] AT %IX."P3_IO_Master".Module011_Bit_1_Bit_1;
	Cyclic#1.P3_Pracovisko.COM_Festo.DI3_6_8DI[2] AT %IX."P3_IO_Master".Module011_Bit_2_Bit_2;
	Cyclic#1.P3_Pracovisko.COM_Festo.DI3_6_8DI[3] AT %IX."P3_IO_Master".Module011_Bit_3_Bit_3;
	Cyclic#1.P3_Pracovisko.COM_Festo.DI3_6_8DI[4] AT %IX."P3_IO_Master".Module011_Bit_4_Bit_4;
	Cyclic#1.P3_Pracovisko.COM_Festo.DI3_6_8DI[5] AT %IX."P3_IO_Master".Module011_Bit_5_Bit_5;
	Cyclic#1.P3_Pracovisko.COM_Festo.DI3_6_8DI[6] AT %IX."P3_IO_Master".Module011_Bit_6_Bit_6;
	Cyclic#1.P3_Pracovisko.COM_Festo.DI3_6_8DI[7] AT %IX."P3_IO_Master".Module011_Bit_7_Bit_7;
	Cyclic#1.P3_Pracovisko.COM_Festo.DS3_1_Port0_IN[0] AT %IB."P3_IO_Master".Module012_Inputs001;
	Cyclic#1.P3_Pracovisko.COM_Festo.DS3_1_Port0_IN[1] AT %IB."P3_IO_Master".Module012_Inputs002;
	Cyclic#1.P3_Pracovisko.COM_Festo.DS3_1_Port0_IN[2] AT %IB."P3_IO_Master".Module012_Inputs003;
	Cyclic#1.P3_Pracovisko.COM_Festo.DS3_1_Port0_IN[3] AT %IB."P3_IO_Master".Module012_Inputs004;
	Cyclic#1.P3_Pracovisko.COM_Festo.DS3_1_Port0_IN[4] AT %IB."P3_IO_Master".Module012_Inputs005;
	Cyclic#1.P3_Pracovisko.COM_Festo.DS3_1_Port0_IN[5] AT %IB."P3_IO_Master".Module012_Inputs006;
	Cyclic#1.P3_Pracovisko.COM_Festo.DS3_1_Port0_IN[6] AT %IB."P3_IO_Master".Module012_Inputs007;
	Cyclic#1.P3_Pracovisko.COM_Festo.DS3_1_Port0_IN[7] AT %IB."P3_IO_Master".Module012_Inputs008;
	Cyclic#1.P3_Pracovisko.COM_Festo.DS3_1_Port0_IN[8] AT %IB."P3_IO_Master".Module012_Inputs009;
	Cyclic#1.P3_Pracovisko.COM_Festo.DS3_1_Port0_IN[9] AT %IB."P3_IO_Master".Module012_Inputs010;
	Cyclic#1.P3_Pracovisko.COM_Festo.DS3_1_Port0_IN[10] AT %IB."P3_IO_Master".Module012_Inputs011;
	Cyclic#1.P3_Pracovisko.COM_Festo.DS3_1_Port0_IN[11] AT %IB."P3_IO_Master".Module012_Inputs012;
	Cyclic#1.P3_Pracovisko.COM_Festo.DS3_1_Port0_IN[12] AT %IB."P3_IO_Master".Module012_Inputs013;
	Cyclic#1.P3_Pracovisko.COM_Festo.DS3_1_Port0_IN[13] AT %IB."P3_IO_Master".Module012_Inputs014;
	Cyclic#1.P3_Pracovisko.COM_Festo.DS3_1_Port0_IN[14] AT %IB."P3_IO_Master".Module012_Inputs015;
	Cyclic#1.P3_Pracovisko.COM_Festo.DS3_1_Port0_IN[15] AT %IB."P3_IO_Master".Module012_Inputs016;
	Cyclic#1.P3_Pracovisko.COM_Festo.DS3_1_Port0_IN[16] AT %IB."P3_IO_Master".Module012_Inputs017;
	Cyclic#1.P3_Pracovisko.COM_Festo.DS3_1_Port0_IN[17] AT %IB."P3_IO_Master".Module012_Inputs018;
	Cyclic#1.P3_Pracovisko.COM_Festo.DS3_1_Port0_IN[18] AT %IB."P3_IO_Master".Module012_Inputs019;
	Cyclic#1.P3_Pracovisko.COM_Festo.DS3_1_Port0_IN[19] AT %IB."P3_IO_Master".Module012_Inputs020;
	Cyclic#1.P3_Pracovisko.COM_Festo.DS3_1_Port0_IN[20] AT %IB."P3_IO_Master".Module012_Inputs021;
	Cyclic#1.P3_Pracovisko.COM_Festo.DS3_1_Port0_IN[21] AT %IB."P3_IO_Master".Module012_Inputs022;
	Cyclic#1.P3_Pracovisko.COM_Festo.DS3_1_Port0_IN[22] AT %IB."P3_IO_Master".Module012_Inputs023;
	Cyclic#1.P3_Pracovisko.COM_Festo.DS3_1_Port0_IN[23] AT %IB."P3_IO_Master".Module012_Inputs024;
	Cyclic#1.P3_Pracovisko.COM_Festo.DS3_1_Port0_IN[24] AT %IB."P3_IO_Master".Module012_Inputs025;
	Cyclic#1.P3_Pracovisko.COM_Festo.DS3_1_Port0_IN[25] AT %IB."P3_IO_Master".Module012_Inputs026;
	Cyclic#1.P3_Pracovisko.COM_Festo.DS3_1_Port0_IN[26] AT %IB."P3_IO_Master".Module012_Inputs027;
	Cyclic#1.P3_Pracovisko.COM_Festo.DS3_1_Port0_IN[27] AT %IB."P3_IO_Master".Module012_Inputs028;
	Cyclic#1.P3_Pracovisko.COM_Festo.DS3_1_Port0_IN[28] AT %IB."P3_IO_Master".Module012_Inputs029;
	Cyclic#1.P3_Pracovisko.COM_Festo.DS3_1_Port0_IN[29] AT %IB."P3_IO_Master".Module012_Inputs030;
	Cyclic#1.P3_Pracovisko.COM_Festo.DS3_1_Port0_IN[30] AT %IB."P3_IO_Master".Module012_Inputs031;
	Cyclic#1.P3_Pracovisko.COM_Festo.DS3_1_Port0_IN[31] AT %IB."P3_IO_Master".Module012_Inputs032;
	Cyclic#1.P3_Pracovisko.COM_Festo.DS3_1_Port1_IN[0] AT %IB."P3_IO_Master".Module012_Inputs033;
	Cyclic#1.P3_Pracovisko.COM_Festo.DS3_1_Port1_IN[1] AT %IB."P3_IO_Master".Module012_Inputs034;
	Cyclic#1.P3_Pracovisko.COM_Festo.DS3_1_Port1_IN[2] AT %IB."P3_IO_Master".Module012_Inputs035;
	Cyclic#1.P3_Pracovisko.COM_Festo.DS3_1_Port1_IN[3] AT %IB."P3_IO_Master".Module012_Inputs036;
	Cyclic#1.P3_Pracovisko.COM_Festo.DS3_1_Port1_IN[4] AT %IB."P3_IO_Master".Module012_Inputs037;
	Cyclic#1.P3_Pracovisko.COM_Festo.DS3_1_Port1_IN[5] AT %IB."P3_IO_Master".Module012_Inputs038;
	Cyclic#1.P3_Pracovisko.COM_Festo.DS3_1_Port1_IN[6] AT %IB."P3_IO_Master".Module012_Inputs039;
	Cyclic#1.P3_Pracovisko.COM_Festo.DS3_1_Port1_IN[7] AT %IB."P3_IO_Master".Module012_Inputs040;
	Cyclic#1.P3_Pracovisko.COM_Festo.DS3_1_Port1_IN[8] AT %IB."P3_IO_Master".Module012_Inputs041;
	Cyclic#1.P3_Pracovisko.COM_Festo.DS3_1_Port1_IN[9] AT %IB."P3_IO_Master".Module012_Inputs042;
	Cyclic#1.P3_Pracovisko.COM_Festo.DS3_1_Port1_IN[10] AT %IB."P3_IO_Master".Module012_Inputs043;
	Cyclic#1.P3_Pracovisko.COM_Festo.DS3_1_Port1_IN[11] AT %IB."P3_IO_Master".Module012_Inputs044;
	Cyclic#1.P3_Pracovisko.COM_Festo.DS3_1_Port1_IN[12] AT %IB."P3_IO_Master".Module012_Inputs045;
	Cyclic#1.P3_Pracovisko.COM_Festo.DS3_1_Port1_IN[13] AT %IB."P3_IO_Master".Module012_Inputs046;
	Cyclic#1.P3_Pracovisko.COM_Festo.DS3_1_Port1_IN[14] AT %IB."P3_IO_Master".Module012_Inputs047;
	Cyclic#1.P3_Pracovisko.COM_Festo.DS3_1_Port1_IN[15] AT %IB."P3_IO_Master".Module012_Inputs048;
	Cyclic#1.P3_Pracovisko.COM_Festo.DS3_1_Port1_IN[16] AT %IB."P3_IO_Master".Module012_Inputs049;
	Cyclic#1.P3_Pracovisko.COM_Festo.DS3_1_Port1_IN[17] AT %IB."P3_IO_Master".Module012_Inputs050;
	Cyclic#1.P3_Pracovisko.COM_Festo.DS3_1_Port1_IN[18] AT %IB."P3_IO_Master".Module012_Inputs051;
	Cyclic#1.P3_Pracovisko.COM_Festo.DS3_1_Port1_IN[19] AT %IB."P3_IO_Master".Module012_Inputs052;
	Cyclic#1.P3_Pracovisko.COM_Festo.DS3_1_Port1_IN[20] AT %IB."P3_IO_Master".Module012_Inputs053;
	Cyclic#1.P3_Pracovisko.COM_Festo.DS3_1_Port1_IN[21] AT %IB."P3_IO_Master".Module012_Inputs054;
	Cyclic#1.P3_Pracovisko.COM_Festo.DS3_1_Port1_IN[22] AT %IB."P3_IO_Master".Module012_Inputs055;
	Cyclic#1.P3_Pracovisko.COM_Festo.DS3_1_Port1_IN[23] AT %IB."P3_IO_Master".Module012_Inputs056;
	Cyclic#1.P3_Pracovisko.COM_Festo.DS3_1_Port1_IN[24] AT %IB."P3_IO_Master".Module012_Inputs057;
	Cyclic#1.P3_Pracovisko.COM_Festo.DS3_1_Port1_IN[25] AT %IB."P3_IO_Master".Module012_Inputs058;
	Cyclic#1.P3_Pracovisko.COM_Festo.DS3_1_Port1_IN[26] AT %IB."P3_IO_Master".Module012_Inputs059;
	Cyclic#1.P3_Pracovisko.COM_Festo.DS3_1_Port1_IN[27] AT %IB."P3_IO_Master".Module012_Inputs060;
	Cyclic#1.P3_Pracovisko.COM_Festo.DS3_1_Port1_IN[28] AT %IB."P3_IO_Master".Module012_Inputs061;
	Cyclic#1.P3_Pracovisko.COM_Festo.DS3_1_Port1_IN[29] AT %IB."P3_IO_Master".Module012_Inputs062;
	Cyclic#1.P3_Pracovisko.COM_Festo.DS3_1_Port1_IN[30] AT %IB."P3_IO_Master".Module012_Inputs063;
	Cyclic#1.P3_Pracovisko.COM_Festo.DS3_1_Port1_IN[31] AT %IB."P3_IO_Master".Module012_Inputs064;
	Cyclic#1.P3_Pracovisko.COM_Festo.DS3_1_Port2_IN[0] AT %IB."P3_IO_Master".Module012_Inputs065;
	Cyclic#1.P3_Pracovisko.COM_Festo.DS3_1_Port2_IN[1] AT %IB."P3_IO_Master".Module012_Inputs066;
	Cyclic#1.P3_Pracovisko.COM_Festo.DS3_1_Port2_IN[2] AT %IB."P3_IO_Master".Module012_Inputs067;
	Cyclic#1.P3_Pracovisko.COM_Festo.DS3_1_Port2_IN[3] AT %IB."P3_IO_Master".Module012_Inputs068;
	Cyclic#1.P3_Pracovisko.COM_Festo.DS3_1_Port2_IN[4] AT %IB."P3_IO_Master".Module012_Inputs069;
	Cyclic#1.P3_Pracovisko.COM_Festo.DS3_1_Port2_IN[5] AT %IB."P3_IO_Master".Module012_Inputs070;
	Cyclic#1.P3_Pracovisko.COM_Festo.DS3_1_Port2_IN[6] AT %IB."P3_IO_Master".Module012_Inputs071;
	Cyclic#1.P3_Pracovisko.COM_Festo.DS3_1_Port2_IN[7] AT %IB."P3_IO_Master".Module012_Inputs072;
	Cyclic#1.P3_Pracovisko.COM_Festo.DS3_1_Port2_IN[8] AT %IB."P3_IO_Master".Module012_Inputs073;
	Cyclic#1.P3_Pracovisko.COM_Festo.DS3_1_Port2_IN[9] AT %IB."P3_IO_Master".Module012_Inputs074;
	Cyclic#1.P3_Pracovisko.COM_Festo.DS3_1_Port2_IN[10] AT %IB."P3_IO_Master".Module012_Inputs075;
	Cyclic#1.P3_Pracovisko.COM_Festo.DS3_1_Port2_IN[11] AT %IB."P3_IO_Master".Module012_Inputs076;
	Cyclic#1.P3_Pracovisko.COM_Festo.DS3_1_Port2_IN[12] AT %IB."P3_IO_Master".Module012_Inputs077;
	Cyclic#1.P3_Pracovisko.COM_Festo.DS3_1_Port2_IN[13] AT %IB."P3_IO_Master".Module012_Inputs078;
	Cyclic#1.P3_Pracovisko.COM_Festo.DS3_1_Port2_IN[14] AT %IB."P3_IO_Master".Module012_Inputs079;
	Cyclic#1.P3_Pracovisko.COM_Festo.DS3_1_Port2_IN[15] AT %IB."P3_IO_Master".Module012_Inputs080;
	Cyclic#1.P3_Pracovisko.COM_Festo.DS3_1_Port2_IN[16] AT %IB."P3_IO_Master".Module012_Inputs081;
	Cyclic#1.P3_Pracovisko.COM_Festo.DS3_1_Port2_IN[17] AT %IB."P3_IO_Master".Module012_Inputs082;
	Cyclic#1.P3_Pracovisko.COM_Festo.DS3_1_Port2_IN[18] AT %IB."P3_IO_Master".Module012_Inputs083;
	Cyclic#1.P3_Pracovisko.COM_Festo.DS3_1_Port2_IN[19] AT %IB."P3_IO_Master".Module012_Inputs084;
	Cyclic#1.P3_Pracovisko.COM_Festo.DS3_1_Port2_IN[20] AT %IB."P3_IO_Master".Module012_Inputs085;
	Cyclic#1.P3_Pracovisko.COM_Festo.DS3_1_Port2_IN[21] AT %IB."P3_IO_Master".Module012_Inputs086;
	Cyclic#1.P3_Pracovisko.COM_Festo.DS3_1_Port2_IN[22] AT %IB."P3_IO_Master".Module012_Inputs087;
	Cyclic#1.P3_Pracovisko.COM_Festo.DS3_1_Port2_IN[23] AT %IB."P3_IO_Master".Module012_Inputs088;
	Cyclic#1.P3_Pracovisko.COM_Festo.DS3_1_Port2_IN[24] AT %IB."P3_IO_Master".Module012_Inputs089;
	Cyclic#1.P3_Pracovisko.COM_Festo.DS3_1_Port2_IN[25] AT %IB."P3_IO_Master".Module012_Inputs090;
	Cyclic#1.P3_Pracovisko.COM_Festo.DS3_1_Port2_IN[26] AT %IB."P3_IO_Master".Module012_Inputs091;
	Cyclic#1.P3_Pracovisko.COM_Festo.DS3_1_Port2_IN[27] AT %IB."P3_IO_Master".Module012_Inputs092;
	Cyclic#1.P3_Pracovisko.COM_Festo.DS3_1_Port2_IN[28] AT %IB."P3_IO_Master".Module012_Inputs093;
	Cyclic#1.P3_Pracovisko.COM_Festo.DS3_1_Port2_IN[29] AT %IB."P3_IO_Master".Module012_Inputs094;
	Cyclic#1.P3_Pracovisko.COM_Festo.DS3_1_Port2_IN[30] AT %IB."P3_IO_Master".Module012_Inputs095;
	Cyclic#1.P3_Pracovisko.COM_Festo.DS3_1_Port2_IN[31] AT %IB."P3_IO_Master".Module012_Inputs096;
	Cyclic#1.P3_Pracovisko.COM_Festo.DS3_1_Port3_IN[0] AT %IB."P3_IO_Master".Module012_Inputs097;
	Cyclic#1.P3_Pracovisko.COM_Festo.DS3_1_Port3_IN[1] AT %IB."P3_IO_Master".Module012_Inputs098;
	Cyclic#1.P3_Pracovisko.COM_Festo.DS3_1_Port3_IN[2] AT %IB."P3_IO_Master".Module012_Inputs099;
	Cyclic#1.P3_Pracovisko.COM_Festo.DS3_1_Port3_IN[3] AT %IB."P3_IO_Master".Module012_Inputs100;
	Cyclic#1.P3_Pracovisko.COM_Festo.DS3_1_Port3_IN[4] AT %IB."P3_IO_Master".Module012_Inputs101;
	Cyclic#1.P3_Pracovisko.COM_Festo.DS3_1_Port3_IN[5] AT %IB."P3_IO_Master".Module012_Inputs102;
	Cyclic#1.P3_Pracovisko.COM_Festo.DS3_1_Port3_IN[6] AT %IB."P3_IO_Master".Module012_Inputs103;
	Cyclic#1.P3_Pracovisko.COM_Festo.DS3_1_Port3_IN[7] AT %IB."P3_IO_Master".Module012_Inputs104;
	Cyclic#1.P3_Pracovisko.COM_Festo.DS3_1_Port3_IN[8] AT %IB."P3_IO_Master".Module012_Inputs105;
	Cyclic#1.P3_Pracovisko.COM_Festo.DS3_1_Port3_IN[9] AT %IB."P3_IO_Master".Module012_Inputs106;
	Cyclic#1.P3_Pracovisko.COM_Festo.DS3_1_Port3_IN[10] AT %IB."P3_IO_Master".Module012_Inputs107;
	Cyclic#1.P3_Pracovisko.COM_Festo.DS3_1_Port3_IN[11] AT %IB."P3_IO_Master".Module012_Inputs108;
	Cyclic#1.P3_Pracovisko.COM_Festo.DS3_1_Port3_IN[12] AT %IB."P3_IO_Master".Module012_Inputs109;
	Cyclic#1.P3_Pracovisko.COM_Festo.DS3_1_Port3_IN[13] AT %IB."P3_IO_Master".Module012_Inputs110;
	Cyclic#1.P3_Pracovisko.COM_Festo.DS3_1_Port3_IN[14] AT %IB."P3_IO_Master".Module012_Inputs111;
	Cyclic#1.P3_Pracovisko.COM_Festo.DS3_1_Port3_IN[15] AT %IB."P3_IO_Master".Module012_Inputs112;
	Cyclic#1.P3_Pracovisko.COM_Festo.DS3_1_Port3_IN[16] AT %IB."P3_IO_Master".Module012_Inputs113;
	Cyclic#1.P3_Pracovisko.COM_Festo.DS3_1_Port3_IN[17] AT %IB."P3_IO_Master".Module012_Inputs114;
	Cyclic#1.P3_Pracovisko.COM_Festo.DS3_1_Port3_IN[18] AT %IB."P3_IO_Master".Module012_Inputs115;
	Cyclic#1.P3_Pracovisko.COM_Festo.DS3_1_Port3_IN[19] AT %IB."P3_IO_Master".Module012_Inputs116;
	Cyclic#1.P3_Pracovisko.COM_Festo.DS3_1_Port3_IN[20] AT %IB."P3_IO_Master".Module012_Inputs117;
	Cyclic#1.P3_Pracovisko.COM_Festo.DS3_1_Port3_IN[21] AT %IB."P3_IO_Master".Module012_Inputs118;
	Cyclic#1.P3_Pracovisko.COM_Festo.DS3_1_Port3_IN[22] AT %IB."P3_IO_Master".Module012_Inputs119;
	Cyclic#1.P3_Pracovisko.COM_Festo.DS3_1_Port3_IN[23] AT %IB."P3_IO_Master".Module012_Inputs120;
	Cyclic#1.P3_Pracovisko.COM_Festo.DS3_1_Port3_IN[24] AT %IB."P3_IO_Master".Module012_Inputs121;
	Cyclic#1.P3_Pracovisko.COM_Festo.DS3_1_Port3_IN[25] AT %IB."P3_IO_Master".Module012_Inputs122;
	Cyclic#1.P3_Pracovisko.COM_Festo.DS3_1_Port3_IN[26] AT %IB."P3_IO_Master".Module012_Inputs123;
	Cyclic#1.P3_Pracovisko.COM_Festo.DS3_1_Port3_IN[27] AT %IB."P3_IO_Master".Module012_Inputs124;
	Cyclic#1.P3_Pracovisko.COM_Festo.DS3_1_Port3_IN[28] AT %IB."P3_IO_Master".Module012_Inputs125;
	Cyclic#1.P3_Pracovisko.COM_Festo.DS3_1_Port3_IN[29] AT %IB."P3_IO_Master".Module012_Inputs126;
	Cyclic#1.P3_Pracovisko.COM_Festo.DS3_1_Port3_IN[30] AT %IB."P3_IO_Master".Module012_Inputs127;
	Cyclic#1.P3_Pracovisko.COM_Festo.DS3_1_Port3_IN[31] AT %IB."P3_IO_Master".Module012_Inputs128;
	Cyclic#1.P3_Pracovisko.COM_Festo.DS3_1_Port0_OUT[0] AT %QB."P3_IO_Master".Module012_Outputs001;
	Cyclic#1.P3_Pracovisko.COM_Festo.DS3_1_Port0_OUT[1] AT %QB."P3_IO_Master".Module012_Outputs002;
	Cyclic#1.P3_Pracovisko.COM_Festo.DS3_1_Port0_OUT[2] AT %QB."P3_IO_Master".Module012_Outputs003;
	Cyclic#1.P3_Pracovisko.COM_Festo.DS3_1_Port0_OUT[3] AT %QB."P3_IO_Master".Module012_Outputs004;
	Cyclic#1.P3_Pracovisko.COM_Festo.DS3_1_Port0_OUT[4] AT %QB."P3_IO_Master".Module012_Outputs005;
	Cyclic#1.P3_Pracovisko.COM_Festo.DS3_1_Port0_OUT[5] AT %QB."P3_IO_Master".Module012_Outputs006;
	Cyclic#1.P3_Pracovisko.COM_Festo.DS3_1_Port0_OUT[6] AT %QB."P3_IO_Master".Module012_Outputs007;
	Cyclic#1.P3_Pracovisko.COM_Festo.DS3_1_Port0_OUT[7] AT %QB."P3_IO_Master".Module012_Outputs008;
	Cyclic#1.P3_Pracovisko.COM_Festo.DS3_1_Port0_OUT[8] AT %QB."P3_IO_Master".Module012_Outputs009;
	Cyclic#1.P3_Pracovisko.COM_Festo.DS3_1_Port0_OUT[9] AT %QB."P3_IO_Master".Module012_Outputs010;
	Cyclic#1.P3_Pracovisko.COM_Festo.DS3_1_Port0_OUT[10] AT %QB."P3_IO_Master".Module012_Outputs011;
	Cyclic#1.P3_Pracovisko.COM_Festo.DS3_1_Port0_OUT[11] AT %QB."P3_IO_Master".Module012_Outputs012;
	Cyclic#1.P3_Pracovisko.COM_Festo.DS3_1_Port0_OUT[12] AT %QB."P3_IO_Master".Module012_Outputs013;
	Cyclic#1.P3_Pracovisko.COM_Festo.DS3_1_Port0_OUT[13] AT %QB."P3_IO_Master".Module012_Outputs014;
	Cyclic#1.P3_Pracovisko.COM_Festo.DS3_1_Port0_OUT[14] AT %QB."P3_IO_Master".Module012_Outputs015;
	Cyclic#1.P3_Pracovisko.COM_Festo.DS3_1_Port0_OUT[15] AT %QB."P3_IO_Master".Module012_Outputs016;
	Cyclic#1.P3_Pracovisko.COM_Festo.DS3_1_Port0_OUT[16] AT %QB."P3_IO_Master".Module012_Outputs017;
	Cyclic#1.P3_Pracovisko.COM_Festo.DS3_1_Port0_OUT[17] AT %QB."P3_IO_Master".Module012_Outputs018;
	Cyclic#1.P3_Pracovisko.COM_Festo.DS3_1_Port0_OUT[18] AT %QB."P3_IO_Master".Module012_Outputs019;
	Cyclic#1.P3_Pracovisko.COM_Festo.DS3_1_Port0_OUT[19] AT %QB."P3_IO_Master".Module012_Outputs020;
	Cyclic#1.P3_Pracovisko.COM_Festo.DS3_1_Port0_OUT[20] AT %QB."P3_IO_Master".Module012_Outputs021;
	Cyclic#1.P3_Pracovisko.COM_Festo.DS3_1_Port0_OUT[21] AT %QB."P3_IO_Master".Module012_Outputs022;
	Cyclic#1.P3_Pracovisko.COM_Festo.DS3_1_Port0_OUT[22] AT %QB."P3_IO_Master".Module012_Outputs023;
	Cyclic#1.P3_Pracovisko.COM_Festo.DS3_1_Port0_OUT[23] AT %QB."P3_IO_Master".Module012_Outputs024;
	Cyclic#1.P3_Pracovisko.COM_Festo.DS3_1_Port0_OUT[24] AT %QB."P3_IO_Master".Module012_Outputs025;
	Cyclic#1.P3_Pracovisko.COM_Festo.DS3_1_Port0_OUT[25] AT %QB."P3_IO_Master".Module012_Outputs026;
	Cyclic#1.P3_Pracovisko.COM_Festo.DS3_1_Port0_OUT[26] AT %QB."P3_IO_Master".Module012_Outputs027;
	Cyclic#1.P3_Pracovisko.COM_Festo.DS3_1_Port0_OUT[27] AT %QB."P3_IO_Master".Module012_Outputs028;
	Cyclic#1.P3_Pracovisko.COM_Festo.DS3_1_Port0_OUT[28] AT %QB."P3_IO_Master".Module012_Outputs029;
	Cyclic#1.P3_Pracovisko.COM_Festo.DS3_1_Port0_OUT[29] AT %QB."P3_IO_Master".Module012_Outputs030;
	Cyclic#1.P3_Pracovisko.COM_Festo.DS3_1_Port0_OUT[30] AT %QB."P3_IO_Master".Module012_Outputs031;
	Cyclic#1.P3_Pracovisko.COM_Festo.DS3_1_Port0_OUT[31] AT %QB."P3_IO_Master".Module012_Outputs032;
	Cyclic#1.P3_Pracovisko.COM_Festo.DS3_1_Port1_OUT[0] AT %QB."P3_IO_Master".Module012_Outputs033;
	Cyclic#1.P3_Pracovisko.COM_Festo.DS3_1_Port1_OUT[1] AT %QB."P3_IO_Master".Module012_Outputs034;
	Cyclic#1.P3_Pracovisko.COM_Festo.DS3_1_Port1_OUT[2] AT %QB."P3_IO_Master".Module012_Outputs035;
	Cyclic#1.P3_Pracovisko.COM_Festo.DS3_1_Port1_OUT[3] AT %QB."P3_IO_Master".Module012_Outputs036;
	Cyclic#1.P3_Pracovisko.COM_Festo.DS3_1_Port1_OUT[4] AT %QB."P3_IO_Master".Module012_Outputs037;
	Cyclic#1.P3_Pracovisko.COM_Festo.DS3_1_Port1_OUT[5] AT %QB."P3_IO_Master".Module012_Outputs038;
	Cyclic#1.P3_Pracovisko.COM_Festo.DS3_1_Port1_OUT[6] AT %QB."P3_IO_Master".Module012_Outputs039;
	Cyclic#1.P3_Pracovisko.COM_Festo.DS3_1_Port1_OUT[7] AT %QB."P3_IO_Master".Module012_Outputs040;
	Cyclic#1.P3_Pracovisko.COM_Festo.DS3_1_Port1_OUT[8] AT %QB."P3_IO_Master".Module012_Outputs041;
	Cyclic#1.P3_Pracovisko.COM_Festo.DS3_1_Port1_OUT[9] AT %QB."P3_IO_Master".Module012_Outputs042;
	Cyclic#1.P3_Pracovisko.COM_Festo.DS3_1_Port1_OUT[10] AT %QB."P3_IO_Master".Module012_Outputs043;
	Cyclic#1.P3_Pracovisko.COM_Festo.DS3_1_Port1_OUT[11] AT %QB."P3_IO_Master".Module012_Outputs044;
	Cyclic#1.P3_Pracovisko.COM_Festo.DS3_1_Port1_OUT[12] AT %QB."P3_IO_Master".Module012_Outputs045;
	Cyclic#1.P3_Pracovisko.COM_Festo.DS3_1_Port1_OUT[13] AT %QB."P3_IO_Master".Module012_Outputs046;
	Cyclic#1.P3_Pracovisko.COM_Festo.DS3_1_Port1_OUT[14] AT %QB."P3_IO_Master".Module012_Outputs047;
	Cyclic#1.P3_Pracovisko.COM_Festo.DS3_1_Port1_OUT[15] AT %QB."P3_IO_Master".Module012_Outputs048;
	Cyclic#1.P3_Pracovisko.COM_Festo.DS3_1_Port1_OUT[16] AT %QB."P3_IO_Master".Module012_Outputs049;
	Cyclic#1.P3_Pracovisko.COM_Festo.DS3_1_Port1_OUT[17] AT %QB."P3_IO_Master".Module012_Outputs050;
	Cyclic#1.P3_Pracovisko.COM_Festo.DS3_1_Port1_OUT[18] AT %QB."P3_IO_Master".Module012_Outputs051;
	Cyclic#1.P3_Pracovisko.COM_Festo.DS3_1_Port1_OUT[19] AT %QB."P3_IO_Master".Module012_Outputs052;
	Cyclic#1.P3_Pracovisko.COM_Festo.DS3_1_Port1_OUT[20] AT %QB."P3_IO_Master".Module012_Outputs053;
	Cyclic#1.P3_Pracovisko.COM_Festo.DS3_1_Port1_OUT[21] AT %QB."P3_IO_Master".Module012_Outputs054;
	Cyclic#1.P3_Pracovisko.COM_Festo.DS3_1_Port1_OUT[22] AT %QB."P3_IO_Master".Module012_Outputs055;
	Cyclic#1.P3_Pracovisko.COM_Festo.DS3_1_Port1_OUT[23] AT %QB."P3_IO_Master".Module012_Outputs056;
	Cyclic#1.P3_Pracovisko.COM_Festo.DS3_1_Port1_OUT[24] AT %QB."P3_IO_Master".Module012_Outputs057;
	Cyclic#1.P3_Pracovisko.COM_Festo.DS3_1_Port1_OUT[25] AT %QB."P3_IO_Master".Module012_Outputs058;
	Cyclic#1.P3_Pracovisko.COM_Festo.DS3_1_Port1_OUT[26] AT %QB."P3_IO_Master".Module012_Outputs059;
	Cyclic#1.P3_Pracovisko.COM_Festo.DS3_1_Port1_OUT[27] AT %QB."P3_IO_Master".Module012_Outputs060;
	Cyclic#1.P3_Pracovisko.COM_Festo.DS3_1_Port1_OUT[28] AT %QB."P3_IO_Master".Module012_Outputs061;
	Cyclic#1.P3_Pracovisko.COM_Festo.DS3_1_Port1_OUT[29] AT %QB."P3_IO_Master".Module012_Outputs062;
	Cyclic#1.P3_Pracovisko.COM_Festo.DS3_1_Port1_OUT[30] AT %QB."P3_IO_Master".Module012_Outputs063;
	Cyclic#1.P3_Pracovisko.COM_Festo.DS3_1_Port1_OUT[31] AT %QB."P3_IO_Master".Module012_Outputs064;
	Cyclic#1.P3_Pracovisko.COM_Festo.DS3_1_Port2_OUT[0] AT %QB."P3_IO_Master".Module012_Outputs065;
	Cyclic#1.P3_Pracovisko.COM_Festo.DS3_1_Port2_OUT[1] AT %QB."P3_IO_Master".Module012_Outputs066;
	Cyclic#1.P3_Pracovisko.COM_Festo.DS3_1_Port2_OUT[2] AT %QB."P3_IO_Master".Module012_Outputs067;
	Cyclic#1.P3_Pracovisko.COM_Festo.DS3_1_Port2_OUT[3] AT %QB."P3_IO_Master".Module012_Outputs068;
	Cyclic#1.P3_Pracovisko.COM_Festo.DS3_1_Port2_OUT[4] AT %QB."P3_IO_Master".Module012_Outputs069;
	Cyclic#1.P3_Pracovisko.COM_Festo.DS3_1_Port2_OUT[5] AT %QB."P3_IO_Master".Module012_Outputs070;
	Cyclic#1.P3_Pracovisko.COM_Festo.DS3_1_Port2_OUT[6] AT %QB."P3_IO_Master".Module012_Outputs071;
	Cyclic#1.P3_Pracovisko.COM_Festo.DS3_1_Port2_OUT[7] AT %QB."P3_IO_Master".Module012_Outputs072;
	Cyclic#1.P3_Pracovisko.COM_Festo.DS3_1_Port2_OUT[8] AT %QB."P3_IO_Master".Module012_Outputs073;
	Cyclic#1.P3_Pracovisko.COM_Festo.DS3_1_Port2_OUT[9] AT %QB."P3_IO_Master".Module012_Outputs074;
	Cyclic#1.P3_Pracovisko.COM_Festo.DS3_1_Port2_OUT[10] AT %QB."P3_IO_Master".Module012_Outputs075;
	Cyclic#1.P3_Pracovisko.COM_Festo.DS3_1_Port2_OUT[11] AT %QB."P3_IO_Master".Module012_Outputs076;
	Cyclic#1.P3_Pracovisko.COM_Festo.DS3_1_Port2_OUT[12] AT %QB."P3_IO_Master".Module012_Outputs077;
	Cyclic#1.P3_Pracovisko.COM_Festo.DS3_1_Port2_OUT[13] AT %QB."P3_IO_Master".Module012_Outputs078;
	Cyclic#1.P3_Pracovisko.COM_Festo.DS3_1_Port2_OUT[14] AT %QB."P3_IO_Master".Module012_Outputs079;
	Cyclic#1.P3_Pracovisko.COM_Festo.DS3_1_Port2_OUT[15] AT %QB."P3_IO_Master".Module012_Outputs080;
	Cyclic#1.P3_Pracovisko.COM_Festo.DS3_1_Port2_OUT[16] AT %QB."P3_IO_Master".Module012_Outputs081;
	Cyclic#1.P3_Pracovisko.COM_Festo.DS3_1_Port2_OUT[17] AT %QB."P3_IO_Master".Module012_Outputs082;
	Cyclic#1.P3_Pracovisko.COM_Festo.DS3_1_Port2_OUT[18] AT %QB."P3_IO_Master".Module012_Outputs083;
	Cyclic#1.P3_Pracovisko.COM_Festo.DS3_1_Port2_OUT[19] AT %QB."P3_IO_Master".Module012_Outputs084;
	Cyclic#1.P3_Pracovisko.COM_Festo.DS3_1_Port2_OUT[20] AT %QB."P3_IO_Master".Module012_Outputs085;
	Cyclic#1.P3_Pracovisko.COM_Festo.DS3_1_Port2_OUT[21] AT %QB."P3_IO_Master".Module012_Outputs086;
	Cyclic#1.P3_Pracovisko.COM_Festo.DS3_1_Port2_OUT[22] AT %QB."P3_IO_Master".Module012_Outputs087;
	Cyclic#1.P3_Pracovisko.COM_Festo.DS3_1_Port2_OUT[23] AT %QB."P3_IO_Master".Module012_Outputs088;
	Cyclic#1.P3_Pracovisko.COM_Festo.DS3_1_Port2_OUT[24] AT %QB."P3_IO_Master".Module012_Outputs089;
	Cyclic#1.P3_Pracovisko.COM_Festo.DS3_1_Port2_OUT[25] AT %QB."P3_IO_Master".Module012_Outputs090;
	Cyclic#1.P3_Pracovisko.COM_Festo.DS3_1_Port2_OUT[26] AT %QB."P3_IO_Master".Module012_Outputs091;
	Cyclic#1.P3_Pracovisko.COM_Festo.DS3_1_Port2_OUT[27] AT %QB."P3_IO_Master".Module012_Outputs092;
	Cyclic#1.P3_Pracovisko.COM_Festo.DS3_1_Port2_OUT[28] AT %QB."P3_IO_Master".Module012_Outputs093;
	Cyclic#1.P3_Pracovisko.COM_Festo.DS3_1_Port2_OUT[29] AT %QB."P3_IO_Master".Module012_Outputs094;
	Cyclic#1.P3_Pracovisko.COM_Festo.DS3_1_Port2_OUT[30] AT %QB."P3_IO_Master".Module012_Outputs095;
	Cyclic#1.P3_Pracovisko.COM_Festo.DS3_1_Port2_OUT[31] AT %QB."P3_IO_Master".Module012_Outputs096;
	Cyclic#1.P3_Pracovisko.COM_Festo.DS3_1_Port3_OUT[0] AT %QB."P3_IO_Master".Module012_Outputs097;
	Cyclic#1.P3_Pracovisko.COM_Festo.DS3_1_Port3_OUT[1] AT %QB."P3_IO_Master".Module012_Outputs098;
	Cyclic#1.P3_Pracovisko.COM_Festo.DS3_1_Port3_OUT[2] AT %QB."P3_IO_Master".Module012_Outputs099;
	Cyclic#1.P3_Pracovisko.COM_Festo.DS3_1_Port3_OUT[3] AT %QB."P3_IO_Master".Module012_Outputs100;
	Cyclic#1.P3_Pracovisko.COM_Festo.DS3_1_Port3_OUT[4] AT %QB."P3_IO_Master".Module012_Outputs101;
	Cyclic#1.P3_Pracovisko.COM_Festo.DS3_1_Port3_OUT[5] AT %QB."P3_IO_Master".Module012_Outputs102;
	Cyclic#1.P3_Pracovisko.COM_Festo.DS3_1_Port3_OUT[6] AT %QB."P3_IO_Master".Module012_Outputs103;
	Cyclic#1.P3_Pracovisko.COM_Festo.DS3_1_Port3_OUT[7] AT %QB."P3_IO_Master".Module012_Outputs104;
	Cyclic#1.P3_Pracovisko.COM_Festo.DS3_1_Port3_OUT[8] AT %QB."P3_IO_Master".Module012_Outputs105;
	Cyclic#1.P3_Pracovisko.COM_Festo.DS3_1_Port3_OUT[9] AT %QB."P3_IO_Master".Module012_Outputs106;
	Cyclic#1.P3_Pracovisko.COM_Festo.DS3_1_Port3_OUT[10] AT %QB."P3_IO_Master".Module012_Outputs107;
	Cyclic#1.P3_Pracovisko.COM_Festo.DS3_1_Port3_OUT[11] AT %QB."P3_IO_Master".Module012_Outputs108;
	Cyclic#1.P3_Pracovisko.COM_Festo.DS3_1_Port3_OUT[12] AT %QB."P3_IO_Master".Module012_Outputs109;
	Cyclic#1.P3_Pracovisko.COM_Festo.DS3_1_Port3_OUT[13] AT %QB."P3_IO_Master".Module012_Outputs110;
	Cyclic#1.P3_Pracovisko.COM_Festo.DS3_1_Port3_OUT[14] AT %QB."P3_IO_Master".Module012_Outputs111;
	Cyclic#1.P3_Pracovisko.COM_Festo.DS3_1_Port3_OUT[15] AT %QB."P3_IO_Master".Module012_Outputs112;
	Cyclic#1.P3_Pracovisko.COM_Festo.DS3_1_Port3_OUT[16] AT %QB."P3_IO_Master".Module012_Outputs113;
	Cyclic#1.P3_Pracovisko.COM_Festo.DS3_1_Port3_OUT[17] AT %QB."P3_IO_Master".Module012_Outputs114;
	Cyclic#1.P3_Pracovisko.COM_Festo.DS3_1_Port3_OUT[18] AT %QB."P3_IO_Master".Module012_Outputs115;
	Cyclic#1.P3_Pracovisko.COM_Festo.DS3_1_Port3_OUT[19] AT %QB."P3_IO_Master".Module012_Outputs116;
	Cyclic#1.P3_Pracovisko.COM_Festo.DS3_1_Port3_OUT[20] AT %QB."P3_IO_Master".Module012_Outputs117;
	Cyclic#1.P3_Pracovisko.COM_Festo.DS3_1_Port3_OUT[21] AT %QB."P3_IO_Master".Module012_Outputs118;
	Cyclic#1.P3_Pracovisko.COM_Festo.DS3_1_Port3_OUT[22] AT %QB."P3_IO_Master".Module012_Outputs119;
	Cyclic#1.P3_Pracovisko.COM_Festo.DS3_1_Port3_OUT[23] AT %QB."P3_IO_Master".Module012_Outputs120;
	Cyclic#1.P3_Pracovisko.COM_Festo.DS3_1_Port3_OUT[24] AT %QB."P3_IO_Master".Module012_Outputs121;
	Cyclic#1.P3_Pracovisko.COM_Festo.DS3_1_Port3_OUT[25] AT %QB."P3_IO_Master".Module012_Outputs122;
	Cyclic#1.P3_Pracovisko.COM_Festo.DS3_1_Port3_OUT[26] AT %QB."P3_IO_Master".Module012_Outputs123;
	Cyclic#1.P3_Pracovisko.COM_Festo.DS3_1_Port3_OUT[27] AT %QB."P3_IO_Master".Module012_Outputs124;
	Cyclic#1.P3_Pracovisko.COM_Festo.DS3_1_Port3_OUT[28] AT %QB."P3_IO_Master".Module012_Outputs125;
	Cyclic#1.P3_Pracovisko.COM_Festo.DS3_1_Port3_OUT[29] AT %QB."P3_IO_Master".Module012_Outputs126;
	Cyclic#1.P3_Pracovisko.COM_Festo.DS3_1_Port3_OUT[30] AT %QB."P3_IO_Master".Module012_Outputs127;
	Cyclic#1.P3_Pracovisko.COM_Festo.DS3_1_Port3_OUT[31] AT %QB."P3_IO_Master".Module012_Outputs128;
	Cyclic#1.P3_Pracovisko.COM_Festo.DS3_2_Port0_IN[0] AT %IB."P3_IO_Master".Module013_Inputs001;
	Cyclic#1.P3_Pracovisko.COM_Festo.DS3_2_Port0_IN[1] AT %IB."P3_IO_Master".Module013_Inputs002;
	Cyclic#1.P3_Pracovisko.COM_Festo.DS3_2_Port1_IN[0] AT %IB."P3_IO_Master".Module013_Inputs003;
	Cyclic#1.P3_Pracovisko.COM_Festo.DS3_2_Port1_IN[1] AT %IB."P3_IO_Master".Module013_Inputs004;
	Cyclic#1.P3_Pracovisko.COM_Festo.DS3_2_Port2_IN[0] AT %IB."P3_IO_Master".Module013_Inputs005;
	Cyclic#1.P3_Pracovisko.COM_Festo.DS3_2_Port2_IN[1] AT %IB."P3_IO_Master".Module013_Inputs006;
	Cyclic#1.P3_Pracovisko.COM_Festo.DS3_2_Port0_OUT[0] AT %QB."P3_IO_Master".Module013_Outputs001;
	Cyclic#1.P3_Pracovisko.COM_Festo.DS3_2_Port0_OUT[1] AT %QB."P3_IO_Master".Module013_Outputs002;
	Cyclic#1.P3_Pracovisko.COM_Festo.DS3_2_Port1_OUT[0] AT %QB."P3_IO_Master".Module013_Outputs003;
	Cyclic#1.P3_Pracovisko.COM_Festo.DS3_2_Port1_OUT[1] AT %QB."P3_IO_Master".Module013_Outputs004;
	Cyclic#1.P3_Pracovisko.COM_Festo.DS3_2_Port2_OUT[0] AT %QB."P3_IO_Master".Module013_Outputs005;
	Cyclic#1.P3_Pracovisko.COM_Festo.DS3_2_Port2_OUT[1] AT %QB."P3_IO_Master".Module013_Outputs006;
	Cyclic#1.P3_Pracovisko.IN.Kamery_ControlUnit_KomOK AT %IX."WenglorControl_Unit".ModuleOk;
	Cyclic#1.ControlUnit.Profinet_PLC_INPUTS[0] AT %IB."WenglorControl_Unit".Module001_Inputs001;
	Cyclic#1.ControlUnit.Profinet_PLC_INPUTS[1] AT %IB."WenglorControl_Unit".Module001_Inputs002;
	Cyclic#1.CAM2.Profinet_PLC_INPUTS[0] AT %IB."WenglorControl_Unit".Module002_Inputs001;
	Cyclic#1.CAM2.Profinet_PLC_INPUTS[1] AT %IB."WenglorControl_Unit".Module002_Inputs002;
	Cyclic#1.CAM2.Profinet_PLC_INPUTS[2] AT %IB."WenglorControl_Unit".Module002_Inputs003;
	Cyclic#1.CAM2.Profinet_PLC_INPUTS[3] AT %IB."WenglorControl_Unit".Module002_Inputs004;
	Cyclic#1.CAM2.Profinet_PLC_INPUTS[4] AT %IB."WenglorControl_Unit".Module002_Inputs005;
	Cyclic#1.CAM4.Profinet_PLC_INPUTS[0] AT %IB."WenglorControl_Unit".Module004_Inputs001;
	Cyclic#1.CAM4.Profinet_PLC_INPUTS[1] AT %IB."WenglorControl_Unit".Module004_Inputs002;
	Cyclic#1.CAM4.Profinet_PLC_INPUTS[2] AT %IB."WenglorControl_Unit".Module004_Inputs003;
	Cyclic#1.CAM4.Profinet_PLC_INPUTS[3] AT %IB."WenglorControl_Unit".Module004_Inputs004;
	Cyclic#1.CAM6.Profinet_PLC_INPUTS[0] AT %IB."WenglorControl_Unit".Module006_Inputs001;
	Cyclic#1.CAM6.Profinet_PLC_INPUTS[1] AT %IB."WenglorControl_Unit".Module006_Inputs002;
	Cyclic#1.CAM6.Profinet_PLC_INPUTS[2] AT %IB."WenglorControl_Unit".Module006_Inputs003;
	Cyclic#1.CAM6.Profinet_PLC_INPUTS[3] AT %IB."WenglorControl_Unit".Module006_Inputs004;
	Cyclic#1.CAM6.Profinet_PLC_INPUTS[4] AT %IB."WenglorControl_Unit".Module006_Inputs005;
	Cyclic#1.CAM6.Profinet_PLC_INPUTS[5] AT %IB."WenglorControl_Unit".Module006_Inputs006;
	Cyclic#1.CAM1.Profinet_PLC_INPUTS[0] AT %IB."WenglorControl_Unit".Module008_Inputs001;
	Cyclic#1.CAM1.Profinet_PLC_INPUTS[1] AT %IB."WenglorControl_Unit".Module008_Inputs002;
	Cyclic#1.CAM1.Profinet_PLC_INPUTS[2] AT %IB."WenglorControl_Unit".Module008_Inputs003;
	Cyclic#1.CAM1.Profinet_PLC_INPUTS[3] AT %IB."WenglorControl_Unit".Module008_Inputs004;
	Cyclic#1.CAM7.Profinet_QRkod_Znaky[0] AT %IB."WenglorControl_Unit".Module011_Inputs001;
	Cyclic#1.CAM7.Profinet_QRkod_Znaky[1] AT %IB."WenglorControl_Unit".Module011_Inputs002;
	Cyclic#1.CAM7.Profinet_QRkod_Znaky[2] AT %IB."WenglorControl_Unit".Module011_Inputs003;
	Cyclic#1.CAM7.Profinet_QRkod_Znaky[3] AT %IB."WenglorControl_Unit".Module011_Inputs004;
	Cyclic#1.CAM7.Profinet_QRkod_Znaky[4] AT %IB."WenglorControl_Unit".Module011_Inputs005;
	Cyclic#1.CAM7.Profinet_QRkod_Znaky[5] AT %IB."WenglorControl_Unit".Module011_Inputs006;
	Cyclic#1.CAM17.Profinet_PLC_INPUTS[0] AT %IB."WenglorControl_Unit".Module012_Inputs001;
	Cyclic#1.CAM17.Profinet_PLC_INPUTS[1] AT %IB."WenglorControl_Unit".Module012_Inputs002;
	Cyclic#1.CAM17.Profinet_PLC_INPUTS[2] AT %IB."WenglorControl_Unit".Module012_Inputs003;
	Cyclic#1.CAM17.Profinet_PLC_INPUTS[3] AT %IB."WenglorControl_Unit".Module012_Inputs004;
	Cyclic#1.CAM7.Profinet_QRkod_Znaky[6] AT %IB."WenglorControl_Unit".Module011_Inputs007;
	Cyclic#1.CAM7.Profinet_QRkod_Znaky[7] AT %IB."WenglorControl_Unit".Module011_Inputs008;
	Cyclic#1.CAM7.Profinet_QRkod_Znaky[8] AT %IB."WenglorControl_Unit".Module011_Inputs009;
	Cyclic#1.CAM7.Profinet_QRkod_Znaky[9] AT %IB."WenglorControl_Unit".Module011_Inputs010;
	Cyclic#1.CAM7.Profinet_QRkod_Znaky[10] AT %IB."WenglorControl_Unit".Module011_Inputs011;
	Cyclic#1.CAM7.Profinet_QRkod_Znaky[11] AT %IB."WenglorControl_Unit".Module011_Inputs012;
	Cyclic#1.CAM7.Profinet_QRkod_Znaky[12] AT %IB."WenglorControl_Unit".Module011_Inputs013;
	Cyclic#1.CAM7.Profinet_QRkod_Znaky[13] AT %IB."WenglorControl_Unit".Module011_Inputs014;
	Cyclic#1.CAM7.Profinet_QRkod_Znaky[14] AT %IB."WenglorControl_Unit".Module011_Inputs015;
	Cyclic#1.CAM7.Profinet_QRkod_Znaky[15] AT %IB."WenglorControl_Unit".Module011_Inputs016;
	Cyclic#1.CAM7.Profinet_QRkod_Znaky[16] AT %IB."WenglorControl_Unit".Module011_Inputs017;
	Cyclic#1.CAM7.Profinet_QRkod_Znaky[17] AT %IB."WenglorControl_Unit".Module011_Inputs018;
	Cyclic#1.CAM7.Profinet_QRkod_Znaky[18] AT %IB."WenglorControl_Unit".Module011_Inputs019;
	Cyclic#1.CAM7.Profinet_QRkod_Znaky[19] AT %IB."WenglorControl_Unit".Module011_Inputs020;
	Cyclic#1.CAM7.Profinet_QRkod_Znaky[20] AT %IB."WenglorControl_Unit".Module011_Inputs021;
	Cyclic#1.CAM7.Profinet_QRkod_Znaky[21] AT %IB."WenglorControl_Unit".Module011_Inputs022;
	Cyclic#1.CAM7.Profinet_QRkod_Znaky[22] AT %IB."WenglorControl_Unit".Module011_Inputs023;
	Cyclic#1.CAM7.Profinet_QRkod_Znaky[23] AT %IB."WenglorControl_Unit".Module011_Inputs024;
	Cyclic#1.CAM7.Profinet_QRkod_Znaky[24] AT %IB."WenglorControl_Unit".Module011_Inputs025;
	Cyclic#1.CAM7.Profinet_QRkod_Znaky[25] AT %IB."WenglorControl_Unit".Module011_Inputs026;
	Cyclic#1.CAM7.Profinet_QRkod_Znaky[26] AT %IB."WenglorControl_Unit".Module011_Inputs027;
	Cyclic#1.CAM7.Profinet_QRkod_Znaky[27] AT %IB."WenglorControl_Unit".Module011_Inputs028;
	Cyclic#1.CAM7.Profinet_QRkod_Znaky[28] AT %IB."WenglorControl_Unit".Module011_Inputs029;
	Cyclic#1.CAM7.Profinet_QRkod_Znaky[29] AT %IB."WenglorControl_Unit".Module011_Inputs030;
	Cyclic#1.CAM7.Profinet_QRkod_Znaky[30] AT %IB."WenglorControl_Unit".Module011_Inputs031;
	Cyclic#1.CAM7.Profinet_QRkod_Znaky[31] AT %IB."WenglorControl_Unit".Module011_Inputs032;
	Cyclic#1.CAM10.Profinet_PLC_INPUTS[0] AT %IB."WenglorControl_Unit".Module015_Inputs001;
	Cyclic#1.CAM10.Profinet_PLC_INPUTS[1] AT %IB."WenglorControl_Unit".Module015_Inputs002;
	Cyclic#1.CAM10.Profinet_PLC_INPUTS[2] AT %IB."WenglorControl_Unit".Module015_Inputs003;
	Cyclic#1.CAM10.Profinet_PLC_INPUTS[3] AT %IB."WenglorControl_Unit".Module015_Inputs004;
	Cyclic#1.CAM11.Profinet_PLC_INPUTS[0] AT %IB."WenglorControl_Unit".Module017_Inputs001;
	Cyclic#1.CAM11.Profinet_PLC_INPUTS[1] AT %IB."WenglorControl_Unit".Module017_Inputs002;
	Cyclic#1.CAM11.Profinet_PLC_INPUTS[2] AT %IB."WenglorControl_Unit".Module017_Inputs003;
	Cyclic#1.CAM11.Profinet_PLC_INPUTS[3] AT %IB."WenglorControl_Unit".Module017_Inputs004;
	Cyclic#1.CAM12.Profinet_PLC_INPUTS[0] AT %IB."WenglorControl_Unit".Module019_Inputs001;
	Cyclic#1.CAM12.Profinet_PLC_INPUTS[1] AT %IB."WenglorControl_Unit".Module019_Inputs002;
	Cyclic#1.CAM12.Profinet_PLC_INPUTS[2] AT %IB."WenglorControl_Unit".Module019_Inputs003;
	Cyclic#1.CAM12.Profinet_PLC_INPUTS[3] AT %IB."WenglorControl_Unit".Module019_Inputs004;
	Cyclic#1.CAM15.Profinet_PLC_INPUTS[0] AT %IB."WenglorControl_Unit".Module021_Inputs001;
	Cyclic#1.CAM15.Profinet_PLC_INPUTS[1] AT %IB."WenglorControl_Unit".Module021_Inputs002;
	Cyclic#1.CAM15.Profinet_PLC_INPUTS[2] AT %IB."WenglorControl_Unit".Module021_Inputs003;
	Cyclic#1.CAM15.Profinet_PLC_INPUTS[3] AT %IB."WenglorControl_Unit".Module021_Inputs004;
	Cyclic#1.CAM16.Profinet_PLC_INPUTS[0] AT %IB."WenglorControl_Unit".Module023_Inputs001;
	Cyclic#1.CAM16.Profinet_PLC_INPUTS[1] AT %IB."WenglorControl_Unit".Module023_Inputs002;
	Cyclic#1.CAM16.Profinet_PLC_INPUTS[2] AT %IB."WenglorControl_Unit".Module023_Inputs003;
	Cyclic#1.CAM16.Profinet_PLC_INPUTS[3] AT %IB."WenglorControl_Unit".Module023_Inputs004;
	Cyclic#1.CAM15.Profinet_QRkod_Znaky[0] AT %IB."WenglorControl_Unit".Module021_Inputs033;
	Cyclic#1.CAM15.Profinet_QRkod_Znaky[1] AT %IB."WenglorControl_Unit".Module021_Inputs034;
	Cyclic#1.CAM15.Profinet_QRkod_Znaky[2] AT %IB."WenglorControl_Unit".Module021_Inputs035;
	Cyclic#1.CAM15.Profinet_QRkod_Znaky[3] AT %IB."WenglorControl_Unit".Module021_Inputs036;
	Cyclic#1.CAM15.Profinet_QRkod_Znaky[4] AT %IB."WenglorControl_Unit".Module021_Inputs037;
	Cyclic#1.CAM15.Profinet_QRkod_Znaky[5] AT %IB."WenglorControl_Unit".Module021_Inputs038;
	Cyclic#1.CAM15.Profinet_QRkod_Znaky[6] AT %IB."WenglorControl_Unit".Module021_Inputs039;
	Cyclic#1.CAM15.Profinet_QRkod_Znaky[7] AT %IB."WenglorControl_Unit".Module021_Inputs040;
	Cyclic#1.CAM15.Profinet_QRkod_Znaky[8] AT %IB."WenglorControl_Unit".Module021_Inputs041;
	Cyclic#1.CAM15.Profinet_QRkod_Znaky[9] AT %IB."WenglorControl_Unit".Module021_Inputs042;
	Cyclic#1.CAM15.Profinet_QRkod_Znaky[10] AT %IB."WenglorControl_Unit".Module021_Inputs043;
	Cyclic#1.CAM15.Profinet_QRkod_Znaky[11] AT %IB."WenglorControl_Unit".Module021_Inputs044;
	Cyclic#1.CAM15.Profinet_QRkod_Znaky[12] AT %IB."WenglorControl_Unit".Module021_Inputs045;
	Cyclic#1.CAM15.Profinet_QRkod_Znaky[13] AT %IB."WenglorControl_Unit".Module021_Inputs046;
	Cyclic#1.CAM15.Profinet_QRkod_Znaky[14] AT %IB."WenglorControl_Unit".Module021_Inputs047;
	Cyclic#1.CAM15.Profinet_QRkod_Znaky[15] AT %IB."WenglorControl_Unit".Module021_Inputs048;
	Cyclic#1.CAM15.Profinet_QRkod_Znaky[16] AT %IB."WenglorControl_Unit".Module021_Inputs049;
	Cyclic#1.CAM15.Profinet_QRkod_Znaky[17] AT %IB."WenglorControl_Unit".Module021_Inputs050;
	Cyclic#1.CAM15.Profinet_QRkod_Znaky[18] AT %IB."WenglorControl_Unit".Module021_Inputs051;
	Cyclic#1.CAM15.Profinet_QRkod_Znaky[19] AT %IB."WenglorControl_Unit".Module021_Inputs052;
	Cyclic#1.CAM15.Profinet_QRkod_Znaky[20] AT %IB."WenglorControl_Unit".Module021_Inputs053;
	Cyclic#1.CAM15.Profinet_QRkod_Znaky[21] AT %IB."WenglorControl_Unit".Module021_Inputs054;
	Cyclic#1.CAM15.Profinet_QRkod_Znaky[22] AT %IB."WenglorControl_Unit".Module021_Inputs055;
	Cyclic#1.CAM15.Profinet_QRkod_Znaky[23] AT %IB."WenglorControl_Unit".Module021_Inputs056;
	Cyclic#1.CAM15.Profinet_QRkod_Znaky[24] AT %IB."WenglorControl_Unit".Module021_Inputs057;
	Cyclic#1.CAM15.Profinet_QRkod_Znaky[25] AT %IB."WenglorControl_Unit".Module021_Inputs058;
	Cyclic#1.CAM15.Profinet_QRkod_Znaky[26] AT %IB."WenglorControl_Unit".Module021_Inputs059;
	Cyclic#1.CAM15.Profinet_QRkod_Znaky[27] AT %IB."WenglorControl_Unit".Module021_Inputs060;
	Cyclic#1.CAM15.Profinet_QRkod_Znaky[28] AT %IB."WenglorControl_Unit".Module021_Inputs061;
	Cyclic#1.CAM15.Profinet_QRkod_Znaky[29] AT %IB."WenglorControl_Unit".Module021_Inputs062;
	Cyclic#1.CAM15.Profinet_QRkod_Znaky[30] AT %IB."WenglorControl_Unit".Module021_Inputs063;
	Cyclic#1.CAM15.Profinet_QRkod_Znaky[31] AT %IB."WenglorControl_Unit".Module021_Inputs064;
	Cyclic#1.CAM2.Profinet_PLC_OUTPUTS[0] AT %QB."WenglorControl_Unit".Module026_Outputs001;
	Cyclic#1.CAM4.Profinet_PLC_OUTPUTS[0] AT %QB."WenglorControl_Unit".Module027_Outputs001;
	Cyclic#1.CAM6.Profinet_PLC_OUTPUTS[0] AT %QB."WenglorControl_Unit".Module028_Outputs001;
	Cyclic#1.CAM1.Profinet_PLC_OUTPUTS[0] AT %QB."WenglorControl_Unit".Module029_Outputs001;
	Cyclic#1.CAM7.Profinet_PLC_OUTPUTS[0] AT %QB."WenglorControl_Unit".Module030_Outputs001;
	Cyclic#1.CAM17.Profinet_PLC_OUTPUTS[0] AT %QB."WenglorControl_Unit".Module031_Outputs001;
	Cyclic#1.CAM10.Profinet_PLC_OUTPUTS[0] AT %QB."WenglorControl_Unit".Module032_Outputs001;
	Cyclic#1.CAM11.Profinet_PLC_OUTPUTS[0] AT %QB."WenglorControl_Unit".Module033_Outputs001;
	Cyclic#1.CAM12.Profinet_PLC_OUTPUTS[0] AT %QB."WenglorControl_Unit".Module034_Outputs001;
	Cyclic#1.CAM15.Profinet_PLC_OUTPUTS[0] AT %QB."WenglorControl_Unit".Module035_Outputs001;
	Cyclic#1.CAM16.Profinet_PLC_OUTPUTS[0] AT %QB."WenglorControl_Unit".Module036_Outputs001;
	Cyclic#1.Safety.Mapping_BYTE_IN[16] AT %IB."P2_SafetyMaster".Module002_External_Output_status_EQ_byte_0;
	Cyclic#1.Safety.Mapping_BYTE_IN[17] AT %IB."P2_SafetyMaster".Module002_External_Output_status_EQ_byte_1;
	Cyclic#1.Safety.Mapping_BYTE_IN[18] AT %IB."P2_SafetyMaster".Module002_External_Output_status_EQ_byte_2;
	Cyclic#1.Safety.Mapping_BYTE_IN[19] AT %IB."P2_SafetyMaster".Module002_External_Output_status_EQ_byte_3;
	Cyclic#1.CAM3.Profinet_PLC_OUTPUTS[0] AT %QB."P1_CAM_3".Module003_Output_1_Byte;
	Cyclic#1.CAM3.Profinet_QRkod_Znaky[0] AT %IB."P1_CAM_3".Module004_Input_64_Byte001;
	Cyclic#1.CAM3.Profinet_QRkod_Znaky[1] AT %IB."P1_CAM_3".Module004_Input_64_Byte002;
	Cyclic#1.CAM3.Profinet_QRkod_Znaky[2] AT %IB."P1_CAM_3".Module004_Input_64_Byte003;
	Cyclic#1.CAM3.Profinet_QRkod_Znaky[3] AT %IB."P1_CAM_3".Module004_Input_64_Byte004;
	Cyclic#1.CAM3.Profinet_QRkod_Znaky[4] AT %IB."P1_CAM_3".Module004_Input_64_Byte005;
	Cyclic#1.CAM3.Profinet_QRkod_Znaky[5] AT %IB."P1_CAM_3".Module004_Input_64_Byte006;
	Cyclic#1.CAM3.Profinet_QRkod_Znaky[6] AT %IB."P1_CAM_3".Module004_Input_64_Byte007;
	Cyclic#1.CAM3.Profinet_QRkod_Znaky[7] AT %IB."P1_CAM_3".Module004_Input_64_Byte008;
	Cyclic#1.CAM3.Profinet_QRkod_Znaky[8] AT %IB."P1_CAM_3".Module004_Input_64_Byte009;
	Cyclic#1.CAM3.Profinet_QRkod_Znaky[9] AT %IB."P1_CAM_3".Module004_Input_64_Byte010;
	Cyclic#1.CAM3.Profinet_QRkod_Znaky[10] AT %IB."P1_CAM_3".Module004_Input_64_Byte011;
	Cyclic#1.CAM3.Profinet_QRkod_Znaky[11] AT %IB."P1_CAM_3".Module004_Input_64_Byte012;
	Cyclic#1.CAM3.Profinet_QRkod_Znaky[12] AT %IB."P1_CAM_3".Module004_Input_64_Byte013;
	Cyclic#1.CAM3.Profinet_QRkod_Znaky[13] AT %IB."P1_CAM_3".Module004_Input_64_Byte014;
	Cyclic#1.CAM3.Profinet_QRkod_Znaky[14] AT %IB."P1_CAM_3".Module004_Input_64_Byte015;
	Cyclic#1.CAM3.Profinet_QRkod_Znaky[15] AT %IB."P1_CAM_3".Module004_Input_64_Byte016;
	Cyclic#1.CAM3.Profinet_QRkod_Znaky[16] AT %IB."P1_CAM_3".Module004_Input_64_Byte017;
	Cyclic#1.CAM3.Profinet_QRkod_Znaky[17] AT %IB."P1_CAM_3".Module004_Input_64_Byte018;
	Cyclic#1.CAM3.Profinet_QRkod_Znaky[18] AT %IB."P1_CAM_3".Module004_Input_64_Byte019;
	Cyclic#1.CAM3.Profinet_QRkod_Znaky[19] AT %IB."P1_CAM_3".Module004_Input_64_Byte020;
	Cyclic#1.CAM3.Profinet_QRkod_Znaky[20] AT %IB."P1_CAM_3".Module004_Input_64_Byte021;
	Cyclic#1.CAM3.Profinet_QRkod_Znaky[21] AT %IB."P1_CAM_3".Module004_Input_64_Byte022;
	Cyclic#1.CAM3.Profinet_QRkod_Znaky[22] AT %IB."P1_CAM_3".Module004_Input_64_Byte023;
	Cyclic#1.CAM3.Profinet_QRkod_Znaky[23] AT %IB."P1_CAM_3".Module004_Input_64_Byte024;
	Cyclic#1.CAM3.Profinet_QRkod_Znaky[24] AT %IB."P1_CAM_3".Module004_Input_64_Byte025;
	Cyclic#1.CAM3.Profinet_QRkod_Znaky[25] AT %IB."P1_CAM_3".Module004_Input_64_Byte026;
	Cyclic#1.CAM3.Profinet_QRkod_Znaky[26] AT %IB."P1_CAM_3".Module004_Input_64_Byte027;
	Cyclic#1.CAM3.Profinet_QRkod_Znaky[27] AT %IB."P1_CAM_3".Module004_Input_64_Byte028;
	Cyclic#1.CAM3.Profinet_QRkod_Znaky[28] AT %IB."P1_CAM_3".Module004_Input_64_Byte029;
	Cyclic#1.CAM3.Profinet_QRkod_Znaky[29] AT %IB."P1_CAM_3".Module004_Input_64_Byte030;
	Cyclic#1.CAM3.Profinet_QRkod_Znaky[30] AT %IB."P1_CAM_3".Module004_Input_64_Byte031;
	Cyclic#1.CAM3.Profinet_QRkod_Znaky[31] AT %IB."P1_CAM_3".Module004_Input_64_Byte032;
	Cyclic#1.CAM3.Profinet_PLC_INPUTS[0] AT %IB."P1_CAM_3".Module005_Input_1_Byte;
	Cyclic#1.CAM3.Profinet_PLC_INPUTS[12] AT %IB."P1_CAM_3".Module006_Input_16_Byte012;
	Cyclic#1.CAM5.Profinet_PLC_OUTPUTS[0] AT %QB."P1_CAM_5".Module003_Output_1_Byte;
	Cyclic#1.CAM5.Profinet_QRkod_Znaky[0] AT %IB."P1_CAM_5".Module004_Input_64_Byte001;
	Cyclic#1.CAM5.Profinet_QRkod_Znaky[1] AT %IB."P1_CAM_5".Module004_Input_64_Byte002;
	Cyclic#1.CAM5.Profinet_QRkod_Znaky[2] AT %IB."P1_CAM_5".Module004_Input_64_Byte003;
	Cyclic#1.CAM5.Profinet_QRkod_Znaky[3] AT %IB."P1_CAM_5".Module004_Input_64_Byte004;
	Cyclic#1.CAM5.Profinet_QRkod_Znaky[4] AT %IB."P1_CAM_5".Module004_Input_64_Byte005;
	Cyclic#1.CAM5.Profinet_QRkod_Znaky[5] AT %IB."P1_CAM_5".Module004_Input_64_Byte006;
	Cyclic#1.CAM5.Profinet_QRkod_Znaky[6] AT %IB."P1_CAM_5".Module004_Input_64_Byte007;
	Cyclic#1.CAM5.Profinet_QRkod_Znaky[7] AT %IB."P1_CAM_5".Module004_Input_64_Byte008;
	Cyclic#1.CAM5.Profinet_QRkod_Znaky[8] AT %IB."P1_CAM_5".Module004_Input_64_Byte009;
	Cyclic#1.CAM5.Profinet_QRkod_Znaky[9] AT %IB."P1_CAM_5".Module004_Input_64_Byte010;
	Cyclic#1.CAM5.Profinet_QRkod_Znaky[10] AT %IB."P1_CAM_5".Module004_Input_64_Byte011;
	Cyclic#1.CAM5.Profinet_QRkod_Znaky[11] AT %IB."P1_CAM_5".Module004_Input_64_Byte012;
	Cyclic#1.CAM5.Profinet_QRkod_Znaky[12] AT %IB."P1_CAM_5".Module004_Input_64_Byte013;
	Cyclic#1.CAM5.Profinet_QRkod_Znaky[13] AT %IB."P1_CAM_5".Module004_Input_64_Byte014;
	Cyclic#1.CAM5.Profinet_QRkod_Znaky[14] AT %IB."P1_CAM_5".Module004_Input_64_Byte015;
	Cyclic#1.CAM5.Profinet_QRkod_Znaky[15] AT %IB."P1_CAM_5".Module004_Input_64_Byte016;
	Cyclic#1.CAM5.Profinet_QRkod_Znaky[16] AT %IB."P1_CAM_5".Module004_Input_64_Byte017;
	Cyclic#1.CAM5.Profinet_QRkod_Znaky[17] AT %IB."P1_CAM_5".Module004_Input_64_Byte018;
	Cyclic#1.CAM5.Profinet_QRkod_Znaky[18] AT %IB."P1_CAM_5".Module004_Input_64_Byte019;
	Cyclic#1.CAM5.Profinet_QRkod_Znaky[19] AT %IB."P1_CAM_5".Module004_Input_64_Byte020;
	Cyclic#1.CAM5.Profinet_QRkod_Znaky[20] AT %IB."P1_CAM_5".Module004_Input_64_Byte021;
	Cyclic#1.CAM5.Profinet_QRkod_Znaky[21] AT %IB."P1_CAM_5".Module004_Input_64_Byte022;
	Cyclic#1.CAM5.Profinet_QRkod_Znaky[22] AT %IB."P1_CAM_5".Module004_Input_64_Byte023;
	Cyclic#1.CAM5.Profinet_QRkod_Znaky[23] AT %IB."P1_CAM_5".Module004_Input_64_Byte024;
	Cyclic#1.CAM5.Profinet_QRkod_Znaky[24] AT %IB."P1_CAM_5".Module004_Input_64_Byte025;
	Cyclic#1.CAM5.Profinet_QRkod_Znaky[25] AT %IB."P1_CAM_5".Module004_Input_64_Byte026;
	Cyclic#1.CAM5.Profinet_QRkod_Znaky[26] AT %IB."P1_CAM_5".Module004_Input_64_Byte027;
	Cyclic#1.CAM5.Profinet_QRkod_Znaky[27] AT %IB."P1_CAM_5".Module004_Input_64_Byte028;
	Cyclic#1.CAM5.Profinet_QRkod_Znaky[28] AT %IB."P1_CAM_5".Module004_Input_64_Byte029;
	Cyclic#1.CAM5.Profinet_QRkod_Znaky[29] AT %IB."P1_CAM_5".Module004_Input_64_Byte030;
	Cyclic#1.CAM5.Profinet_QRkod_Znaky[30] AT %IB."P1_CAM_5".Module004_Input_64_Byte031;
	Cyclic#1.CAM5.Profinet_QRkod_Znaky[31] AT %IB."P1_CAM_5".Module004_Input_64_Byte032;
	Cyclic#1.CAM5.Profinet_PLC_INPUTS[0] AT %IB."P1_CAM_5".Module005_Input_1_Byte;
	Cyclic#1.CAM5.Profinet_PLC_INPUTS[12] AT %IB."P1_CAM_5".Module006_Input_16_Byte012;
	Cyclic#1.CAM14.Profinet_PLC_OUTPUTS[0] AT %QB."P4_CAM_14".Module003_Output_1_Byte;
	Cyclic#1.CAM14.Profinet_QRkod_Znaky[0] AT %IB."P4_CAM_14".Module004_Input_64_Byte001;
	Cyclic#1.CAM14.Profinet_QRkod_Znaky[1] AT %IB."P4_CAM_14".Module004_Input_64_Byte002;
	Cyclic#1.CAM14.Profinet_QRkod_Znaky[2] AT %IB."P4_CAM_14".Module004_Input_64_Byte003;
	Cyclic#1.CAM14.Profinet_QRkod_Znaky[3] AT %IB."P4_CAM_14".Module004_Input_64_Byte004;
	Cyclic#1.CAM14.Profinet_QRkod_Znaky[4] AT %IB."P4_CAM_14".Module004_Input_64_Byte005;
	Cyclic#1.CAM14.Profinet_QRkod_Znaky[5] AT %IB."P4_CAM_14".Module004_Input_64_Byte006;
	Cyclic#1.CAM14.Profinet_QRkod_Znaky[6] AT %IB."P4_CAM_14".Module004_Input_64_Byte007;
	Cyclic#1.CAM14.Profinet_QRkod_Znaky[7] AT %IB."P4_CAM_14".Module004_Input_64_Byte008;
	Cyclic#1.CAM14.Profinet_QRkod_Znaky[8] AT %IB."P4_CAM_14".Module004_Input_64_Byte009;
	Cyclic#1.CAM14.Profinet_QRkod_Znaky[9] AT %IB."P4_CAM_14".Module004_Input_64_Byte010;
	Cyclic#1.CAM14.Profinet_QRkod_Znaky[10] AT %IB."P4_CAM_14".Module004_Input_64_Byte011;
	Cyclic#1.CAM14.Profinet_QRkod_Znaky[11] AT %IB."P4_CAM_14".Module004_Input_64_Byte012;
	Cyclic#1.CAM14.Profinet_QRkod_Znaky[12] AT %IB."P4_CAM_14".Module004_Input_64_Byte013;
	Cyclic#1.CAM14.Profinet_QRkod_Znaky[13] AT %IB."P4_CAM_14".Module004_Input_64_Byte014;
	Cyclic#1.CAM14.Profinet_QRkod_Znaky[14] AT %IB."P4_CAM_14".Module004_Input_64_Byte015;
	Cyclic#1.CAM14.Profinet_QRkod_Znaky[15] AT %IB."P4_CAM_14".Module004_Input_64_Byte016;
	Cyclic#1.CAM14.Profinet_QRkod_Znaky[16] AT %IB."P4_CAM_14".Module004_Input_64_Byte017;
	Cyclic#1.CAM14.Profinet_QRkod_Znaky[17] AT %IB."P4_CAM_14".Module004_Input_64_Byte018;
	Cyclic#1.CAM14.Profinet_QRkod_Znaky[18] AT %IB."P4_CAM_14".Module004_Input_64_Byte019;
	Cyclic#1.CAM14.Profinet_QRkod_Znaky[19] AT %IB."P4_CAM_14".Module004_Input_64_Byte020;
	Cyclic#1.CAM14.Profinet_QRkod_Znaky[20] AT %IB."P4_CAM_14".Module004_Input_64_Byte021;
	Cyclic#1.CAM14.Profinet_QRkod_Znaky[21] AT %IB."P4_CAM_14".Module004_Input_64_Byte022;
	Cyclic#1.CAM14.Profinet_QRkod_Znaky[22] AT %IB."P4_CAM_14".Module004_Input_64_Byte023;
	Cyclic#1.CAM14.Profinet_QRkod_Znaky[23] AT %IB."P4_CAM_14".Module004_Input_64_Byte024;
	Cyclic#1.CAM14.Profinet_QRkod_Znaky[24] AT %IB."P4_CAM_14".Module004_Input_64_Byte025;
	Cyclic#1.CAM14.Profinet_QRkod_Znaky[25] AT %IB."P4_CAM_14".Module004_Input_64_Byte026;
	Cyclic#1.CAM14.Profinet_QRkod_Znaky[26] AT %IB."P4_CAM_14".Module004_Input_64_Byte027;
	Cyclic#1.CAM14.Profinet_QRkod_Znaky[27] AT %IB."P4_CAM_14".Module004_Input_64_Byte028;
	Cyclic#1.CAM14.Profinet_QRkod_Znaky[28] AT %IB."P4_CAM_14".Module004_Input_64_Byte029;
	Cyclic#1.CAM14.Profinet_QRkod_Znaky[29] AT %IB."P4_CAM_14".Module004_Input_64_Byte030;
	Cyclic#1.CAM14.Profinet_QRkod_Znaky[30] AT %IB."P4_CAM_14".Module004_Input_64_Byte031;
	Cyclic#1.CAM14.Profinet_QRkod_Znaky[31] AT %IB."P4_CAM_14".Module004_Input_64_Byte032;
	Cyclic#1.CAM14.Profinet_PLC_INPUTS[0] AT %IB."P4_CAM_14".Module005_Input_1_Byte;
	Cyclic#1.CAM14.Profinet_PLC_INPUTS[4] AT %IB."P4_CAM_14".Module006_Input_16_Byte004;
	Cyclic#1.CAM14.Profinet_PLC_INPUTS[12] AT %IB."P4_CAM_14".Module006_Input_16_Byte012;
	Cyclic#1.CAM9.Profinet_PLC_OUTPUTS[0] AT %QB."P2_CAM_9".Module003_Output_1_Byte;
	Cyclic#1.CAM9.Profinet_PLC_INPUTS[0] AT %IB."P2_CAM_9".Module005_Input_1_Byte;
	Cyclic#1.CAM9.Profinet_PLC_INPUTS[12] AT %IB."P2_CAM_9".Module006_Input_16_Byte012;
	Cyclic#1.CAM8.Profinet_PLC_OUTPUTS[0] AT %QB."P2_CAM_8".Module003_Output_1_Byte;
	Cyclic#1.CAM8.Profinet_QRkod_Znaky[0] AT %IB."P2_CAM_8".Module004_Input_64_Byte001;
	Cyclic#1.CAM8.Profinet_QRkod_Znaky[1] AT %IB."P2_CAM_8".Module004_Input_64_Byte002;
	Cyclic#1.CAM8.Profinet_QRkod_Znaky[2] AT %IB."P2_CAM_8".Module004_Input_64_Byte003;
	Cyclic#1.CAM8.Profinet_QRkod_Znaky[3] AT %IB."P2_CAM_8".Module004_Input_64_Byte004;
	Cyclic#1.CAM8.Profinet_QRkod_Znaky[4] AT %IB."P2_CAM_8".Module004_Input_64_Byte005;
	Cyclic#1.CAM8.Profinet_QRkod_Znaky[5] AT %IB."P2_CAM_8".Module004_Input_64_Byte006;
	Cyclic#1.CAM8.Profinet_QRkod_Znaky[6] AT %IB."P2_CAM_8".Module004_Input_64_Byte007;
	Cyclic#1.CAM8.Profinet_QRkod_Znaky[7] AT %IB."P2_CAM_8".Module004_Input_64_Byte008;
	Cyclic#1.CAM8.Profinet_QRkod_Znaky[8] AT %IB."P2_CAM_8".Module004_Input_64_Byte009;
	Cyclic#1.CAM8.Profinet_QRkod_Znaky[9] AT %IB."P2_CAM_8".Module004_Input_64_Byte010;
	Cyclic#1.CAM8.Profinet_QRkod_Znaky[10] AT %IB."P2_CAM_8".Module004_Input_64_Byte011;
	Cyclic#1.CAM8.Profinet_QRkod_Znaky[11] AT %IB."P2_CAM_8".Module004_Input_64_Byte012;
	Cyclic#1.CAM8.Profinet_QRkod_Znaky[12] AT %IB."P2_CAM_8".Module004_Input_64_Byte013;
	Cyclic#1.CAM8.Profinet_QRkod_Znaky[13] AT %IB."P2_CAM_8".Module004_Input_64_Byte014;
	Cyclic#1.CAM8.Profinet_QRkod_Znaky[14] AT %IB."P2_CAM_8".Module004_Input_64_Byte015;
	Cyclic#1.CAM8.Profinet_QRkod_Znaky[15] AT %IB."P2_CAM_8".Module004_Input_64_Byte016;
	Cyclic#1.CAM8.Profinet_QRkod_Znaky[16] AT %IB."P2_CAM_8".Module004_Input_64_Byte017;
	Cyclic#1.CAM8.Profinet_QRkod_Znaky[17] AT %IB."P2_CAM_8".Module004_Input_64_Byte018;
	Cyclic#1.CAM8.Profinet_QRkod_Znaky[18] AT %IB."P2_CAM_8".Module004_Input_64_Byte019;
	Cyclic#1.CAM8.Profinet_QRkod_Znaky[19] AT %IB."P2_CAM_8".Module004_Input_64_Byte020;
	Cyclic#1.CAM8.Profinet_QRkod_Znaky[20] AT %IB."P2_CAM_8".Module004_Input_64_Byte021;
	Cyclic#1.CAM8.Profinet_QRkod_Znaky[21] AT %IB."P2_CAM_8".Module004_Input_64_Byte022;
	Cyclic#1.CAM8.Profinet_QRkod_Znaky[22] AT %IB."P2_CAM_8".Module004_Input_64_Byte023;
	Cyclic#1.CAM8.Profinet_QRkod_Znaky[23] AT %IB."P2_CAM_8".Module004_Input_64_Byte024;
	Cyclic#1.CAM8.Profinet_QRkod_Znaky[24] AT %IB."P2_CAM_8".Module004_Input_64_Byte025;
	Cyclic#1.CAM8.Profinet_QRkod_Znaky[25] AT %IB."P2_CAM_8".Module004_Input_64_Byte026;
	Cyclic#1.CAM8.Profinet_QRkod_Znaky[26] AT %IB."P2_CAM_8".Module004_Input_64_Byte027;
	Cyclic#1.CAM8.Profinet_QRkod_Znaky[27] AT %IB."P2_CAM_8".Module004_Input_64_Byte028;
	Cyclic#1.CAM8.Profinet_QRkod_Znaky[28] AT %IB."P2_CAM_8".Module004_Input_64_Byte029;
	Cyclic#1.CAM8.Profinet_QRkod_Znaky[29] AT %IB."P2_CAM_8".Module004_Input_64_Byte030;
	Cyclic#1.CAM8.Profinet_QRkod_Znaky[30] AT %IB."P2_CAM_8".Module004_Input_64_Byte031;
	Cyclic#1.CAM8.Profinet_QRkod_Znaky[31] AT %IB."P2_CAM_8".Module004_Input_64_Byte032;
	Cyclic#1.CAM8.Profinet_PLC_INPUTS[0] AT %IB."P2_CAM_8".Module005_Input_1_Byte;
	Cyclic#1.CAM8.Profinet_PLC_INPUTS[12] AT %IB."P2_CAM_8".Module006_Input_16_Byte012;
	Cyclic#1.CAM7.Profinet_PLC_INPUTS[0] AT %IB."WenglorControl_Unit".Module010_Inputs001;
	Cyclic#1.CAM7.Profinet_PLC_INPUTS[1] AT %IB."WenglorControl_Unit".Module010_Inputs002;
	Cyclic#1.CAM7.Profinet_PLC_INPUTS[2] AT %IB."WenglorControl_Unit".Module010_Inputs003;
	Cyclic#1.CAM7.Profinet_PLC_INPUTS[3] AT %IB."WenglorControl_Unit".Module010_Inputs004;
	Cyclic#1.CAM2.STAV.RunCounter_Byte0 AT %IB."WenglorControl_Unit".Module002_Inputs031;
	Cyclic#1.CAM2.STAV.RunCounter_Byte1  AT %IB."WenglorControl_Unit".Module002_Inputs032;
	Cyclic#1.CAM3.STAV.RunCounter_Byte0 AT %IB."P1_CAM_3".Module006_Input_16_Byte007;
	Cyclic#1.CAM3.STAV.RunCounter_Byte1  AT %IB."P1_CAM_3".Module006_Input_16_Byte008;
	Cyclic#1.CAM5.STAV.RunCounter_Byte0 AT %IB."P1_CAM_5".Module006_Input_16_Byte007;
	Cyclic#1.CAM5.STAV.RunCounter_Byte1  AT %IB."P1_CAM_5".Module006_Input_16_Byte008;
	Cyclic#1.CAM14.STAV.RunCounter_Byte0 AT %IB."P4_CAM_14".Module006_Input_16_Byte007;
	Cyclic#1.CAM14.STAV.RunCounter_Byte1  AT %IB."P4_CAM_14".Module006_Input_16_Byte008;
	Cyclic#1.CAM8.STAV.RunCounter_Byte0 AT %IB."P2_CAM_8".Module006_Input_16_Byte007;
	Cyclic#1.CAM8.STAV.RunCounter_Byte1  AT %IB."P2_CAM_8".Module006_Input_16_Byte008;
	Cyclic#1.CAM9.STAV.RunCounter_Byte0 AT %IB."P2_CAM_9".Module006_Input_16_Byte007;
	Cyclic#1.CAM9.STAV.RunCounter_Byte1  AT %IB."P2_CAM_9".Module006_Input_16_Byte008;
	Cyclic#1.CAM4.STAV.RunCounter_Byte0 AT %IB."WenglorControl_Unit".Module004_Inputs031;
	Cyclic#1.CAM4.STAV.RunCounter_Byte1  AT %IB."WenglorControl_Unit".Module004_Inputs032;
	Cyclic#1.CAM6.STAV.RunCounter_Byte0  AT %IB."WenglorControl_Unit".Module006_Inputs031;
	Cyclic#1.CAM6.STAV.RunCounter_Byte1  AT %IB."WenglorControl_Unit".Module006_Inputs032;
	Cyclic#1.CAM1.STAV.RunCounter_Byte0  AT %IB."WenglorControl_Unit".Module008_Inputs031;
	Cyclic#1.CAM1.STAV.RunCounter_Byte1  AT %IB."WenglorControl_Unit".Module008_Inputs032;
	Cyclic#1.CAM7.STAV.RunCounter_Byte0   AT %IB."WenglorControl_Unit".Module010_Inputs031;
	Cyclic#1.CAM7.STAV.RunCounter_Byte1  AT %IB."WenglorControl_Unit".Module010_Inputs032;
	Cyclic#1.CAM17.STAV.RunCounter_Byte0   AT %IB."WenglorControl_Unit".Module012_Inputs031;
	Cyclic#1.CAM17.STAV.RunCounter_Byte1  AT %IB."WenglorControl_Unit".Module012_Inputs032;
	Cyclic#1.CAM10.STAV.RunCounter_Byte0    AT %IB."WenglorControl_Unit".Module015_Inputs031;
	Cyclic#1.CAM10.STAV.RunCounter_Byte1  AT %IB."WenglorControl_Unit".Module015_Inputs032;
	Cyclic#1.CAM11.STAV.RunCounter_Byte0    AT %IB."WenglorControl_Unit".Module017_Inputs031;
	Cyclic#1.CAM11.STAV.RunCounter_Byte1  AT %IB."WenglorControl_Unit".Module017_Inputs032;
	Cyclic#1.CAM12.STAV.RunCounter_Byte0     AT %IB."WenglorControl_Unit".Module019_Inputs031;
	Cyclic#1.CAM12.STAV.RunCounter_Byte1  AT %IB."WenglorControl_Unit".Module019_Inputs032;
	Cyclic#1.CAM15.STAV.RunCounter_Byte0      AT %IB."WenglorControl_Unit".Module021_Inputs031;
	Cyclic#1.CAM15.STAV.RunCounter_Byte1  AT %IB."WenglorControl_Unit".Module021_Inputs032;
	Cyclic#1.CAM16.STAV.RunCounter_Byte0       AT %IB."WenglorControl_Unit".Module023_Inputs031;
	Cyclic#1.CAM16.STAV.RunCounter_Byte1  AT %IB."WenglorControl_Unit".Module023_Inputs032;
END_VAR
```
